(* CODESYS project 20260622.project

Project tree, tasks and I/O mapping:
  Device : AM522-0808TP/TN, Shenzhen Inovance Control Technology, version 3.5.11.50
      settings: PersistentStartAdddr = 0; PersistentStartEndAddr = 524287; Mode = 1; OPC UA Mode = 0
    application Application
      libraries: Standard, * (System); CmpEventMgr, 3.5.8.0 (System); Component Manager, 3.5.9.0 (System); CmpApp, 3.5.11.0 (System); CmpIecTask, 3.5.9.0 (System); SM3_Math, 4.10.0.0 (3S - Smart Software Solutions GmbH); SM3_Math, 4.10.0.0 (3S - Smart Software Solutions GmbH); HC_OmronUtils, 1.5.8.0 (Inovance); SM3_Basic, 4.10.13.1 (3S - Smart Software Solutions GmbH)
      task MainTask (cyclic, interval 10 ms, priority 1) calls PLC_MainPRG
      task ETHERCAT1 (cyclic, interval 4000 µs, priority 0) calls ETHERCAT1.EtherCAT_Task, PLC_Servo_伺服, PLC_HandWheel_手轮, PLC_CNC
      50_action/
        program PLC_Pump_泵管理 [ST]
        program PhotoScrape_L2 [ST]: A10_init_初始化, A32_cam_定位, A35_cam_回零, A34_cam_相机位, A33_cam_下压, A31_cam_移轴335, A40_scrape_刮取, A52_取料停旋转, A51_取料松压, A41_scrape_收尾
        program FeedLift_L2 [ST]: A11_feed_raise, A22_unload_bury, A12_feed_lower, A21_unload_ready
        program Sampling_L2 [ST]: A50_absorb_吸收液体, A31_放板移轴, A40_prep_上样准备, A32_放板定位, A20_clean_清洗, A10_init_初始化, A60_spray_点样, A61_喷涂移轴
        program Collect_L2 [ST]: A23_缩回升降下压, A22_伸缩伸出, A21_夹持夹紧, A30_collect_收集, A10_init_初始化, A42_伸缩缩回, A41_复位伸出, A43_松夹持
        program Rail_Sync [ST]
        program Rail_L2 [ST]
        program Develop_L2 [ST]: A31_放板缸回原点, A21_rinse_润洗展缸, A20_pipeline_清洗管路, A32_放板缸到动点, A22_up_liquid_上液, A10_init_初始化, A26_rinse_suction
        program Pump_L2 [ST]: A10_vacuum_on, A20_vacuum_off
      DifferentialMonitor
      25_FB_功能块/
        function block FB_Teach [ST]
        function block FB_SERVOAXIS [ST]
        function block FB_cylinder [ST]
        function block FB_HandWheel [ST]
        function block FB_RB_Control [ST]
        function block FB_Mode [ST]
      10_数据结构/
        data type HMI_Servo
        data type servo
        data type EN_功能块状态
      Symbols
      30_Ethercat任务/
        program PLC_Servo_伺服 [ST]: 伺服一键回原点, 伺服调用, 位置示教
        program PLC_CNC [CFC]
        program PLC_HandWheel_手轮 [ST]
      global variables PersistentVars
      20_变量Date/
        global variables HMI_Date
        global variables cyinder_date
        global variables IO
        global variables servoaxisdate
        global variables GVL
        global variables Host_Computer
        global variables RB_Date
      trace Trace (task ETHERCAT1): 玻璃上料轴1ZDATE.fActPos, 玻璃上料轴1ZDATE.fActVel
      CNC设置
      TaskEventPreStart
      text CNC_1
      40_Man/
        program Expand_process_展开流程 [ST]: Develop_L2_Dispatch, A00_initialization_初始化, A10_pipeline_cleaning_清洗管路, A20_clean_expand_润洗展缸, A40_up_liquid_上液, A30_silica_gel_plate_放硅胶板
        program Robotic_Process_机器人流程 [ST]: A30_取展缸硅胶板, A60_取收集器放暂存工位, A00_取放工具, A35_放拍照硅胶板, A65_放废料硅胶板, A41_取收集瓶组放暂存工位, A40_取收集器组放暂存工位, A15_放点样硅胶板, A55_取刮板收集器放到收集工位, A45_取暂存收集器放刮板位, A20_取点样硅胶板, A25_放展缸硅胶板, A50_取暂存收集瓶放收集工位, A71_取暂存收集瓶放仓库, A65_取收集瓶放暂存工位, A10_取升降机硅胶板, A70_取暂存收集器组放仓库, A32_取拍照硅胶板
        program Sample_point_sampling_上样点样 [ST]: A20_Place_materials_放硅胶板, A30_Sample_preparation_上样准备, A00_initialization_初始化, A50_Spray_sample_点样, A40_absorb_liquid_吸收液体, Sampling_L2_Dispatch, A10_clean_清洗
        program Collection_process_收集流程 [ST]: A20_collect_收集, A00_initialization_初始化, Collect_L2_Dispatch, A30_transport_物料搬运, A10_preparation_准备
        program PLC_MainPRG [ST]: A10_上下料伺服流程, A00_设备状态显示及控制, A20_机器人, A30_急停
        program initialization [ST]
        program Develop_TankDrain [ST]: A50_Expand_liquid_discharge_排液
        program Photo_scraper_拍照刮板 [ST]: A00_initialization_初始化, A10_Material_camera_拍照硅胶板, PhotoScrape_L2_Dispatch, A20_Scraper_collection_刮板收集, A30_Robot_material_retrieval_机器人取粉末收集器
        program PLC_Cyinder_气缸动作 [ST]
    ConfigStorage
    Network Configuration
      EtherCAT Config
      LocalBus Config
    Resources List
    HardWare Configuration
    Device Diagnosis
    EXP_A : 扩展卡, 汇川技术股份有限公司, version 00.00.00.10
    LocalHSIO : 本地高速IO, 汇川技术股份有限公司, version 2.0.0.0
        unmapped channels: %IB0 DigitalInput, DigitalOutput
      Counter0 : 高速计数器, 汇川技术股份有限公司, version 1.0.0.0
          settings: GeneralConfiguration.Value = 25; SignalSource.Value = 3; ResetPin.Value = 138; PresetPin.Value = 14; PositionComparePin.Value = 2; TouchProbePin1.Value = 10; TouchProbePin2.Value = 12
          unmapped channels: Statusword, Counter Value, Preset Status, Compare Status, Touch Probe Status1, Touch Probe Status2, Latch rising pos1, Latch rising pos2, Latch falling pos1, Latch falling pos2, Latch rising time1 low, Latch rising time1 high, Latch rising time2 low, Latch rising time2 high, Latch falling time1 low, Latch falling time1 high, Latch falling time2 low, Latch falling time2 high, Current frequency, ErrorCode, Controlword, Preset Value, Preset command, Compare Mode, Compare Parameter, Compare Value, Output Type, Output Parameter, Compare command, Touch probe command1, Touch probe command2
        Encoder : 编码器, 汇川技术股份有限公司, version 1.0.0.0
            settings: wDriveID = 0; 5050 = 10; Units = 1; LogicId = 0; AdrOffset_8010 = 64; BitOffset_8010 = 0; BitLength_8010 = 16; Address_ = '%QW32'; TYPE_ = 'WORD'; Address_Pointer = ADR(%QW32); AdrOffset_8020 = 72; BitOffset_8020 = 0; BitLength_8020 = 16; Address_ = '%QW36'; TYPE_ = 'WORD'; Address_Pointer = ADR(%QW36); AdrOffset_8030 = 68; BitOffset_8030 = 0; BitLength_8030 = 32; Address_ = '%QD17'; TYPE_ = 'DWORD'; Address_Pointer = ADR(%QD17); AdrOffset_8040 = 88; BitOffset_8040 = 0; BitLength_8040 = 16; Address_ = '%QW44'; TYPE_ = 'WORD'; Address_Pointer = ADR(%QW44); AdrOffset_8050 = 74; BitOffset_8050 = 0; BitLength_8050 = 16; Address_ = '%QW37'; TYPE_ = 'WORD'; Address_Pointer = ADR(%QW37); AdrOffset_8060 = 76; BitOffset_8060 = 0; BitLength_8060 = 32; Address_ = '%QD19'; TYPE_ = 'DWORD'; Address_Pointer = ADR(%QD19);
              AdrOffset_8070 = 80; BitOffset_8070 = 0; BitLength_8070 = 32; Address_ = '%QD20'; TYPE_ = 'DWORD'; Address_Pointer = ADR(%QD20); AdrOffset_8080 = 84; BitOffset_8080 = 0; BitLength_8080 = 16; Address_ = '%QW42'; TYPE_ = 'WORD'; Address_Pointer = ADR(%QW42); AdrOffset_8090 = 86; BitOffset_8090 = 0; BitLength_8090 = 16; Address_ = '%QW43'; TYPE_ = 'WORD'; Address_Pointer = ADR(%QW43); AdrOffset_8100 = 90; BitOffset_8100 = 0; BitLength_8100 = 16; Address_ = '%QW45'; TYPE_ = 'WORD'; Address_Pointer = ADR(%QW45); AdrOffset_8110 = 92; BitOffset_8110 = 0; BitLength_8110 = 16; Address_ = '%QW46'; TYPE_ = 'WORD'; Address_Pointer = ADR(%QW46); AdrOffset_8510 = 104; BitOffset_8510 = 0; BitLength_8510 = 16; Address_ = '%IW52'; TYPE_ = 'WORD'; Address_Pointer = ADR(%IW52); AdrOffset_8520 = 108; BitOffset_8520 = 0; BitLength_8520 = 32; Address_ = '%ID27';
              TYPE_ = 'DWORD'; Address_Pointer = ADR(%ID27); AdrOffset_8530 = 112; BitOffset_8530 = 0; BitLength_8530 = 16; Address_ = '%IW56'; TYPE_ = 'WORD'; Address_Pointer = ADR(%IW56); AdrOffset_8540 = 114; BitOffset_8540 = 0; BitLength_8540 = 16; Address_ = '%IW57'; TYPE_ = 'WORD'; Address_Pointer = ADR(%IW57); AdrOffset_8550 = 116; BitOffset_8550 = 0; BitLength_8550 = 16; Address_ = '%IW58'; TYPE_ = 'WORD'; Address_Pointer = ADR(%IW58); AdrOffset_8560 = 118; BitOffset_8560 = 0; BitLength_8560 = 16; Address_ = '%IW59'; TYPE_ = 'WORD'; Address_Pointer = ADR(%IW59); AdrOffset_8570 = 120; BitOffset_8570 = 0; BitLength_8570 = 32; Address_ = '%ID30'; TYPE_ = 'DWORD'; Address_Pointer = ADR(%ID30); AdrOffset_8580 = 124; BitOffset_8580 = 0; BitLength_8580 = 32; Address_ = '%ID31'; TYPE_ = 'DWORD'; Address_Pointer = ADR(%ID31); AdrOffset_8590 = 128; BitOffset_8590 = 0;
              BitLength_8590 = 32; Address_ = '%ID32'; TYPE_ = 'DWORD'; Address_Pointer = ADR(%ID32); AdrOffset_8600 = 132; BitOffset_8600 = 0; BitLength_8600 = 32; Address_ = '%ID33'; TYPE_ = 'DWORD'; Address_Pointer = ADR(%ID33); AdrOffset_8610 = 136; BitOffset_8610 = 0; BitLength_8610 = 32; Address_ = '%ID34'; TYPE_ = 'DWORD'; Address_Pointer = ADR(%ID34); AdrOffset_8620 = 140; BitOffset_8620 = 0; BitLength_8620 = 32; Address_ = '%ID35'; TYPE_ = 'DWORD'; Address_Pointer = ADR(%ID35); AdrOffset_8630 = 144; BitOffset_8630 = 0; BitLength_8630 = 32; Address_ = '%ID36'; TYPE_ = 'DWORD'; Address_Pointer = ADR(%ID36); AdrOffset_8640 = 148; BitOffset_8640 = 0; BitLength_8640 = 32; Address_ = '%ID37'; TYPE_ = 'DWORD'; Address_Pointer = ADR(%ID37); AdrOffset_8650 = 152; BitOffset_8650 = 0; BitLength_8650 = 32; Address_ = '%ID38'; TYPE_ = 'DWORD'; Address_Pointer = ADR(%ID38);
              AdrOffset_8660 = 156; BitOffset_8660 = 0; BitLength_8660 = 32; Address_ = '%ID39'; TYPE_ = 'DWORD'; Address_Pointer = ADR(%ID39); AdrOffset_8670 = 160; BitOffset_8670 = 0; BitLength_8670 = 32; Address_ = '%ID40'; TYPE_ = 'DWORD'; Address_Pointer = ADR(%ID40); AdrOffset_8680 = 164; BitOffset_8680 = 0; BitLength_8680 = 32; Address_ = '%ID41'; TYPE_ = 'DWORD'; Address_Pointer = ADR(%ID41); AdrOffset_8690 = 168; BitOffset_8690 = 0; BitLength_8690 = 32; Address_ = '%ID42'; TYPE_ = 'DWORD'; Address_Pointer = ADR(%ID42); AdrOffset_8700 = 172; BitOffset_8700 = 0; BitLength_8700 = 32; Address_ = '%ID43'; TYPE_ = 'DWORD'; Address_Pointer = ADR(%ID43)
    Serial : 串行接口, 汇川技术股份有限公司, version 00.00.00.10
      COM : Serial Port, Inovance, version 00.00.00.10
          settings: Device = AM522-0808TP/TN; devGuid = 'ea0913c2-01c3-4246-ae88-1c6b39cb02f1'
        串口自由协议 : 串口自由协议, inovance, version 00.00.00.10
            settings: Vendor.parameterset.Bit7 = FALSE; slave device set.RxCount = 1000; slave device set.RxAddrNum = 1001; slave device set.TxCount = 1300; slave device set.TxAddrNum = 1301
    EXP_B : 扩展卡, 汇川技术股份有限公司, version 00.00.00.10
    MODBUS_TCP_1 : ModbusTCP主站, inovance, version 00.00.00.10
        settings:  = 0
      modbusTcp : ModbusTCP Slave, Inovance, version 00.00.00.10 (disabled)
          settings: UseDec = True; ModbusTcpSlave.ChannelNum = 4; ModbusTcpSlave.EnableSlaveVariable = 3001; ModbusTcpSlave.IpAddr = 251701440; channel.PremeterSet.Bit2 = TRUE; channel.PremeterSet.Bit3 = TRUE; channel.PremeterSet.Bit4 = TRUE; channel.CycleTimes = 200; channel.ReadRegOffSet = 0; channel.WriteRegOffSet = 3100; channel.WriteRegLeg = 13; channel.IOChannel = 0; channel.ResendCount = 5; channel.ChannelName = 'write'; channel.ChannelNote = ''; channel.PremeterSet.Bit3 = TRUE; channel.CycleTimes = 200; channel.ReadRegOffSet = 3200; channel.ReadRegLeg = 13; channel.WriteRegOffSet = 0; channel.ResendCount = 5; channel.ChannelName = 'read'; channel.ChannelNote = ''; channel.PremeterSet.Bit2 = TRUE; channel.CycleTimes = 200; channel.ReadRegOffSet = 0; channel.ReadRegLeg = 12; channel.WriteRegOffSet = 0; channel.IOChannel = 2; channel.ResendCount = 5; channel.ChannelName = 'read_bool'; channel.ChannelNote = ''; channel.PremeterSet.Bit3 = TRUE; channel.PremeterSet.Bit4 = TRUE; channel.CycleTimes = 200; channel.ReadRegOffSet = 0; channel.WriteRegOffSet = 0; channel.WriteRegLeg = 7; channel.IOChannel = 3; channel.ResendCount = 5;
            channel.ChannelName = 'write_bool'; channel.ChannelNote = ''
          input  Application.Status : WORD  // read.read
          input  Application.Point : WORD  // read.read
          input  Application.ErrorID : WORD  // read.read
          input  Application.RO_ParameterList1 : WORD  // read.read
          input  Application.RO_ParameterList2 : WORD  // read.read
          input  Application.RO_ParameterList3 : WORD  // read.read
          input  Application.RO_ParameterList4 : WORD  // read.read
          input  Application.RO_ParameterList5 : WORD  // read.read
          input  Application.RO_ParameterList6 : WORD  // read.read
          input  Application.RO_ParameterList7 : WORD  // read.read
          input  Application.RO_ParameterList8 : WORD  // read.read
          input  Application.RO_ParameterList9 : WORD  // read.read
          input  Application.RO_ParameterList10 : WORD  // read.read
          output Application.Execute : WORD  // write.write
          output Application.Reset : WORD  // write.write
          output Application.FunctionID : WORD  // write.write
          output Application.ParameterList1 : WORD  // write.write
          output Application.ParameterList2 : WORD  // write.write
          output Application.ParameterList3 : WORD  // write.write
          output Application.ParameterList4 : WORD  // write.write
          output Application.ParameterList5 : WORD  // write.write
          output Application.ParameterList6 : WORD  // write.write
          output Application.ParameterList7 : WORD  // write.write
          output Application.ParameterList8 : WORD  // write.write
          output Application.ParameterList9 : WORD  // write.write
          output Application.ParameterList10 : WORD  // write.write
          unmapped channels: read, read_bool, write, write_bool
    ETHERCAT1 : EtherCAT Master SoftMotion, 3S - Smart Software Solutions GmbH, version 3.5.11.10
        settings:  = 0; NetworkName = 'eth1'; SelectNetworkByName = TRUE; DisableTaskGeneration = True; SyncOffset = 50; SlaveArrayName = ADR(_EC1_Node)
      InoSV660N_3 : SV660_1Axis_00915, Inovance, order no. InoSV660N, version Revision=16#00010000
          settings: FunCodeList = H02;H02-01;; WriteValueList = H02-01_8194_2_1_UINT_RW;; Number of Outputs = 6; Number of Inputs = 10; Number of Infos about Outputs = 6; Number of Infos about Inputs = 10; Configuration address of the slave = 5; Sync.Length = 18; Sync.Length = 32; FMMU.Length = 18; FMMU.Length = 32; AutoUpdate = False; DC sync0 cycletime = 4000; DC sync1 cycletime = 4000; Number of SDO = 10; Homing method.Index = 16#6098; Homing method.Subindex = 16#00; Homing method.Value = 27; Homing method.Size = 8; Homing method.AbortIfError = FALSE; Homing method.JumpToLine = FALSE; Homing method.Line = 0; Homing method.CompleteAccess = FALSE; Actual Position Calculation Method.Index = 16#60E6; Actual Position Calculation Method.Subindex = 16#00; Actual Position Calculation Method.Value = 0; Actual Position Calculation Method.Size = 8; Actual Position Calculation Method.AbortIfError = FALSE; Actual Position Calculation Method.JumpToLine = FALSE; Actual Position Calculation Method.Line = 0; Actual Position Calculation Method.CompleteAccess = FALSE; Speed during search for switch.Index = 16#6099; Speed during search for switch.Subindex = 16#01; Speed during search for switch.Value = 83886080; Speed during search for switch.Size = 32; Speed during search for switch.AbortIfError = FALSE; Speed during search for switch.JumpToLine = FALSE; Speed during search for switch.Line = 0; Speed during search for switch.CompleteAccess = FALSE; Homing acceleration.Index = 16#609A;
            Homing acceleration.Subindex = 16#00; Homing acceleration.Value = 279620266; Homing acceleration.Size = 32; Homing acceleration.AbortIfError = FALSE; Homing acceleration.JumpToLine = FALSE; Homing acceleration.Line = 0; Homing acceleration.CompleteAccess = FALSE; Speed during search for zero.Index = 16#6099; Speed during search for zero.Subindex = 16#02; Speed during search for zero.Value = 33554432; Speed during search for zero.Size = 32; Speed during search for zero.AbortIfError = FALSE; Speed during search for zero.JumpToLine = FALSE; Speed during search for zero.Line = 0; Speed during search for zero.CompleteAccess = FALSE; Time of home searching.Index = 16#2005; Time of home searching.Subindex = 16#24; Time of home searching.Value = 50000; Time of home searching.Size = 16; Time of home searching.AbortIfError = FALSE; Time of home searching.JumpToLine = FALSE; Time of home searching.Line = 0; Time of home searching.CompleteAccess = FALSE; Positive torque limit value.Index = 16#60E0; Positive torque limit value.Subindex = 16#00; Positive torque limit value.Value = 3500; Positive torque limit value.Size = 16; Positive torque limit value.AbortIfError = FALSE; Positive torque limit value.JumpToLine = FALSE; Positive torque limit value.Line = 0; Positive torque limit value.CompleteAccess = FALSE; Negative torque limit value.Index = 16#60E1; Negative torque limit value.Subindex = 16#00; Negative torque limit value.Value = 3500; Negative torque limit value.Size = 16; Negative torque limit value.AbortIfError = FALSE; Negative torque limit value.JumpToLine = FALSE; Negative torque limit value.Line = 0; Negative torque limit value.CompleteAccess = FALSE; Max profile velocity.Index = 16#607F;
            Max profile velocity.Subindex = 16#00; Max profile velocity.Value = 167772160; Max profile velocity.Size = 32; Max profile velocity.AbortIfError = FALSE; Max profile velocity.JumpToLine = FALSE; Max profile velocity.Line = 0; Max profile velocity.CompleteAccess = FALSE; RxTxPdo.NumberofEntries = 6; RxTxPdo.Sm = 2; Controlword.Index = 16#6040; Controlword.SubIndex = 0; Controlword.Size = 16; Controlword.DependOnSlot = false; Controlword.DependOnSlotGroup = false; Target position.Index = 16#607A; Target position.SubIndex = 0; Target position.Size = 32; Target position.DependOnSlot = false; Target position.DependOnSlotGroup = false; Touch probe function.Index = 16#60B8; Touch probe function.SubIndex = 0; Touch probe function.Size = 16; Touch probe function.DependOnSlot = false; Touch probe function.DependOnSlotGroup = false; Physical outputs.Index = 16#60FE; Physical outputs.SubIndex = 1; Physical outputs.Size = 32; Physical outputs.DependOnSlot = false; Physical outputs.DependOnSlotGroup = false; Target velocity.Index = 16#60FF; Target velocity.SubIndex = 0; Target velocity.Size = 32; Target velocity.DependOnSlot = false; Target velocity.DependOnSlotGroup = false; Target torque.Index = 16#6071; Target torque.SubIndex = 0; Target torque.Size = 16; Target torque.DependOnSlot = false; Target torque.DependOnSlotGroup = false; RxTxPdo.Sm = -1;
            RxTxPdo.NumberofEntries = 10; RxTxPdo.Sm = 3; Error code.Index = 16#603F; Error code.SubIndex = 0; Error code.Size = 16; Error code.DependOnSlot = false; Error code.DependOnSlotGroup = false; Statusword.Index = 16#6041; Statusword.SubIndex = 0; Statusword.Size = 16; Statusword.DependOnSlot = false; Statusword.DependOnSlotGroup = false; Position actual value.Index = 16#6064; Position actual value.SubIndex = 0; Position actual value.Size = 32; Position actual value.DependOnSlot = false; Position actual value.DependOnSlotGroup = false; Torque actual value.Index = 16#6077; Torque actual value.SubIndex = 0; Torque actual value.Size = 16; Torque actual value.DependOnSlot = false; Torque actual value.DependOnSlotGroup = false; Following error actual value.Index = 16#60F4; Following error actual value.SubIndex = 0; Following error actual value.Size = 32; Following error actual value.DependOnSlot = false; Following error actual value.DependOnSlotGroup = false; Touch probe status.Index = 16#60B9; Touch probe status.SubIndex = 0; Touch probe status.Size = 16; Touch probe status.DependOnSlot = false; Touch probe status.DependOnSlotGroup = false; Touch probe pos1 pos value.Index = 16#60BA; Touch probe pos1 pos value.SubIndex = 0; Touch probe pos1 pos value.Size = 32; Touch probe pos1 pos value.DependOnSlot = false; Touch probe pos1 pos value.DependOnSlotGroup = false; Touch probe pos2 pos value.Index = 16#60BC; Touch probe pos2 pos value.SubIndex = 0; Touch probe pos2 pos value.Size = 32;
            Touch probe pos2 pos value.DependOnSlot = false; Touch probe pos2 pos value.DependOnSlotGroup = false; Digital inputs.Index = 16#60FD; Digital inputs.SubIndex = 0; Digital inputs.Size = 32; Digital inputs.DependOnSlot = false; Digital inputs.DependOnSlotGroup = false; Velocity actual value.Index = 16#606C; Velocity actual value.SubIndex = 0; Velocity actual value.Size = 32; Velocity actual value.DependOnSlot = false; Velocity actual value.DependOnSlotGroup = false; RxTxPdo.Sm = -1; Controlword.Name = 'Controlword'; Controlword.DataType = 'UINT'; Target position.Name = 'Target position'; Target position.DataType = 'DINT'; Touch probe function.Name = 'Touch probe function'; Touch probe function.DataType = 'UINT'; Physical outputs.Name = 'Physical outputs'; Physical outputs.DataType = 'UDINT'; Target velocity.Name = 'Target velocity'; Target velocity.DataType = 'DINT'; Target torque.Name = 'Target torque'; Target torque.DataType = 'INT'; Error code.Name = 'Error code'; Error code.DataType = 'UINT'; Statusword.Name = 'Statusword'; Statusword.DataType = 'UINT'; Position actual value.Name = 'Position actual value'; Position actual value.DataType = 'DINT'; Torque actual value.Name = 'Torque actual value'; Torque actual value.DataType = 'INT'; Following error actual value.Name = 'Following error actual value'; Following error actual value.DataType = 'DINT'; Touch probe status.Name = 'Touch probe status'; Touch probe status.DataType = 'UINT'; Touch probe pos1 pos value.Name = 'Touch probe pos1 pos value'; Touch probe pos1 pos value.DataType = 'DINT'; Touch probe pos2 pos value.Name = 'Touch probe pos2 pos value';
            Touch probe pos2 pos value.DataType = 'DINT'; Digital inputs.Name = 'Digital inputs'; Digital inputs.DataType = 'UDINT'; Velocity actual value.Name = 'Velocity actual value'; Velocity actual value.DataType = 'DINT'
          unmapped channels: Controlword, Target position, Touch probe function, Physical outputs, Target velocity, Target torque, Error code, Statusword, Position actual value, Torque actual value, Following error actual value, Touch probe status, Touch probe pos1 pos value, Touch probe pos2 pos value, Digital inputs, Velocity actual value
        点样轴6X : Axis, Inovance, order no. 0, version 1.0.0.0
            settings: wDriveID = 3; dwRatioTechUnitsDenom = 8388608; iRatioTechUnitsNum = 5; iEncoderType = 1; iAbsEncoderOption = 2; HomingMode = 10; ZeroSignal = 0; StartDirction = 1; EndDirection = 1; PosLimitMode = 0; NegLimitMode = 0; HomingVelocity = 10; HomingApproachVelocity = 2; HomingAcceleration = 100; HomingDeceleration = 100; HomingJerk = 0; HomeMaskDistance = 0; HomePositionOffset = 0; HomePushTime = 0; HomeCompensation = 0; HomeTimeout = 0; HomeCompensationVelocity = 1000; 4000 = 1; 4001 = 0; 4003 = true; 4004 = 27; 4005 = 0; 4006 = 50.0; 4007 = 166.666666; 4008 = 20.0; 4009 = 50000; 4010 = 3500; 4011 = 3500; 4012 = 100.000000; ScalingIncs = 16#800000; 6005 = 5; AdrOffset_8010 = 2072; BitOffset_8010 = 0; BitLength_8010 = 16; Address_8010 = '%QW1036';
              Type_8010 = 'UINT'; AddressPointer_8010 = ADR(%QW1036); AdrOffset_8020 = 2076; BitOffset_8020 = 0; BitLength_8020 = 32; Address_8020 = '%QD519'; Type_8020 = 'DINT'; AddressPointer_8020 = ADR(%QD519); AdrOffset_8030 = 2088; BitOffset_8030 = 0; BitLength_8030 = 32; Address_8030 = '%QD522'; Type_8030 = 'DINT'; AddressPointer_8030 = ADR(%QD522); AdrOffset_8040 = 2092; BitOffset_8040 = 0; BitLength_8040 = 16; Address_8040 = '%QW1046'; Type_8040 = 'INT'; AddressPointer_8040 = ADR(%QW1046); AdrOffset_8050 = 4294967295; BitOffset_8050 = 0; BitLength_8050 = 0; Address_8050 = ''; Type_8050 = ''; AddressPointer_8050 = 0; AdrOffset_8060 = 2080; BitOffset_8060 = 0; BitLength_8060 = 16; Address_8060 = '%QW1040'; Type_8060 = 'UINT'; AddressPointer_8060 = ADR(%QW1040); AdrOffset_8070 = 4294967295; BitOffset_8070 = 0; BitLength_8070 = 0; Address_8070 = ''; Type_8070 = ''; AddressPointer_8070 = 0; AdrOffset_8080 = 4294967295; BitOffset_8080 = 0;
              BitLength_8080 = 0; Address_8080 = ''; Type_8080 = ''; AddressPointer_8080 = 0; AdrOffset_8090 = 2084; BitOffset_8090 = 0; BitLength_8090 = 32; Address_8090 = '%QD521'; Type_8090 = 'UDINT'; AddressPointer_8090 = ADR(%QD521); AdrOffset_8100 = 4294967295; BitOffset_8100 = 0; BitLength_8100 = 0; Address_8100 = ''; Type_8100 = ''; AddressPointer_8100 = 0; AdrOffset_8510 = 2110; BitOffset_8510 = 0; BitLength_8510 = 16; Address_8510 = '%IW1055'; Type_8510 = 'UINT'; AddressPointer_8510 = ADR(%IW1055); AdrOffset_8520 = 2112; BitOffset_8520 = 0; BitLength_8520 = 32; Address_8520 = '%ID528'; Type_8520 = 'DINT'; AddressPointer_8520 = ADR(%ID528); AdrOffset_8530 = 2140; BitOffset_8530 = 0; BitLength_8530 = 32; Address_8530 = '%ID535'; Type_8530 = 'DINT'; AddressPointer_8530 = ADR(%ID535); AdrOffset_8540 = 2116; BitOffset_8540 = 0; BitLength_8540 = 16; Address_8540 = '%IW1058'; Type_8540 = 'INT'; AddressPointer_8540 = ADR(%IW1058);
              AdrOffset_8550 = 4294967295; BitOffset_8550 = 0; BitLength_8550 = 0; Address_8550 = ''; Type_8550 = ''; AddressPointer_8550 = 0; AdrOffset_8560 = 2136; BitOffset_8560 = 0; BitLength_8560 = 32; Address_8560 = '%ID534'; Type_8560 = 'UDINT'; AddressPointer_8560 = ADR(%ID534); AdrOffset_8570 = 2124; BitOffset_8570 = 0; BitLength_8570 = 16; Address_8570 = '%IW1062'; Type_8570 = 'UINT'; AddressPointer_8570 = ADR(%IW1062); AdrOffset_8580 = 2128; BitOffset_8580 = 0; BitLength_8580 = 32; Address_8580 = '%ID532'; Type_8580 = 'DINT'; AddressPointer_8580 = ADR(%ID532); AdrOffset_8590 = 4294967295; BitOffset_8590 = 0; BitLength_8590 = 0; Address_8590 = ''; Type_8590 = ''; AddressPointer_8590 = 0; AdrOffset_8600 = 2132; BitOffset_8600 = 0; BitLength_8600 = 32; Address_8600 = '%ID533'; Type_8600 = 'DINT'; AddressPointer_8600 = ADR(%ID533); AdrOffset_8600 = 4294967295; BitOffset_8600 = 0; BitLength_8600 = 0; Address_8610 = '';
              Type_8610 = ''; AddressPointer_8610 = 0; AdrOffset_8620 = 2108; BitOffset_8620 = 0; BitLength_8620 = 16; Address_8620 = '%IW1054'; Type_8620 = 'UINT'; AddressPointer_8620 = ADR(%IW1054); IsValid = True; AxisNumber = 4; IsHostHoming = False; PulseSelectIndex = 4; SERVO_MAX_ID = 167772160
      InoSV660N_6 : SV660_1Axis_00915, Inovance, order no. InoSV660N, version Revision=16#00010000
          settings: FunCodeList = H02;H02-01;H03;H03-03;H03-05;; WriteValueList = H02-01_8194_2_1_UINT_RW;H03-03_8195_4_1_UINT_RW;H03-05_8195_6_1_UINT_RW;; Number of Outputs = 6; Number of Inputs = 10; Number of Infos about Outputs = 6; Number of Infos about Inputs = 10; Configuration address of the slave = 8; Sync.Length = 18; Sync.Length = 32; FMMU.Length = 18; FMMU.Length = 32; AutoUpdate = False; DC sync0 cycletime = 4000; DC sync1 cycletime = 4000; Number of SDO = 10; Homing method.Index = 16#6098; Homing method.Subindex = 16#00; Homing method.Value = 27; Homing method.Size = 8; Homing method.AbortIfError = FALSE; Homing method.JumpToLine = FALSE; Homing method.Line = 0; Homing method.CompleteAccess = FALSE; Actual Position Calculation Method.Index = 16#60E6; Actual Position Calculation Method.Subindex = 16#00; Actual Position Calculation Method.Value = 0; Actual Position Calculation Method.Size = 8; Actual Position Calculation Method.AbortIfError = FALSE; Actual Position Calculation Method.JumpToLine = FALSE; Actual Position Calculation Method.Line = 0; Actual Position Calculation Method.CompleteAccess = FALSE; Speed during search for switch.Index = 16#6099; Speed during search for switch.Subindex = 16#01; Speed during search for switch.Value = 15534459; Speed during search for switch.Size = 32; Speed during search for switch.AbortIfError = FALSE; Speed during search for switch.JumpToLine = FALSE; Speed during search for switch.Line = 0; Speed during search for switch.CompleteAccess = FALSE; Homing acceleration.Index = 16#609A;
            Homing acceleration.Subindex = 16#00; Homing acceleration.Value = 51781531; Homing acceleration.Size = 32; Homing acceleration.AbortIfError = FALSE; Homing acceleration.JumpToLine = FALSE; Homing acceleration.Line = 0; Homing acceleration.CompleteAccess = FALSE; Speed during search for zero.Index = 16#6099; Speed during search for zero.Subindex = 16#02; Speed during search for zero.Value = 6213784; Speed during search for zero.Size = 32; Speed during search for zero.AbortIfError = FALSE; Speed during search for zero.JumpToLine = FALSE; Speed during search for zero.Line = 0; Speed during search for zero.CompleteAccess = FALSE; Time of home searching.Index = 16#2005; Time of home searching.Subindex = 16#24; Time of home searching.Value = 50000; Time of home searching.Size = 16; Time of home searching.AbortIfError = FALSE; Time of home searching.JumpToLine = FALSE; Time of home searching.Line = 0; Time of home searching.CompleteAccess = FALSE; Positive torque limit value.Index = 16#60E0; Positive torque limit value.Subindex = 16#00; Positive torque limit value.Value = 3500; Positive torque limit value.Size = 16; Positive torque limit value.AbortIfError = FALSE; Positive torque limit value.JumpToLine = FALSE; Positive torque limit value.Line = 0; Positive torque limit value.CompleteAccess = FALSE; Negative torque limit value.Index = 16#60E1; Negative torque limit value.Subindex = 16#00; Negative torque limit value.Value = 3500; Negative torque limit value.Size = 16; Negative torque limit value.AbortIfError = FALSE; Negative torque limit value.JumpToLine = FALSE; Negative torque limit value.Line = 0; Negative torque limit value.CompleteAccess = FALSE; Max profile velocity.Index = 16#607F;
            Max profile velocity.Subindex = 16#00; Max profile velocity.Value = 31068919; Max profile velocity.Size = 32; Max profile velocity.AbortIfError = FALSE; Max profile velocity.JumpToLine = FALSE; Max profile velocity.Line = 0; Max profile velocity.CompleteAccess = FALSE; RxTxPdo.NumberofEntries = 6; RxTxPdo.Sm = 2; Controlword.Index = 16#6040; Controlword.SubIndex = 0; Controlword.Size = 16; Controlword.DependOnSlot = false; Controlword.DependOnSlotGroup = false; Target position.Index = 16#607A; Target position.SubIndex = 0; Target position.Size = 32; Target position.DependOnSlot = false; Target position.DependOnSlotGroup = false; Touch probe function.Index = 16#60B8; Touch probe function.SubIndex = 0; Touch probe function.Size = 16; Touch probe function.DependOnSlot = false; Touch probe function.DependOnSlotGroup = false; Physical outputs.Index = 16#60FE; Physical outputs.SubIndex = 1; Physical outputs.Size = 32; Physical outputs.DependOnSlot = false; Physical outputs.DependOnSlotGroup = false; Target velocity.Index = 16#60FF; Target velocity.SubIndex = 0; Target velocity.Size = 32; Target velocity.DependOnSlot = false; Target velocity.DependOnSlotGroup = false; Target torque.Index = 16#6071; Target torque.SubIndex = 0; Target torque.Size = 16; Target torque.DependOnSlot = false; Target torque.DependOnSlotGroup = false; RxTxPdo.Sm = -1;
            RxTxPdo.NumberofEntries = 10; RxTxPdo.Sm = 3; Error code.Index = 16#603F; Error code.SubIndex = 0; Error code.Size = 16; Error code.DependOnSlot = false; Error code.DependOnSlotGroup = false; Statusword.Index = 16#6041; Statusword.SubIndex = 0; Statusword.Size = 16; Statusword.DependOnSlot = false; Statusword.DependOnSlotGroup = false; Position actual value.Index = 16#6064; Position actual value.SubIndex = 0; Position actual value.Size = 32; Position actual value.DependOnSlot = false; Position actual value.DependOnSlotGroup = false; Torque actual value.Index = 16#6077; Torque actual value.SubIndex = 0; Torque actual value.Size = 16; Torque actual value.DependOnSlot = false; Torque actual value.DependOnSlotGroup = false; Following error actual value.Index = 16#60F4; Following error actual value.SubIndex = 0; Following error actual value.Size = 32; Following error actual value.DependOnSlot = false; Following error actual value.DependOnSlotGroup = false; Touch probe status.Index = 16#60B9; Touch probe status.SubIndex = 0; Touch probe status.Size = 16; Touch probe status.DependOnSlot = false; Touch probe status.DependOnSlotGroup = false; Touch probe pos1 pos value.Index = 16#60BA; Touch probe pos1 pos value.SubIndex = 0; Touch probe pos1 pos value.Size = 32; Touch probe pos1 pos value.DependOnSlot = false; Touch probe pos1 pos value.DependOnSlotGroup = false; Touch probe pos2 pos value.Index = 16#60BC; Touch probe pos2 pos value.SubIndex = 0; Touch probe pos2 pos value.Size = 32;
            Touch probe pos2 pos value.DependOnSlot = false; Touch probe pos2 pos value.DependOnSlotGroup = false; Digital inputs.Index = 16#60FD; Digital inputs.SubIndex = 0; Digital inputs.Size = 32; Digital inputs.DependOnSlot = false; Digital inputs.DependOnSlotGroup = false; Velocity actual value.Index = 16#606C; Velocity actual value.SubIndex = 0; Velocity actual value.Size = 32; Velocity actual value.DependOnSlot = false; Velocity actual value.DependOnSlotGroup = false; RxTxPdo.Sm = -1; Controlword.Name = 'Controlword'; Controlword.DataType = 'UINT'; Target position.Name = 'Target position'; Target position.DataType = 'DINT'; Touch probe function.Name = 'Touch probe function'; Touch probe function.DataType = 'UINT'; Physical outputs.Name = 'Physical outputs'; Physical outputs.DataType = 'UDINT'; Target velocity.Name = 'Target velocity'; Target velocity.DataType = 'DINT'; Target torque.Name = 'Target torque'; Target torque.DataType = 'INT'; Error code.Name = 'Error code'; Error code.DataType = 'UINT'; Statusword.Name = 'Statusword'; Statusword.DataType = 'UINT'; Position actual value.Name = 'Position actual value'; Position actual value.DataType = 'DINT'; Torque actual value.Name = 'Torque actual value'; Torque actual value.DataType = 'INT'; Following error actual value.Name = 'Following error actual value'; Following error actual value.DataType = 'DINT'; Touch probe status.Name = 'Touch probe status'; Touch probe status.DataType = 'UINT'; Touch probe pos1 pos value.Name = 'Touch probe pos1 pos value'; Touch probe pos1 pos value.DataType = 'DINT'; Touch probe pos2 pos value.Name = 'Touch probe pos2 pos value';
            Touch probe pos2 pos value.DataType = 'DINT'; Digital inputs.Name = 'Digital inputs'; Digital inputs.DataType = 'UDINT'; Velocity actual value.Name = 'Velocity actual value'; Velocity actual value.DataType = 'DINT'
          unmapped channels: Controlword, Target position, Touch probe function, Physical outputs, Target velocity, Target torque, Error code, Statusword, Position actual value, Torque actual value, Following error actual value, Touch probe status, Touch probe pos1 pos value, Touch probe pos2 pos value, Digital inputs, Velocity actual value
        刮板轴9X : Axis, Inovance, order no. 0, version 1.0.0.0
            settings: wDriveID = 6; dwRatioTechUnitsDenom = 8388608; iRatioTechUnitsNum = 27; iEncoderType = 1; iAbsEncoderOption = 2; HomingMode = 10; ZeroSignal = 0; StartDirction = 1; EndDirection = 1; PosLimitMode = 0; NegLimitMode = 0; HomingVelocity = 10; HomingApproachVelocity = 2; HomingAcceleration = 100; HomingDeceleration = 100; HomingJerk = 0; HomeMaskDistance = 0; HomePositionOffset = 0; HomePushTime = 0; HomeCompensation = 0; HomeTimeout = 0; HomeCompensationVelocity = 1000; 4000 = 1; 4001 = 0; 4003 = true; 4004 = 27; 4005 = 0; 4006 = 50.0; 4007 = 166.666666; 4008 = 20.0; 4009 = 50000; 4010 = 3500; 4011 = 3500; 4012 = 100.000000; ScalingIncs = 16#800000; 6005 = 27; AdrOffset_8010 = 2144; BitOffset_8010 = 0; BitLength_8010 = 16; Address_8010 = '%QW1072';
              Type_8010 = 'UINT'; AddressPointer_8010 = ADR(%QW1072); AdrOffset_8020 = 2148; BitOffset_8020 = 0; BitLength_8020 = 32; Address_8020 = '%QD537'; Type_8020 = 'DINT'; AddressPointer_8020 = ADR(%QD537); AdrOffset_8030 = 2160; BitOffset_8030 = 0; BitLength_8030 = 32; Address_8030 = '%QD540'; Type_8030 = 'DINT'; AddressPointer_8030 = ADR(%QD540); AdrOffset_8040 = 2164; BitOffset_8040 = 0; BitLength_8040 = 16; Address_8040 = '%QW1082'; Type_8040 = 'INT'; AddressPointer_8040 = ADR(%QW1082); AdrOffset_8050 = 4294967295; BitOffset_8050 = 0; BitLength_8050 = 0; Address_8050 = ''; Type_8050 = ''; AddressPointer_8050 = 0; AdrOffset_8060 = 2152; BitOffset_8060 = 0; BitLength_8060 = 16; Address_8060 = '%QW1076'; Type_8060 = 'UINT'; AddressPointer_8060 = ADR(%QW1076); AdrOffset_8070 = 4294967295; BitOffset_8070 = 0; BitLength_8070 = 0; Address_8070 = ''; Type_8070 = ''; AddressPointer_8070 = 0; AdrOffset_8080 = 4294967295; BitOffset_8080 = 0;
              BitLength_8080 = 0; Address_8080 = ''; Type_8080 = ''; AddressPointer_8080 = 0; AdrOffset_8090 = 2156; BitOffset_8090 = 0; BitLength_8090 = 32; Address_8090 = '%QD539'; Type_8090 = 'UDINT'; AddressPointer_8090 = ADR(%QD539); AdrOffset_8100 = 4294967295; BitOffset_8100 = 0; BitLength_8100 = 0; Address_8100 = ''; Type_8100 = ''; AddressPointer_8100 = 0; AdrOffset_8510 = 2218; BitOffset_8510 = 0; BitLength_8510 = 16; Address_8510 = '%IW1109'; Type_8510 = 'UINT'; AddressPointer_8510 = ADR(%IW1109); AdrOffset_8520 = 2220; BitOffset_8520 = 0; BitLength_8520 = 32; Address_8520 = '%ID555'; Type_8520 = 'DINT'; AddressPointer_8520 = ADR(%ID555); AdrOffset_8530 = 2248; BitOffset_8530 = 0; BitLength_8530 = 32; Address_8530 = '%ID562'; Type_8530 = 'DINT'; AddressPointer_8530 = ADR(%ID562); AdrOffset_8540 = 2224; BitOffset_8540 = 0; BitLength_8540 = 16; Address_8540 = '%IW1112'; Type_8540 = 'INT'; AddressPointer_8540 = ADR(%IW1112);
              AdrOffset_8550 = 4294967295; BitOffset_8550 = 0; BitLength_8550 = 0; Address_8550 = ''; Type_8550 = ''; AddressPointer_8550 = 0; AdrOffset_8560 = 2244; BitOffset_8560 = 0; BitLength_8560 = 32; Address_8560 = '%ID561'; Type_8560 = 'UDINT'; AddressPointer_8560 = ADR(%ID561); AdrOffset_8570 = 2232; BitOffset_8570 = 0; BitLength_8570 = 16; Address_8570 = '%IW1116'; Type_8570 = 'UINT'; AddressPointer_8570 = ADR(%IW1116); AdrOffset_8580 = 2236; BitOffset_8580 = 0; BitLength_8580 = 32; Address_8580 = '%ID559'; Type_8580 = 'DINT'; AddressPointer_8580 = ADR(%ID559); AdrOffset_8590 = 4294967295; BitOffset_8590 = 0; BitLength_8590 = 0; Address_8590 = ''; Type_8590 = ''; AddressPointer_8590 = 0; AdrOffset_8600 = 2240; BitOffset_8600 = 0; BitLength_8600 = 32; Address_8600 = '%ID560'; Type_8600 = 'DINT'; AddressPointer_8600 = ADR(%ID560); AdrOffset_8600 = 4294967295; BitOffset_8600 = 0; BitLength_8600 = 0; Address_8610 = '';
              Type_8610 = ''; AddressPointer_8610 = 0; AdrOffset_8620 = 2216; BitOffset_8620 = 0; BitLength_8620 = 16; Address_8620 = '%IW1108'; Type_8620 = 'UINT'; AddressPointer_8620 = ADR(%IW1108); IsValid = True; AxisNumber = 7; IsHostHoming = False; PulseSelectIndex = 4; SERVO_MAX_ID = 31068919
      InoSV660N_2 : SV660_1Axis_00915, Inovance, order no. InoSV660N, version Revision=16#00010000
          settings: FunCodeList = H02;H02-01;H03;H03-03;H03-05;; WriteValueList = H02-01_8194_2_1_UINT_RW;H03-03_8195_4_1_UINT_RW;H03-05_8195_6_1_UINT_RW;; Number of Outputs = 6; Number of Inputs = 10; Number of Infos about Outputs = 6; Number of Infos about Inputs = 10; Configuration address of the slave = 4; Sync.Length = 18; Sync.Length = 32; FMMU.Length = 18; FMMU.Length = 32; AutoUpdate = False; DC sync0 cycletime = 4000; DC sync1 cycletime = 4000; Number of SDO = 10; Homing method.Index = 16#6098; Homing method.Subindex = 16#00; Homing method.Value = 26; Homing method.Size = 8; Homing method.AbortIfError = FALSE; Homing method.JumpToLine = FALSE; Homing method.Line = 0; Homing method.CompleteAccess = FALSE; Actual Position Calculation Method.Index = 16#60E6; Actual Position Calculation Method.Subindex = 16#00; Actual Position Calculation Method.Value = 0; Actual Position Calculation Method.Size = 8; Actual Position Calculation Method.AbortIfError = FALSE; Actual Position Calculation Method.JumpToLine = FALSE; Actual Position Calculation Method.Line = 0; Actual Position Calculation Method.CompleteAccess = FALSE; Speed during search for switch.Index = 16#6099; Speed during search for switch.Subindex = 16#01; Speed during search for switch.Value = 15534459; Speed during search for switch.Size = 32; Speed during search for switch.AbortIfError = FALSE; Speed during search for switch.JumpToLine = FALSE; Speed during search for switch.Line = 0; Speed during search for switch.CompleteAccess = FALSE; Homing acceleration.Index = 16#609A;
            Homing acceleration.Subindex = 16#00; Homing acceleration.Value = 51781531; Homing acceleration.Size = 32; Homing acceleration.AbortIfError = FALSE; Homing acceleration.JumpToLine = FALSE; Homing acceleration.Line = 0; Homing acceleration.CompleteAccess = FALSE; Speed during search for zero.Index = 16#6099; Speed during search for zero.Subindex = 16#02; Speed during search for zero.Value = 6213784; Speed during search for zero.Size = 32; Speed during search for zero.AbortIfError = FALSE; Speed during search for zero.JumpToLine = FALSE; Speed during search for zero.Line = 0; Speed during search for zero.CompleteAccess = FALSE; Time of home searching.Index = 16#2005; Time of home searching.Subindex = 16#24; Time of home searching.Value = 50000; Time of home searching.Size = 16; Time of home searching.AbortIfError = FALSE; Time of home searching.JumpToLine = FALSE; Time of home searching.Line = 0; Time of home searching.CompleteAccess = FALSE; Positive torque limit value.Index = 16#60E0; Positive torque limit value.Subindex = 16#00; Positive torque limit value.Value = 3500; Positive torque limit value.Size = 16; Positive torque limit value.AbortIfError = FALSE; Positive torque limit value.JumpToLine = FALSE; Positive torque limit value.Line = 0; Positive torque limit value.CompleteAccess = FALSE; Negative torque limit value.Index = 16#60E1; Negative torque limit value.Subindex = 16#00; Negative torque limit value.Value = 3500; Negative torque limit value.Size = 16; Negative torque limit value.AbortIfError = FALSE; Negative torque limit value.JumpToLine = FALSE; Negative torque limit value.Line = 0; Negative torque limit value.CompleteAccess = FALSE; Max profile velocity.Index = 16#607F;
            Max profile velocity.Subindex = 16#00; Max profile velocity.Value = 31068919; Max profile velocity.Size = 32; Max profile velocity.AbortIfError = FALSE; Max profile velocity.JumpToLine = FALSE; Max profile velocity.Line = 0; Max profile velocity.CompleteAccess = FALSE; RxTxPdo.NumberofEntries = 6; RxTxPdo.Sm = 2; Controlword.Index = 16#6040; Controlword.SubIndex = 0; Controlword.Size = 16; Controlword.DependOnSlot = false; Controlword.DependOnSlotGroup = false; Target position.Index = 16#607A; Target position.SubIndex = 0; Target position.Size = 32; Target position.DependOnSlot = false; Target position.DependOnSlotGroup = false; Touch probe function.Index = 16#60B8; Touch probe function.SubIndex = 0; Touch probe function.Size = 16; Touch probe function.DependOnSlot = false; Touch probe function.DependOnSlotGroup = false; Physical outputs.Index = 16#60FE; Physical outputs.SubIndex = 1; Physical outputs.Size = 32; Physical outputs.DependOnSlot = false; Physical outputs.DependOnSlotGroup = false; Target velocity.Index = 16#60FF; Target velocity.SubIndex = 0; Target velocity.Size = 32; Target velocity.DependOnSlot = false; Target velocity.DependOnSlotGroup = false; Target torque.Index = 16#6071; Target torque.SubIndex = 0; Target torque.Size = 16; Target torque.DependOnSlot = false; Target torque.DependOnSlotGroup = false; RxTxPdo.Sm = -1;
            RxTxPdo.NumberofEntries = 10; RxTxPdo.Sm = 3; Error code.Index = 16#603F; Error code.SubIndex = 0; Error code.Size = 16; Error code.DependOnSlot = false; Error code.DependOnSlotGroup = false; Statusword.Index = 16#6041; Statusword.SubIndex = 0; Statusword.Size = 16; Statusword.DependOnSlot = false; Statusword.DependOnSlotGroup = false; Position actual value.Index = 16#6064; Position actual value.SubIndex = 0; Position actual value.Size = 32; Position actual value.DependOnSlot = false; Position actual value.DependOnSlotGroup = false; Torque actual value.Index = 16#6077; Torque actual value.SubIndex = 0; Torque actual value.Size = 16; Torque actual value.DependOnSlot = false; Torque actual value.DependOnSlotGroup = false; Following error actual value.Index = 16#60F4; Following error actual value.SubIndex = 0; Following error actual value.Size = 32; Following error actual value.DependOnSlot = false; Following error actual value.DependOnSlotGroup = false; Touch probe status.Index = 16#60B9; Touch probe status.SubIndex = 0; Touch probe status.Size = 16; Touch probe status.DependOnSlot = false; Touch probe status.DependOnSlotGroup = false; Touch probe pos1 pos value.Index = 16#60BA; Touch probe pos1 pos value.SubIndex = 0; Touch probe pos1 pos value.Size = 32; Touch probe pos1 pos value.DependOnSlot = false; Touch probe pos1 pos value.DependOnSlotGroup = false; Touch probe pos2 pos value.Index = 16#60BC; Touch probe pos2 pos value.SubIndex = 0; Touch probe pos2 pos value.Size = 32;
            Touch probe pos2 pos value.DependOnSlot = false; Touch probe pos2 pos value.DependOnSlotGroup = false; Digital inputs.Index = 16#60FD; Digital inputs.SubIndex = 0; Digital inputs.Size = 32; Digital inputs.DependOnSlot = false; Digital inputs.DependOnSlotGroup = false; Velocity actual value.Index = 16#606C; Velocity actual value.SubIndex = 0; Velocity actual value.Size = 32; Velocity actual value.DependOnSlot = false; Velocity actual value.DependOnSlotGroup = false; RxTxPdo.Sm = -1; Controlword.Name = 'Controlword'; Controlword.DataType = 'UINT'; Target position.Name = 'Target position'; Target position.DataType = 'DINT'; Touch probe function.Name = 'Touch probe function'; Touch probe function.DataType = 'UINT'; Physical outputs.Name = 'Physical outputs'; Physical outputs.DataType = 'UDINT'; Target velocity.Name = 'Target velocity'; Target velocity.DataType = 'DINT'; Target torque.Name = 'Target torque'; Target torque.DataType = 'INT'; Error code.Name = 'Error code'; Error code.DataType = 'UINT'; Statusword.Name = 'Statusword'; Statusword.DataType = 'UINT'; Position actual value.Name = 'Position actual value'; Position actual value.DataType = 'DINT'; Torque actual value.Name = 'Torque actual value'; Torque actual value.DataType = 'INT'; Following error actual value.Name = 'Following error actual value'; Following error actual value.DataType = 'DINT'; Touch probe status.Name = 'Touch probe status'; Touch probe status.DataType = 'UINT'; Touch probe pos1 pos value.Name = 'Touch probe pos1 pos value'; Touch probe pos1 pos value.DataType = 'DINT'; Touch probe pos2 pos value.Name = 'Touch probe pos2 pos value';
            Touch probe pos2 pos value.DataType = 'DINT'; Digital inputs.Name = 'Digital inputs'; Digital inputs.DataType = 'UDINT'; Velocity actual value.Name = 'Velocity actual value'; Velocity actual value.DataType = 'DINT'
          unmapped channels: Controlword, Target position, Touch probe function, Physical outputs, Target velocity, Target torque, Error code, Statusword, Position actual value, Torque actual value, Following error actual value, Touch probe status, Touch probe pos1 pos value, Touch probe pos2 pos value, Digital inputs, Velocity actual value
        打样瓶上料轴3Y : Axis, Inovance, order no. 0, version 1.0.0.0
            settings: wDriveID = 2; dwRatioTechUnitsDenom = 8388608; iRatioTechUnitsNum = -27; iEncoderType = 1; iAbsEncoderOption = 2; HomingMode = 10; ZeroSignal = 0; StartDirction = 1; EndDirection = 1; PosLimitMode = 0; NegLimitMode = 0; HomingVelocity = 10; HomingApproachVelocity = 2; HomingAcceleration = 100; HomingDeceleration = 100; HomingJerk = 0; HomeMaskDistance = 0; HomePositionOffset = 0; HomePushTime = 0; HomeCompensation = 0; HomeTimeout = 0; HomeCompensationVelocity = 1000; 4000 = 1; 4001 = 0; 4003 = true; 4004 = 26; 4005 = 0; 4006 = 50.0; 4007 = 166.666666; 4008 = 20.0; 4009 = 50000; 4010 = 3500; 4011 = 3500; 4012 = 100.000000; ScalingIncs = 16#800000; InvertDirection = TRUE; 6005 = 27; AdrOffset_8010 = 2048; BitOffset_8010 = 0; BitLength_8010 = 16;
              Address_8010 = '%QW1024'; Type_8010 = 'UINT'; AddressPointer_8010 = ADR(%QW1024); AdrOffset_8020 = 2052; BitOffset_8020 = 0; BitLength_8020 = 32; Address_8020 = '%QD513'; Type_8020 = 'DINT'; AddressPointer_8020 = ADR(%QD513); AdrOffset_8030 = 2064; BitOffset_8030 = 0; BitLength_8030 = 32; Address_8030 = '%QD516'; Type_8030 = 'DINT'; AddressPointer_8030 = ADR(%QD516); AdrOffset_8040 = 2068; BitOffset_8040 = 0; BitLength_8040 = 16; Address_8040 = '%QW1034'; Type_8040 = 'INT'; AddressPointer_8040 = ADR(%QW1034); AdrOffset_8050 = 4294967295; BitOffset_8050 = 0; BitLength_8050 = 0; Address_8050 = ''; Type_8050 = ''; AddressPointer_8050 = 0; AdrOffset_8060 = 2056; BitOffset_8060 = 0; BitLength_8060 = 16; Address_8060 = '%QW1028'; Type_8060 = 'UINT'; AddressPointer_8060 = ADR(%QW1028); AdrOffset_8070 = 4294967295; BitOffset_8070 = 0; BitLength_8070 = 0; Address_8070 = ''; Type_8070 = ''; AddressPointer_8070 = 0; AdrOffset_8080 = 4294967295;
              BitOffset_8080 = 0; BitLength_8080 = 0; Address_8080 = ''; Type_8080 = ''; AddressPointer_8080 = 0; AdrOffset_8090 = 2060; BitOffset_8090 = 0; BitLength_8090 = 32; Address_8090 = '%QD515'; Type_8090 = 'UDINT'; AddressPointer_8090 = ADR(%QD515); AdrOffset_8100 = 4294967295; BitOffset_8100 = 0; BitLength_8100 = 0; Address_8100 = ''; Type_8100 = ''; AddressPointer_8100 = 0; AdrOffset_8510 = 2074; BitOffset_8510 = 0; BitLength_8510 = 16; Address_8510 = '%IW1037'; Type_8510 = 'UINT'; AddressPointer_8510 = ADR(%IW1037); AdrOffset_8520 = 2076; BitOffset_8520 = 0; BitLength_8520 = 32; Address_8520 = '%ID519'; Type_8520 = 'DINT'; AddressPointer_8520 = ADR(%ID519); AdrOffset_8530 = 2104; BitOffset_8530 = 0; BitLength_8530 = 32; Address_8530 = '%ID526'; Type_8530 = 'DINT'; AddressPointer_8530 = ADR(%ID526); AdrOffset_8540 = 2080; BitOffset_8540 = 0; BitLength_8540 = 16; Address_8540 = '%IW1040'; Type_8540 = 'INT';
              AddressPointer_8540 = ADR(%IW1040); AdrOffset_8550 = 4294967295; BitOffset_8550 = 0; BitLength_8550 = 0; Address_8550 = ''; Type_8550 = ''; AddressPointer_8550 = 0; AdrOffset_8560 = 2100; BitOffset_8560 = 0; BitLength_8560 = 32; Address_8560 = '%ID525'; Type_8560 = 'UDINT'; AddressPointer_8560 = ADR(%ID525); AdrOffset_8570 = 2088; BitOffset_8570 = 0; BitLength_8570 = 16; Address_8570 = '%IW1044'; Type_8570 = 'UINT'; AddressPointer_8570 = ADR(%IW1044); AdrOffset_8580 = 2092; BitOffset_8580 = 0; BitLength_8580 = 32; Address_8580 = '%ID523'; Type_8580 = 'DINT'; AddressPointer_8580 = ADR(%ID523); AdrOffset_8590 = 4294967295; BitOffset_8590 = 0; BitLength_8590 = 0; Address_8590 = ''; Type_8590 = ''; AddressPointer_8590 = 0; AdrOffset_8600 = 2096; BitOffset_8600 = 0; BitLength_8600 = 32; Address_8600 = '%ID524'; Type_8600 = 'DINT'; AddressPointer_8600 = ADR(%ID524); AdrOffset_8600 = 4294967295; BitOffset_8600 = 0; BitLength_8600 = 0;
              Address_8610 = ''; Type_8610 = ''; AddressPointer_8610 = 0; AdrOffset_8620 = 2072; BitOffset_8620 = 0; BitLength_8620 = 16; Address_8620 = '%IW1036'; Type_8620 = 'UINT'; AddressPointer_8620 = ADR(%IW1036); IsValid = True; AxisNumber = 3; IsHostHoming = False; PulseSelectIndex = 4; SERVO_MAX_ID = 31068919
      InoSV660N_7 : SV660_1Axis_00915, Inovance, order no. InoSV660N, version Revision=16#00010000
          settings: FunCodeList = H02;H02-01;H03;H03-03;H03-05;; WriteValueList = H02-01_8194_2_1_UINT_RW;H03-03_8195_4_1_UINT_RW;H03-05_8195_6_1_UINT_RW;; Number of Outputs = 6; Number of Inputs = 10; Number of Infos about Outputs = 6; Number of Infos about Inputs = 10; Configuration address of the slave = 9; Sync.Length = 18; Sync.Length = 32; FMMU.Length = 18; FMMU.Length = 32; AutoUpdate = False; DC sync0 cycletime = 4000; DC sync1 cycletime = 4000; Number of SDO = 10; Homing method.Index = 16#6098; Homing method.Subindex = 16#00; Homing method.Value = 26; Homing method.Size = 8; Homing method.AbortIfError = FALSE; Homing method.JumpToLine = FALSE; Homing method.Line = 0; Homing method.CompleteAccess = FALSE; Actual Position Calculation Method.Index = 16#60E6; Actual Position Calculation Method.Subindex = 16#00; Actual Position Calculation Method.Value = 0; Actual Position Calculation Method.Size = 8; Actual Position Calculation Method.AbortIfError = FALSE; Actual Position Calculation Method.JumpToLine = FALSE; Actual Position Calculation Method.Line = 0; Actual Position Calculation Method.CompleteAccess = FALSE; Speed during search for switch.Index = 16#6099; Speed during search for switch.Subindex = 16#01; Speed during search for switch.Value = 83886080; Speed during search for switch.Size = 32; Speed during search for switch.AbortIfError = FALSE; Speed during search for switch.JumpToLine = FALSE; Speed during search for switch.Line = 0; Speed during search for switch.CompleteAccess = FALSE; Homing acceleration.Index = 16#609A;
            Homing acceleration.Subindex = 16#00; Homing acceleration.Value = 279620266; Homing acceleration.Size = 32; Homing acceleration.AbortIfError = FALSE; Homing acceleration.JumpToLine = FALSE; Homing acceleration.Line = 0; Homing acceleration.CompleteAccess = FALSE; Speed during search for zero.Index = 16#6099; Speed during search for zero.Subindex = 16#02; Speed during search for zero.Value = 33554432; Speed during search for zero.Size = 32; Speed during search for zero.AbortIfError = FALSE; Speed during search for zero.JumpToLine = FALSE; Speed during search for zero.Line = 0; Speed during search for zero.CompleteAccess = FALSE; Time of home searching.Index = 16#2005; Time of home searching.Subindex = 16#24; Time of home searching.Value = 50000; Time of home searching.Size = 16; Time of home searching.AbortIfError = FALSE; Time of home searching.JumpToLine = FALSE; Time of home searching.Line = 0; Time of home searching.CompleteAccess = FALSE; Positive torque limit value.Index = 16#60E0; Positive torque limit value.Subindex = 16#00; Positive torque limit value.Value = 3500; Positive torque limit value.Size = 16; Positive torque limit value.AbortIfError = FALSE; Positive torque limit value.JumpToLine = FALSE; Positive torque limit value.Line = 0; Positive torque limit value.CompleteAccess = FALSE; Negative torque limit value.Index = 16#60E1; Negative torque limit value.Subindex = 16#00; Negative torque limit value.Value = 3500; Negative torque limit value.Size = 16; Negative torque limit value.AbortIfError = FALSE; Negative torque limit value.JumpToLine = FALSE; Negative torque limit value.Line = 0; Negative torque limit value.CompleteAccess = FALSE; Max profile velocity.Index = 16#607F;
            Max profile velocity.Subindex = 16#00; Max profile velocity.Value = 167772160; Max profile velocity.Size = 32; Max profile velocity.AbortIfError = FALSE; Max profile velocity.JumpToLine = FALSE; Max profile velocity.Line = 0; Max profile velocity.CompleteAccess = FALSE; RxTxPdo.NumberofEntries = 6; RxTxPdo.Sm = 2; Controlword.Index = 16#6040; Controlword.SubIndex = 0; Controlword.Size = 16; Controlword.DependOnSlot = false; Controlword.DependOnSlotGroup = false; Target position.Index = 16#607A; Target position.SubIndex = 0; Target position.Size = 32; Target position.DependOnSlot = false; Target position.DependOnSlotGroup = false; Touch probe function.Index = 16#60B8; Touch probe function.SubIndex = 0; Touch probe function.Size = 16; Touch probe function.DependOnSlot = false; Touch probe function.DependOnSlotGroup = false; Physical outputs.Index = 16#60FE; Physical outputs.SubIndex = 1; Physical outputs.Size = 32; Physical outputs.DependOnSlot = false; Physical outputs.DependOnSlotGroup = false; Target velocity.Index = 16#60FF; Target velocity.SubIndex = 0; Target velocity.Size = 32; Target velocity.DependOnSlot = false; Target velocity.DependOnSlotGroup = false; Target torque.Index = 16#6071; Target torque.SubIndex = 0; Target torque.Size = 16; Target torque.DependOnSlot = false; Target torque.DependOnSlotGroup = false; RxTxPdo.Sm = -1;
            RxTxPdo.NumberofEntries = 10; RxTxPdo.Sm = 3; Error code.Index = 16#603F; Error code.SubIndex = 0; Error code.Size = 16; Error code.DependOnSlot = false; Error code.DependOnSlotGroup = false; Statusword.Index = 16#6041; Statusword.SubIndex = 0; Statusword.Size = 16; Statusword.DependOnSlot = false; Statusword.DependOnSlotGroup = false; Position actual value.Index = 16#6064; Position actual value.SubIndex = 0; Position actual value.Size = 32; Position actual value.DependOnSlot = false; Position actual value.DependOnSlotGroup = false; Torque actual value.Index = 16#6077; Torque actual value.SubIndex = 0; Torque actual value.Size = 16; Torque actual value.DependOnSlot = false; Torque actual value.DependOnSlotGroup = false; Following error actual value.Index = 16#60F4; Following error actual value.SubIndex = 0; Following error actual value.Size = 32; Following error actual value.DependOnSlot = false; Following error actual value.DependOnSlotGroup = false; Touch probe status.Index = 16#60B9; Touch probe status.SubIndex = 0; Touch probe status.Size = 16; Touch probe status.DependOnSlot = false; Touch probe status.DependOnSlotGroup = false; Touch probe pos1 pos value.Index = 16#60BA; Touch probe pos1 pos value.SubIndex = 0; Touch probe pos1 pos value.Size = 32; Touch probe pos1 pos value.DependOnSlot = false; Touch probe pos1 pos value.DependOnSlotGroup = false; Touch probe pos2 pos value.Index = 16#60BC; Touch probe pos2 pos value.SubIndex = 0; Touch probe pos2 pos value.Size = 32;
            Touch probe pos2 pos value.DependOnSlot = false; Touch probe pos2 pos value.DependOnSlotGroup = false; Digital inputs.Index = 16#60FD; Digital inputs.SubIndex = 0; Digital inputs.Size = 32; Digital inputs.DependOnSlot = false; Digital inputs.DependOnSlotGroup = false; Velocity actual value.Index = 16#606C; Velocity actual value.SubIndex = 0; Velocity actual value.Size = 32; Velocity actual value.DependOnSlot = false; Velocity actual value.DependOnSlotGroup = false; RxTxPdo.Sm = -1; Controlword.Name = 'Controlword'; Controlword.DataType = 'UINT'; Target position.Name = 'Target position'; Target position.DataType = 'DINT'; Touch probe function.Name = 'Touch probe function'; Touch probe function.DataType = 'UINT'; Physical outputs.Name = 'Physical outputs'; Physical outputs.DataType = 'UDINT'; Target velocity.Name = 'Target velocity'; Target velocity.DataType = 'DINT'; Target torque.Name = 'Target torque'; Target torque.DataType = 'INT'; Error code.Name = 'Error code'; Error code.DataType = 'UINT'; Statusword.Name = 'Statusword'; Statusword.DataType = 'UINT'; Position actual value.Name = 'Position actual value'; Position actual value.DataType = 'DINT'; Torque actual value.Name = 'Torque actual value'; Torque actual value.DataType = 'INT'; Following error actual value.Name = 'Following error actual value'; Following error actual value.DataType = 'DINT'; Touch probe status.Name = 'Touch probe status'; Touch probe status.DataType = 'UINT'; Touch probe pos1 pos value.Name = 'Touch probe pos1 pos value'; Touch probe pos1 pos value.DataType = 'DINT'; Touch probe pos2 pos value.Name = 'Touch probe pos2 pos value';
            Touch probe pos2 pos value.DataType = 'DINT'; Digital inputs.Name = 'Digital inputs'; Digital inputs.DataType = 'UDINT'; Velocity actual value.Name = 'Velocity actual value'; Velocity actual value.DataType = 'DINT'
          unmapped channels: Controlword, Target position, Touch probe function, Physical outputs, Target velocity, Target torque, Error code, Statusword, Position actual value, Torque actual value, Following error actual value, Touch probe status, Touch probe pos1 pos value, Touch probe pos2 pos value, Digital inputs, Velocity actual value
        刮板轴10Z : Axis, Inovance, order no. 0, version 1.0.0.0
            settings: wDriveID = 7; dwRatioTechUnitsDenom = 8388608; iRatioTechUnitsNum = -5; iEncoderType = 1; iAbsEncoderOption = 2; HomingMode = 10; ZeroSignal = 0; StartDirction = 1; EndDirection = 1; PosLimitMode = 0; NegLimitMode = 0; HomingVelocity = 10; HomingApproachVelocity = 2; HomingAcceleration = 100; HomingDeceleration = 100; HomingJerk = 0; HomeMaskDistance = 0; HomePositionOffset = 0; HomePushTime = 0; HomeCompensation = 0; HomeTimeout = 0; HomeCompensationVelocity = 1000; 4000 = 1; 4001 = 0; 4003 = true; 4004 = 26; 4005 = 0; 4006 = 50.0; 4007 = 166.666666; 4008 = 20.0; 4009 = 50000; 4010 = 3500; 4011 = 3500; 4012 = 100.000000; ScalingIncs = 16#800000; InvertDirection = TRUE; 6005 = 5; AdrOffset_8010 = 2168; BitOffset_8010 = 0; BitLength_8010 = 16;
              Address_8010 = '%QW1084'; Type_8010 = 'UINT'; AddressPointer_8010 = ADR(%QW1084); AdrOffset_8020 = 2172; BitOffset_8020 = 0; BitLength_8020 = 32; Address_8020 = '%QD543'; Type_8020 = 'DINT'; AddressPointer_8020 = ADR(%QD543); AdrOffset_8030 = 2184; BitOffset_8030 = 0; BitLength_8030 = 32; Address_8030 = '%QD546'; Type_8030 = 'DINT'; AddressPointer_8030 = ADR(%QD546); AdrOffset_8040 = 2188; BitOffset_8040 = 0; BitLength_8040 = 16; Address_8040 = '%QW1094'; Type_8040 = 'INT'; AddressPointer_8040 = ADR(%QW1094); AdrOffset_8050 = 4294967295; BitOffset_8050 = 0; BitLength_8050 = 0; Address_8050 = ''; Type_8050 = ''; AddressPointer_8050 = 0; AdrOffset_8060 = 2176; BitOffset_8060 = 0; BitLength_8060 = 16; Address_8060 = '%QW1088'; Type_8060 = 'UINT'; AddressPointer_8060 = ADR(%QW1088); AdrOffset_8070 = 4294967295; BitOffset_8070 = 0; BitLength_8070 = 0; Address_8070 = ''; Type_8070 = ''; AddressPointer_8070 = 0; AdrOffset_8080 = 4294967295;
              BitOffset_8080 = 0; BitLength_8080 = 0; Address_8080 = ''; Type_8080 = ''; AddressPointer_8080 = 0; AdrOffset_8090 = 2180; BitOffset_8090 = 0; BitLength_8090 = 32; Address_8090 = '%QD545'; Type_8090 = 'UDINT'; AddressPointer_8090 = ADR(%QD545); AdrOffset_8100 = 4294967295; BitOffset_8100 = 0; BitLength_8100 = 0; Address_8100 = ''; Type_8100 = ''; AddressPointer_8100 = 0; AdrOffset_8510 = 2254; BitOffset_8510 = 0; BitLength_8510 = 16; Address_8510 = '%IW1127'; Type_8510 = 'UINT'; AddressPointer_8510 = ADR(%IW1127); AdrOffset_8520 = 2256; BitOffset_8520 = 0; BitLength_8520 = 32; Address_8520 = '%ID564'; Type_8520 = 'DINT'; AddressPointer_8520 = ADR(%ID564); AdrOffset_8530 = 2284; BitOffset_8530 = 0; BitLength_8530 = 32; Address_8530 = '%ID571'; Type_8530 = 'DINT'; AddressPointer_8530 = ADR(%ID571); AdrOffset_8540 = 2260; BitOffset_8540 = 0; BitLength_8540 = 16; Address_8540 = '%IW1130'; Type_8540 = 'INT';
              AddressPointer_8540 = ADR(%IW1130); AdrOffset_8550 = 4294967295; BitOffset_8550 = 0; BitLength_8550 = 0; Address_8550 = ''; Type_8550 = ''; AddressPointer_8550 = 0; AdrOffset_8560 = 2280; BitOffset_8560 = 0; BitLength_8560 = 32; Address_8560 = '%ID570'; Type_8560 = 'UDINT'; AddressPointer_8560 = ADR(%ID570); AdrOffset_8570 = 2268; BitOffset_8570 = 0; BitLength_8570 = 16; Address_8570 = '%IW1134'; Type_8570 = 'UINT'; AddressPointer_8570 = ADR(%IW1134); AdrOffset_8580 = 2272; BitOffset_8580 = 0; BitLength_8580 = 32; Address_8580 = '%ID568'; Type_8580 = 'DINT'; AddressPointer_8580 = ADR(%ID568); AdrOffset_8590 = 4294967295; BitOffset_8590 = 0; BitLength_8590 = 0; Address_8590 = ''; Type_8590 = ''; AddressPointer_8590 = 0; AdrOffset_8600 = 2276; BitOffset_8600 = 0; BitLength_8600 = 32; Address_8600 = '%ID569'; Type_8600 = 'DINT'; AddressPointer_8600 = ADR(%ID569); AdrOffset_8600 = 4294967295; BitOffset_8600 = 0; BitLength_8600 = 0;
              Address_8610 = ''; Type_8610 = ''; AddressPointer_8610 = 0; AdrOffset_8620 = 2252; BitOffset_8620 = 0; BitLength_8620 = 16; Address_8620 = '%IW1126'; Type_8620 = 'UINT'; AddressPointer_8620 = ADR(%IW1126); IsValid = True; AxisNumber = 8; IsHostHoming = False; PulseSelectIndex = 4; SERVO_MAX_ID = 167772160
      InoSV660N : SV660_1Axis_00915, Inovance, order no. InoSV660N, version Revision=16#00010000
          settings: WriteValueList = H02-01_8194_2_1_UINT_RW;H03-03_8195_4_1_UINT_RW;H03-05_8195_6_1_UINT_RW;; Number of Outputs = 6; Number of Inputs = 10; Number of Infos about Outputs = 6; Number of Infos about Inputs = 10; StationAlias = 1002; Optional = False; DeviceIdenticationADO = 0; DeviceIdenticationMode = 0; Configuration address of the slave = 2; Sync.Length = 18; Sync.Length = 32; FMMU.Length = 18; FMMU.Length = 32; AutoUpdate = False; DC sync0 cycletime = 2000; DC sync0 cycletime = 4000000; DC sync1 cycletime = 2000; DC sync1 cycletime = 4000000; Number of SDO = 10; Homing method.Index = 16#6098; Homing method.Subindex = 16#00; Homing method.Value = 27; Homing method.Size = 8; Homing method.AbortIfError = FALSE; Homing method.JumpToLine = FALSE; Homing method.Line = 0; Homing method.CompleteAccess = FALSE; Actual Position Calculation Method.Index = 16#60E6; Actual Position Calculation Method.Subindex = 16#00; Actual Position Calculation Method.Value = 0; Actual Position Calculation Method.Size = 8; Actual Position Calculation Method.AbortIfError = FALSE; Actual Position Calculation Method.JumpToLine = FALSE; Actual Position Calculation Method.Line = 0; Actual Position Calculation Method.CompleteAccess = FALSE; Speed during search for switch.Index = 16#6099; Speed during search for switch.Subindex = 16#01; Speed during search for switch.Value = 83886080; Speed during search for switch.Size = 32;
            Speed during search for switch.AbortIfError = FALSE; Speed during search for switch.JumpToLine = FALSE; Speed during search for switch.Line = 0; Speed during search for switch.CompleteAccess = FALSE; Homing acceleration.Index = 16#609A; Homing acceleration.Subindex = 16#00; Homing acceleration.Value = 279620266; Homing acceleration.Size = 32; Homing acceleration.AbortIfError = FALSE; Homing acceleration.JumpToLine = FALSE; Homing acceleration.Line = 0; Homing acceleration.CompleteAccess = FALSE; Speed during search for zero.Index = 16#6099; Speed during search for zero.Subindex = 16#02; Speed during search for zero.Value = 33554432; Speed during search for zero.Size = 32; Speed during search for zero.AbortIfError = FALSE; Speed during search for zero.JumpToLine = FALSE; Speed during search for zero.Line = 0; Speed during search for zero.CompleteAccess = FALSE; Time of home searching.Index = 16#2005; Time of home searching.Subindex = 16#24; Time of home searching.Value = 50000; Time of home searching.Size = 16; Time of home searching.AbortIfError = FALSE; Time of home searching.JumpToLine = FALSE; Time of home searching.Line = 0; Time of home searching.CompleteAccess = FALSE; Positive torque limit value.Index = 16#60E0; Positive torque limit value.Subindex = 16#00; Positive torque limit value.Value = 3500; Positive torque limit value.Size = 16; Positive torque limit value.AbortIfError = FALSE; Positive torque limit value.JumpToLine = FALSE; Positive torque limit value.Line = 0; Positive torque limit value.CompleteAccess = FALSE; Negative torque limit value.Index = 16#60E1; Negative torque limit value.Subindex = 16#00; Negative torque limit value.Value = 3500; Negative torque limit value.Size = 16;
            Negative torque limit value.AbortIfError = FALSE; Negative torque limit value.JumpToLine = FALSE; Negative torque limit value.Line = 0; Negative torque limit value.CompleteAccess = FALSE; Max profile velocity.Index = 16#607F; Max profile velocity.Subindex = 16#00; Max profile velocity.Value = 167772160; Max profile velocity.Size = 32; Max profile velocity.AbortIfError = FALSE; Max profile velocity.JumpToLine = FALSE; Max profile velocity.Line = 0; Max profile velocity.CompleteAccess = FALSE; RxTxPdo.NumberofEntries = 6; RxTxPdo.Sm = 2; Controlword.Index = 16#6040; Controlword.SubIndex = 0; Controlword.Size = 16; Controlword.DependOnSlot = false; Controlword.DependOnSlotGroup = false; Target position.Index = 16#607A; Target position.SubIndex = 0; Target position.Size = 32; Target position.DependOnSlot = false; Target position.DependOnSlotGroup = false; Touch probe function.Index = 16#60B8; Touch probe function.SubIndex = 0; Touch probe function.Size = 16; Touch probe function.DependOnSlot = false; Touch probe function.DependOnSlotGroup = false; Physical outputs.Index = 16#60FE; Physical outputs.SubIndex = 1; Physical outputs.Size = 32; Physical outputs.DependOnSlot = false; Physical outputs.DependOnSlotGroup = false; Target velocity.Index = 16#60FF; Target velocity.SubIndex = 0; Target velocity.Size = 32; Target velocity.DependOnSlot = false; Target velocity.DependOnSlotGroup = false; Target torque.Index = 16#6071;
            Target torque.SubIndex = 0; Target torque.Size = 16; Target torque.DependOnSlot = false; Target torque.DependOnSlotGroup = false; RxTxPdo.Sm = -1; RxTxPdo.NumberofEntries = 10; RxTxPdo.Sm = 3; Error code.Index = 16#603F; Error code.SubIndex = 0; Error code.Size = 16; Error code.DependOnSlot = false; Error code.DependOnSlotGroup = false; Statusword.Index = 16#6041; Statusword.SubIndex = 0; Statusword.Size = 16; Statusword.DependOnSlot = false; Statusword.DependOnSlotGroup = false; Position actual value.Index = 16#6064; Position actual value.SubIndex = 0; Position actual value.Size = 32; Position actual value.DependOnSlot = false; Position actual value.DependOnSlotGroup = false; Torque actual value.Index = 16#6077; Torque actual value.SubIndex = 0; Torque actual value.Size = 16; Torque actual value.DependOnSlot = false; Torque actual value.DependOnSlotGroup = false; Following error actual value.Index = 16#60F4; Following error actual value.SubIndex = 0; Following error actual value.Size = 32; Following error actual value.DependOnSlot = false; Following error actual value.DependOnSlotGroup = false; Touch probe status.Index = 16#60B9; Touch probe status.SubIndex = 0; Touch probe status.Size = 16; Touch probe status.DependOnSlot = false; Touch probe status.DependOnSlotGroup = false; Touch probe pos1 pos value.Index = 16#60BA; Touch probe pos1 pos value.SubIndex = 0; Touch probe pos1 pos value.Size = 32;
            Touch probe pos1 pos value.DependOnSlot = false; Touch probe pos1 pos value.DependOnSlotGroup = false; Touch probe pos2 pos value.Index = 16#60BC; Touch probe pos2 pos value.SubIndex = 0; Touch probe pos2 pos value.Size = 32; Touch probe pos2 pos value.DependOnSlot = false; Touch probe pos2 pos value.DependOnSlotGroup = false; Digital inputs.Index = 16#60FD; Digital inputs.SubIndex = 0; Digital inputs.Size = 32; Digital inputs.DependOnSlot = false; Digital inputs.DependOnSlotGroup = false; Velocity actual value.Index = 16#606C; Velocity actual value.SubIndex = 0; Velocity actual value.Size = 32; Velocity actual value.DependOnSlot = false; Velocity actual value.DependOnSlotGroup = false; RxTxPdo.Sm = -1; Controlword.Name = 'Controlword'; Controlword.DataType = 'UINT'; Target position.Name = 'Target position'; Target position.DataType = 'DINT'; Touch probe function.Name = 'Touch probe function'; Touch probe function.DataType = 'UINT'; Physical outputs.Name = 'Physical outputs'; Physical outputs.DataType = 'UDINT'; Target velocity.Name = 'Target velocity'; Target velocity.DataType = 'DINT'; Target torque.Name = 'Target torque'; Target torque.DataType = 'INT'; Error code.Name = 'Error code'; Error code.DataType = 'UINT'; Statusword.Name = 'Statusword'; Statusword.DataType = 'UINT'; Position actual value.Name = 'Position actual value'; Position actual value.DataType = 'DINT'; Torque actual value.Name = 'Torque actual value'; Torque actual value.DataType = 'INT'; Following error actual value.Name = 'Following error actual value'; Following error actual value.DataType = 'DINT';
            Touch probe status.Name = 'Touch probe status'; Touch probe status.DataType = 'UINT'; Touch probe pos1 pos value.Name = 'Touch probe pos1 pos value'; Touch probe pos1 pos value.DataType = 'DINT'; Touch probe pos2 pos value.Name = 'Touch probe pos2 pos value'; Touch probe pos2 pos value.DataType = 'DINT'; Digital inputs.Name = 'Digital inputs'; Digital inputs.DataType = 'UDINT'; Velocity actual value.Name = 'Velocity actual value'; Velocity actual value.DataType = 'DINT'
          unmapped channels: %QW1000 Controlword, Target position, Touch probe function, Physical outputs, Target velocity, Target torque, %IW1000 Error code, Statusword, Position actual value, Torque actual value, Following error actual value, Touch probe status, Touch probe pos1 pos value, Touch probe pos2 pos value, Digital inputs, Velocity actual value
        玻璃上料轴1Z : Axis, Inovance, order no. 0, version 1.0.0.0
            settings: wDriveID = 0; dwRatioTechUnitsDenom = 8388608; iRatioTechUnitsNum = 5; iEncoderType = 1; iAbsEncoderOption = 2; HomingMode = 4; ZeroSignal = 0; StartDirction = -1; EndDirection = 1; PosLimitMode = 1; NegLimitMode = 1; HomingVelocity = 10; HomingApproachVelocity = 2; HomingAcceleration = 100; HomingDeceleration = 100; HomingJerk = 0; HomeMaskDistance = 0; HomePositionOffset = 0; HomePushTime = 0; HomeCompensation = 0; HomeTimeout = 0; HomeCompensationVelocity = 1000; 4000 = 1; 4001 = 0; 4003 = true; 4004 = 27; 4005 = 0; 4006 = 50.0; 4007 = 166.666666; 4008 = 20.0; 4009 = 50000; 4010 = 3500; 4011 = 3500; 4012 = 100.000000; ScalingIncs = 16#800000; 6005 = 5; AdrOffset_8010 = 2000; BitOffset_8010 = 0; BitLength_8010 = 16; Address_8010 = '%QW1000';
              Type_8010 = 'UINT'; AddressPointer_8010 = ADR(%QW1000); AdrOffset_8020 = 2004; BitOffset_8020 = 0; BitLength_8020 = 32; Address_8020 = '%QD501'; Type_8020 = 'DINT'; AddressPointer_8020 = ADR(%QD501); AdrOffset_8030 = 2016; BitOffset_8030 = 0; BitLength_8030 = 32; Address_8030 = '%QD504'; Type_8030 = 'DINT'; AddressPointer_8030 = ADR(%QD504); AdrOffset_8040 = 2020; BitOffset_8040 = 0; BitLength_8040 = 16; Address_8040 = '%QW1010'; Type_8040 = 'INT'; AddressPointer_8040 = ADR(%QW1010); AdrOffset_8050 = 4294967295; BitOffset_8050 = 0; BitLength_8050 = 0; Address_8050 = ''; Type_8050 = ''; AddressPointer_8050 = 0; AdrOffset_8060 = 2008; BitOffset_8060 = 0; BitLength_8060 = 16; Address_8060 = '%QW1004'; Type_8060 = 'UINT'; AddressPointer_8060 = ADR(%QW1004); AdrOffset_8070 = 4294967295; BitOffset_8070 = 0; BitLength_8070 = 0; Address_8070 = ''; Type_8070 = ''; AddressPointer_8070 = 0; AdrOffset_8080 = 4294967295; BitOffset_8080 = 0;
              BitLength_8080 = 0; Address_8080 = ''; Type_8080 = ''; AddressPointer_8080 = 0; AdrOffset_8090 = 2012; BitOffset_8090 = 0; BitLength_8090 = 32; Address_8090 = '%QD503'; Type_8090 = 'UDINT'; AddressPointer_8090 = ADR(%QD503); AdrOffset_8100 = 4294967295; BitOffset_8100 = 0; BitLength_8100 = 0; Address_8100 = ''; Type_8100 = ''; AddressPointer_8100 = 0; AdrOffset_8510 = 2002; BitOffset_8510 = 0; BitLength_8510 = 16; Address_8510 = '%IW1001'; Type_8510 = 'UINT'; AddressPointer_8510 = ADR(%IW1001); AdrOffset_8520 = 2004; BitOffset_8520 = 0; BitLength_8520 = 32; Address_8520 = '%ID501'; Type_8520 = 'DINT'; AddressPointer_8520 = ADR(%ID501); AdrOffset_8530 = 2032; BitOffset_8530 = 0; BitLength_8530 = 32; Address_8530 = '%ID508'; Type_8530 = 'DINT'; AddressPointer_8530 = ADR(%ID508); AdrOffset_8540 = 2008; BitOffset_8540 = 0; BitLength_8540 = 16; Address_8540 = '%IW1004'; Type_8540 = 'INT'; AddressPointer_8540 = ADR(%IW1004);
              AdrOffset_8550 = 4294967295; BitOffset_8550 = 0; BitLength_8550 = 0; Address_8550 = ''; Type_8550 = ''; AddressPointer_8550 = 0; AdrOffset_8560 = 2028; BitOffset_8560 = 0; BitLength_8560 = 32; Address_8560 = '%ID507'; Type_8560 = 'UDINT'; AddressPointer_8560 = ADR(%ID507); AdrOffset_8570 = 2016; BitOffset_8570 = 0; BitLength_8570 = 16; Address_8570 = '%IW1008'; Type_8570 = 'UINT'; AddressPointer_8570 = ADR(%IW1008); AdrOffset_8580 = 2020; BitOffset_8580 = 0; BitLength_8580 = 32; Address_8580 = '%ID505'; Type_8580 = 'DINT'; AddressPointer_8580 = ADR(%ID505); AdrOffset_8590 = 4294967295; BitOffset_8590 = 0; BitLength_8590 = 0; Address_8590 = ''; Type_8590 = ''; AddressPointer_8590 = 0; AdrOffset_8600 = 2024; BitOffset_8600 = 0; BitLength_8600 = 32; Address_8600 = '%ID506'; Type_8600 = 'DINT'; AddressPointer_8600 = ADR(%ID506); AdrOffset_8600 = 4294967295; BitOffset_8600 = 0; BitLength_8600 = 0; Address_8610 = '';
              Type_8610 = ''; AddressPointer_8610 = 0; AdrOffset_8620 = 2000; BitOffset_8620 = 0; BitLength_8620 = 16; Address_8620 = '%IW1000'; Type_8620 = 'UINT'; AddressPointer_8620 = ADR(%IW1000); IsValid = True; AxisNumber = 1; IsHostHoming = False; PulseSelectIndex = 4; SERVO_MAX_ID = 167772160
      CL3C_EC503_1 : CL3C-EC503(COE), Leadshine Technology Co.,Ltd., order no. CL3C-EC503, version Revision=16#00000001
          settings: Number of Outputs = 4; Number of Infos about Outputs = 4; Configuration address of the slave = 12; Sync.Length = 9; FMMU.Length = 9; AutoUpdate = False; DC sync0 cycletime = 4000; DC sync1 cycletime = 4000; RxTxPdo.NumberofEntries = 4; RxTxPdo.DependOnSlot = False; RxTxPdo.DependOnSlotGroup = False; RxTxPdo.OverwrittenByModule = False; Homing Method.Index = 16#6098; Homing Method.SubIndex = 0; Homing Method.Size = 8; Homing Method.Offset = 0; Homing Method.DependOnSlot = False; Homing Method.DependOnSlotGroup = False; Control Word.Index = 16#6040; Control Word.SubIndex = 0; Control Word.Size = 16; Control Word.Offset = 0; Control Word.DependOnSlot = False; Control Word.DependOnSlotGroup = False; Profile Target Position.Index = 16#607A; Profile Target Position.SubIndex = 0; Profile Target Position.Size = 32; Profile Target Position.Offset = 0; Profile Target Position.DependOnSlot = False; Profile Target Position.DependOnSlotGroup = False; Touch Probe Function.Index = 16#60B8; Touch Probe Function.SubIndex = 0; Touch Probe Function.Size = 16; Touch Probe Function.Offset = 0; Touch Probe Function.DependOnSlot = False; Touch Probe Function.DependOnSlotGroup = False; Homing Method.Name = 'Homing Method'; Homing Method.DataType = 'SINT'; Homing Method.Default = ''; Homing Method.Comment = '';
            Control Word.Name = 'Control Word'; Control Word.DataType = 'UINT'; Control Word.Default = ''; Control Word.Comment = ''; Profile Target Position.Name = 'Profile Target Position'; Profile Target Position.DataType = 'DINT'; Profile Target Position.Default = ''; Profile Target Position.Comment = ''; Touch Probe Function.Name = 'Touch Probe Function'; Touch Probe Function.DataType = 'UINT'; Touch Probe Function.Default = ''; Touch Probe Function.Comment = ''
          unmapped channels: Homing Method, Control Word, Profile Target Position, Touch Probe Function, Last Error Code, Status Word, Modes of Operation display, Position Actual Value, Touch Probe Status, Touch Probe 1 Positive Value, Digital Inputs
        上样轴5Z轴 : Axis, Inovance, order no. 0, version 4.0.0.0
            settings: wDriveID = 10; dwRatioTechUnitsDenom = 100; HomingMode = 4; ZeroSignal = 0; StartDirction = -1; EndDirection = -1; PosLimitMode = 1; NegLimitMode = 1; HomingVelocity = 10; HomingApproachVelocity = 2; HomingAcceleration = 100; HomingDeceleration = 100; HomingJerk = 0; HomeMaskDistance = 0; HomePositionOffset = 0; HomePushTime = 0; HomeCompensation = 0; HomeTimeout = 0; HomeCompensationVelocity = 1000; 4000 = 1; 4001 = 0; ScalingIncs = 7500; 6005 = 75; AdrOffset_8010 = 2230; BitOffset_8010 = 0; BitLength_8010 = 16; Address_8010 = '%QW1115'; Type_8010 = 'UINT'; AddressPointer_8010 = ADR(%QW1115); AdrOffset_8020 = 2232; BitOffset_8020 = 0; BitLength_8020 = 32; Address_8020 = '%QD558'; Type_8020 = 'DINT'; AddressPointer_8020 = ADR(%QD558); AdrOffset_8030 = 4294967295; BitOffset_8030 = 0; BitLength_8030 = 0; Address_8030 = ''; Type_8030 = '';
              AddressPointer_8030 = 0; AdrOffset_8040 = 4294967295; BitOffset_8040 = 0; BitLength_8040 = 0; Address_8040 = ''; Type_8040 = ''; AddressPointer_8040 = 0; AdrOffset_8050 = 4294967295; BitOffset_8050 = 0; BitLength_8050 = 0; Address_8050 = ''; Type_8050 = ''; AddressPointer_8050 = 0; AdrOffset_8060 = 2236; BitOffset_8060 = 0; BitLength_8060 = 16; Address_8060 = '%QW1118'; Type_8060 = 'UINT'; AddressPointer_8060 = ADR(%QW1118); AdrOffset_8070 = 4294967295; BitOffset_8070 = 0; BitLength_8070 = 0; Address_8070 = ''; Type_8070 = ''; AddressPointer_8070 = 0; AdrOffset_8080 = 4294967295; BitOffset_8080 = 0; BitLength_8080 = 0; Address_8080 = ''; Type_8080 = ''; AddressPointer_8080 = 0; AdrOffset_8090 = 4294967295; BitOffset_8090 = 0; BitLength_8090 = 0; Address_8090 = ''; Type_8090 = ''; AddressPointer_8090 = 0; AdrOffset_8100 = 4294967295; BitOffset_8100 = 0; BitLength_8100 = 0;
              Address_8100 = ''; Type_8100 = ''; AddressPointer_8100 = 0; AdrOffset_8510 = 2350; BitOffset_8510 = 0; BitLength_8510 = 16; Address_8510 = '%IW1175'; Type_8510 = 'UINT'; AddressPointer_8510 = ADR(%IW1175); AdrOffset_8520 = 2356; BitOffset_8520 = 0; BitLength_8520 = 32; Address_8520 = '%ID589'; Type_8520 = 'DINT'; AddressPointer_8520 = ADR(%ID589); AdrOffset_8530 = 4294967295; BitOffset_8530 = 0; BitLength_8530 = 0; Address_8530 = ''; Type_8530 = ''; AddressPointer_8530 = 0; AdrOffset_8540 = 4294967295; BitOffset_8540 = 0; BitLength_8540 = 0; Address_8540 = ''; Type_8540 = ''; AddressPointer_8540 = 0; AdrOffset_8550 = 2352; BitOffset_8550 = 0; BitLength_8550 = 8; Address_8550 = '%IB2352'; Type_8550 = 'SINT'; AddressPointer_8550 = ADR(%IB2352); AdrOffset_8560 = 2368; BitOffset_8560 = 0; BitLength_8560 = 32; Address_8560 = '%ID592'; Type_8560 = 'UDINT'; AddressPointer_8560 = ADR(%ID592); AdrOffset_8570 = 2360;
              BitOffset_8570 = 0; BitLength_8570 = 16; Address_8570 = '%IW1180'; Type_8570 = 'UINT'; AddressPointer_8570 = ADR(%IW1180); AdrOffset_8580 = 2364; BitOffset_8580 = 0; BitLength_8580 = 32; Address_8580 = '%ID591'; Type_8580 = 'DINT'; AddressPointer_8580 = ADR(%ID591); AdrOffset_8590 = 4294967295; BitOffset_8590 = 0; BitLength_8590 = 0; Address_8590 = ''; Type_8590 = ''; AddressPointer_8590 = 0; AdrOffset_8600 = 4294967295; BitOffset_8600 = 0; BitLength_8600 = 0; Address_8600 = ''; Type_8600 = ''; AddressPointer_8600 = 0; AdrOffset_8600 = 4294967295; BitOffset_8600 = 0; BitLength_8600 = 0; Address_8610 = ''; Type_8610 = ''; AddressPointer_8610 = 0; AdrOffset_8620 = 2348; BitOffset_8620 = 0; BitLength_8620 = 16; Address_8620 = '%IW1174'; Type_8620 = 'UINT'; AddressPointer_8620 = ADR(%IW1174); IsValid = True; AxisNumber = 11; IsHostHoming = True; PulseSelectIndex = 0
      InoSV660N_1 : SV660_1Axis_00915, Inovance, order no. InoSV660N, version Revision=16#00010000
          settings: FunCodeList = H02;H02-01;; WriteValueList = H02-01_8194_2_1_UINT_RW;; Number of Outputs = 6; Number of Inputs = 10; Number of Infos about Outputs = 6; Number of Infos about Inputs = 10; Configuration address of the slave = 3; Sync.Length = 18; Sync.Length = 32; FMMU.Length = 18; FMMU.Length = 32; AutoUpdate = False; DC sync0 cycletime = 4000; DC sync1 cycletime = 4000; Number of SDO = 10; Homing method.Index = 16#6098; Homing method.Subindex = 16#00; Homing method.Value = 27; Homing method.Size = 8; Homing method.AbortIfError = FALSE; Homing method.JumpToLine = FALSE; Homing method.Line = 0; Homing method.CompleteAccess = FALSE; Actual Position Calculation Method.Index = 16#60E6; Actual Position Calculation Method.Subindex = 16#00; Actual Position Calculation Method.Value = 0; Actual Position Calculation Method.Size = 8; Actual Position Calculation Method.AbortIfError = FALSE; Actual Position Calculation Method.JumpToLine = FALSE; Actual Position Calculation Method.Line = 0; Actual Position Calculation Method.CompleteAccess = FALSE; Speed during search for switch.Index = 16#6099; Speed during search for switch.Subindex = 16#01; Speed during search for switch.Value = 83886080; Speed during search for switch.Size = 32; Speed during search for switch.AbortIfError = FALSE; Speed during search for switch.JumpToLine = FALSE; Speed during search for switch.Line = 0; Speed during search for switch.CompleteAccess = FALSE; Homing acceleration.Index = 16#609A;
            Homing acceleration.Subindex = 16#00; Homing acceleration.Value = 279620266; Homing acceleration.Size = 32; Homing acceleration.AbortIfError = FALSE; Homing acceleration.JumpToLine = FALSE; Homing acceleration.Line = 0; Homing acceleration.CompleteAccess = FALSE; Speed during search for zero.Index = 16#6099; Speed during search for zero.Subindex = 16#02; Speed during search for zero.Value = 33554432; Speed during search for zero.Size = 32; Speed during search for zero.AbortIfError = FALSE; Speed during search for zero.JumpToLine = FALSE; Speed during search for zero.Line = 0; Speed during search for zero.CompleteAccess = FALSE; Time of home searching.Index = 16#2005; Time of home searching.Subindex = 16#24; Time of home searching.Value = 50000; Time of home searching.Size = 16; Time of home searching.AbortIfError = FALSE; Time of home searching.JumpToLine = FALSE; Time of home searching.Line = 0; Time of home searching.CompleteAccess = FALSE; Positive torque limit value.Index = 16#60E0; Positive torque limit value.Subindex = 16#00; Positive torque limit value.Value = 3500; Positive torque limit value.Size = 16; Positive torque limit value.AbortIfError = FALSE; Positive torque limit value.JumpToLine = FALSE; Positive torque limit value.Line = 0; Positive torque limit value.CompleteAccess = FALSE; Negative torque limit value.Index = 16#60E1; Negative torque limit value.Subindex = 16#00; Negative torque limit value.Value = 3500; Negative torque limit value.Size = 16; Negative torque limit value.AbortIfError = FALSE; Negative torque limit value.JumpToLine = FALSE; Negative torque limit value.Line = 0; Negative torque limit value.CompleteAccess = FALSE; Max profile velocity.Index = 16#607F;
            Max profile velocity.Subindex = 16#00; Max profile velocity.Value = 167772160; Max profile velocity.Size = 32; Max profile velocity.AbortIfError = FALSE; Max profile velocity.JumpToLine = FALSE; Max profile velocity.Line = 0; Max profile velocity.CompleteAccess = FALSE; RxTxPdo.NumberofEntries = 6; RxTxPdo.Sm = 2; Controlword.Index = 16#6040; Controlword.SubIndex = 0; Controlword.Size = 16; Controlword.DependOnSlot = false; Controlword.DependOnSlotGroup = false; Target position.Index = 16#607A; Target position.SubIndex = 0; Target position.Size = 32; Target position.DependOnSlot = false; Target position.DependOnSlotGroup = false; Touch probe function.Index = 16#60B8; Touch probe function.SubIndex = 0; Touch probe function.Size = 16; Touch probe function.DependOnSlot = false; Touch probe function.DependOnSlotGroup = false; Physical outputs.Index = 16#60FE; Physical outputs.SubIndex = 1; Physical outputs.Size = 32; Physical outputs.DependOnSlot = false; Physical outputs.DependOnSlotGroup = false; Target velocity.Index = 16#60FF; Target velocity.SubIndex = 0; Target velocity.Size = 32; Target velocity.DependOnSlot = false; Target velocity.DependOnSlotGroup = false; Target torque.Index = 16#6071; Target torque.SubIndex = 0; Target torque.Size = 16; Target torque.DependOnSlot = false; Target torque.DependOnSlotGroup = false; RxTxPdo.Sm = -1;
            RxTxPdo.NumberofEntries = 10; RxTxPdo.Sm = 3; Error code.Index = 16#603F; Error code.SubIndex = 0; Error code.Size = 16; Error code.DependOnSlot = false; Error code.DependOnSlotGroup = false; Statusword.Index = 16#6041; Statusword.SubIndex = 0; Statusword.Size = 16; Statusword.DependOnSlot = false; Statusword.DependOnSlotGroup = false; Position actual value.Index = 16#6064; Position actual value.SubIndex = 0; Position actual value.Size = 32; Position actual value.DependOnSlot = false; Position actual value.DependOnSlotGroup = false; Torque actual value.Index = 16#6077; Torque actual value.SubIndex = 0; Torque actual value.Size = 16; Torque actual value.DependOnSlot = false; Torque actual value.DependOnSlotGroup = false; Following error actual value.Index = 16#60F4; Following error actual value.SubIndex = 0; Following error actual value.Size = 32; Following error actual value.DependOnSlot = false; Following error actual value.DependOnSlotGroup = false; Touch probe status.Index = 16#60B9; Touch probe status.SubIndex = 0; Touch probe status.Size = 16; Touch probe status.DependOnSlot = false; Touch probe status.DependOnSlotGroup = false; Touch probe pos1 pos value.Index = 16#60BA; Touch probe pos1 pos value.SubIndex = 0; Touch probe pos1 pos value.Size = 32; Touch probe pos1 pos value.DependOnSlot = false; Touch probe pos1 pos value.DependOnSlotGroup = false; Touch probe pos2 pos value.Index = 16#60BC; Touch probe pos2 pos value.SubIndex = 0; Touch probe pos2 pos value.Size = 32;
            Touch probe pos2 pos value.DependOnSlot = false; Touch probe pos2 pos value.DependOnSlotGroup = false; Digital inputs.Index = 16#60FD; Digital inputs.SubIndex = 0; Digital inputs.Size = 32; Digital inputs.DependOnSlot = false; Digital inputs.DependOnSlotGroup = false; Velocity actual value.Index = 16#606C; Velocity actual value.SubIndex = 0; Velocity actual value.Size = 32; Velocity actual value.DependOnSlot = false; Velocity actual value.DependOnSlotGroup = false; RxTxPdo.Sm = -1; Controlword.Name = 'Controlword'; Controlword.DataType = 'UINT'; Target position.Name = 'Target position'; Target position.DataType = 'DINT'; Touch probe function.Name = 'Touch probe function'; Touch probe function.DataType = 'UINT'; Physical outputs.Name = 'Physical outputs'; Physical outputs.DataType = 'UDINT'; Target velocity.Name = 'Target velocity'; Target velocity.DataType = 'DINT'; Target torque.Name = 'Target torque'; Target torque.DataType = 'INT'; Error code.Name = 'Error code'; Error code.DataType = 'UINT'; Statusword.Name = 'Statusword'; Statusword.DataType = 'UINT'; Position actual value.Name = 'Position actual value'; Position actual value.DataType = 'DINT'; Torque actual value.Name = 'Torque actual value'; Torque actual value.DataType = 'INT'; Following error actual value.Name = 'Following error actual value'; Following error actual value.DataType = 'DINT'; Touch probe status.Name = 'Touch probe status'; Touch probe status.DataType = 'UINT'; Touch probe pos1 pos value.Name = 'Touch probe pos1 pos value'; Touch probe pos1 pos value.DataType = 'DINT'; Touch probe pos2 pos value.Name = 'Touch probe pos2 pos value';
            Touch probe pos2 pos value.DataType = 'DINT'; Digital inputs.Name = 'Digital inputs'; Digital inputs.DataType = 'UDINT'; Velocity actual value.Name = 'Velocity actual value'; Velocity actual value.DataType = 'DINT'
          unmapped channels: Controlword, Target position, Touch probe function, Physical outputs, Target velocity, Target torque, Error code, Statusword, Position actual value, Torque actual value, Following error actual value, Touch probe status, Touch probe pos1 pos value, Touch probe pos2 pos value, Digital inputs, Velocity actual value
        玻璃上料轴2Z : Axis, Inovance, order no. 0, version 1.0.0.0
            settings: dwRatioTechUnitsDenom = 8388608; iRatioTechUnitsNum = 5; iEncoderType = 1; iAbsEncoderOption = 2; HomingMode = 10; ZeroSignal = 0; StartDirction = 1; EndDirection = 1; PosLimitMode = 0; NegLimitMode = 0; HomingVelocity = 10; HomingApproachVelocity = 2; HomingAcceleration = 100; HomingDeceleration = 100; HomingJerk = 0; HomeMaskDistance = 0; HomePositionOffset = 0; HomePushTime = 0; HomeCompensation = 0; HomeTimeout = 0; HomeCompensationVelocity = 1000; 4000 = 1; 4001 = 0; 4003 = true; 4004 = 27; 4005 = 0; 4006 = 50.0; 4007 = 166.666666; 4008 = 20.0; 4009 = 50000; 4010 = 3500; 4011 = 3500; 4012 = 100.000000; ScalingIncs = 16#800000; 6005 = 5; AdrOffset_8010 = 2024; BitOffset_8010 = 0; BitLength_8010 = 16; Address_8010 = '%QW1012'; Type_8010 = 'UINT';
              AddressPointer_8010 = ADR(%QW1012); AdrOffset_8020 = 2028; BitOffset_8020 = 0; BitLength_8020 = 32; Address_8020 = '%QD507'; Type_8020 = 'DINT'; AddressPointer_8020 = ADR(%QD507); AdrOffset_8030 = 2040; BitOffset_8030 = 0; BitLength_8030 = 32; Address_8030 = '%QD510'; Type_8030 = 'DINT'; AddressPointer_8030 = ADR(%QD510); AdrOffset_8040 = 2044; BitOffset_8040 = 0; BitLength_8040 = 16; Address_8040 = '%QW1022'; Type_8040 = 'INT'; AddressPointer_8040 = ADR(%QW1022); AdrOffset_8050 = 4294967295; BitOffset_8050 = 0; BitLength_8050 = 0; Address_8050 = ''; Type_8050 = ''; AddressPointer_8050 = 0; AdrOffset_8060 = 2032; BitOffset_8060 = 0; BitLength_8060 = 16; Address_8060 = '%QW1016'; Type_8060 = 'UINT'; AddressPointer_8060 = ADR(%QW1016); AdrOffset_8070 = 4294967295; BitOffset_8070 = 0; BitLength_8070 = 0; Address_8070 = ''; Type_8070 = ''; AddressPointer_8070 = 0; AdrOffset_8080 = 4294967295; BitOffset_8080 = 0; BitLength_8080 = 0;
              Address_8080 = ''; Type_8080 = ''; AddressPointer_8080 = 0; AdrOffset_8090 = 2036; BitOffset_8090 = 0; BitLength_8090 = 32; Address_8090 = '%QD509'; Type_8090 = 'UDINT'; AddressPointer_8090 = ADR(%QD509); AdrOffset_8100 = 4294967295; BitOffset_8100 = 0; BitLength_8100 = 0; Address_8100 = ''; Type_8100 = ''; AddressPointer_8100 = 0; AdrOffset_8510 = 2038; BitOffset_8510 = 0; BitLength_8510 = 16; Address_8510 = '%IW1019'; Type_8510 = 'UINT'; AddressPointer_8510 = ADR(%IW1019); AdrOffset_8520 = 2040; BitOffset_8520 = 0; BitLength_8520 = 32; Address_8520 = '%ID510'; Type_8520 = 'DINT'; AddressPointer_8520 = ADR(%ID510); AdrOffset_8530 = 2068; BitOffset_8530 = 0; BitLength_8530 = 32; Address_8530 = '%ID517'; Type_8530 = 'DINT'; AddressPointer_8530 = ADR(%ID517); AdrOffset_8540 = 2044; BitOffset_8540 = 0; BitLength_8540 = 16; Address_8540 = '%IW1022'; Type_8540 = 'INT'; AddressPointer_8540 = ADR(%IW1022); AdrOffset_8550 = 4294967295;
              BitOffset_8550 = 0; BitLength_8550 = 0; Address_8550 = ''; Type_8550 = ''; AddressPointer_8550 = 0; AdrOffset_8560 = 2064; BitOffset_8560 = 0; BitLength_8560 = 32; Address_8560 = '%ID516'; Type_8560 = 'UDINT'; AddressPointer_8560 = ADR(%ID516); AdrOffset_8570 = 2052; BitOffset_8570 = 0; BitLength_8570 = 16; Address_8570 = '%IW1026'; Type_8570 = 'UINT'; AddressPointer_8570 = ADR(%IW1026); AdrOffset_8580 = 2056; BitOffset_8580 = 0; BitLength_8580 = 32; Address_8580 = '%ID514'; Type_8580 = 'DINT'; AddressPointer_8580 = ADR(%ID514); AdrOffset_8590 = 4294967295; BitOffset_8590 = 0; BitLength_8590 = 0; Address_8590 = ''; Type_8590 = ''; AddressPointer_8590 = 0; AdrOffset_8600 = 2060; BitOffset_8600 = 0; BitLength_8600 = 32; Address_8600 = '%ID515'; Type_8600 = 'DINT'; AddressPointer_8600 = ADR(%ID515); AdrOffset_8600 = 4294967295; BitOffset_8600 = 0; BitLength_8600 = 0; Address_8610 = ''; Type_8610 = '';
              AddressPointer_8610 = 0; AdrOffset_8620 = 2036; BitOffset_8620 = 0; BitLength_8620 = 16; Address_8620 = '%IW1018'; Type_8620 = 'UINT'; AddressPointer_8620 = ADR(%IW1018); IsValid = True; AxisNumber = 2; IsHostHoming = False; PulseSelectIndex = 4; SERVO_MAX_ID = 167772160
      CL3C_EC503 : CL3C-EC503(COE), Leadshine Technology Co.,Ltd., order no. CL3C-EC503, version Revision=16#00000001
          settings: Number of Outputs = 4; Number of Infos about Outputs = 4; Configuration address of the slave = 11; Sync.Length = 9; FMMU.Length = 9; Number of RxPDOs of the Slave = 1; Number of TxPDOs of the Slave = 1; AutoUpdate = False; DC sync0 cycletime = 4000; DC sync1 cycletime = 4000; Number of SDO = 1; Modes of Operation.Index = 16#6060; Modes of Operation.Subindex = 16#00; Modes of Operation.Value = 8; Modes of Operation.Size = 8; Modes of Operation.AbortIfError = FALSE; Modes of Operation.JumpToLine = FALSE; Modes of Operation.Line = 0; Modes of Operation.CompleteAccess = False; RxTxPdo.NumberofExcludes = 0; RxTxPdo.NumberofEntries = 4; RxTxPdo.Index = 16#1600; RxTxPdo.Fixed = False; RxTxPdo.Mandatory = False; RxTxPdo.Virtual = False; RxTxPdo.Sm = 2; RxTxPdo.Su = 0; RxTxPdo.Name = 'RXPDO 1 Mapping Parameter'; RxTxPdo.DependOnSlot = False; RxTxPdo.DependOnSlotGroup = False; RxTxPdo.OverwrittenByModule = False; Homing Method.Index = 16#6098; Homing Method.SubIndex = 0; Homing Method.Size = 8; Homing Method.Offset = 0; Homing Method.DependOnSlot = False; Homing Method.DependOnSlotGroup = False; Control Word.Index = 16#6040; Control Word.SubIndex = 0; Control Word.Size = 16;
            Control Word.Offset = 0; Control Word.DependOnSlot = False; Control Word.DependOnSlotGroup = False; Profile Target Position.Index = 16#607A; Profile Target Position.SubIndex = 0; Profile Target Position.Size = 32; Profile Target Position.Offset = 0; Profile Target Position.DependOnSlot = False; Profile Target Position.DependOnSlotGroup = False; Touch Probe Function.Index = 16#60B8; Touch Probe Function.SubIndex = 0; Touch Probe Function.Size = 16; Touch Probe Function.Offset = 0; Touch Probe Function.DependOnSlot = False; Touch Probe Function.DependOnSlotGroup = False; RxTxPdo.NumberofExcludes = 0; RxTxPdo.NumberofEntries = 7; RxTxPdo.Index = 16#1A00; RxTxPdo.Fixed = False; RxTxPdo.Mandatory = False; RxTxPdo.Virtual = False; RxTxPdo.Sm = 3; RxTxPdo.Su = 0; RxTxPdo.Name = 'TXPDO 1 Mapping Parameter'; RxTxPdo.DependOnSlot = False; RxTxPdo.DependOnSlotGroup = False; RxTxPdo.OverwrittenByModule = False; Last Error Code.Index = 16#603F; Last Error Code.SubIndex = 0; Last Error Code.Size = 16; Last Error Code.Offset = 0; Last Error Code.DependOnSlot = False; Last Error Code.DependOnSlotGroup = False; Status Word.Index = 16#6041; Status Word.SubIndex = 0; Status Word.Size = 16; Status Word.Offset = 0; Status Word.DependOnSlot = False; Status Word.DependOnSlotGroup = False; Modes of Operation Display.Index = 16#6061;
            Modes of Operation Display.SubIndex = 0; Modes of Operation Display.Size = 8; Modes of Operation Display.Offset = 0; Modes of Operation Display.DependOnSlot = False; Modes of Operation Display.DependOnSlotGroup = False; Actual Position.Index = 16#6064; Actual Position.SubIndex = 0; Actual Position.Size = 32; Actual Position.Offset = 0; Actual Position.DependOnSlot = False; Actual Position.DependOnSlotGroup = False; Touch Probe Status.Index = 16#60B9; Touch Probe Status.SubIndex = 0; Touch Probe Status.Size = 16; Touch Probe Status.Offset = 0; Touch Probe Status.DependOnSlot = False; Touch Probe Status.DependOnSlotGroup = False; Touch Probe 1 Positive Value.Index = 16#60BA; Touch Probe 1 Positive Value.SubIndex = 0; Touch Probe 1 Positive Value.Size = 32; Touch Probe 1 Positive Value.Offset = 0; Touch Probe 1 Positive Value.DependOnSlot = False; Touch Probe 1 Positive Value.DependOnSlotGroup = False; Digital Inputs.Index = 16#60FD; Digital Inputs.SubIndex = 0; Digital Inputs.Size = 32; Digital Inputs.Offset = 0; Digital Inputs.DependOnSlot = False; Digital Inputs.DependOnSlotGroup = False; Homing Method.Name = 'Homing Method'; Homing Method.DataType = 'SINT'; Homing Method.Default = ''; Homing Method.Comment = ''; Control Word.Name = 'Control Word'; Control Word.DataType = 'UINT'; Control Word.Default = ''; Control Word.Comment = ''; Profile Target Position.Name = 'Profile Target Position'; Profile Target Position.DataType = 'DINT'; Profile Target Position.Default = '';
            Profile Target Position.Comment = ''; Touch Probe Function.Name = 'Touch Probe Function'; Touch Probe Function.DataType = 'UINT'; Touch Probe Function.Default = ''; Touch Probe Function.Comment = ''; Last Error Code.Name = 'Last Error Code'; Last Error Code.DataType = 'UINT'; Last Error Code.Default = ''; Last Error Code.Comment = ''; Status Word.Name = 'Status Word'; Status Word.DataType = 'UINT'; Status Word.Default = ''; Status Word.Comment = ''; Modes of Operation Display.Name = 'Modes of Operation Display'; Modes of Operation Display.DataType = 'SINT'; Modes of Operation Display.Default = ''; Modes of Operation Display.Comment = ''; Actual Position.Name = 'Actual Position'; Actual Position.DataType = 'DINT'; Actual Position.Default = ''; Actual Position.Comment = ''; Touch Probe Status.Name = 'Touch Probe Status'; Touch Probe Status.DataType = 'UINT'; Touch Probe Status.Default = ''; Touch Probe Status.Comment = ''; Touch Probe 1 Positive Value.Name = 'Touch Probe 1 Positive Value'; Touch Probe 1 Positive Value.DataType = 'DINT'; Touch Probe 1 Positive Value.Default = ''; Touch Probe 1 Positive Value.Comment = ''; Digital Inputs.Name = 'Digital Inputs'; Digital Inputs.DataType = 'UDINT'; Digital Inputs.Default = ''; Digital Inputs.Comment = ''
          unmapped channels: Homing Method, Control Word, Profile Target Position, Touch Probe Function, Last Error Code, Status Word, Modes of Operation Display, Actual Position, Touch Probe Status, Touch Probe 1 Positive Value, Digital Inputs
        上样轴4X轴 : Axis, Inovance, order no. 0, version 4.0.0.0
            settings: wDriveID = 9; dwRatioTechUnitsDenom = 2800; iRatioTechUnitsNum = 3; HomingMode = 4; ZeroSignal = 0; StartDirction = -1; EndDirection = -1; PosLimitMode = 1; NegLimitMode = 1; HomingVelocity = 10; HomingApproachVelocity = 2; HomingAcceleration = 100; HomingDeceleration = 100; HomingJerk = 0; HomeMaskDistance = 0; HomePositionOffset = 0; HomePushTime = 0; HomeCompensation = 0; HomeTimeout = 0; HomeCompensationVelocity = 1000; 4000 = 1; 4001 = 0; ScalingIncs = 35000; 6005 = 37.5; AdrOffset_8010 = 2218; BitOffset_8010 = 0; BitLength_8010 = 16; Address_8010 = '%QW1109'; Type_8010 = 'UINT'; AddressPointer_8010 = ADR(%QW1109); AdrOffset_8020 = 2220; BitOffset_8020 = 0; BitLength_8020 = 32; Address_8020 = '%QD555'; Type_8020 = 'DINT'; AddressPointer_8020 = ADR(%QD555); AdrOffset_8030 = 4294967295; BitOffset_8030 = 0; BitLength_8030 = 0; Address_8030 = '';
              Type_8030 = ''; AddressPointer_8030 = 0; AdrOffset_8040 = 4294967295; BitOffset_8040 = 0; BitLength_8040 = 0; Address_8040 = ''; Type_8040 = ''; AddressPointer_8040 = 0; AdrOffset_8050 = 4294967295; BitOffset_8050 = 0; BitLength_8050 = 0; Address_8050 = ''; Type_8050 = ''; AddressPointer_8050 = 0; AdrOffset_8060 = 2224; BitOffset_8060 = 0; BitLength_8060 = 16; Address_8060 = '%QW1112'; Type_8060 = 'UINT'; AddressPointer_8060 = ADR(%QW1112); AdrOffset_8070 = 4294967295; BitOffset_8070 = 0; BitLength_8070 = 0; Address_8070 = ''; Type_8070 = ''; AddressPointer_8070 = 0; AdrOffset_8080 = 4294967295; BitOffset_8080 = 0; BitLength_8080 = 0; Address_8080 = ''; Type_8080 = ''; AddressPointer_8080 = 0; AdrOffset_8090 = 4294967295; BitOffset_8090 = 0; BitLength_8090 = 0; Address_8090 = ''; Type_8090 = ''; AddressPointer_8090 = 0; AdrOffset_8100 = 4294967295; BitOffset_8100 = 0;
              BitLength_8100 = 0; Address_8100 = ''; Type_8100 = ''; AddressPointer_8100 = 0; AdrOffset_8510 = 2326; BitOffset_8510 = 0; BitLength_8510 = 16; Address_8510 = '%IW1163'; Type_8510 = 'UINT'; AddressPointer_8510 = ADR(%IW1163); AdrOffset_8520 = 2332; BitOffset_8520 = 0; BitLength_8520 = 32; Address_8520 = '%ID583'; Type_8520 = 'DINT'; AddressPointer_8520 = ADR(%ID583); AdrOffset_8530 = 4294967295; BitOffset_8530 = 0; BitLength_8530 = 0; Address_8530 = ''; Type_8530 = ''; AddressPointer_8530 = 0; AdrOffset_8540 = 4294967295; BitOffset_8540 = 0; BitLength_8540 = 0; Address_8540 = ''; Type_8540 = ''; AddressPointer_8540 = 0; AdrOffset_8550 = 2328; BitOffset_8550 = 0; BitLength_8550 = 8; Address_8550 = '%IB2328'; Type_8550 = 'SINT'; AddressPointer_8550 = ADR(%IB2328); AdrOffset_8560 = 2344; BitOffset_8560 = 0; BitLength_8560 = 32; Address_8560 = '%ID586'; Type_8560 = 'UDINT'; AddressPointer_8560 = ADR(%ID586);
              AdrOffset_8570 = 2336; BitOffset_8570 = 0; BitLength_8570 = 16; Address_8570 = '%IW1168'; Type_8570 = 'UINT'; AddressPointer_8570 = ADR(%IW1168); AdrOffset_8580 = 2340; BitOffset_8580 = 0; BitLength_8580 = 32; Address_8580 = '%ID585'; Type_8580 = 'DINT'; AddressPointer_8580 = ADR(%ID585); AdrOffset_8590 = 4294967295; BitOffset_8590 = 0; BitLength_8590 = 0; Address_8590 = ''; Type_8590 = ''; AddressPointer_8590 = 0; AdrOffset_8600 = 4294967295; BitOffset_8600 = 0; BitLength_8600 = 0; Address_8600 = ''; Type_8600 = ''; AddressPointer_8600 = 0; AdrOffset_8600 = 4294967295; BitOffset_8600 = 0; BitLength_8600 = 0; Address_8610 = ''; Type_8610 = ''; AddressPointer_8610 = 0; AdrOffset_8620 = 2324; BitOffset_8620 = 0; BitLength_8620 = 16; Address_8620 = '%IW1162'; Type_8620 = 'UINT'; AddressPointer_8620 = ADR(%IW1162); Automatic Mapping = True; IsValid = True; AxisNumber = 10; IsHostHoming = True;
              PulseSelectIndex = 0
      AU7_877_ECT22_H : AU7 877-ECT22-H, AUTO, order no. AU7 877-ECT22-H, version Revision=16#00001000
          settings:  = '30d8641a-a89f-41d9-9860-5b1d09cb5afa';  = '30d8641a-a89f-41d9-9860-5b1d09cb5afa';  = '30d8641a-a89f-41d9-9860-5b1d09cb5afa';  = '30d8641a-a89f-41d9-9860-5b1d09cb5afa';  = '30d8641a-a89f-41d9-9860-5b1d09cb5afa';  = '2b5b7a91-b0ea-458b-8a5e-2a35da436682';  = '2b5b7a91-b0ea-458b-8a5e-2a35da436682';  = '2b5b7a91-b0ea-458b-8a5e-2a35da436682';  = '2b5b7a91-b0ea-458b-8a5e-2a35da436682';  = '2b5b7a91-b0ea-458b-8a5e-2a35da436682';  = '1e06bf35-6cb5-4a2d-8bf5-5f44f972a574';  = '1e06bf35-6cb5-4a2d-8bf5-5f44f972a574';  = '1e06bf35-6cb5-4a2d-8bf5-5f44f972a574';  = '1e06bf35-6cb5-4a2d-8bf5-5f44f972a574';  = '1e06bf35-6cb5-4a2d-8bf5-5f44f972a574';  = 'd126d70a-8f54-4883-a11e-5bdc58f1a2b5';  = 'd126d70a-8f54-4883-a11e-5bdc58f1a2b5';  = 'd126d70a-8f54-4883-a11e-5bdc58f1a2b5';  = 'd126d70a-8f54-4883-a11e-5bdc58f1a2b5';  = 'd126d70a-8f54-4883-a11e-5bdc58f1a2b5';  = '3ad5e0e7-27d0-4bc5-8bf1-3c35b9d3bbe6';  = '3ad5e0e7-27d0-4bc5-8bf1-3c35b9d3bbe6';  = '3ad5e0e7-27d0-4bc5-8bf1-3c35b9d3bbe6';  = '3ad5e0e7-27d0-4bc5-8bf1-3c35b9d3bbe6';  = '3ad5e0e7-27d0-4bc5-8bf1-3c35b9d3bbe6';  = '30d8641a-a89f-41d9-9860-5b1d09cb5afa';  = '30d8641a-a89f-41d9-9860-5b1d09cb5afa';  = '30d8641a-a89f-41d9-9860-5b1d09cb5afa';  = '30d8641a-a89f-41d9-9860-5b1d09cb5afa';  = '30d8641a-a89f-41d9-9860-5b1d09cb5afa';  = '2b5b7a91-b0ea-458b-8a5e-2a35da436682';  = '2b5b7a91-b0ea-458b-8a5e-2a35da436682';  = '2b5b7a91-b0ea-458b-8a5e-2a35da436682';  = '2b5b7a91-b0ea-458b-8a5e-2a35da436682';  = '2b5b7a91-b0ea-458b-8a5e-2a35da436682';  = '1e06bf35-6cb5-4a2d-8bf5-5f44f972a574';  = '1e06bf35-6cb5-4a2d-8bf5-5f44f972a574';  = '1e06bf35-6cb5-4a2d-8bf5-5f44f972a574';  = '1e06bf35-6cb5-4a2d-8bf5-5f44f972a574';  = '1e06bf35-6cb5-4a2d-8bf5-5f44f972a574';
             = 'd126d70a-8f54-4883-a11e-5bdc58f1a2b5';  = 'd126d70a-8f54-4883-a11e-5bdc58f1a2b5';  = 'd126d70a-8f54-4883-a11e-5bdc58f1a2b5';  = 'd126d70a-8f54-4883-a11e-5bdc58f1a2b5';  = 'd126d70a-8f54-4883-a11e-5bdc58f1a2b5';  = '3ad5e0e7-27d0-4bc5-8bf1-3c35b9d3bbe6';  = '3ad5e0e7-27d0-4bc5-8bf1-3c35b9d3bbe6';  = '3ad5e0e7-27d0-4bc5-8bf1-3c35b9d3bbe6';  = '3ad5e0e7-27d0-4bc5-8bf1-3c35b9d3bbe6';  = '3ad5e0e7-27d0-4bc5-8bf1-3c35b9d3bbe6'; Number of Outputs = 80; Number of Inputs = 81; IOModuleSize = 5; IOModuleName = "AU7_823_1ML22_MIL,AU7_823_1ML22_MIL_1,AU7_823_1ML22_MIL_2,AU7_823_1ML22_MIL_3,AU7_823_1ML22_MIL_4"; Number of Infos about Outputs = 80; Number of Infos about Inputs = 81; Configuration address of the slave = 1; Sync.Length = 10; Sync.Length = 12; FMMU.Length = 10; FMMU.Length = 12; Number of RxPDOs of the Slave = 25; Number of TxPDOs of the Slave = 26; AutoUpdate = False; DC sync0 cycletime = 4000; DC sync1 cycletime = 4000; Number of SDO = 5; Command_0.Index = 16#8000; Command_0.Subindex = 16#01; Command_0.Value = 4256; Command_0.Size = 16; Command_0.AbortIfError = FALSE; Command_0.JumpToLine = FALSE; Command_0.Line = 0; Command_0.CompleteAccess = False; Command_0.Index = 16#8010; Command_0.Subindex = 16#01; Command_0.Value = 4256; Command_0.Size = 16; Command_0.AbortIfError = FALSE;
            Command_0.JumpToLine = FALSE; Command_0.Line = 0; Command_0.CompleteAccess = False; Command_0.Index = 16#8020; Command_0.Subindex = 16#01; Command_0.Value = 4256; Command_0.Size = 16; Command_0.AbortIfError = FALSE; Command_0.JumpToLine = FALSE; Command_0.Line = 0; Command_0.CompleteAccess = False; Command_0.Index = 16#8030; Command_0.Subindex = 16#01; Command_0.Value = 4256; Command_0.Size = 16; Command_0.AbortIfError = FALSE; Command_0.JumpToLine = FALSE; Command_0.Line = 0; Command_0.CompleteAccess = False; Command_0.Index = 16#8040; Command_0.Subindex = 16#01; Command_0.Value = 4256; Command_0.Size = 16; Command_0.AbortIfError = FALSE; Command_0.JumpToLine = FALSE; Command_0.Line = 0; Command_0.CompleteAccess = False; RxTxPdo.NumberofExcludes = 4; RxTxPdo.NumberofEntries = 16; RxTxPdo.Index = 16#1660; RxTxPdo.Fixed = True; RxTxPdo.Mandatory = False; RxTxPdo.Virtual = False; RxTxPdo.Sm = 2; RxTxPdo.Su = 0; RxTxPdo.Name = 'Digital Outputs(Bit)'; RxTxPdo.DependOnSlot = True; RxTxPdo.DependOnSlotGroup = False; RxTxPdo.OverwrittenByModule = True; Exclude = [16#1661,16#1662,16#1663,16#1664];
            AU7_823_1ML22_MIL Channel 1.Index = 16#7600; AU7_823_1ML22_MIL Channel 1.SubIndex = 1; AU7_823_1ML22_MIL Channel 1.Size = 1; AU7_823_1ML22_MIL Channel 1.Offset = 0; AU7_823_1ML22_MIL Channel 1.DependOnSlot = True; AU7_823_1ML22_MIL Channel 1.DependOnSlotGroup = False; AU7_823_1ML22_MIL Channel 2.Index = 16#7600; AU7_823_1ML22_MIL Channel 2.SubIndex = 2; AU7_823_1ML22_MIL Channel 2.Size = 1; AU7_823_1ML22_MIL Channel 2.Offset = 0; AU7_823_1ML22_MIL Channel 2.DependOnSlot = True; AU7_823_1ML22_MIL Channel 2.DependOnSlotGroup = False; AU7_823_1ML22_MIL Channel 3.Index = 16#7600; AU7_823_1ML22_MIL Channel 3.SubIndex = 3; AU7_823_1ML22_MIL Channel 3.Size = 1; AU7_823_1ML22_MIL Channel 3.Offset = 0; AU7_823_1ML22_MIL Channel 3.DependOnSlot = True; AU7_823_1ML22_MIL Channel 3.DependOnSlotGroup = False; AU7_823_1ML22_MIL Channel 4.Index = 16#7600; AU7_823_1ML22_MIL Channel 4.SubIndex = 4; AU7_823_1ML22_MIL Channel 4.Size = 1; AU7_823_1ML22_MIL Channel 4.Offset = 0; AU7_823_1ML22_MIL Channel 4.DependOnSlot = True; AU7_823_1ML22_MIL Channel 4.DependOnSlotGroup = False; AU7_823_1ML22_MIL Channel 5.Index = 16#7600; AU7_823_1ML22_MIL Channel 5.SubIndex = 5; AU7_823_1ML22_MIL Channel 5.Size = 1; AU7_823_1ML22_MIL Channel 5.Offset = 0; AU7_823_1ML22_MIL Channel 5.DependOnSlot = True; AU7_823_1ML22_MIL Channel 5.DependOnSlotGroup = False; AU7_823_1ML22_MIL Channel 6.Index = 16#7600; AU7_823_1ML22_MIL Channel 6.SubIndex = 6; AU7_823_1ML22_MIL Channel 6.Size = 1; AU7_823_1ML22_MIL Channel 6.Offset = 0; AU7_823_1ML22_MIL Channel 6.DependOnSlot = True; AU7_823_1ML22_MIL Channel 6.DependOnSlotGroup = False; AU7_823_1ML22_MIL Channel 7.Index = 16#7600; AU7_823_1ML22_MIL Channel 7.SubIndex = 7; AU7_823_1ML22_MIL Channel 7.Size = 1; AU7_823_1ML22_MIL Channel 7.Offset = 0;
            AU7_823_1ML22_MIL Channel 7.DependOnSlot = True; AU7_823_1ML22_MIL Channel 7.DependOnSlotGroup = False; AU7_823_1ML22_MIL Channel 8.Index = 16#7600; AU7_823_1ML22_MIL Channel 8.SubIndex = 8; AU7_823_1ML22_MIL Channel 8.Size = 1; AU7_823_1ML22_MIL Channel 8.Offset = 0; AU7_823_1ML22_MIL Channel 8.DependOnSlot = True; AU7_823_1ML22_MIL Channel 8.DependOnSlotGroup = False; AU7_823_1ML22_MIL Channel 9.Index = 16#7600; AU7_823_1ML22_MIL Channel 9.SubIndex = 9; AU7_823_1ML22_MIL Channel 9.Size = 1; AU7_823_1ML22_MIL Channel 9.Offset = 0; AU7_823_1ML22_MIL Channel 9.DependOnSlot = True; AU7_823_1ML22_MIL Channel 9.DependOnSlotGroup = False; AU7_823_1ML22_MIL Channel 10.Index = 16#7600; AU7_823_1ML22_MIL Channel 10.SubIndex = 10; AU7_823_1ML22_MIL Channel 10.Size = 1; AU7_823_1ML22_MIL Channel 10.Offset = 0; AU7_823_1ML22_MIL Channel 10.DependOnSlot = True; AU7_823_1ML22_MIL Channel 10.DependOnSlotGroup = False; AU7_823_1ML22_MIL Channel 11.Index = 16#7600; AU7_823_1ML22_MIL Channel 11.SubIndex = 11; AU7_823_1ML22_MIL Channel 11.Size = 1; AU7_823_1ML22_MIL Channel 11.Offset = 0; AU7_823_1ML22_MIL Channel 11.DependOnSlot = True; AU7_823_1ML22_MIL Channel 11.DependOnSlotGroup = False; AU7_823_1ML22_MIL Channel 12.Index = 16#7600; AU7_823_1ML22_MIL Channel 12.SubIndex = 12; AU7_823_1ML22_MIL Channel 12.Size = 1; AU7_823_1ML22_MIL Channel 12.Offset = 0; AU7_823_1ML22_MIL Channel 12.DependOnSlot = True; AU7_823_1ML22_MIL Channel 12.DependOnSlotGroup = False; AU7_823_1ML22_MIL Channel 13.Index = 16#7600; AU7_823_1ML22_MIL Channel 13.SubIndex = 13; AU7_823_1ML22_MIL Channel 13.Size = 1; AU7_823_1ML22_MIL Channel 13.Offset = 0; AU7_823_1ML22_MIL Channel 13.DependOnSlot = True; AU7_823_1ML22_MIL Channel 13.DependOnSlotGroup = False; AU7_823_1ML22_MIL Channel 14.Index = 16#7600; AU7_823_1ML22_MIL Channel 14.SubIndex = 14;
            AU7_823_1ML22_MIL Channel 14.Size = 1; AU7_823_1ML22_MIL Channel 14.Offset = 0; AU7_823_1ML22_MIL Channel 14.DependOnSlot = True; AU7_823_1ML22_MIL Channel 14.DependOnSlotGroup = False; AU7_823_1ML22_MIL Channel 15.Index = 16#7600; AU7_823_1ML22_MIL Channel 15.SubIndex = 15; AU7_823_1ML22_MIL Channel 15.Size = 1; AU7_823_1ML22_MIL Channel 15.Offset = 0; AU7_823_1ML22_MIL Channel 15.DependOnSlot = True; AU7_823_1ML22_MIL Channel 15.DependOnSlotGroup = False; AU7_823_1ML22_MIL Channel 16.Index = 16#7600; AU7_823_1ML22_MIL Channel 16.SubIndex = 16; AU7_823_1ML22_MIL Channel 16.Size = 1; AU7_823_1ML22_MIL Channel 16.Offset = 0; AU7_823_1ML22_MIL Channel 16.DependOnSlot = True; AU7_823_1ML22_MIL Channel 16.DependOnSlotGroup = False; RxTxPdo.NumberofExcludes = 4; RxTxPdo.NumberofEntries = 2; RxTxPdo.Index = 16#1661; RxTxPdo.Fixed = True; RxTxPdo.Mandatory = False; RxTxPdo.Virtual = False; RxTxPdo.Sm = -1; RxTxPdo.Su = 0; RxTxPdo.Name = 'Digital Outputs(Byte)'; RxTxPdo.DependOnSlot = True; RxTxPdo.DependOnSlotGroup = False; RxTxPdo.OverwrittenByModule = True; Exclude = [16#1660,16#1662,16#1663,16#1664]; AU7_823_1ML22_MIL Channel 1-8.Index = 16#7601; AU7_823_1ML22_MIL Channel 1-8.SubIndex = 1; AU7_823_1ML22_MIL Channel 1-8.Size = 8; AU7_823_1ML22_MIL Channel 1-8.Offset = 0; AU7_823_1ML22_MIL Channel 1-8.DependOnSlot = True; AU7_823_1ML22_MIL Channel 1-8.DependOnSlotGroup = False; AU7_823_1ML22_MIL Channel 9-16.Index = 16#7601; AU7_823_1ML22_MIL Channel 9-16.SubIndex = 2; AU7_823_1ML22_MIL Channel 9-16.Size = 8; AU7_823_1ML22_MIL Channel 9-16.Offset = 0; AU7_823_1ML22_MIL Channel 9-16.DependOnSlot = True;
            AU7_823_1ML22_MIL Channel 9-16.DependOnSlotGroup = False; RxTxPdo.NumberofExcludes = 4; RxTxPdo.NumberofEntries = 2; RxTxPdo.Index = 16#1662; RxTxPdo.Fixed = True; RxTxPdo.Mandatory = False; RxTxPdo.Virtual = False; RxTxPdo.Sm = -1; RxTxPdo.Su = 0; RxTxPdo.Name = 'Digital Outputs(Arr 8Bit)'; RxTxPdo.DependOnSlot = True; RxTxPdo.DependOnSlotGroup = False; RxTxPdo.OverwrittenByModule = True; Exclude = [16#1660,16#1661,16#1663,16#1664]; AU7_823_1ML22_MIL Channel 1-8.Index = 16#7602; AU7_823_1ML22_MIL Channel 1-8.SubIndex = 1; AU7_823_1ML22_MIL Channel 1-8.Size = 8; AU7_823_1ML22_MIL Channel 1-8.Offset = 0; AU7_823_1ML22_MIL Channel 1-8.DependOnSlot = True; AU7_823_1ML22_MIL Channel 1-8.DependOnSlotGroup = False; AU7_823_1ML22_MIL Channel 9-16.Index = 16#7602; AU7_823_1ML22_MIL Channel 9-16.SubIndex = 2; AU7_823_1ML22_MIL Channel 9-16.Size = 8; AU7_823_1ML22_MIL Channel 9-16.Offset = 0; AU7_823_1ML22_MIL Channel 9-16.DependOnSlot = True; AU7_823_1ML22_MIL Channel 9-16.DependOnSlotGroup = False; RxTxPdo.NumberofExcludes = 4; RxTxPdo.NumberofEntries = 1; RxTxPdo.Index = 16#1663; RxTxPdo.Fixed = True; RxTxPdo.Mandatory = False; RxTxPdo.Virtual = False; RxTxPdo.Sm = -1; RxTxPdo.Su = 0; RxTxPdo.Name = 'Digital Outputs(Arr 16Bit)'; RxTxPdo.DependOnSlot = True; RxTxPdo.DependOnSlotGroup = False; RxTxPdo.OverwrittenByModule = True; Exclude = [16#1660,16#1661,16#1662,16#1664]; AU7_823_1ML22_MIL Channel 1-16.Index = 16#7603;
            AU7_823_1ML22_MIL Channel 1-16.SubIndex = 1; AU7_823_1ML22_MIL Channel 1-16.Size = 16; AU7_823_1ML22_MIL Channel 1-16.Offset = 0; AU7_823_1ML22_MIL Channel 1-16.DependOnSlot = True; AU7_823_1ML22_MIL Channel 1-16.DependOnSlotGroup = False; RxTxPdo.NumberofExcludes = 4; RxTxPdo.NumberofEntries = 1; RxTxPdo.Index = 16#1664; RxTxPdo.Fixed = True; RxTxPdo.Mandatory = False; RxTxPdo.Virtual = False; RxTxPdo.Sm = -1; RxTxPdo.Su = 0; RxTxPdo.Name = 'Digital Outputs(Word)'; RxTxPdo.DependOnSlot = True; RxTxPdo.DependOnSlotGroup = False; RxTxPdo.OverwrittenByModule = True; Exclude = [16#1660,16#1661,16#1662,16#1663]; AU7_823_1ML22_MIL Channel 1-16.Index = 16#7604; AU7_823_1ML22_MIL Channel 1-16.SubIndex = 1; AU7_823_1ML22_MIL Channel 1-16.Size = 16; AU7_823_1ML22_MIL Channel 1-16.Offset = 0; AU7_823_1ML22_MIL Channel 1-16.DependOnSlot = True; AU7_823_1ML22_MIL Channel 1-16.DependOnSlotGroup = False; RxTxPdo.NumberofExcludes = 4; RxTxPdo.NumberofEntries = 16; RxTxPdo.Index = 16#1665; RxTxPdo.Fixed = True; RxTxPdo.Mandatory = False; RxTxPdo.Virtual = False; RxTxPdo.Sm = 2; RxTxPdo.Su = 0; RxTxPdo.Name = 'Digital Outputs(Bit)'; RxTxPdo.DependOnSlot = True; RxTxPdo.DependOnSlotGroup = False; RxTxPdo.OverwrittenByModule = True; Exclude = [16#1666,16#1667,16#1668,16#1669]; AU7_823_1ML22_MIL_1 Channel 1.Index = 16#7610; AU7_823_1ML22_MIL_1 Channel 1.SubIndex = 1; AU7_823_1ML22_MIL_1 Channel 1.Size = 1;
            AU7_823_1ML22_MIL_1 Channel 1.Offset = 0; AU7_823_1ML22_MIL_1 Channel 1.DependOnSlot = True; AU7_823_1ML22_MIL_1 Channel 1.DependOnSlotGroup = False; AU7_823_1ML22_MIL_1 Channel 2.Index = 16#7610; AU7_823_1ML22_MIL_1 Channel 2.SubIndex = 2; AU7_823_1ML22_MIL_1 Channel 2.Size = 1; AU7_823_1ML22_MIL_1 Channel 2.Offset = 0; AU7_823_1ML22_MIL_1 Channel 2.DependOnSlot = True; AU7_823_1ML22_MIL_1 Channel 2.DependOnSlotGroup = False; AU7_823_1ML22_MIL_1 Channel 3.Index = 16#7610; AU7_823_1ML22_MIL_1 Channel 3.SubIndex = 3; AU7_823_1ML22_MIL_1 Channel 3.Size = 1; AU7_823_1ML22_MIL_1 Channel 3.Offset = 0; AU7_823_1ML22_MIL_1 Channel 3.DependOnSlot = True; AU7_823_1ML22_MIL_1 Channel 3.DependOnSlotGroup = False; AU7_823_1ML22_MIL_1 Channel 4.Index = 16#7610; AU7_823_1ML22_MIL_1 Channel 4.SubIndex = 4; AU7_823_1ML22_MIL_1 Channel 4.Size = 1; AU7_823_1ML22_MIL_1 Channel 4.Offset = 0; AU7_823_1ML22_MIL_1 Channel 4.DependOnSlot = True; AU7_823_1ML22_MIL_1 Channel 4.DependOnSlotGroup = False; AU7_823_1ML22_MIL_1 Channel 5.Index = 16#7610; AU7_823_1ML22_MIL_1 Channel 5.SubIndex = 5; AU7_823_1ML22_MIL_1 Channel 5.Size = 1; AU7_823_1ML22_MIL_1 Channel 5.Offset = 0; AU7_823_1ML22_MIL_1 Channel 5.DependOnSlot = True; AU7_823_1ML22_MIL_1 Channel 5.DependOnSlotGroup = False; AU7_823_1ML22_MIL_1 Channel 6.Index = 16#7610; AU7_823_1ML22_MIL_1 Channel 6.SubIndex = 6; AU7_823_1ML22_MIL_1 Channel 6.Size = 1; AU7_823_1ML22_MIL_1 Channel 6.Offset = 0; AU7_823_1ML22_MIL_1 Channel 6.DependOnSlot = True; AU7_823_1ML22_MIL_1 Channel 6.DependOnSlotGroup = False; AU7_823_1ML22_MIL_1 Channel 7.Index = 16#7610; AU7_823_1ML22_MIL_1 Channel 7.SubIndex = 7; AU7_823_1ML22_MIL_1 Channel 7.Size = 1; AU7_823_1ML22_MIL_1 Channel 7.Offset = 0; AU7_823_1ML22_MIL_1 Channel 7.DependOnSlot = True; AU7_823_1ML22_MIL_1 Channel 7.DependOnSlotGroup = False; AU7_823_1ML22_MIL_1 Channel 8.Index = 16#7610;
            AU7_823_1ML22_MIL_1 Channel 8.SubIndex = 8; AU7_823_1ML22_MIL_1 Channel 8.Size = 1; AU7_823_1ML22_MIL_1 Channel 8.Offset = 0; AU7_823_1ML22_MIL_1 Channel 8.DependOnSlot = True; AU7_823_1ML22_MIL_1 Channel 8.DependOnSlotGroup = False; AU7_823_1ML22_MIL_1 Channel 9.Index = 16#7610; AU7_823_1ML22_MIL_1 Channel 9.SubIndex = 9; AU7_823_1ML22_MIL_1 Channel 9.Size = 1; AU7_823_1ML22_MIL_1 Channel 9.Offset = 0; AU7_823_1ML22_MIL_1 Channel 9.DependOnSlot = True; AU7_823_1ML22_MIL_1 Channel 9.DependOnSlotGroup = False; AU7_823_1ML22_MIL_1 Channel 10.Index = 16#7610; AU7_823_1ML22_MIL_1 Channel 10.SubIndex = 10; AU7_823_1ML22_MIL_1 Channel 10.Size = 1; AU7_823_1ML22_MIL_1 Channel 10.Offset = 0; AU7_823_1ML22_MIL_1 Channel 10.DependOnSlot = True; AU7_823_1ML22_MIL_1 Channel 10.DependOnSlotGroup = False; AU7_823_1ML22_MIL_1 Channel 11.Index = 16#7610; AU7_823_1ML22_MIL_1 Channel 11.SubIndex = 11; AU7_823_1ML22_MIL_1 Channel 11.Size = 1; AU7_823_1ML22_MIL_1 Channel 11.Offset = 0; AU7_823_1ML22_MIL_1 Channel 11.DependOnSlot = True; AU7_823_1ML22_MIL_1 Channel 11.DependOnSlotGroup = False; AU7_823_1ML22_MIL_1 Channel 12.Index = 16#7610; AU7_823_1ML22_MIL_1 Channel 12.SubIndex = 12; AU7_823_1ML22_MIL_1 Channel 12.Size = 1; AU7_823_1ML22_MIL_1 Channel 12.Offset = 0; AU7_823_1ML22_MIL_1 Channel 12.DependOnSlot = True; AU7_823_1ML22_MIL_1 Channel 12.DependOnSlotGroup = False; AU7_823_1ML22_MIL_1 Channel 13.Index = 16#7610; AU7_823_1ML22_MIL_1 Channel 13.SubIndex = 13; AU7_823_1ML22_MIL_1 Channel 13.Size = 1; AU7_823_1ML22_MIL_1 Channel 13.Offset = 0; AU7_823_1ML22_MIL_1 Channel 13.DependOnSlot = True; AU7_823_1ML22_MIL_1 Channel 13.DependOnSlotGroup = False; AU7_823_1ML22_MIL_1 Channel 14.Index = 16#7610; AU7_823_1ML22_MIL_1 Channel 14.SubIndex = 14; AU7_823_1ML22_MIL_1 Channel 14.Size = 1; AU7_823_1ML22_MIL_1 Channel 14.Offset = 0; AU7_823_1ML22_MIL_1 Channel 14.DependOnSlot = True;
            AU7_823_1ML22_MIL_1 Channel 14.DependOnSlotGroup = False; AU7_823_1ML22_MIL_1 Channel 15.Index = 16#7610; AU7_823_1ML22_MIL_1 Channel 15.SubIndex = 15; AU7_823_1ML22_MIL_1 Channel 15.Size = 1; AU7_823_1ML22_MIL_1 Channel 15.Offset = 0; AU7_823_1ML22_MIL_1 Channel 15.DependOnSlot = True; AU7_823_1ML22_MIL_1 Channel 15.DependOnSlotGroup = False; AU7_823_1ML22_MIL_1 Channel 16.Index = 16#7610; AU7_823_1ML22_MIL_1 Channel 16.SubIndex = 16; AU7_823_1ML22_MIL_1 Channel 16.Size = 1; AU7_823_1ML22_MIL_1 Channel 16.Offset = 0; AU7_823_1ML22_MIL_1 Channel 16.DependOnSlot = True; AU7_823_1ML22_MIL_1 Channel 16.DependOnSlotGroup = False; RxTxPdo.NumberofExcludes = 4; RxTxPdo.NumberofEntries = 2; RxTxPdo.Index = 16#1666; RxTxPdo.Fixed = True; RxTxPdo.Mandatory = False; RxTxPdo.Virtual = False; RxTxPdo.Sm = -1; RxTxPdo.Su = 0; RxTxPdo.Name = 'Digital Outputs(Byte)'; RxTxPdo.DependOnSlot = True; RxTxPdo.DependOnSlotGroup = False; RxTxPdo.OverwrittenByModule = True; Exclude = [16#1665,16#1667,16#1668,16#1669]; AU7_823_1ML22_MIL_1 Channel 1-8.Index = 16#7611; AU7_823_1ML22_MIL_1 Channel 1-8.SubIndex = 1; AU7_823_1ML22_MIL_1 Channel 1-8.Size = 8; AU7_823_1ML22_MIL_1 Channel 1-8.Offset = 0; AU7_823_1ML22_MIL_1 Channel 1-8.DependOnSlot = True; AU7_823_1ML22_MIL_1 Channel 1-8.DependOnSlotGroup = False; AU7_823_1ML22_MIL_1 Channel 9-16.Index = 16#7611; AU7_823_1ML22_MIL_1 Channel 9-16.SubIndex = 2; AU7_823_1ML22_MIL_1 Channel 9-16.Size = 8; AU7_823_1ML22_MIL_1 Channel 9-16.Offset = 0; AU7_823_1ML22_MIL_1 Channel 9-16.DependOnSlot = True; AU7_823_1ML22_MIL_1 Channel 9-16.DependOnSlotGroup = False; RxTxPdo.NumberofExcludes = 4; RxTxPdo.NumberofEntries = 2;
            RxTxPdo.Index = 16#1667; RxTxPdo.Fixed = True; RxTxPdo.Mandatory = False; RxTxPdo.Virtual = False; RxTxPdo.Sm = -1; RxTxPdo.Su = 0; RxTxPdo.Name = 'Digital Outputs(Arr 8Bit)'; RxTxPdo.DependOnSlot = True; RxTxPdo.DependOnSlotGroup = False; RxTxPdo.OverwrittenByModule = True; Exclude = [16#1665,16#1666,16#1668,16#1669]; AU7_823_1ML22_MIL_1 Channel 1-8.Index = 16#7612; AU7_823_1ML22_MIL_1 Channel 1-8.SubIndex = 1; AU7_823_1ML22_MIL_1 Channel 1-8.Size = 8; AU7_823_1ML22_MIL_1 Channel 1-8.Offset = 0; AU7_823_1ML22_MIL_1 Channel 1-8.DependOnSlot = True; AU7_823_1ML22_MIL_1 Channel 1-8.DependOnSlotGroup = False; AU7_823_1ML22_MIL_1 Channel 9-16.Index = 16#7612; AU7_823_1ML22_MIL_1 Channel 9-16.SubIndex = 2; AU7_823_1ML22_MIL_1 Channel 9-16.Size = 8; AU7_823_1ML22_MIL_1 Channel 9-16.Offset = 0; AU7_823_1ML22_MIL_1 Channel 9-16.DependOnSlot = True; AU7_823_1ML22_MIL_1 Channel 9-16.DependOnSlotGroup = False; RxTxPdo.NumberofExcludes = 4; RxTxPdo.NumberofEntries = 1; RxTxPdo.Index = 16#1668; RxTxPdo.Fixed = True; RxTxPdo.Mandatory = False; RxTxPdo.Virtual = False; RxTxPdo.Sm = -1; RxTxPdo.Su = 0; RxTxPdo.Name = 'Digital Outputs(Arr 16Bit)'; RxTxPdo.DependOnSlot = True; RxTxPdo.DependOnSlotGroup = False; RxTxPdo.OverwrittenByModule = True; Exclude = [16#1665,16#1666,16#1667,16#1669]; AU7_823_1ML22_MIL_1 Channel 1-16.Index = 16#7613; AU7_823_1ML22_MIL_1 Channel 1-16.SubIndex = 1; AU7_823_1ML22_MIL_1 Channel 1-16.Size = 16; AU7_823_1ML22_MIL_1 Channel 1-16.Offset = 0;
            AU7_823_1ML22_MIL_1 Channel 1-16.DependOnSlot = True; AU7_823_1ML22_MIL_1 Channel 1-16.DependOnSlotGroup = False; RxTxPdo.NumberofExcludes = 4; RxTxPdo.NumberofEntries = 1; RxTxPdo.Index = 16#1669; RxTxPdo.Fixed = True; RxTxPdo.Mandatory = False; RxTxPdo.Virtual = False; RxTxPdo.Sm = -1; RxTxPdo.Su = 0; RxTxPdo.Name = 'Digital Outputs(Word)'; RxTxPdo.DependOnSlot = True; RxTxPdo.DependOnSlotGroup = False; RxTxPdo.OverwrittenByModule = True; Exclude = [16#1665,16#1666,16#1667,16#1668]; AU7_823_1ML22_MIL_1 Channel 1-16.Index = 16#7614; AU7_823_1ML22_MIL_1 Channel 1-16.SubIndex = 1; AU7_823_1ML22_MIL_1 Channel 1-16.Size = 16; AU7_823_1ML22_MIL_1 Channel 1-16.Offset = 0; AU7_823_1ML22_MIL_1 Channel 1-16.DependOnSlot = True; AU7_823_1ML22_MIL_1 Channel 1-16.DependOnSlotGroup = False; RxTxPdo.NumberofExcludes = 4; RxTxPdo.NumberofEntries = 16; RxTxPdo.Index = 16#166A; RxTxPdo.Fixed = True; RxTxPdo.Mandatory = False; RxTxPdo.Virtual = False; RxTxPdo.Sm = 2; RxTxPdo.Su = 0; RxTxPdo.Name = 'Digital Outputs(Bit)'; RxTxPdo.DependOnSlot = True; RxTxPdo.DependOnSlotGroup = False; RxTxPdo.OverwrittenByModule = True; Exclude = [16#166B,16#166C,16#166D,16#166E]; AU7_823_1ML22_MIL_2 Channel 1.Index = 16#7620; AU7_823_1ML22_MIL_2 Channel 1.SubIndex = 1; AU7_823_1ML22_MIL_2 Channel 1.Size = 1; AU7_823_1ML22_MIL_2 Channel 1.Offset = 0; AU7_823_1ML22_MIL_2 Channel 1.DependOnSlot = True; AU7_823_1ML22_MIL_2 Channel 1.DependOnSlotGroup = False;
            AU7_823_1ML22_MIL_2 Channel 2.Index = 16#7620; AU7_823_1ML22_MIL_2 Channel 2.SubIndex = 2; AU7_823_1ML22_MIL_2 Channel 2.Size = 1; AU7_823_1ML22_MIL_2 Channel 2.Offset = 0; AU7_823_1ML22_MIL_2 Channel 2.DependOnSlot = True; AU7_823_1ML22_MIL_2 Channel 2.DependOnSlotGroup = False; AU7_823_1ML22_MIL_2 Channel 3.Index = 16#7620; AU7_823_1ML22_MIL_2 Channel 3.SubIndex = 3; AU7_823_1ML22_MIL_2 Channel 3.Size = 1; AU7_823_1ML22_MIL_2 Channel 3.Offset = 0; AU7_823_1ML22_MIL_2 Channel 3.DependOnSlot = True; AU7_823_1ML22_MIL_2 Channel 3.DependOnSlotGroup = False; AU7_823_1ML22_MIL_2 Channel 4.Index = 16#7620; AU7_823_1ML22_MIL_2 Channel 4.SubIndex = 4; AU7_823_1ML22_MIL_2 Channel 4.Size = 1; AU7_823_1ML22_MIL_2 Channel 4.Offset = 0; AU7_823_1ML22_MIL_2 Channel 4.DependOnSlot = True; AU7_823_1ML22_MIL_2 Channel 4.DependOnSlotGroup = False; AU7_823_1ML22_MIL_2 Channel 5.Index = 16#7620; AU7_823_1ML22_MIL_2 Channel 5.SubIndex = 5; AU7_823_1ML22_MIL_2 Channel 5.Size = 1; AU7_823_1ML22_MIL_2 Channel 5.Offset = 0; AU7_823_1ML22_MIL_2 Channel 5.DependOnSlot = True; AU7_823_1ML22_MIL_2 Channel 5.DependOnSlotGroup = False; AU7_823_1ML22_MIL_2 Channel 6.Index = 16#7620; AU7_823_1ML22_MIL_2 Channel 6.SubIndex = 6; AU7_823_1ML22_MIL_2 Channel 6.Size = 1; AU7_823_1ML22_MIL_2 Channel 6.Offset = 0; AU7_823_1ML22_MIL_2 Channel 6.DependOnSlot = True; AU7_823_1ML22_MIL_2 Channel 6.DependOnSlotGroup = False; AU7_823_1ML22_MIL_2 Channel 7.Index = 16#7620; AU7_823_1ML22_MIL_2 Channel 7.SubIndex = 7; AU7_823_1ML22_MIL_2 Channel 7.Size = 1; AU7_823_1ML22_MIL_2 Channel 7.Offset = 0; AU7_823_1ML22_MIL_2 Channel 7.DependOnSlot = True; AU7_823_1ML22_MIL_2 Channel 7.DependOnSlotGroup = False; AU7_823_1ML22_MIL_2 Channel 8.Index = 16#7620; AU7_823_1ML22_MIL_2 Channel 8.SubIndex = 8; AU7_823_1ML22_MIL_2 Channel 8.Size = 1; AU7_823_1ML22_MIL_2 Channel 8.Offset = 0;
            AU7_823_1ML22_MIL_2 Channel 8.DependOnSlot = True; AU7_823_1ML22_MIL_2 Channel 8.DependOnSlotGroup = False; AU7_823_1ML22_MIL_2 Channel 9.Index = 16#7620; AU7_823_1ML22_MIL_2 Channel 9.SubIndex = 9; AU7_823_1ML22_MIL_2 Channel 9.Size = 1; AU7_823_1ML22_MIL_2 Channel 9.Offset = 0; AU7_823_1ML22_MIL_2 Channel 9.DependOnSlot = True; AU7_823_1ML22_MIL_2 Channel 9.DependOnSlotGroup = False; AU7_823_1ML22_MIL_2 Channel 10.Index = 16#7620; AU7_823_1ML22_MIL_2 Channel 10.SubIndex = 10; AU7_823_1ML22_MIL_2 Channel 10.Size = 1; AU7_823_1ML22_MIL_2 Channel 10.Offset = 0; AU7_823_1ML22_MIL_2 Channel 10.DependOnSlot = True; AU7_823_1ML22_MIL_2 Channel 10.DependOnSlotGroup = False; AU7_823_1ML22_MIL_2 Channel 11.Index = 16#7620; AU7_823_1ML22_MIL_2 Channel 11.SubIndex = 11; AU7_823_1ML22_MIL_2 Channel 11.Size = 1; AU7_823_1ML22_MIL_2 Channel 11.Offset = 0; AU7_823_1ML22_MIL_2 Channel 11.DependOnSlot = True; AU7_823_1ML22_MIL_2 Channel 11.DependOnSlotGroup = False; AU7_823_1ML22_MIL_2 Channel 12.Index = 16#7620; AU7_823_1ML22_MIL_2 Channel 12.SubIndex = 12; AU7_823_1ML22_MIL_2 Channel 12.Size = 1; AU7_823_1ML22_MIL_2 Channel 12.Offset = 0; AU7_823_1ML22_MIL_2 Channel 12.DependOnSlot = True; AU7_823_1ML22_MIL_2 Channel 12.DependOnSlotGroup = False; AU7_823_1ML22_MIL_2 Channel 13.Index = 16#7620; AU7_823_1ML22_MIL_2 Channel 13.SubIndex = 13; AU7_823_1ML22_MIL_2 Channel 13.Size = 1; AU7_823_1ML22_MIL_2 Channel 13.Offset = 0; AU7_823_1ML22_MIL_2 Channel 13.DependOnSlot = True; AU7_823_1ML22_MIL_2 Channel 13.DependOnSlotGroup = False; AU7_823_1ML22_MIL_2 Channel 14.Index = 16#7620; AU7_823_1ML22_MIL_2 Channel 14.SubIndex = 14; AU7_823_1ML22_MIL_2 Channel 14.Size = 1; AU7_823_1ML22_MIL_2 Channel 14.Offset = 0; AU7_823_1ML22_MIL_2 Channel 14.DependOnSlot = True; AU7_823_1ML22_MIL_2 Channel 14.DependOnSlotGroup = False; AU7_823_1ML22_MIL_2 Channel 15.Index = 16#7620; AU7_823_1ML22_MIL_2 Channel 15.SubIndex = 15;
            AU7_823_1ML22_MIL_2 Channel 15.Size = 1; AU7_823_1ML22_MIL_2 Channel 15.Offset = 0; AU7_823_1ML22_MIL_2 Channel 15.DependOnSlot = True; AU7_823_1ML22_MIL_2 Channel 15.DependOnSlotGroup = False; AU7_823_1ML22_MIL_2 Channel 16.Index = 16#7620; AU7_823_1ML22_MIL_2 Channel 16.SubIndex = 16; AU7_823_1ML22_MIL_2 Channel 16.Size = 1; AU7_823_1ML22_MIL_2 Channel 16.Offset = 0; AU7_823_1ML22_MIL_2 Channel 16.DependOnSlot = True; AU7_823_1ML22_MIL_2 Channel 16.DependOnSlotGroup = False; RxTxPdo.NumberofExcludes = 4; RxTxPdo.NumberofEntries = 2; RxTxPdo.Index = 16#166B; RxTxPdo.Fixed = True; RxTxPdo.Mandatory = False; RxTxPdo.Virtual = False; RxTxPdo.Sm = -1; RxTxPdo.Su = 0; RxTxPdo.Name = 'Digital Outputs(Byte)'; RxTxPdo.DependOnSlot = True; RxTxPdo.DependOnSlotGroup = False; RxTxPdo.OverwrittenByModule = True; Exclude = [16#166A,16#166C,16#166D,16#166E]; AU7_823_1ML22_MIL_2 Channel 1-8.Index = 16#7621; AU7_823_1ML22_MIL_2 Channel 1-8.SubIndex = 1; AU7_823_1ML22_MIL_2 Channel 1-8.Size = 8; AU7_823_1ML22_MIL_2 Channel 1-8.Offset = 0; AU7_823_1ML22_MIL_2 Channel 1-8.DependOnSlot = True; AU7_823_1ML22_MIL_2 Channel 1-8.DependOnSlotGroup = False; AU7_823_1ML22_MIL_2 Channel 9-16.Index = 16#7621; AU7_823_1ML22_MIL_2 Channel 9-16.SubIndex = 2; AU7_823_1ML22_MIL_2 Channel 9-16.Size = 8; AU7_823_1ML22_MIL_2 Channel 9-16.Offset = 0; AU7_823_1ML22_MIL_2 Channel 9-16.DependOnSlot = True; AU7_823_1ML22_MIL_2 Channel 9-16.DependOnSlotGroup = False; RxTxPdo.NumberofExcludes = 4; RxTxPdo.NumberofEntries = 2; RxTxPdo.Index = 16#166C; RxTxPdo.Fixed = True; RxTxPdo.Mandatory = False;
            RxTxPdo.Virtual = False; RxTxPdo.Sm = -1; RxTxPdo.Su = 0; RxTxPdo.Name = 'Digital Outputs(Arr 8Bit)'; RxTxPdo.DependOnSlot = True; RxTxPdo.DependOnSlotGroup = False; RxTxPdo.OverwrittenByModule = True; Exclude = [16#166A,16#166B,16#166D,16#166E]; AU7_823_1ML22_MIL_2 Channel 1-8.Index = 16#7622; AU7_823_1ML22_MIL_2 Channel 1-8.SubIndex = 1; AU7_823_1ML22_MIL_2 Channel 1-8.Size = 8; AU7_823_1ML22_MIL_2 Channel 1-8.Offset = 0; AU7_823_1ML22_MIL_2 Channel 1-8.DependOnSlot = True; AU7_823_1ML22_MIL_2 Channel 1-8.DependOnSlotGroup = False; AU7_823_1ML22_MIL_2 Channel 9-16.Index = 16#7622; AU7_823_1ML22_MIL_2 Channel 9-16.SubIndex = 2; AU7_823_1ML22_MIL_2 Channel 9-16.Size = 8; AU7_823_1ML22_MIL_2 Channel 9-16.Offset = 0; AU7_823_1ML22_MIL_2 Channel 9-16.DependOnSlot = True; AU7_823_1ML22_MIL_2 Channel 9-16.DependOnSlotGroup = False; RxTxPdo.NumberofExcludes = 4; RxTxPdo.NumberofEntries = 1; RxTxPdo.Index = 16#166D; RxTxPdo.Fixed = True; RxTxPdo.Mandatory = False; RxTxPdo.Virtual = False; RxTxPdo.Sm = -1; RxTxPdo.Su = 0; RxTxPdo.Name = 'Digital Outputs(Arr 16Bit)'; RxTxPdo.DependOnSlot = True; RxTxPdo.DependOnSlotGroup = False; RxTxPdo.OverwrittenByModule = True; Exclude = [16#166A,16#166B,16#166C,16#166E]; AU7_823_1ML22_MIL_2 Channel 1-16.Index = 16#7623; AU7_823_1ML22_MIL_2 Channel 1-16.SubIndex = 1; AU7_823_1ML22_MIL_2 Channel 1-16.Size = 16; AU7_823_1ML22_MIL_2 Channel 1-16.Offset = 0; AU7_823_1ML22_MIL_2 Channel 1-16.DependOnSlot = True; AU7_823_1ML22_MIL_2 Channel 1-16.DependOnSlotGroup = False; RxTxPdo.NumberofExcludes = 4;
            RxTxPdo.NumberofEntries = 1; RxTxPdo.Index = 16#166E; RxTxPdo.Fixed = True; RxTxPdo.Mandatory = False; RxTxPdo.Virtual = False; RxTxPdo.Sm = -1; RxTxPdo.Su = 0; RxTxPdo.Name = 'Digital Outputs(Word)'; RxTxPdo.DependOnSlot = True; RxTxPdo.DependOnSlotGroup = False; RxTxPdo.OverwrittenByModule = True; Exclude = [16#166A,16#166B,16#166C,16#166D]; AU7_823_1ML22_MIL_2 Channel 1-16.Index = 16#7624; AU7_823_1ML22_MIL_2 Channel 1-16.SubIndex = 1; AU7_823_1ML22_MIL_2 Channel 1-16.Size = 16; AU7_823_1ML22_MIL_2 Channel 1-16.Offset = 0; AU7_823_1ML22_MIL_2 Channel 1-16.DependOnSlot = True; AU7_823_1ML22_MIL_2 Channel 1-16.DependOnSlotGroup = False; RxTxPdo.NumberofExcludes = 4; RxTxPdo.NumberofEntries = 16; RxTxPdo.Index = 16#166F; RxTxPdo.Fixed = True; RxTxPdo.Mandatory = False; RxTxPdo.Virtual = False; RxTxPdo.Sm = 2; RxTxPdo.Su = 0; RxTxPdo.Name = 'Digital Outputs(Bit)'; RxTxPdo.DependOnSlot = True; RxTxPdo.DependOnSlotGroup = False; RxTxPdo.OverwrittenByModule = True; Exclude = [16#1670,16#1671,16#1672,16#1673]; AU7_823_1ML22_MIL_3 Channel 1.Index = 16#7630; AU7_823_1ML22_MIL_3 Channel 1.SubIndex = 1; AU7_823_1ML22_MIL_3 Channel 1.Size = 1; AU7_823_1ML22_MIL_3 Channel 1.Offset = 0; AU7_823_1ML22_MIL_3 Channel 1.DependOnSlot = True; AU7_823_1ML22_MIL_3 Channel 1.DependOnSlotGroup = False; AU7_823_1ML22_MIL_3 Channel 2.Index = 16#7630; AU7_823_1ML22_MIL_3 Channel 2.SubIndex = 2; AU7_823_1ML22_MIL_3 Channel 2.Size = 1;
            AU7_823_1ML22_MIL_3 Channel 2.Offset = 0; AU7_823_1ML22_MIL_3 Channel 2.DependOnSlot = True; AU7_823_1ML22_MIL_3 Channel 2.DependOnSlotGroup = False; AU7_823_1ML22_MIL_3 Channel 3.Index = 16#7630; AU7_823_1ML22_MIL_3 Channel 3.SubIndex = 3; AU7_823_1ML22_MIL_3 Channel 3.Size = 1; AU7_823_1ML22_MIL_3 Channel 3.Offset = 0; AU7_823_1ML22_MIL_3 Channel 3.DependOnSlot = True; AU7_823_1ML22_MIL_3 Channel 3.DependOnSlotGroup = False; AU7_823_1ML22_MIL_3 Channel 4.Index = 16#7630; AU7_823_1ML22_MIL_3 Channel 4.SubIndex = 4; AU7_823_1ML22_MIL_3 Channel 4.Size = 1; AU7_823_1ML22_MIL_3 Channel 4.Offset = 0; AU7_823_1ML22_MIL_3 Channel 4.DependOnSlot = True; AU7_823_1ML22_MIL_3 Channel 4.DependOnSlotGroup = False; AU7_823_1ML22_MIL_3 Channel 5.Index = 16#7630; AU7_823_1ML22_MIL_3 Channel 5.SubIndex = 5; AU7_823_1ML22_MIL_3 Channel 5.Size = 1; AU7_823_1ML22_MIL_3 Channel 5.Offset = 0; AU7_823_1ML22_MIL_3 Channel 5.DependOnSlot = True; AU7_823_1ML22_MIL_3 Channel 5.DependOnSlotGroup = False; AU7_823_1ML22_MIL_3 Channel 6.Index = 16#7630; AU7_823_1ML22_MIL_3 Channel 6.SubIndex = 6; AU7_823_1ML22_MIL_3 Channel 6.Size = 1; AU7_823_1ML22_MIL_3 Channel 6.Offset = 0; AU7_823_1ML22_MIL_3 Channel 6.DependOnSlot = True; AU7_823_1ML22_MIL_3 Channel 6.DependOnSlotGroup = False; AU7_823_1ML22_MIL_3 Channel 7.Index = 16#7630; AU7_823_1ML22_MIL_3 Channel 7.SubIndex = 7; AU7_823_1ML22_MIL_3 Channel 7.Size = 1; AU7_823_1ML22_MIL_3 Channel 7.Offset = 0; AU7_823_1ML22_MIL_3 Channel 7.DependOnSlot = True; AU7_823_1ML22_MIL_3 Channel 7.DependOnSlotGroup = False; AU7_823_1ML22_MIL_3 Channel 8.Index = 16#7630; AU7_823_1ML22_MIL_3 Channel 8.SubIndex = 8; AU7_823_1ML22_MIL_3 Channel 8.Size = 1; AU7_823_1ML22_MIL_3 Channel 8.Offset = 0; AU7_823_1ML22_MIL_3 Channel 8.DependOnSlot = True; AU7_823_1ML22_MIL_3 Channel 8.DependOnSlotGroup = False; AU7_823_1ML22_MIL_3 Channel 9.Index = 16#7630;
            AU7_823_1ML22_MIL_3 Channel 9.SubIndex = 9; AU7_823_1ML22_MIL_3 Channel 9.Size = 1; AU7_823_1ML22_MIL_3 Channel 9.Offset = 0; AU7_823_1ML22_MIL_3 Channel 9.DependOnSlot = True; AU7_823_1ML22_MIL_3 Channel 9.DependOnSlotGroup = False; AU7_823_1ML22_MIL_3 Channel 10.Index = 16#7630; AU7_823_1ML22_MIL_3 Channel 10.SubIndex = 10; AU7_823_1ML22_MIL_3 Channel 10.Size = 1; AU7_823_1ML22_MIL_3 Channel 10.Offset = 0; AU7_823_1ML22_MIL_3 Channel 10.DependOnSlot = True; AU7_823_1ML22_MIL_3 Channel 10.DependOnSlotGroup = False; AU7_823_1ML22_MIL_3 Channel 11.Index = 16#7630; AU7_823_1ML22_MIL_3 Channel 11.SubIndex = 11; AU7_823_1ML22_MIL_3 Channel 11.Size = 1; AU7_823_1ML22_MIL_3 Channel 11.Offset = 0; AU7_823_1ML22_MIL_3 Channel 11.DependOnSlot = True; AU7_823_1ML22_MIL_3 Channel 11.DependOnSlotGroup = False; AU7_823_1ML22_MIL_3 Channel 12.Index = 16#7630; AU7_823_1ML22_MIL_3 Channel 12.SubIndex = 12; AU7_823_1ML22_MIL_3 Channel 12.Size = 1; AU7_823_1ML22_MIL_3 Channel 12.Offset = 0; AU7_823_1ML22_MIL_3 Channel 12.DependOnSlot = True; AU7_823_1ML22_MIL_3 Channel 12.DependOnSlotGroup = False; AU7_823_1ML22_MIL_3 Channel 13.Index = 16#7630; AU7_823_1ML22_MIL_3 Channel 13.SubIndex = 13; AU7_823_1ML22_MIL_3 Channel 13.Size = 1; AU7_823_1ML22_MIL_3 Channel 13.Offset = 0; AU7_823_1ML22_MIL_3 Channel 13.DependOnSlot = True; AU7_823_1ML22_MIL_3 Channel 13.DependOnSlotGroup = False; AU7_823_1ML22_MIL_3 Channel 14.Index = 16#7630; AU7_823_1ML22_MIL_3 Channel 14.SubIndex = 14; AU7_823_1ML22_MIL_3 Channel 14.Size = 1; AU7_823_1ML22_MIL_3 Channel 14.Offset = 0; AU7_823_1ML22_MIL_3 Channel 14.DependOnSlot = True; AU7_823_1ML22_MIL_3 Channel 14.DependOnSlotGroup = False; AU7_823_1ML22_MIL_3 Channel 15.Index = 16#7630; AU7_823_1ML22_MIL_3 Channel 15.SubIndex = 15; AU7_823_1ML22_MIL_3 Channel 15.Size = 1; AU7_823_1ML22_MIL_3 Channel 15.Offset = 0; AU7_823_1ML22_MIL_3 Channel 15.DependOnSlot = True;
            AU7_823_1ML22_MIL_3 Channel 15.DependOnSlotGroup = False; AU7_823_1ML22_MIL_3 Channel 16.Index = 16#7630; AU7_823_1ML22_MIL_3 Channel 16.SubIndex = 16; AU7_823_1ML22_MIL_3 Channel 16.Size = 1; AU7_823_1ML22_MIL_3 Channel 16.Offset = 0; AU7_823_1ML22_MIL_3 Channel 16.DependOnSlot = True; AU7_823_1ML22_MIL_3 Channel 16.DependOnSlotGroup = False; RxTxPdo.NumberofExcludes = 4; RxTxPdo.NumberofEntries = 2; RxTxPdo.Index = 16#1670; RxTxPdo.Fixed = True; RxTxPdo.Mandatory = False; RxTxPdo.Virtual = False; RxTxPdo.Sm = -1; RxTxPdo.Su = 0; RxTxPdo.Name = 'Digital Outputs(Byte)'; RxTxPdo.DependOnSlot = True; RxTxPdo.DependOnSlotGroup = False; RxTxPdo.OverwrittenByModule = True; Exclude = [16#166F,16#1671,16#1672,16#1673]; AU7_823_1ML22_MIL_3 Channel 1-8.Index = 16#7631; AU7_823_1ML22_MIL_3 Channel 1-8.SubIndex = 1; AU7_823_1ML22_MIL_3 Channel 1-8.Size = 8; AU7_823_1ML22_MIL_3 Channel 1-8.Offset = 0; AU7_823_1ML22_MIL_3 Channel 1-8.DependOnSlot = True; AU7_823_1ML22_MIL_3 Channel 1-8.DependOnSlotGroup = False; AU7_823_1ML22_MIL_3 Channel 9-16.Index = 16#7631; AU7_823_1ML22_MIL_3 Channel 9-16.SubIndex = 2; AU7_823_1ML22_MIL_3 Channel 9-16.Size = 8; AU7_823_1ML22_MIL_3 Channel 9-16.Offset = 0; AU7_823_1ML22_MIL_3 Channel 9-16.DependOnSlot = True; AU7_823_1ML22_MIL_3 Channel 9-16.DependOnSlotGroup = False; RxTxPdo.NumberofExcludes = 4; RxTxPdo.NumberofEntries = 2; RxTxPdo.Index = 16#1671; RxTxPdo.Fixed = True; RxTxPdo.Mandatory = False; RxTxPdo.Virtual = False; RxTxPdo.Sm = -1; RxTxPdo.Su = 0;
            RxTxPdo.Name = 'Digital Outputs(Arr 8Bit)'; RxTxPdo.DependOnSlot = True; RxTxPdo.DependOnSlotGroup = False; RxTxPdo.OverwrittenByModule = True; Exclude = [16#166F,16#1670,16#1672,16#1673]; AU7_823_1ML22_MIL_3 Channel 1-8.Index = 16#7632; AU7_823_1ML22_MIL_3 Channel 1-8.SubIndex = 1; AU7_823_1ML22_MIL_3 Channel 1-8.Size = 8; AU7_823_1ML22_MIL_3 Channel 1-8.Offset = 0; AU7_823_1ML22_MIL_3 Channel 1-8.DependOnSlot = True; AU7_823_1ML22_MIL_3 Channel 1-8.DependOnSlotGroup = False; AU7_823_1ML22_MIL_3 Channel 9-16.Index = 16#7632; AU7_823_1ML22_MIL_3 Channel 9-16.SubIndex = 2; AU7_823_1ML22_MIL_3 Channel 9-16.Size = 8; AU7_823_1ML22_MIL_3 Channel 9-16.Offset = 0; AU7_823_1ML22_MIL_3 Channel 9-16.DependOnSlot = True; AU7_823_1ML22_MIL_3 Channel 9-16.DependOnSlotGroup = False; RxTxPdo.NumberofExcludes = 4; RxTxPdo.NumberofEntries = 1; RxTxPdo.Index = 16#1672; RxTxPdo.Fixed = True; RxTxPdo.Mandatory = False; RxTxPdo.Virtual = False; RxTxPdo.Sm = -1; RxTxPdo.Su = 0; RxTxPdo.Name = 'Digital Outputs(Arr 16Bit)'; RxTxPdo.DependOnSlot = True; RxTxPdo.DependOnSlotGroup = False; RxTxPdo.OverwrittenByModule = True; Exclude = [16#166F,16#1670,16#1671,16#1673]; AU7_823_1ML22_MIL_3 Channel 1-16.Index = 16#7633; AU7_823_1ML22_MIL_3 Channel 1-16.SubIndex = 1; AU7_823_1ML22_MIL_3 Channel 1-16.Size = 16; AU7_823_1ML22_MIL_3 Channel 1-16.Offset = 0; AU7_823_1ML22_MIL_3 Channel 1-16.DependOnSlot = True; AU7_823_1ML22_MIL_3 Channel 1-16.DependOnSlotGroup = False; RxTxPdo.NumberofExcludes = 4; RxTxPdo.NumberofEntries = 1; RxTxPdo.Index = 16#1673; RxTxPdo.Fixed = True;
            RxTxPdo.Mandatory = False; RxTxPdo.Virtual = False; RxTxPdo.Sm = -1; RxTxPdo.Su = 0; RxTxPdo.Name = 'Digital Outputs(Word)'; RxTxPdo.DependOnSlot = True; RxTxPdo.DependOnSlotGroup = False; RxTxPdo.OverwrittenByModule = True; Exclude = [16#166F,16#1670,16#1671,16#1672]; AU7_823_1ML22_MIL_3 Channel 1-16.Index = 16#7634; AU7_823_1ML22_MIL_3 Channel 1-16.SubIndex = 1; AU7_823_1ML22_MIL_3 Channel 1-16.Size = 16; AU7_823_1ML22_MIL_3 Channel 1-16.Offset = 0; AU7_823_1ML22_MIL_3 Channel 1-16.DependOnSlot = True; AU7_823_1ML22_MIL_3 Channel 1-16.DependOnSlotGroup = False; RxTxPdo.NumberofExcludes = 4; RxTxPdo.NumberofEntries = 16; RxTxPdo.Index = 16#1674; RxTxPdo.Fixed = True; RxTxPdo.Mandatory = False; RxTxPdo.Virtual = False; RxTxPdo.Sm = 2; RxTxPdo.Su = 0; RxTxPdo.Name = 'Digital Outputs(Bit)'; RxTxPdo.DependOnSlot = True; RxTxPdo.DependOnSlotGroup = False; RxTxPdo.OverwrittenByModule = True; Exclude = [16#1675,16#1676,16#1677,16#1678]; AU7_823_1ML22_MIL_4 Channel 1.Index = 16#7640; AU7_823_1ML22_MIL_4 Channel 1.SubIndex = 1; AU7_823_1ML22_MIL_4 Channel 1.Size = 1; AU7_823_1ML22_MIL_4 Channel 1.Offset = 0; AU7_823_1ML22_MIL_4 Channel 1.DependOnSlot = True; AU7_823_1ML22_MIL_4 Channel 1.DependOnSlotGroup = False; AU7_823_1ML22_MIL_4 Channel 2.Index = 16#7640; AU7_823_1ML22_MIL_4 Channel 2.SubIndex = 2; AU7_823_1ML22_MIL_4 Channel 2.Size = 1; AU7_823_1ML22_MIL_4 Channel 2.Offset = 0; AU7_823_1ML22_MIL_4 Channel 2.DependOnSlot = True; AU7_823_1ML22_MIL_4 Channel 2.DependOnSlotGroup = False;
            AU7_823_1ML22_MIL_4 Channel 3.Index = 16#7640; AU7_823_1ML22_MIL_4 Channel 3.SubIndex = 3; AU7_823_1ML22_MIL_4 Channel 3.Size = 1; AU7_823_1ML22_MIL_4 Channel 3.Offset = 0; AU7_823_1ML22_MIL_4 Channel 3.DependOnSlot = True; AU7_823_1ML22_MIL_4 Channel 3.DependOnSlotGroup = False; AU7_823_1ML22_MIL_4 Channel 4.Index = 16#7640; AU7_823_1ML22_MIL_4 Channel 4.SubIndex = 4; AU7_823_1ML22_MIL_4 Channel 4.Size = 1; AU7_823_1ML22_MIL_4 Channel 4.Offset = 0; AU7_823_1ML22_MIL_4 Channel 4.DependOnSlot = True; AU7_823_1ML22_MIL_4 Channel 4.DependOnSlotGroup = False; AU7_823_1ML22_MIL_4 Channel 5.Index = 16#7640; AU7_823_1ML22_MIL_4 Channel 5.SubIndex = 5; AU7_823_1ML22_MIL_4 Channel 5.Size = 1; AU7_823_1ML22_MIL_4 Channel 5.Offset = 0; AU7_823_1ML22_MIL_4 Channel 5.DependOnSlot = True; AU7_823_1ML22_MIL_4 Channel 5.DependOnSlotGroup = False; AU7_823_1ML22_MIL_4 Channel 6.Index = 16#7640; AU7_823_1ML22_MIL_4 Channel 6.SubIndex = 6; AU7_823_1ML22_MIL_4 Channel 6.Size = 1; AU7_823_1ML22_MIL_4 Channel 6.Offset = 0; AU7_823_1ML22_MIL_4 Channel 6.DependOnSlot = True; AU7_823_1ML22_MIL_4 Channel 6.DependOnSlotGroup = False; AU7_823_1ML22_MIL_4 Channel 7.Index = 16#7640; AU7_823_1ML22_MIL_4 Channel 7.SubIndex = 7; AU7_823_1ML22_MIL_4 Channel 7.Size = 1; AU7_823_1ML22_MIL_4 Channel 7.Offset = 0; AU7_823_1ML22_MIL_4 Channel 7.DependOnSlot = True; AU7_823_1ML22_MIL_4 Channel 7.DependOnSlotGroup = False; AU7_823_1ML22_MIL_4 Channel 8.Index = 16#7640; AU7_823_1ML22_MIL_4 Channel 8.SubIndex = 8; AU7_823_1ML22_MIL_4 Channel 8.Size = 1; AU7_823_1ML22_MIL_4 Channel 8.Offset = 0; AU7_823_1ML22_MIL_4 Channel 8.DependOnSlot = True; AU7_823_1ML22_MIL_4 Channel 8.DependOnSlotGroup = False; AU7_823_1ML22_MIL_4 Channel 9.Index = 16#7640; AU7_823_1ML22_MIL_4 Channel 9.SubIndex = 9; AU7_823_1ML22_MIL_4 Channel 9.Size = 1; AU7_823_1ML22_MIL_4 Channel 9.Offset = 0;
            AU7_823_1ML22_MIL_4 Channel 9.DependOnSlot = True; AU7_823_1ML22_MIL_4 Channel 9.DependOnSlotGroup = False; AU7_823_1ML22_MIL_4 Channel 10.Index = 16#7640; AU7_823_1ML22_MIL_4 Channel 10.SubIndex = 10; AU7_823_1ML22_MIL_4 Channel 10.Size = 1; AU7_823_1ML22_MIL_4 Channel 10.Offset = 0; AU7_823_1ML22_MIL_4 Channel 10.DependOnSlot = True; AU7_823_1ML22_MIL_4 Channel 10.DependOnSlotGroup = False; AU7_823_1ML22_MIL_4 Channel 11.Index = 16#7640; AU7_823_1ML22_MIL_4 Channel 11.SubIndex = 11; AU7_823_1ML22_MIL_4 Channel 11.Size = 1; AU7_823_1ML22_MIL_4 Channel 11.Offset = 0; AU7_823_1ML22_MIL_4 Channel 11.DependOnSlot = True; AU7_823_1ML22_MIL_4 Channel 11.DependOnSlotGroup = False; AU7_823_1ML22_MIL_4 Channel 12.Index = 16#7640; AU7_823_1ML22_MIL_4 Channel 12.SubIndex = 12; AU7_823_1ML22_MIL_4 Channel 12.Size = 1; AU7_823_1ML22_MIL_4 Channel 12.Offset = 0; AU7_823_1ML22_MIL_4 Channel 12.DependOnSlot = True; AU7_823_1ML22_MIL_4 Channel 12.DependOnSlotGroup = False; AU7_823_1ML22_MIL_4 Channel 13.Index = 16#7640; AU7_823_1ML22_MIL_4 Channel 13.SubIndex = 13; AU7_823_1ML22_MIL_4 Channel 13.Size = 1; AU7_823_1ML22_MIL_4 Channel 13.Offset = 0; AU7_823_1ML22_MIL_4 Channel 13.DependOnSlot = True; AU7_823_1ML22_MIL_4 Channel 13.DependOnSlotGroup = False; AU7_823_1ML22_MIL_4 Channel 14.Index = 16#7640; AU7_823_1ML22_MIL_4 Channel 14.SubIndex = 14; AU7_823_1ML22_MIL_4 Channel 14.Size = 1; AU7_823_1ML22_MIL_4 Channel 14.Offset = 0; AU7_823_1ML22_MIL_4 Channel 14.DependOnSlot = True; AU7_823_1ML22_MIL_4 Channel 14.DependOnSlotGroup = False; AU7_823_1ML22_MIL_4 Channel 15.Index = 16#7640; AU7_823_1ML22_MIL_4 Channel 15.SubIndex = 15; AU7_823_1ML22_MIL_4 Channel 15.Size = 1; AU7_823_1ML22_MIL_4 Channel 15.Offset = 0; AU7_823_1ML22_MIL_4 Channel 15.DependOnSlot = True; AU7_823_1ML22_MIL_4 Channel 15.DependOnSlotGroup = False; AU7_823_1ML22_MIL_4 Channel 16.Index = 16#7640; AU7_823_1ML22_MIL_4 Channel 16.SubIndex = 16;
            AU7_823_1ML22_MIL_4 Channel 16.Size = 1; AU7_823_1ML22_MIL_4 Channel 16.Offset = 0; AU7_823_1ML22_MIL_4 Channel 16.DependOnSlot = True; AU7_823_1ML22_MIL_4 Channel 16.DependOnSlotGroup = False; RxTxPdo.NumberofExcludes = 4; RxTxPdo.NumberofEntries = 2; RxTxPdo.Index = 16#1675; RxTxPdo.Fixed = True; RxTxPdo.Mandatory = False; RxTxPdo.Virtual = False; RxTxPdo.Sm = -1; RxTxPdo.Su = 0; RxTxPdo.Name = 'Digital Outputs(Byte)'; RxTxPdo.DependOnSlot = True; RxTxPdo.DependOnSlotGroup = False; RxTxPdo.OverwrittenByModule = True; Exclude = [16#1674,16#1676,16#1677,16#1678]; AU7_823_1ML22_MIL_4 Channel 1-8.Index = 16#7641; AU7_823_1ML22_MIL_4 Channel 1-8.SubIndex = 1; AU7_823_1ML22_MIL_4 Channel 1-8.Size = 8; AU7_823_1ML22_MIL_4 Channel 1-8.Offset = 0; AU7_823_1ML22_MIL_4 Channel 1-8.DependOnSlot = True; AU7_823_1ML22_MIL_4 Channel 1-8.DependOnSlotGroup = False; AU7_823_1ML22_MIL_4 Channel 9-16.Index = 16#7641; AU7_823_1ML22_MIL_4 Channel 9-16.SubIndex = 2; AU7_823_1ML22_MIL_4 Channel 9-16.Size = 8; AU7_823_1ML22_MIL_4 Channel 9-16.Offset = 0; AU7_823_1ML22_MIL_4 Channel 9-16.DependOnSlot = True; AU7_823_1ML22_MIL_4 Channel 9-16.DependOnSlotGroup = False; RxTxPdo.NumberofExcludes = 4; RxTxPdo.NumberofEntries = 2; RxTxPdo.Index = 16#1676; RxTxPdo.Fixed = True; RxTxPdo.Mandatory = False; RxTxPdo.Virtual = False; RxTxPdo.Sm = -1; RxTxPdo.Su = 0; RxTxPdo.Name = 'Digital Outputs(Arr 8Bit)'; RxTxPdo.DependOnSlot = True; RxTxPdo.DependOnSlotGroup = False;
            RxTxPdo.OverwrittenByModule = True; Exclude = [16#1674,16#1675,16#1677,16#1678]; AU7_823_1ML22_MIL_4 Channel 1-8.Index = 16#7642; AU7_823_1ML22_MIL_4 Channel 1-8.SubIndex = 1; AU7_823_1ML22_MIL_4 Channel 1-8.Size = 8; AU7_823_1ML22_MIL_4 Channel 1-8.Offset = 0; AU7_823_1ML22_MIL_4 Channel 1-8.DependOnSlot = True; AU7_823_1ML22_MIL_4 Channel 1-8.DependOnSlotGroup = False; AU7_823_1ML22_MIL_4 Channel 9-16.Index = 16#7642; AU7_823_1ML22_MIL_4 Channel 9-16.SubIndex = 2; AU7_823_1ML22_MIL_4 Channel 9-16.Size = 8; AU7_823_1ML22_MIL_4 Channel 9-16.Offset = 0; AU7_823_1ML22_MIL_4 Channel 9-16.DependOnSlot = True; AU7_823_1ML22_MIL_4 Channel 9-16.DependOnSlotGroup = False; RxTxPdo.NumberofExcludes = 4; RxTxPdo.NumberofEntries = 1; RxTxPdo.Index = 16#1677; RxTxPdo.Fixed = True; RxTxPdo.Mandatory = False; RxTxPdo.Virtual = False; RxTxPdo.Sm = -1; RxTxPdo.Su = 0; RxTxPdo.Name = 'Digital Outputs(Arr 16Bit)'; RxTxPdo.DependOnSlot = True; RxTxPdo.DependOnSlotGroup = False; RxTxPdo.OverwrittenByModule = True; Exclude = [16#1674,16#1675,16#1676,16#1678]; AU7_823_1ML22_MIL_4 Channel 1-16.Index = 16#7643; AU7_823_1ML22_MIL_4 Channel 1-16.SubIndex = 1; AU7_823_1ML22_MIL_4 Channel 1-16.Size = 16; AU7_823_1ML22_MIL_4 Channel 1-16.Offset = 0; AU7_823_1ML22_MIL_4 Channel 1-16.DependOnSlot = True; AU7_823_1ML22_MIL_4 Channel 1-16.DependOnSlotGroup = False; RxTxPdo.NumberofExcludes = 4; RxTxPdo.NumberofEntries = 1; RxTxPdo.Index = 16#1678; RxTxPdo.Fixed = True; RxTxPdo.Mandatory = False; RxTxPdo.Virtual = False; RxTxPdo.Sm = -1;
            RxTxPdo.Su = 0; RxTxPdo.Name = 'Digital Outputs(Word)'; RxTxPdo.DependOnSlot = True; RxTxPdo.DependOnSlotGroup = False; RxTxPdo.OverwrittenByModule = True; Exclude = [16#1674,16#1675,16#1676,16#1677]; AU7_823_1ML22_MIL_4 Channel 1-16.Index = 16#7644; AU7_823_1ML22_MIL_4 Channel 1-16.SubIndex = 1; AU7_823_1ML22_MIL_4 Channel 1-16.Size = 16; AU7_823_1ML22_MIL_4 Channel 1-16.Offset = 0; AU7_823_1ML22_MIL_4 Channel 1-16.DependOnSlot = True; AU7_823_1ML22_MIL_4 Channel 1-16.DependOnSlotGroup = False; RxTxPdo.NumberofExcludes = 0; RxTxPdo.NumberofEntries = 1; RxTxPdo.Index = 16#1A00; RxTxPdo.Fixed = True; RxTxPdo.Mandatory = True; RxTxPdo.Virtual = False; RxTxPdo.Sm = 3; RxTxPdo.Su = 3; RxTxPdo.Name = 'ID'; RxTxPdo.DependOnSlot = False; RxTxPdo.DependOnSlotGroup = False; RxTxPdo.OverwrittenByModule = False; ID.Index = 16#6000; ID.SubIndex = 1; ID.Size = 16; ID.Offset = 0; ID.DependOnSlot = False; ID.DependOnSlotGroup = False; RxTxPdo.NumberofExcludes = 4; RxTxPdo.NumberofEntries = 16; RxTxPdo.Index = 16#1A60; RxTxPdo.Fixed = True; RxTxPdo.Mandatory = False; RxTxPdo.Virtual = False; RxTxPdo.Sm = 3; RxTxPdo.Su = 0; RxTxPdo.Name = 'Digital Inputs(Bit)'; RxTxPdo.DependOnSlot = True;
            RxTxPdo.DependOnSlotGroup = False; RxTxPdo.OverwrittenByModule = True; Exclude = [16#1A61,16#1A62,16#1A63,16#1A64]; AU7_823_1ML22_MIL Channel 1.Index = 16#6600; AU7_823_1ML22_MIL Channel 1.SubIndex = 1; AU7_823_1ML22_MIL Channel 1.Size = 1; AU7_823_1ML22_MIL Channel 1.Offset = 0; AU7_823_1ML22_MIL Channel 1.DependOnSlot = True; AU7_823_1ML22_MIL Channel 1.DependOnSlotGroup = False; AU7_823_1ML22_MIL Channel 2.Index = 16#6600; AU7_823_1ML22_MIL Channel 2.SubIndex = 2; AU7_823_1ML22_MIL Channel 2.Size = 1; AU7_823_1ML22_MIL Channel 2.Offset = 0; AU7_823_1ML22_MIL Channel 2.DependOnSlot = True; AU7_823_1ML22_MIL Channel 2.DependOnSlotGroup = False; AU7_823_1ML22_MIL Channel 3.Index = 16#6600; AU7_823_1ML22_MIL Channel 3.SubIndex = 3; AU7_823_1ML22_MIL Channel 3.Size = 1; AU7_823_1ML22_MIL Channel 3.Offset = 0; AU7_823_1ML22_MIL Channel 3.DependOnSlot = True; AU7_823_1ML22_MIL Channel 3.DependOnSlotGroup = False; AU7_823_1ML22_MIL Channel 4.Index = 16#6600; AU7_823_1ML22_MIL Channel 4.SubIndex = 4; AU7_823_1ML22_MIL Channel 4.Size = 1; AU7_823_1ML22_MIL Channel 4.Offset = 0; AU7_823_1ML22_MIL Channel 4.DependOnSlot = True; AU7_823_1ML22_MIL Channel 4.DependOnSlotGroup = False; AU7_823_1ML22_MIL Channel 5.Index = 16#6600; AU7_823_1ML22_MIL Channel 5.SubIndex = 5; AU7_823_1ML22_MIL Channel 5.Size = 1; AU7_823_1ML22_MIL Channel 5.Offset = 0; AU7_823_1ML22_MIL Channel 5.DependOnSlot = True; AU7_823_1ML22_MIL Channel 5.DependOnSlotGroup = False; AU7_823_1ML22_MIL Channel 6.Index = 16#6600; AU7_823_1ML22_MIL Channel 6.SubIndex = 6; AU7_823_1ML22_MIL Channel 6.Size = 1; AU7_823_1ML22_MIL Channel 6.Offset = 0; AU7_823_1ML22_MIL Channel 6.DependOnSlot = True; AU7_823_1ML22_MIL Channel 6.DependOnSlotGroup = False; AU7_823_1ML22_MIL Channel 7.Index = 16#6600;
            AU7_823_1ML22_MIL Channel 7.SubIndex = 7; AU7_823_1ML22_MIL Channel 7.Size = 1; AU7_823_1ML22_MIL Channel 7.Offset = 0; AU7_823_1ML22_MIL Channel 7.DependOnSlot = True; AU7_823_1ML22_MIL Channel 7.DependOnSlotGroup = False; AU7_823_1ML22_MIL Channel 8.Index = 16#6600; AU7_823_1ML22_MIL Channel 8.SubIndex = 8; AU7_823_1ML22_MIL Channel 8.Size = 1; AU7_823_1ML22_MIL Channel 8.Offset = 0; AU7_823_1ML22_MIL Channel 8.DependOnSlot = True; AU7_823_1ML22_MIL Channel 8.DependOnSlotGroup = False; AU7_823_1ML22_MIL Channel 9.Index = 16#6600; AU7_823_1ML22_MIL Channel 9.SubIndex = 9; AU7_823_1ML22_MIL Channel 9.Size = 1; AU7_823_1ML22_MIL Channel 9.Offset = 0; AU7_823_1ML22_MIL Channel 9.DependOnSlot = True; AU7_823_1ML22_MIL Channel 9.DependOnSlotGroup = False; AU7_823_1ML22_MIL Channel 10.Index = 16#6600; AU7_823_1ML22_MIL Channel 10.SubIndex = 10; AU7_823_1ML22_MIL Channel 10.Size = 1; AU7_823_1ML22_MIL Channel 10.Offset = 0; AU7_823_1ML22_MIL Channel 10.DependOnSlot = True; AU7_823_1ML22_MIL Channel 10.DependOnSlotGroup = False; AU7_823_1ML22_MIL Channel 11.Index = 16#6600; AU7_823_1ML22_MIL Channel 11.SubIndex = 11; AU7_823_1ML22_MIL Channel 11.Size = 1; AU7_823_1ML22_MIL Channel 11.Offset = 0; AU7_823_1ML22_MIL Channel 11.DependOnSlot = True; AU7_823_1ML22_MIL Channel 11.DependOnSlotGroup = False; AU7_823_1ML22_MIL Channel 12.Index = 16#6600; AU7_823_1ML22_MIL Channel 12.SubIndex = 12; AU7_823_1ML22_MIL Channel 12.Size = 1; AU7_823_1ML22_MIL Channel 12.Offset = 0; AU7_823_1ML22_MIL Channel 12.DependOnSlot = True; AU7_823_1ML22_MIL Channel 12.DependOnSlotGroup = False; AU7_823_1ML22_MIL Channel 13.Index = 16#6600; AU7_823_1ML22_MIL Channel 13.SubIndex = 13; AU7_823_1ML22_MIL Channel 13.Size = 1; AU7_823_1ML22_MIL Channel 13.Offset = 0; AU7_823_1ML22_MIL Channel 13.DependOnSlot = True;
            AU7_823_1ML22_MIL Channel 13.DependOnSlotGroup = False; AU7_823_1ML22_MIL Channel 14.Index = 16#6600; AU7_823_1ML22_MIL Channel 14.SubIndex = 14; AU7_823_1ML22_MIL Channel 14.Size = 1; AU7_823_1ML22_MIL Channel 14.Offset = 0; AU7_823_1ML22_MIL Channel 14.DependOnSlot = True; AU7_823_1ML22_MIL Channel 14.DependOnSlotGroup = False; AU7_823_1ML22_MIL Channel 15.Index = 16#6600; AU7_823_1ML22_MIL Channel 15.SubIndex = 15; AU7_823_1ML22_MIL Channel 15.Size = 1; AU7_823_1ML22_MIL Channel 15.Offset = 0; AU7_823_1ML22_MIL Channel 15.DependOnSlot = True; AU7_823_1ML22_MIL Channel 15.DependOnSlotGroup = False; AU7_823_1ML22_MIL Channel 16.Index = 16#6600; AU7_823_1ML22_MIL Channel 16.SubIndex = 16; AU7_823_1ML22_MIL Channel 16.Size = 1; AU7_823_1ML22_MIL Channel 16.Offset = 0; AU7_823_1ML22_MIL Channel 16.DependOnSlot = True; AU7_823_1ML22_MIL Channel 16.DependOnSlotGroup = False; RxTxPdo.NumberofExcludes = 4; RxTxPdo.NumberofEntries = 2; RxTxPdo.Index = 16#1A61; RxTxPdo.Fixed = True; RxTxPdo.Mandatory = False; RxTxPdo.Virtual = False; RxTxPdo.Sm = -1; RxTxPdo.Su = 0; RxTxPdo.Name = 'Digital Inputs(Byte)'; RxTxPdo.DependOnSlot = True; RxTxPdo.DependOnSlotGroup = False; RxTxPdo.OverwrittenByModule = True; Exclude = [16#1A60,16#1A62,16#1A63,16#1A64]; AU7_823_1ML22_MIL Channel 1-8.Index = 16#6601; AU7_823_1ML22_MIL Channel 1-8.SubIndex = 1; AU7_823_1ML22_MIL Channel 1-8.Size = 8; AU7_823_1ML22_MIL Channel 1-8.Offset = 0; AU7_823_1ML22_MIL Channel 1-8.DependOnSlot = True; AU7_823_1ML22_MIL Channel 1-8.DependOnSlotGroup = False; AU7_823_1ML22_MIL Channel 9-16.Index = 16#6601; AU7_823_1ML22_MIL Channel 9-16.SubIndex = 2;
            AU7_823_1ML22_MIL Channel 9-16.Size = 8; AU7_823_1ML22_MIL Channel 9-16.Offset = 0; AU7_823_1ML22_MIL Channel 9-16.DependOnSlot = True; AU7_823_1ML22_MIL Channel 9-16.DependOnSlotGroup = False; RxTxPdo.NumberofExcludes = 4; RxTxPdo.NumberofEntries = 2; RxTxPdo.Index = 16#1A62; RxTxPdo.Fixed = True; RxTxPdo.Mandatory = False; RxTxPdo.Virtual = False; RxTxPdo.Sm = -1; RxTxPdo.Su = 0; RxTxPdo.Name = 'Digital Inputs(Arr 8Bit)'; RxTxPdo.DependOnSlot = True; RxTxPdo.DependOnSlotGroup = False; RxTxPdo.OverwrittenByModule = True; Exclude = [16#1A60,16#1A61,16#1A63,16#1A64]; AU7_823_1ML22_MIL Channel 1-8.Index = 16#6602; AU7_823_1ML22_MIL Channel 1-8.SubIndex = 1; AU7_823_1ML22_MIL Channel 1-8.Size = 8; AU7_823_1ML22_MIL Channel 1-8.Offset = 0; AU7_823_1ML22_MIL Channel 1-8.DependOnSlot = True; AU7_823_1ML22_MIL Channel 1-8.DependOnSlotGroup = False; AU7_823_1ML22_MIL Channel 9-16.Index = 16#6602; AU7_823_1ML22_MIL Channel 9-16.SubIndex = 2; AU7_823_1ML22_MIL Channel 9-16.Size = 8; AU7_823_1ML22_MIL Channel 9-16.Offset = 0; AU7_823_1ML22_MIL Channel 9-16.DependOnSlot = True; AU7_823_1ML22_MIL Channel 9-16.DependOnSlotGroup = False; RxTxPdo.NumberofExcludes = 4; RxTxPdo.NumberofEntries = 1; RxTxPdo.Index = 16#1A63; RxTxPdo.Fixed = True; RxTxPdo.Mandatory = False; RxTxPdo.Virtual = False; RxTxPdo.Sm = -1; RxTxPdo.Su = 0; RxTxPdo.Name = 'Digital Inputs(Arr 16Bit)'; RxTxPdo.DependOnSlot = True; RxTxPdo.DependOnSlotGroup = False;
            RxTxPdo.OverwrittenByModule = True; Exclude = [16#1A60,16#1A61,16#1A62,16#1A64]; AU7_823_1ML22_MIL Channel 1-16.Index = 16#6603; AU7_823_1ML22_MIL Channel 1-16.SubIndex = 1; AU7_823_1ML22_MIL Channel 1-16.Size = 16; AU7_823_1ML22_MIL Channel 1-16.Offset = 0; AU7_823_1ML22_MIL Channel 1-16.DependOnSlot = True; AU7_823_1ML22_MIL Channel 1-16.DependOnSlotGroup = False; RxTxPdo.NumberofExcludes = 4; RxTxPdo.NumberofEntries = 1; RxTxPdo.Index = 16#1A64; RxTxPdo.Fixed = True; RxTxPdo.Mandatory = False; RxTxPdo.Virtual = False; RxTxPdo.Sm = -1; RxTxPdo.Su = 0; RxTxPdo.Name = 'Digital Inputs(Word)'; RxTxPdo.DependOnSlot = True; RxTxPdo.DependOnSlotGroup = False; RxTxPdo.OverwrittenByModule = True; Exclude = [16#1A60,16#1A61,16#1A62,16#1A63]; AU7_823_1ML22_MIL Channel 1-16.Index = 16#6604; AU7_823_1ML22_MIL Channel 1-16.SubIndex = 1; AU7_823_1ML22_MIL Channel 1-16.Size = 16; AU7_823_1ML22_MIL Channel 1-16.Offset = 0; AU7_823_1ML22_MIL Channel 1-16.DependOnSlot = True; AU7_823_1ML22_MIL Channel 1-16.DependOnSlotGroup = False; RxTxPdo.NumberofExcludes = 4; RxTxPdo.NumberofEntries = 16; RxTxPdo.Index = 16#1A65; RxTxPdo.Fixed = True; RxTxPdo.Mandatory = False; RxTxPdo.Virtual = False; RxTxPdo.Sm = 3; RxTxPdo.Su = 0; RxTxPdo.Name = 'Digital Inputs(Bit)'; RxTxPdo.DependOnSlot = True; RxTxPdo.DependOnSlotGroup = False; RxTxPdo.OverwrittenByModule = True; Exclude = [16#1A66,16#1A67,16#1A68,16#1A69];
            AU7_823_1ML22_MIL_1 Channel 1.Index = 16#6610; AU7_823_1ML22_MIL_1 Channel 1.SubIndex = 1; AU7_823_1ML22_MIL_1 Channel 1.Size = 1; AU7_823_1ML22_MIL_1 Channel 1.Offset = 0; AU7_823_1ML22_MIL_1 Channel 1.DependOnSlot = True; AU7_823_1ML22_MIL_1 Channel 1.DependOnSlotGroup = False; AU7_823_1ML22_MIL_1 Channel 2.Index = 16#6610; AU7_823_1ML22_MIL_1 Channel 2.SubIndex = 2; AU7_823_1ML22_MIL_1 Channel 2.Size = 1; AU7_823_1ML22_MIL_1 Channel 2.Offset = 0; AU7_823_1ML22_MIL_1 Channel 2.DependOnSlot = True; AU7_823_1ML22_MIL_1 Channel 2.DependOnSlotGroup = False; AU7_823_1ML22_MIL_1 Channel 3.Index = 16#6610; AU7_823_1ML22_MIL_1 Channel 3.SubIndex = 3; AU7_823_1ML22_MIL_1 Channel 3.Size = 1; AU7_823_1ML22_MIL_1 Channel 3.Offset = 0; AU7_823_1ML22_MIL_1 Channel 3.DependOnSlot = True; AU7_823_1ML22_MIL_1 Channel 3.DependOnSlotGroup = False; AU7_823_1ML22_MIL_1 Channel 4.Index = 16#6610; AU7_823_1ML22_MIL_1 Channel 4.SubIndex = 4; AU7_823_1ML22_MIL_1 Channel 4.Size = 1; AU7_823_1ML22_MIL_1 Channel 4.Offset = 0; AU7_823_1ML22_MIL_1 Channel 4.DependOnSlot = True; AU7_823_1ML22_MIL_1 Channel 4.DependOnSlotGroup = False; AU7_823_1ML22_MIL_1 Channel 5.Index = 16#6610; AU7_823_1ML22_MIL_1 Channel 5.SubIndex = 5; AU7_823_1ML22_MIL_1 Channel 5.Size = 1; AU7_823_1ML22_MIL_1 Channel 5.Offset = 0; AU7_823_1ML22_MIL_1 Channel 5.DependOnSlot = True; AU7_823_1ML22_MIL_1 Channel 5.DependOnSlotGroup = False; AU7_823_1ML22_MIL_1 Channel 6.Index = 16#6610; AU7_823_1ML22_MIL_1 Channel 6.SubIndex = 6; AU7_823_1ML22_MIL_1 Channel 6.Size = 1; AU7_823_1ML22_MIL_1 Channel 6.Offset = 0; AU7_823_1ML22_MIL_1 Channel 6.DependOnSlot = True; AU7_823_1ML22_MIL_1 Channel 6.DependOnSlotGroup = False; AU7_823_1ML22_MIL_1 Channel 7.Index = 16#6610; AU7_823_1ML22_MIL_1 Channel 7.SubIndex = 7; AU7_823_1ML22_MIL_1 Channel 7.Size = 1; AU7_823_1ML22_MIL_1 Channel 7.Offset = 0;
            AU7_823_1ML22_MIL_1 Channel 7.DependOnSlot = True; AU7_823_1ML22_MIL_1 Channel 7.DependOnSlotGroup = False; AU7_823_1ML22_MIL_1 Channel 8.Index = 16#6610; AU7_823_1ML22_MIL_1 Channel 8.SubIndex = 8; AU7_823_1ML22_MIL_1 Channel 8.Size = 1; AU7_823_1ML22_MIL_1 Channel 8.Offset = 0; AU7_823_1ML22_MIL_1 Channel 8.DependOnSlot = True; AU7_823_1ML22_MIL_1 Channel 8.DependOnSlotGroup = False; AU7_823_1ML22_MIL_1 Channel 9.Index = 16#6610; AU7_823_1ML22_MIL_1 Channel 9.SubIndex = 9; AU7_823_1ML22_MIL_1 Channel 9.Size = 1; AU7_823_1ML22_MIL_1 Channel 9.Offset = 0; AU7_823_1ML22_MIL_1 Channel 9.DependOnSlot = True; AU7_823_1ML22_MIL_1 Channel 9.DependOnSlotGroup = False; AU7_823_1ML22_MIL_1 Channel 10.Index = 16#6610; AU7_823_1ML22_MIL_1 Channel 10.SubIndex = 10; AU7_823_1ML22_MIL_1 Channel 10.Size = 1; AU7_823_1ML22_MIL_1 Channel 10.Offset = 0; AU7_823_1ML22_MIL_1 Channel 10.DependOnSlot = True; AU7_823_1ML22_MIL_1 Channel 10.DependOnSlotGroup = False; AU7_823_1ML22_MIL_1 Channel 11.Index = 16#6610; AU7_823_1ML22_MIL_1 Channel 11.SubIndex = 11; AU7_823_1ML22_MIL_1 Channel 11.Size = 1; AU7_823_1ML22_MIL_1 Channel 11.Offset = 0; AU7_823_1ML22_MIL_1 Channel 11.DependOnSlot = True; AU7_823_1ML22_MIL_1 Channel 11.DependOnSlotGroup = False; AU7_823_1ML22_MIL_1 Channel 12.Index = 16#6610; AU7_823_1ML22_MIL_1 Channel 12.SubIndex = 12; AU7_823_1ML22_MIL_1 Channel 12.Size = 1; AU7_823_1ML22_MIL_1 Channel 12.Offset = 0; AU7_823_1ML22_MIL_1 Channel 12.DependOnSlot = True; AU7_823_1ML22_MIL_1 Channel 12.DependOnSlotGroup = False; AU7_823_1ML22_MIL_1 Channel 13.Index = 16#6610; AU7_823_1ML22_MIL_1 Channel 13.SubIndex = 13; AU7_823_1ML22_MIL_1 Channel 13.Size = 1; AU7_823_1ML22_MIL_1 Channel 13.Offset = 0; AU7_823_1ML22_MIL_1 Channel 13.DependOnSlot = True; AU7_823_1ML22_MIL_1 Channel 13.DependOnSlotGroup = False; AU7_823_1ML22_MIL_1 Channel 14.Index = 16#6610; AU7_823_1ML22_MIL_1 Channel 14.SubIndex = 14;
            AU7_823_1ML22_MIL_1 Channel 14.Size = 1; AU7_823_1ML22_MIL_1 Channel 14.Offset = 0; AU7_823_1ML22_MIL_1 Channel 14.DependOnSlot = True; AU7_823_1ML22_MIL_1 Channel 14.DependOnSlotGroup = False; AU7_823_1ML22_MIL_1 Channel 15.Index = 16#6610; AU7_823_1ML22_MIL_1 Channel 15.SubIndex = 15; AU7_823_1ML22_MIL_1 Channel 15.Size = 1; AU7_823_1ML22_MIL_1 Channel 15.Offset = 0; AU7_823_1ML22_MIL_1 Channel 15.DependOnSlot = True; AU7_823_1ML22_MIL_1 Channel 15.DependOnSlotGroup = False; AU7_823_1ML22_MIL_1 Channel 16.Index = 16#6610; AU7_823_1ML22_MIL_1 Channel 16.SubIndex = 16; AU7_823_1ML22_MIL_1 Channel 16.Size = 1; AU7_823_1ML22_MIL_1 Channel 16.Offset = 0; AU7_823_1ML22_MIL_1 Channel 16.DependOnSlot = True; AU7_823_1ML22_MIL_1 Channel 16.DependOnSlotGroup = False; RxTxPdo.NumberofExcludes = 4; RxTxPdo.NumberofEntries = 2; RxTxPdo.Index = 16#1A66; RxTxPdo.Fixed = True; RxTxPdo.Mandatory = False; RxTxPdo.Virtual = False; RxTxPdo.Sm = -1; RxTxPdo.Su = 0; RxTxPdo.Name = 'Digital Inputs(Byte)'; RxTxPdo.DependOnSlot = True; RxTxPdo.DependOnSlotGroup = False; RxTxPdo.OverwrittenByModule = True; Exclude = [16#1A65,16#1A67,16#1A68,16#1A69]; AU7_823_1ML22_MIL_1 Channel 1-8.Index = 16#6611; AU7_823_1ML22_MIL_1 Channel 1-8.SubIndex = 1; AU7_823_1ML22_MIL_1 Channel 1-8.Size = 8; AU7_823_1ML22_MIL_1 Channel 1-8.Offset = 0; AU7_823_1ML22_MIL_1 Channel 1-8.DependOnSlot = True; AU7_823_1ML22_MIL_1 Channel 1-8.DependOnSlotGroup = False; AU7_823_1ML22_MIL_1 Channel 9-16.Index = 16#6611; AU7_823_1ML22_MIL_1 Channel 9-16.SubIndex = 2; AU7_823_1ML22_MIL_1 Channel 9-16.Size = 8; AU7_823_1ML22_MIL_1 Channel 9-16.Offset = 0; AU7_823_1ML22_MIL_1 Channel 9-16.DependOnSlot = True;
            AU7_823_1ML22_MIL_1 Channel 9-16.DependOnSlotGroup = False; RxTxPdo.NumberofExcludes = 4; RxTxPdo.NumberofEntries = 2; RxTxPdo.Index = 16#1A67; RxTxPdo.Fixed = True; RxTxPdo.Mandatory = False; RxTxPdo.Virtual = False; RxTxPdo.Sm = -1; RxTxPdo.Su = 0; RxTxPdo.Name = 'Digital Inputs(Arr 8Bit)'; RxTxPdo.DependOnSlot = True; RxTxPdo.DependOnSlotGroup = False; RxTxPdo.OverwrittenByModule = True; Exclude = [16#1A65,16#1A66,16#1A68,16#1A69]; AU7_823_1ML22_MIL_1 Channel 1-8.Index = 16#6612; AU7_823_1ML22_MIL_1 Channel 1-8.SubIndex = 1; AU7_823_1ML22_MIL_1 Channel 1-8.Size = 8; AU7_823_1ML22_MIL_1 Channel 1-8.Offset = 0; AU7_823_1ML22_MIL_1 Channel 1-8.DependOnSlot = True; AU7_823_1ML22_MIL_1 Channel 1-8.DependOnSlotGroup = False; AU7_823_1ML22_MIL_1 Channel 9-16.Index = 16#6612; AU7_823_1ML22_MIL_1 Channel 9-16.SubIndex = 2; AU7_823_1ML22_MIL_1 Channel 9-16.Size = 8; AU7_823_1ML22_MIL_1 Channel 9-16.Offset = 0; AU7_823_1ML22_MIL_1 Channel 9-16.DependOnSlot = True; AU7_823_1ML22_MIL_1 Channel 9-16.DependOnSlotGroup = False; RxTxPdo.NumberofExcludes = 4; RxTxPdo.NumberofEntries = 1; RxTxPdo.Index = 16#1A68; RxTxPdo.Fixed = True; RxTxPdo.Mandatory = False; RxTxPdo.Virtual = False; RxTxPdo.Sm = -1; RxTxPdo.Su = 0; RxTxPdo.Name = 'Digital Inputs(Arr 16Bit)'; RxTxPdo.DependOnSlot = True; RxTxPdo.DependOnSlotGroup = False; RxTxPdo.OverwrittenByModule = True; Exclude = [16#1A65,16#1A66,16#1A67,16#1A69]; AU7_823_1ML22_MIL_1 Channel 1-16.Index = 16#6613;
            AU7_823_1ML22_MIL_1 Channel 1-16.SubIndex = 1; AU7_823_1ML22_MIL_1 Channel 1-16.Size = 16; AU7_823_1ML22_MIL_1 Channel 1-16.Offset = 0; AU7_823_1ML22_MIL_1 Channel 1-16.DependOnSlot = True; AU7_823_1ML22_MIL_1 Channel 1-16.DependOnSlotGroup = False; RxTxPdo.NumberofExcludes = 4; RxTxPdo.NumberofEntries = 1; RxTxPdo.Index = 16#1A69; RxTxPdo.Fixed = True; RxTxPdo.Mandatory = False; RxTxPdo.Virtual = False; RxTxPdo.Sm = -1; RxTxPdo.Su = 0; RxTxPdo.Name = 'Digital Inputs(Word)'; RxTxPdo.DependOnSlot = True; RxTxPdo.DependOnSlotGroup = False; RxTxPdo.OverwrittenByModule = True; Exclude = [16#1A65,16#1A66,16#1A67,16#1A68]; AU7_823_1ML22_MIL_1 Channel 1-16.Index = 16#6614; AU7_823_1ML22_MIL_1 Channel 1-16.SubIndex = 1; AU7_823_1ML22_MIL_1 Channel 1-16.Size = 16; AU7_823_1ML22_MIL_1 Channel 1-16.Offset = 0; AU7_823_1ML22_MIL_1 Channel 1-16.DependOnSlot = True; AU7_823_1ML22_MIL_1 Channel 1-16.DependOnSlotGroup = False; RxTxPdo.NumberofExcludes = 4; RxTxPdo.NumberofEntries = 16; RxTxPdo.Index = 16#1A6A; RxTxPdo.Fixed = True; RxTxPdo.Mandatory = False; RxTxPdo.Virtual = False; RxTxPdo.Sm = 3; RxTxPdo.Su = 0; RxTxPdo.Name = 'Digital Inputs(Bit)'; RxTxPdo.DependOnSlot = True; RxTxPdo.DependOnSlotGroup = False; RxTxPdo.OverwrittenByModule = True; Exclude = [16#1A6B,16#1A6C,16#1A6D,16#1A6E]; AU7_823_1ML22_MIL_2 Channel 1.Index = 16#6620; AU7_823_1ML22_MIL_2 Channel 1.SubIndex = 1; AU7_823_1ML22_MIL_2 Channel 1.Size = 1;
            AU7_823_1ML22_MIL_2 Channel 1.Offset = 0; AU7_823_1ML22_MIL_2 Channel 1.DependOnSlot = True; AU7_823_1ML22_MIL_2 Channel 1.DependOnSlotGroup = False; AU7_823_1ML22_MIL_2 Channel 2.Index = 16#6620; AU7_823_1ML22_MIL_2 Channel 2.SubIndex = 2; AU7_823_1ML22_MIL_2 Channel 2.Size = 1; AU7_823_1ML22_MIL_2 Channel 2.Offset = 0; AU7_823_1ML22_MIL_2 Channel 2.DependOnSlot = True; AU7_823_1ML22_MIL_2 Channel 2.DependOnSlotGroup = False; AU7_823_1ML22_MIL_2 Channel 3.Index = 16#6620; AU7_823_1ML22_MIL_2 Channel 3.SubIndex = 3; AU7_823_1ML22_MIL_2 Channel 3.Size = 1; AU7_823_1ML22_MIL_2 Channel 3.Offset = 0; AU7_823_1ML22_MIL_2 Channel 3.DependOnSlot = True; AU7_823_1ML22_MIL_2 Channel 3.DependOnSlotGroup = False; AU7_823_1ML22_MIL_2 Channel 4.Index = 16#6620; AU7_823_1ML22_MIL_2 Channel 4.SubIndex = 4; AU7_823_1ML22_MIL_2 Channel 4.Size = 1; AU7_823_1ML22_MIL_2 Channel 4.Offset = 0; AU7_823_1ML22_MIL_2 Channel 4.DependOnSlot = True; AU7_823_1ML22_MIL_2 Channel 4.DependOnSlotGroup = False; AU7_823_1ML22_MIL_2 Channel 5.Index = 16#6620; AU7_823_1ML22_MIL_2 Channel 5.SubIndex = 5; AU7_823_1ML22_MIL_2 Channel 5.Size = 1; AU7_823_1ML22_MIL_2 Channel 5.Offset = 0; AU7_823_1ML22_MIL_2 Channel 5.DependOnSlot = True; AU7_823_1ML22_MIL_2 Channel 5.DependOnSlotGroup = False; AU7_823_1ML22_MIL_2 Channel 6.Index = 16#6620; AU7_823_1ML22_MIL_2 Channel 6.SubIndex = 6; AU7_823_1ML22_MIL_2 Channel 6.Size = 1; AU7_823_1ML22_MIL_2 Channel 6.Offset = 0; AU7_823_1ML22_MIL_2 Channel 6.DependOnSlot = True; AU7_823_1ML22_MIL_2 Channel 6.DependOnSlotGroup = False; AU7_823_1ML22_MIL_2 Channel 7.Index = 16#6620; AU7_823_1ML22_MIL_2 Channel 7.SubIndex = 7; AU7_823_1ML22_MIL_2 Channel 7.Size = 1; AU7_823_1ML22_MIL_2 Channel 7.Offset = 0; AU7_823_1ML22_MIL_2 Channel 7.DependOnSlot = True; AU7_823_1ML22_MIL_2 Channel 7.DependOnSlotGroup = False; AU7_823_1ML22_MIL_2 Channel 8.Index = 16#6620;
            AU7_823_1ML22_MIL_2 Channel 8.SubIndex = 8; AU7_823_1ML22_MIL_2 Channel 8.Size = 1; AU7_823_1ML22_MIL_2 Channel 8.Offset = 0; AU7_823_1ML22_MIL_2 Channel 8.DependOnSlot = True; AU7_823_1ML22_MIL_2 Channel 8.DependOnSlotGroup = False; AU7_823_1ML22_MIL_2 Channel 9.Index = 16#6620; AU7_823_1ML22_MIL_2 Channel 9.SubIndex = 9; AU7_823_1ML22_MIL_2 Channel 9.Size = 1; AU7_823_1ML22_MIL_2 Channel 9.Offset = 0; AU7_823_1ML22_MIL_2 Channel 9.DependOnSlot = True; AU7_823_1ML22_MIL_2 Channel 9.DependOnSlotGroup = False; AU7_823_1ML22_MIL_2 Channel 10.Index = 16#6620; AU7_823_1ML22_MIL_2 Channel 10.SubIndex = 10; AU7_823_1ML22_MIL_2 Channel 10.Size = 1; AU7_823_1ML22_MIL_2 Channel 10.Offset = 0; AU7_823_1ML22_MIL_2 Channel 10.DependOnSlot = True; AU7_823_1ML22_MIL_2 Channel 10.DependOnSlotGroup = False; AU7_823_1ML22_MIL_2 Channel 11.Index = 16#6620; AU7_823_1ML22_MIL_2 Channel 11.SubIndex = 11; AU7_823_1ML22_MIL_2 Channel 11.Size = 1; AU7_823_1ML22_MIL_2 Channel 11.Offset = 0; AU7_823_1ML22_MIL_2 Channel 11.DependOnSlot = True; AU7_823_1ML22_MIL_2 Channel 11.DependOnSlotGroup = False; AU7_823_1ML22_MIL_2 Channel 12.Index = 16#6620; AU7_823_1ML22_MIL_2 Channel 12.SubIndex = 12; AU7_823_1ML22_MIL_2 Channel 12.Size = 1; AU7_823_1ML22_MIL_2 Channel 12.Offset = 0; AU7_823_1ML22_MIL_2 Channel 12.DependOnSlot = True; AU7_823_1ML22_MIL_2 Channel 12.DependOnSlotGroup = False; AU7_823_1ML22_MIL_2 Channel 13.Index = 16#6620; AU7_823_1ML22_MIL_2 Channel 13.SubIndex = 13; AU7_823_1ML22_MIL_2 Channel 13.Size = 1; AU7_823_1ML22_MIL_2 Channel 13.Offset = 0; AU7_823_1ML22_MIL_2 Channel 13.DependOnSlot = True; AU7_823_1ML22_MIL_2 Channel 13.DependOnSlotGroup = False; AU7_823_1ML22_MIL_2 Channel 14.Index = 16#6620; AU7_823_1ML22_MIL_2 Channel 14.SubIndex = 14; AU7_823_1ML22_MIL_2 Channel 14.Size = 1; AU7_823_1ML22_MIL_2 Channel 14.Offset = 0; AU7_823_1ML22_MIL_2 Channel 14.DependOnSlot = True;
            AU7_823_1ML22_MIL_2 Channel 14.DependOnSlotGroup = False; AU7_823_1ML22_MIL_2 Channel 15.Index = 16#6620; AU7_823_1ML22_MIL_2 Channel 15.SubIndex = 15; AU7_823_1ML22_MIL_2 Channel 15.Size = 1; AU7_823_1ML22_MIL_2 Channel 15.Offset = 0; AU7_823_1ML22_MIL_2 Channel 15.DependOnSlot = True; AU7_823_1ML22_MIL_2 Channel 15.DependOnSlotGroup = False; AU7_823_1ML22_MIL_2 Channel 16.Index = 16#6620; AU7_823_1ML22_MIL_2 Channel 16.SubIndex = 16; AU7_823_1ML22_MIL_2 Channel 16.Size = 1; AU7_823_1ML22_MIL_2 Channel 16.Offset = 0; AU7_823_1ML22_MIL_2 Channel 16.DependOnSlot = True; AU7_823_1ML22_MIL_2 Channel 16.DependOnSlotGroup = False; RxTxPdo.NumberofExcludes = 4; RxTxPdo.NumberofEntries = 2; RxTxPdo.Index = 16#1A6B; RxTxPdo.Fixed = True; RxTxPdo.Mandatory = False; RxTxPdo.Virtual = False; RxTxPdo.Sm = -1; RxTxPdo.Su = 0; RxTxPdo.Name = 'Digital Inputs(Byte)'; RxTxPdo.DependOnSlot = True; RxTxPdo.DependOnSlotGroup = False; RxTxPdo.OverwrittenByModule = True; Exclude = [16#1A6A,16#1A6C,16#1A6D,16#1A6E]; AU7_823_1ML22_MIL_2 Channel 1-8.Index = 16#6621; AU7_823_1ML22_MIL_2 Channel 1-8.SubIndex = 1; AU7_823_1ML22_MIL_2 Channel 1-8.Size = 8; AU7_823_1ML22_MIL_2 Channel 1-8.Offset = 0; AU7_823_1ML22_MIL_2 Channel 1-8.DependOnSlot = True; AU7_823_1ML22_MIL_2 Channel 1-8.DependOnSlotGroup = False; AU7_823_1ML22_MIL_2 Channel 9-16.Index = 16#6621; AU7_823_1ML22_MIL_2 Channel 9-16.SubIndex = 2; AU7_823_1ML22_MIL_2 Channel 9-16.Size = 8; AU7_823_1ML22_MIL_2 Channel 9-16.Offset = 0; AU7_823_1ML22_MIL_2 Channel 9-16.DependOnSlot = True; AU7_823_1ML22_MIL_2 Channel 9-16.DependOnSlotGroup = False; RxTxPdo.NumberofExcludes = 4; RxTxPdo.NumberofEntries = 2;
            RxTxPdo.Index = 16#1A6C; RxTxPdo.Fixed = True; RxTxPdo.Mandatory = False; RxTxPdo.Virtual = False; RxTxPdo.Sm = -1; RxTxPdo.Su = 0; RxTxPdo.Name = 'Digital Inputs(Arr 8Bit)'; RxTxPdo.DependOnSlot = True; RxTxPdo.DependOnSlotGroup = False; RxTxPdo.OverwrittenByModule = True; Exclude = [16#1A6A,16#1A6B,16#1A6D,16#1A6E]; AU7_823_1ML22_MIL_2 Channel 1-8.Index = 16#6622; AU7_823_1ML22_MIL_2 Channel 1-8.SubIndex = 1; AU7_823_1ML22_MIL_2 Channel 1-8.Size = 8; AU7_823_1ML22_MIL_2 Channel 1-8.Offset = 0; AU7_823_1ML22_MIL_2 Channel 1-8.DependOnSlot = True; AU7_823_1ML22_MIL_2 Channel 1-8.DependOnSlotGroup = False; AU7_823_1ML22_MIL_2 Channel 9-16.Index = 16#6622; AU7_823_1ML22_MIL_2 Channel 9-16.SubIndex = 2; AU7_823_1ML22_MIL_2 Channel 9-16.Size = 8; AU7_823_1ML22_MIL_2 Channel 9-16.Offset = 0; AU7_823_1ML22_MIL_2 Channel 9-16.DependOnSlot = True; AU7_823_1ML22_MIL_2 Channel 9-16.DependOnSlotGroup = False; RxTxPdo.NumberofExcludes = 4; RxTxPdo.NumberofEntries = 1; RxTxPdo.Index = 16#1A6D; RxTxPdo.Fixed = True; RxTxPdo.Mandatory = False; RxTxPdo.Virtual = False; RxTxPdo.Sm = -1; RxTxPdo.Su = 0; RxTxPdo.Name = 'Digital Inputs(Arr 16Bit)'; RxTxPdo.DependOnSlot = True; RxTxPdo.DependOnSlotGroup = False; RxTxPdo.OverwrittenByModule = True; Exclude = [16#1A6A,16#1A6B,16#1A6C,16#1A6E]; AU7_823_1ML22_MIL_2 Channel 1-16.Index = 16#6623; AU7_823_1ML22_MIL_2 Channel 1-16.SubIndex = 1; AU7_823_1ML22_MIL_2 Channel 1-16.Size = 16; AU7_823_1ML22_MIL_2 Channel 1-16.Offset = 0;
            AU7_823_1ML22_MIL_2 Channel 1-16.DependOnSlot = True; AU7_823_1ML22_MIL_2 Channel 1-16.DependOnSlotGroup = False; RxTxPdo.NumberofExcludes = 4; RxTxPdo.NumberofEntries = 1; RxTxPdo.Index = 16#1A6E; RxTxPdo.Fixed = True; RxTxPdo.Mandatory = False; RxTxPdo.Virtual = False; RxTxPdo.Sm = -1; RxTxPdo.Su = 0; RxTxPdo.Name = 'Digital Inputs(Word)'; RxTxPdo.DependOnSlot = True; RxTxPdo.DependOnSlotGroup = False; RxTxPdo.OverwrittenByModule = True; Exclude = [16#1A6A,16#1A6B,16#1A6C,16#1A6D]; AU7_823_1ML22_MIL_2 Channel 1-16.Index = 16#6624; AU7_823_1ML22_MIL_2 Channel 1-16.SubIndex = 1; AU7_823_1ML22_MIL_2 Channel 1-16.Size = 16; AU7_823_1ML22_MIL_2 Channel 1-16.Offset = 0; AU7_823_1ML22_MIL_2 Channel 1-16.DependOnSlot = True; AU7_823_1ML22_MIL_2 Channel 1-16.DependOnSlotGroup = False; RxTxPdo.NumberofExcludes = 4; RxTxPdo.NumberofEntries = 16; RxTxPdo.Index = 16#1A6F; RxTxPdo.Fixed = True; RxTxPdo.Mandatory = False; RxTxPdo.Virtual = False; RxTxPdo.Sm = 3; RxTxPdo.Su = 0; RxTxPdo.Name = 'Digital Inputs(Bit)'; RxTxPdo.DependOnSlot = True; RxTxPdo.DependOnSlotGroup = False; RxTxPdo.OverwrittenByModule = True; Exclude = [16#1A70,16#1A71,16#1A72,16#1A73]; AU7_823_1ML22_MIL_3 Channel 1.Index = 16#6630; AU7_823_1ML22_MIL_3 Channel 1.SubIndex = 1; AU7_823_1ML22_MIL_3 Channel 1.Size = 1; AU7_823_1ML22_MIL_3 Channel 1.Offset = 0; AU7_823_1ML22_MIL_3 Channel 1.DependOnSlot = True; AU7_823_1ML22_MIL_3 Channel 1.DependOnSlotGroup = False;
            AU7_823_1ML22_MIL_3 Channel 2.Index = 16#6630; AU7_823_1ML22_MIL_3 Channel 2.SubIndex = 2; AU7_823_1ML22_MIL_3 Channel 2.Size = 1; AU7_823_1ML22_MIL_3 Channel 2.Offset = 0; AU7_823_1ML22_MIL_3 Channel 2.DependOnSlot = True; AU7_823_1ML22_MIL_3 Channel 2.DependOnSlotGroup = False; AU7_823_1ML22_MIL_3 Channel 3.Index = 16#6630; AU7_823_1ML22_MIL_3 Channel 3.SubIndex = 3; AU7_823_1ML22_MIL_3 Channel 3.Size = 1; AU7_823_1ML22_MIL_3 Channel 3.Offset = 0; AU7_823_1ML22_MIL_3 Channel 3.DependOnSlot = True; AU7_823_1ML22_MIL_3 Channel 3.DependOnSlotGroup = False; AU7_823_1ML22_MIL_3 Channel 4.Index = 16#6630; AU7_823_1ML22_MIL_3 Channel 4.SubIndex = 4; AU7_823_1ML22_MIL_3 Channel 4.Size = 1; AU7_823_1ML22_MIL_3 Channel 4.Offset = 0; AU7_823_1ML22_MIL_3 Channel 4.DependOnSlot = True; AU7_823_1ML22_MIL_3 Channel 4.DependOnSlotGroup = False; AU7_823_1ML22_MIL_3 Channel 5.Index = 16#6630; AU7_823_1ML22_MIL_3 Channel 5.SubIndex = 5; AU7_823_1ML22_MIL_3 Channel 5.Size = 1; AU7_823_1ML22_MIL_3 Channel 5.Offset = 0; AU7_823_1ML22_MIL_3 Channel 5.DependOnSlot = True; AU7_823_1ML22_MIL_3 Channel 5.DependOnSlotGroup = False; AU7_823_1ML22_MIL_3 Channel 6.Index = 16#6630; AU7_823_1ML22_MIL_3 Channel 6.SubIndex = 6; AU7_823_1ML22_MIL_3 Channel 6.Size = 1; AU7_823_1ML22_MIL_3 Channel 6.Offset = 0; AU7_823_1ML22_MIL_3 Channel 6.DependOnSlot = True; AU7_823_1ML22_MIL_3 Channel 6.DependOnSlotGroup = False; AU7_823_1ML22_MIL_3 Channel 7.Index = 16#6630; AU7_823_1ML22_MIL_3 Channel 7.SubIndex = 7; AU7_823_1ML22_MIL_3 Channel 7.Size = 1; AU7_823_1ML22_MIL_3 Channel 7.Offset = 0; AU7_823_1ML22_MIL_3 Channel 7.DependOnSlot = True; AU7_823_1ML22_MIL_3 Channel 7.DependOnSlotGroup = False; AU7_823_1ML22_MIL_3 Channel 8.Index = 16#6630; AU7_823_1ML22_MIL_3 Channel 8.SubIndex = 8; AU7_823_1ML22_MIL_3 Channel 8.Size = 1; AU7_823_1ML22_MIL_3 Channel 8.Offset = 0;
            AU7_823_1ML22_MIL_3 Channel 8.DependOnSlot = True; AU7_823_1ML22_MIL_3 Channel 8.DependOnSlotGroup = False; AU7_823_1ML22_MIL_3 Channel 9.Index = 16#6630; AU7_823_1ML22_MIL_3 Channel 9.SubIndex = 9; AU7_823_1ML22_MIL_3 Channel 9.Size = 1; AU7_823_1ML22_MIL_3 Channel 9.Offset = 0; AU7_823_1ML22_MIL_3 Channel 9.DependOnSlot = True; AU7_823_1ML22_MIL_3 Channel 9.DependOnSlotGroup = False; AU7_823_1ML22_MIL_3 Channel 10.Index = 16#6630; AU7_823_1ML22_MIL_3 Channel 10.SubIndex = 10; AU7_823_1ML22_MIL_3 Channel 10.Size = 1; AU7_823_1ML22_MIL_3 Channel 10.Offset = 0; AU7_823_1ML22_MIL_3 Channel 10.DependOnSlot = True; AU7_823_1ML22_MIL_3 Channel 10.DependOnSlotGroup = False; AU7_823_1ML22_MIL_3 Channel 11.Index = 16#6630; AU7_823_1ML22_MIL_3 Channel 11.SubIndex = 11; AU7_823_1ML22_MIL_3 Channel 11.Size = 1; AU7_823_1ML22_MIL_3 Channel 11.Offset = 0; AU7_823_1ML22_MIL_3 Channel 11.DependOnSlot = True; AU7_823_1ML22_MIL_3 Channel 11.DependOnSlotGroup = False; AU7_823_1ML22_MIL_3 Channel 12.Index = 16#6630; AU7_823_1ML22_MIL_3 Channel 12.SubIndex = 12; AU7_823_1ML22_MIL_3 Channel 12.Size = 1; AU7_823_1ML22_MIL_3 Channel 12.Offset = 0; AU7_823_1ML22_MIL_3 Channel 12.DependOnSlot = True; AU7_823_1ML22_MIL_3 Channel 12.DependOnSlotGroup = False; AU7_823_1ML22_MIL_3 Channel 13.Index = 16#6630; AU7_823_1ML22_MIL_3 Channel 13.SubIndex = 13; AU7_823_1ML22_MIL_3 Channel 13.Size = 1; AU7_823_1ML22_MIL_3 Channel 13.Offset = 0; AU7_823_1ML22_MIL_3 Channel 13.DependOnSlot = True; AU7_823_1ML22_MIL_3 Channel 13.DependOnSlotGroup = False; AU7_823_1ML22_MIL_3 Channel 14.Index = 16#6630; AU7_823_1ML22_MIL_3 Channel 14.SubIndex = 14; AU7_823_1ML22_MIL_3 Channel 14.Size = 1; AU7_823_1ML22_MIL_3 Channel 14.Offset = 0; AU7_823_1ML22_MIL_3 Channel 14.DependOnSlot = True; AU7_823_1ML22_MIL_3 Channel 14.DependOnSlotGroup = False; AU7_823_1ML22_MIL_3 Channel 15.Index = 16#6630; AU7_823_1ML22_MIL_3 Channel 15.SubIndex = 15;
            AU7_823_1ML22_MIL_3 Channel 15.Size = 1; AU7_823_1ML22_MIL_3 Channel 15.Offset = 0; AU7_823_1ML22_MIL_3 Channel 15.DependOnSlot = True; AU7_823_1ML22_MIL_3 Channel 15.DependOnSlotGroup = False; AU7_823_1ML22_MIL_3 Channel 16.Index = 16#6630; AU7_823_1ML22_MIL_3 Channel 16.SubIndex = 16; AU7_823_1ML22_MIL_3 Channel 16.Size = 1; AU7_823_1ML22_MIL_3 Channel 16.Offset = 0; AU7_823_1ML22_MIL_3 Channel 16.DependOnSlot = True; AU7_823_1ML22_MIL_3 Channel 16.DependOnSlotGroup = False; RxTxPdo.NumberofExcludes = 4; RxTxPdo.NumberofEntries = 2; RxTxPdo.Index = 16#1A70; RxTxPdo.Fixed = True; RxTxPdo.Mandatory = False; RxTxPdo.Virtual = False; RxTxPdo.Sm = -1; RxTxPdo.Su = 0; RxTxPdo.Name = 'Digital Inputs(Byte)'; RxTxPdo.DependOnSlot = True; RxTxPdo.DependOnSlotGroup = False; RxTxPdo.OverwrittenByModule = True; Exclude = [16#1A6F,16#1A71,16#1A72,16#1A73]; AU7_823_1ML22_MIL_3 Channel 1-8.Index = 16#6631; AU7_823_1ML22_MIL_3 Channel 1-8.SubIndex = 1; AU7_823_1ML22_MIL_3 Channel 1-8.Size = 8; AU7_823_1ML22_MIL_3 Channel 1-8.Offset = 0; AU7_823_1ML22_MIL_3 Channel 1-8.DependOnSlot = True; AU7_823_1ML22_MIL_3 Channel 1-8.DependOnSlotGroup = False; AU7_823_1ML22_MIL_3 Channel 9-16.Index = 16#6631; AU7_823_1ML22_MIL_3 Channel 9-16.SubIndex = 2; AU7_823_1ML22_MIL_3 Channel 9-16.Size = 8; AU7_823_1ML22_MIL_3 Channel 9-16.Offset = 0; AU7_823_1ML22_MIL_3 Channel 9-16.DependOnSlot = True; AU7_823_1ML22_MIL_3 Channel 9-16.DependOnSlotGroup = False; RxTxPdo.NumberofExcludes = 4; RxTxPdo.NumberofEntries = 2; RxTxPdo.Index = 16#1A71; RxTxPdo.Fixed = True; RxTxPdo.Mandatory = False;
            RxTxPdo.Virtual = False; RxTxPdo.Sm = -1; RxTxPdo.Su = 0; RxTxPdo.Name = 'Digital Inputs(Arr 8Bit)'; RxTxPdo.DependOnSlot = True; RxTxPdo.DependOnSlotGroup = False; RxTxPdo.OverwrittenByModule = True; Exclude = [16#1A6F,16#1A70,16#1A72,16#1A73]; AU7_823_1ML22_MIL_3 Channel 1-8.Index = 16#6632; AU7_823_1ML22_MIL_3 Channel 1-8.SubIndex = 1; AU7_823_1ML22_MIL_3 Channel 1-8.Size = 8; AU7_823_1ML22_MIL_3 Channel 1-8.Offset = 0; AU7_823_1ML22_MIL_3 Channel 1-8.DependOnSlot = True; AU7_823_1ML22_MIL_3 Channel 1-8.DependOnSlotGroup = False; AU7_823_1ML22_MIL_3 Channel 9-16.Index = 16#6632; AU7_823_1ML22_MIL_3 Channel 9-16.SubIndex = 2; AU7_823_1ML22_MIL_3 Channel 9-16.Size = 8; AU7_823_1ML22_MIL_3 Channel 9-16.Offset = 0; AU7_823_1ML22_MIL_3 Channel 9-16.DependOnSlot = True; AU7_823_1ML22_MIL_3 Channel 9-16.DependOnSlotGroup = False; RxTxPdo.NumberofExcludes = 4; RxTxPdo.NumberofEntries = 1; RxTxPdo.Index = 16#1A72; RxTxPdo.Fixed = True; RxTxPdo.Mandatory = False; RxTxPdo.Virtual = False; RxTxPdo.Sm = -1; RxTxPdo.Su = 0; RxTxPdo.Name = 'Digital Inputs(Arr 16Bit)'; RxTxPdo.DependOnSlot = True; RxTxPdo.DependOnSlotGroup = False; RxTxPdo.OverwrittenByModule = True; Exclude = [16#1A6F,16#1A70,16#1A71,16#1A73]; AU7_823_1ML22_MIL_3 Channel 1-16.Index = 16#6633; AU7_823_1ML22_MIL_3 Channel 1-16.SubIndex = 1; AU7_823_1ML22_MIL_3 Channel 1-16.Size = 16; AU7_823_1ML22_MIL_3 Channel 1-16.Offset = 0; AU7_823_1ML22_MIL_3 Channel 1-16.DependOnSlot = True; AU7_823_1ML22_MIL_3 Channel 1-16.DependOnSlotGroup = False; RxTxPdo.NumberofExcludes = 4;
            RxTxPdo.NumberofEntries = 1; RxTxPdo.Index = 16#1A73; RxTxPdo.Fixed = True; RxTxPdo.Mandatory = False; RxTxPdo.Virtual = False; RxTxPdo.Sm = -1; RxTxPdo.Su = 0; RxTxPdo.Name = 'Digital Inputs(Word)'; RxTxPdo.DependOnSlot = True; RxTxPdo.DependOnSlotGroup = False; RxTxPdo.OverwrittenByModule = True; Exclude = [16#1A6F,16#1A70,16#1A71,16#1A72]; AU7_823_1ML22_MIL_3 Channel 1-16.Index = 16#6634; AU7_823_1ML22_MIL_3 Channel 1-16.SubIndex = 1; AU7_823_1ML22_MIL_3 Channel 1-16.Size = 16; AU7_823_1ML22_MIL_3 Channel 1-16.Offset = 0; AU7_823_1ML22_MIL_3 Channel 1-16.DependOnSlot = True; AU7_823_1ML22_MIL_3 Channel 1-16.DependOnSlotGroup = False; RxTxPdo.NumberofExcludes = 4; RxTxPdo.NumberofEntries = 16; RxTxPdo.Index = 16#1A74; RxTxPdo.Fixed = True; RxTxPdo.Mandatory = False; RxTxPdo.Virtual = False; RxTxPdo.Sm = 3; RxTxPdo.Su = 0; RxTxPdo.Name = 'Digital Inputs(Bit)'; RxTxPdo.DependOnSlot = True; RxTxPdo.DependOnSlotGroup = False; RxTxPdo.OverwrittenByModule = True; Exclude = [16#1A75,16#1A76,16#1A77,16#1A78]; AU7_823_1ML22_MIL_4 Channel 1.Index = 16#6640; AU7_823_1ML22_MIL_4 Channel 1.SubIndex = 1; AU7_823_1ML22_MIL_4 Channel 1.Size = 1; AU7_823_1ML22_MIL_4 Channel 1.Offset = 0; AU7_823_1ML22_MIL_4 Channel 1.DependOnSlot = True; AU7_823_1ML22_MIL_4 Channel 1.DependOnSlotGroup = False; AU7_823_1ML22_MIL_4 Channel 2.Index = 16#6640; AU7_823_1ML22_MIL_4 Channel 2.SubIndex = 2; AU7_823_1ML22_MIL_4 Channel 2.Size = 1;
            AU7_823_1ML22_MIL_4 Channel 2.Offset = 0; AU7_823_1ML22_MIL_4 Channel 2.DependOnSlot = True; AU7_823_1ML22_MIL_4 Channel 2.DependOnSlotGroup = False; AU7_823_1ML22_MIL_4 Channel 3.Index = 16#6640; AU7_823_1ML22_MIL_4 Channel 3.SubIndex = 3; AU7_823_1ML22_MIL_4 Channel 3.Size = 1; AU7_823_1ML22_MIL_4 Channel 3.Offset = 0; AU7_823_1ML22_MIL_4 Channel 3.DependOnSlot = True; AU7_823_1ML22_MIL_4 Channel 3.DependOnSlotGroup = False; AU7_823_1ML22_MIL_4 Channel 4.Index = 16#6640; AU7_823_1ML22_MIL_4 Channel 4.SubIndex = 4; AU7_823_1ML22_MIL_4 Channel 4.Size = 1; AU7_823_1ML22_MIL_4 Channel 4.Offset = 0; AU7_823_1ML22_MIL_4 Channel 4.DependOnSlot = True; AU7_823_1ML22_MIL_4 Channel 4.DependOnSlotGroup = False; AU7_823_1ML22_MIL_4 Channel 5.Index = 16#6640; AU7_823_1ML22_MIL_4 Channel 5.SubIndex = 5; AU7_823_1ML22_MIL_4 Channel 5.Size = 1; AU7_823_1ML22_MIL_4 Channel 5.Offset = 0; AU7_823_1ML22_MIL_4 Channel 5.DependOnSlot = True; AU7_823_1ML22_MIL_4 Channel 5.DependOnSlotGroup = False; AU7_823_1ML22_MIL_4 Channel 6.Index = 16#6640; AU7_823_1ML22_MIL_4 Channel 6.SubIndex = 6; AU7_823_1ML22_MIL_4 Channel 6.Size = 1; AU7_823_1ML22_MIL_4 Channel 6.Offset = 0; AU7_823_1ML22_MIL_4 Channel 6.DependOnSlot = True; AU7_823_1ML22_MIL_4 Channel 6.DependOnSlotGroup = False; AU7_823_1ML22_MIL_4 Channel 7.Index = 16#6640; AU7_823_1ML22_MIL_4 Channel 7.SubIndex = 7; AU7_823_1ML22_MIL_4 Channel 7.Size = 1; AU7_823_1ML22_MIL_4 Channel 7.Offset = 0; AU7_823_1ML22_MIL_4 Channel 7.DependOnSlot = True; AU7_823_1ML22_MIL_4 Channel 7.DependOnSlotGroup = False; AU7_823_1ML22_MIL_4 Channel 8.Index = 16#6640; AU7_823_1ML22_MIL_4 Channel 8.SubIndex = 8; AU7_823_1ML22_MIL_4 Channel 8.Size = 1; AU7_823_1ML22_MIL_4 Channel 8.Offset = 0; AU7_823_1ML22_MIL_4 Channel 8.DependOnSlot = True; AU7_823_1ML22_MIL_4 Channel 8.DependOnSlotGroup = False; AU7_823_1ML22_MIL_4 Channel 9.Index = 16#6640;
            AU7_823_1ML22_MIL_4 Channel 9.SubIndex = 9; AU7_823_1ML22_MIL_4 Channel 9.Size = 1; AU7_823_1ML22_MIL_4 Channel 9.Offset = 0; AU7_823_1ML22_MIL_4 Channel 9.DependOnSlot = True; AU7_823_1ML22_MIL_4 Channel 9.DependOnSlotGroup = False; AU7_823_1ML22_MIL_4 Channel 10.Index = 16#6640; AU7_823_1ML22_MIL_4 Channel 10.SubIndex = 10; AU7_823_1ML22_MIL_4 Channel 10.Size = 1; AU7_823_1ML22_MIL_4 Channel 10.Offset = 0; AU7_823_1ML22_MIL_4 Channel 10.DependOnSlot = True; AU7_823_1ML22_MIL_4 Channel 10.DependOnSlotGroup = False; AU7_823_1ML22_MIL_4 Channel 11.Index = 16#6640; AU7_823_1ML22_MIL_4 Channel 11.SubIndex = 11; AU7_823_1ML22_MIL_4 Channel 11.Size = 1; AU7_823_1ML22_MIL_4 Channel 11.Offset = 0; AU7_823_1ML22_MIL_4 Channel 11.DependOnSlot = True; AU7_823_1ML22_MIL_4 Channel 11.DependOnSlotGroup = False; AU7_823_1ML22_MIL_4 Channel 12.Index = 16#6640; AU7_823_1ML22_MIL_4 Channel 12.SubIndex = 12; AU7_823_1ML22_MIL_4 Channel 12.Size = 1; AU7_823_1ML22_MIL_4 Channel 12.Offset = 0; AU7_823_1ML22_MIL_4 Channel 12.DependOnSlot = True; AU7_823_1ML22_MIL_4 Channel 12.DependOnSlotGroup = False; AU7_823_1ML22_MIL_4 Channel 13.Index = 16#6640; AU7_823_1ML22_MIL_4 Channel 13.SubIndex = 13; AU7_823_1ML22_MIL_4 Channel 13.Size = 1; AU7_823_1ML22_MIL_4 Channel 13.Offset = 0; AU7_823_1ML22_MIL_4 Channel 13.DependOnSlot = True; AU7_823_1ML22_MIL_4 Channel 13.DependOnSlotGroup = False; AU7_823_1ML22_MIL_4 Channel 14.Index = 16#6640; AU7_823_1ML22_MIL_4 Channel 14.SubIndex = 14; AU7_823_1ML22_MIL_4 Channel 14.Size = 1; AU7_823_1ML22_MIL_4 Channel 14.Offset = 0; AU7_823_1ML22_MIL_4 Channel 14.DependOnSlot = True; AU7_823_1ML22_MIL_4 Channel 14.DependOnSlotGroup = False; AU7_823_1ML22_MIL_4 Channel 15.Index = 16#6640; AU7_823_1ML22_MIL_4 Channel 15.SubIndex = 15; AU7_823_1ML22_MIL_4 Channel 15.Size = 1; AU7_823_1ML22_MIL_4 Channel 15.Offset = 0; AU7_823_1ML22_MIL_4 Channel 15.DependOnSlot = True;
            AU7_823_1ML22_MIL_4 Channel 15.DependOnSlotGroup = False; AU7_823_1ML22_MIL_4 Channel 16.Index = 16#6640; AU7_823_1ML22_MIL_4 Channel 16.SubIndex = 16; AU7_823_1ML22_MIL_4 Channel 16.Size = 1; AU7_823_1ML22_MIL_4 Channel 16.Offset = 0; AU7_823_1ML22_MIL_4 Channel 16.DependOnSlot = True; AU7_823_1ML22_MIL_4 Channel 16.DependOnSlotGroup = False; RxTxPdo.NumberofExcludes = 4; RxTxPdo.NumberofEntries = 2; RxTxPdo.Index = 16#1A75; RxTxPdo.Fixed = True; RxTxPdo.Mandatory = False; RxTxPdo.Virtual = False; RxTxPdo.Sm = -1; RxTxPdo.Su = 0; RxTxPdo.Name = 'Digital Inputs(Byte)'; RxTxPdo.DependOnSlot = True; RxTxPdo.DependOnSlotGroup = False; RxTxPdo.OverwrittenByModule = True; Exclude = [16#1A74,16#1A76,16#1A77,16#1A78]; AU7_823_1ML22_MIL_4 Channel 1-8.Index = 16#6641; AU7_823_1ML22_MIL_4 Channel 1-8.SubIndex = 1; AU7_823_1ML22_MIL_4 Channel 1-8.Size = 8; AU7_823_1ML22_MIL_4 Channel 1-8.Offset = 0; AU7_823_1ML22_MIL_4 Channel 1-8.DependOnSlot = True; AU7_823_1ML22_MIL_4 Channel 1-8.DependOnSlotGroup = False; AU7_823_1ML22_MIL_4 Channel 9-16.Index = 16#6641; AU7_823_1ML22_MIL_4 Channel 9-16.SubIndex = 2; AU7_823_1ML22_MIL_4 Channel 9-16.Size = 8; AU7_823_1ML22_MIL_4 Channel 9-16.Offset = 0; AU7_823_1ML22_MIL_4 Channel 9-16.DependOnSlot = True; AU7_823_1ML22_MIL_4 Channel 9-16.DependOnSlotGroup = False; RxTxPdo.NumberofExcludes = 4; RxTxPdo.NumberofEntries = 2; RxTxPdo.Index = 16#1A76; RxTxPdo.Fixed = True; RxTxPdo.Mandatory = False; RxTxPdo.Virtual = False; RxTxPdo.Sm = -1; RxTxPdo.Su = 0;
            RxTxPdo.Name = 'Digital Inputs(Arr 8Bit)'; RxTxPdo.DependOnSlot = True; RxTxPdo.DependOnSlotGroup = False; RxTxPdo.OverwrittenByModule = True; Exclude = [16#1A74,16#1A75,16#1A77,16#1A78]; AU7_823_1ML22_MIL_4 Channel 1-8.Index = 16#6642; AU7_823_1ML22_MIL_4 Channel 1-8.SubIndex = 1; AU7_823_1ML22_MIL_4 Channel 1-8.Size = 8; AU7_823_1ML22_MIL_4 Channel 1-8.Offset = 0; AU7_823_1ML22_MIL_4 Channel 1-8.DependOnSlot = True; AU7_823_1ML22_MIL_4 Channel 1-8.DependOnSlotGroup = False; AU7_823_1ML22_MIL_4 Channel 9-16.Index = 16#6642; AU7_823_1ML22_MIL_4 Channel 9-16.SubIndex = 2; AU7_823_1ML22_MIL_4 Channel 9-16.Size = 8; AU7_823_1ML22_MIL_4 Channel 9-16.Offset = 0; AU7_823_1ML22_MIL_4 Channel 9-16.DependOnSlot = True; AU7_823_1ML22_MIL_4 Channel 9-16.DependOnSlotGroup = False; RxTxPdo.NumberofExcludes = 4; RxTxPdo.NumberofEntries = 1; RxTxPdo.Index = 16#1A77; RxTxPdo.Fixed = True; RxTxPdo.Mandatory = False; RxTxPdo.Virtual = False; RxTxPdo.Sm = -1; RxTxPdo.Su = 0; RxTxPdo.Name = 'Digital Inputs(Arr 16Bit)'; RxTxPdo.DependOnSlot = True; RxTxPdo.DependOnSlotGroup = False; RxTxPdo.OverwrittenByModule = True; Exclude = [16#1A74,16#1A75,16#1A76,16#1A78]; AU7_823_1ML22_MIL_4 Channel 1-16.Index = 16#6643; AU7_823_1ML22_MIL_4 Channel 1-16.SubIndex = 1; AU7_823_1ML22_MIL_4 Channel 1-16.Size = 16; AU7_823_1ML22_MIL_4 Channel 1-16.Offset = 0; AU7_823_1ML22_MIL_4 Channel 1-16.DependOnSlot = True; AU7_823_1ML22_MIL_4 Channel 1-16.DependOnSlotGroup = False; RxTxPdo.NumberofExcludes = 4; RxTxPdo.NumberofEntries = 1; RxTxPdo.Index = 16#1A78; RxTxPdo.Fixed = True;
            RxTxPdo.Mandatory = False; RxTxPdo.Virtual = False; RxTxPdo.Sm = -1; RxTxPdo.Su = 0; RxTxPdo.Name = 'Digital Inputs(Word)'; RxTxPdo.DependOnSlot = True; RxTxPdo.DependOnSlotGroup = False; RxTxPdo.OverwrittenByModule = True; Exclude = [16#1A74,16#1A75,16#1A76,16#1A77]; AU7_823_1ML22_MIL_4 Channel 1-16.Index = 16#6644; AU7_823_1ML22_MIL_4 Channel 1-16.SubIndex = 1; AU7_823_1ML22_MIL_4 Channel 1-16.Size = 16; AU7_823_1ML22_MIL_4 Channel 1-16.Offset = 0; AU7_823_1ML22_MIL_4 Channel 1-16.DependOnSlot = True; AU7_823_1ML22_MIL_4 Channel 1-16.DependOnSlotGroup = False; AU7_823_1ML22_MIL Channel 1.Name = 'AU7_823_1ML22_MIL Channel 1'; AU7_823_1ML22_MIL Channel 1.DataType = 'BOOL'; AU7_823_1ML22_MIL Channel 1.Default = ''; AU7_823_1ML22_MIL Channel 1.Comment = ''; AU7_823_1ML22_MIL Channel 2.Name = 'AU7_823_1ML22_MIL Channel 2'; AU7_823_1ML22_MIL Channel 2.DataType = 'BOOL'; AU7_823_1ML22_MIL Channel 2.Default = ''; AU7_823_1ML22_MIL Channel 2.Comment = ''; AU7_823_1ML22_MIL Channel 3.Name = 'AU7_823_1ML22_MIL Channel 3'; AU7_823_1ML22_MIL Channel 3.DataType = 'BOOL'; AU7_823_1ML22_MIL Channel 3.Default = ''; AU7_823_1ML22_MIL Channel 3.Comment = ''; AU7_823_1ML22_MIL Channel 4.Name = 'AU7_823_1ML22_MIL Channel 4'; AU7_823_1ML22_MIL Channel 4.DataType = 'BOOL'; AU7_823_1ML22_MIL Channel 4.Default = ''; AU7_823_1ML22_MIL Channel 4.Comment = ''; AU7_823_1ML22_MIL Channel 5.Name = 'AU7_823_1ML22_MIL Channel 5'; AU7_823_1ML22_MIL Channel 5.DataType = 'BOOL'; AU7_823_1ML22_MIL Channel 5.Default = ''; AU7_823_1ML22_MIL Channel 5.Comment = ''; AU7_823_1ML22_MIL Channel 6.Name = 'AU7_823_1ML22_MIL Channel 6'; AU7_823_1ML22_MIL Channel 6.DataType = 'BOOL'; AU7_823_1ML22_MIL Channel 6.Default = ''; AU7_823_1ML22_MIL Channel 6.Comment = ''; AU7_823_1ML22_MIL Channel 7.Name = 'AU7_823_1ML22_MIL Channel 7';
            AU7_823_1ML22_MIL Channel 7.DataType = 'BOOL'; AU7_823_1ML22_MIL Channel 7.Default = ''; AU7_823_1ML22_MIL Channel 7.Comment = ''; AU7_823_1ML22_MIL Channel 8.Name = 'AU7_823_1ML22_MIL Channel 8'; AU7_823_1ML22_MIL Channel 8.DataType = 'BOOL'; AU7_823_1ML22_MIL Channel 8.Default = ''; AU7_823_1ML22_MIL Channel 8.Comment = ''; AU7_823_1ML22_MIL Channel 9.Name = 'AU7_823_1ML22_MIL Channel 9'; AU7_823_1ML22_MIL Channel 9.DataType = 'BOOL'; AU7_823_1ML22_MIL Channel 9.Default = ''; AU7_823_1ML22_MIL Channel 9.Comment = ''; AU7_823_1ML22_MIL Channel 10.Name = 'AU7_823_1ML22_MIL Channel 10'; AU7_823_1ML22_MIL Channel 10.DataType = 'BOOL'; AU7_823_1ML22_MIL Channel 10.Default = ''; AU7_823_1ML22_MIL Channel 10.Comment = ''; AU7_823_1ML22_MIL Channel 11.Name = 'AU7_823_1ML22_MIL Channel 11'; AU7_823_1ML22_MIL Channel 11.DataType = 'BOOL'; AU7_823_1ML22_MIL Channel 11.Default = ''; AU7_823_1ML22_MIL Channel 11.Comment = ''; AU7_823_1ML22_MIL Channel 12.Name = 'AU7_823_1ML22_MIL Channel 12'; AU7_823_1ML22_MIL Channel 12.DataType = 'BOOL'; AU7_823_1ML22_MIL Channel 12.Default = ''; AU7_823_1ML22_MIL Channel 12.Comment = ''; AU7_823_1ML22_MIL Channel 13.Name = 'AU7_823_1ML22_MIL Channel 13'; AU7_823_1ML22_MIL Channel 13.DataType = 'BOOL'; AU7_823_1ML22_MIL Channel 13.Default = ''; AU7_823_1ML22_MIL Channel 13.Comment = ''; AU7_823_1ML22_MIL Channel 14.Name = 'AU7_823_1ML22_MIL Channel 14'; AU7_823_1ML22_MIL Channel 14.DataType = 'BOOL'; AU7_823_1ML22_MIL Channel 14.Default = ''; AU7_823_1ML22_MIL Channel 14.Comment = ''; AU7_823_1ML22_MIL Channel 15.Name = 'AU7_823_1ML22_MIL Channel 15'; AU7_823_1ML22_MIL Channel 15.DataType = 'BOOL'; AU7_823_1ML22_MIL Channel 15.Default = ''; AU7_823_1ML22_MIL Channel 15.Comment = ''; AU7_823_1ML22_MIL Channel 16.Name = 'AU7_823_1ML22_MIL Channel 16'; AU7_823_1ML22_MIL Channel 16.DataType = 'BOOL'; AU7_823_1ML22_MIL Channel 16.Default = ''; AU7_823_1ML22_MIL Channel 16.Comment = ''; AU7_823_1ML22_MIL Channel 1-8.Name = 'AU7_823_1ML22_MIL Channel 1-8';
            AU7_823_1ML22_MIL Channel 1-8.DataType = 'USINT'; AU7_823_1ML22_MIL Channel 1-8.Default = ''; AU7_823_1ML22_MIL Channel 1-8.Comment = ''; AU7_823_1ML22_MIL Channel 9-16.Name = 'AU7_823_1ML22_MIL Channel 9-16'; AU7_823_1ML22_MIL Channel 9-16.DataType = 'USINT'; AU7_823_1ML22_MIL Channel 9-16.Default = ''; AU7_823_1ML22_MIL Channel 9-16.Comment = ''; AU7_823_1ML22_MIL Channel 1-8.Name = 'AU7_823_1ML22_MIL Channel 1-8'; AU7_823_1ML22_MIL Channel 1-8.DataType = 'BIT'; AU7_823_1ML22_MIL Channel 1-8.Default = ''; AU7_823_1ML22_MIL Channel 1-8.Comment = ''; AU7_823_1ML22_MIL Channel 9-16.Name = 'AU7_823_1ML22_MIL Channel 9-16'; AU7_823_1ML22_MIL Channel 9-16.DataType = 'BIT'; AU7_823_1ML22_MIL Channel 9-16.Default = ''; AU7_823_1ML22_MIL Channel 9-16.Comment = ''; AU7_823_1ML22_MIL Channel 1-16.Name = 'AU7_823_1ML22_MIL Channel 1-16'; AU7_823_1ML22_MIL Channel 1-16.DataType = 'BIT'; AU7_823_1ML22_MIL Channel 1-16.Default = ''; AU7_823_1ML22_MIL Channel 1-16.Comment = ''; AU7_823_1ML22_MIL Channel 1-16.Name = 'AU7_823_1ML22_MIL Channel 1-16'; AU7_823_1ML22_MIL Channel 1-16.DataType = 'UINT'; AU7_823_1ML22_MIL Channel 1-16.Default = ''; AU7_823_1ML22_MIL Channel 1-16.Comment = ''; AU7_823_1ML22_MIL_1 Channel 1.Name = 'AU7_823_1ML22_MIL_1 Channel 1'; AU7_823_1ML22_MIL_1 Channel 1.DataType = 'BOOL'; AU7_823_1ML22_MIL_1 Channel 1.Default = ''; AU7_823_1ML22_MIL_1 Channel 1.Comment = ''; AU7_823_1ML22_MIL_1 Channel 2.Name = 'AU7_823_1ML22_MIL_1 Channel 2'; AU7_823_1ML22_MIL_1 Channel 2.DataType = 'BOOL'; AU7_823_1ML22_MIL_1 Channel 2.Default = ''; AU7_823_1ML22_MIL_1 Channel 2.Comment = ''; AU7_823_1ML22_MIL_1 Channel 3.Name = 'AU7_823_1ML22_MIL_1 Channel 3'; AU7_823_1ML22_MIL_1 Channel 3.DataType = 'BOOL'; AU7_823_1ML22_MIL_1 Channel 3.Default = ''; AU7_823_1ML22_MIL_1 Channel 3.Comment = ''; AU7_823_1ML22_MIL_1 Channel 4.Name = 'AU7_823_1ML22_MIL_1 Channel 4'; AU7_823_1ML22_MIL_1 Channel 4.DataType = 'BOOL'; AU7_823_1ML22_MIL_1 Channel 4.Default = ''; AU7_823_1ML22_MIL_1 Channel 4.Comment = ''; AU7_823_1ML22_MIL_1 Channel 5.Name = 'AU7_823_1ML22_MIL_1 Channel 5';
            AU7_823_1ML22_MIL_1 Channel 5.DataType = 'BOOL'; AU7_823_1ML22_MIL_1 Channel 5.Default = ''; AU7_823_1ML22_MIL_1 Channel 5.Comment = ''; AU7_823_1ML22_MIL_1 Channel 6.Name = 'AU7_823_1ML22_MIL_1 Channel 6'; AU7_823_1ML22_MIL_1 Channel 6.DataType = 'BOOL'; AU7_823_1ML22_MIL_1 Channel 6.Default = ''; AU7_823_1ML22_MIL_1 Channel 6.Comment = ''; AU7_823_1ML22_MIL_1 Channel 7.Name = 'AU7_823_1ML22_MIL_1 Channel 7'; AU7_823_1ML22_MIL_1 Channel 7.DataType = 'BOOL'; AU7_823_1ML22_MIL_1 Channel 7.Default = ''; AU7_823_1ML22_MIL_1 Channel 7.Comment = ''; AU7_823_1ML22_MIL_1 Channel 8.Name = 'AU7_823_1ML22_MIL_1 Channel 8'; AU7_823_1ML22_MIL_1 Channel 8.DataType = 'BOOL'; AU7_823_1ML22_MIL_1 Channel 8.Default = ''; AU7_823_1ML22_MIL_1 Channel 8.Comment = ''; AU7_823_1ML22_MIL_1 Channel 9.Name = 'AU7_823_1ML22_MIL_1 Channel 9'; AU7_823_1ML22_MIL_1 Channel 9.DataType = 'BOOL'; AU7_823_1ML22_MIL_1 Channel 9.Default = ''; AU7_823_1ML22_MIL_1 Channel 9.Comment = ''; AU7_823_1ML22_MIL_1 Channel 10.Name = 'AU7_823_1ML22_MIL_1 Channel 10'; AU7_823_1ML22_MIL_1 Channel 10.DataType = 'BOOL'; AU7_823_1ML22_MIL_1 Channel 10.Default = ''; AU7_823_1ML22_MIL_1 Channel 10.Comment = ''; AU7_823_1ML22_MIL_1 Channel 11.Name = 'AU7_823_1ML22_MIL_1 Channel 11'; AU7_823_1ML22_MIL_1 Channel 11.DataType = 'BOOL'; AU7_823_1ML22_MIL_1 Channel 11.Default = ''; AU7_823_1ML22_MIL_1 Channel 11.Comment = ''; AU7_823_1ML22_MIL_1 Channel 12.Name = 'AU7_823_1ML22_MIL_1 Channel 12'; AU7_823_1ML22_MIL_1 Channel 12.DataType = 'BOOL'; AU7_823_1ML22_MIL_1 Channel 12.Default = ''; AU7_823_1ML22_MIL_1 Channel 12.Comment = ''; AU7_823_1ML22_MIL_1 Channel 13.Name = 'AU7_823_1ML22_MIL_1 Channel 13'; AU7_823_1ML22_MIL_1 Channel 13.DataType = 'BOOL'; AU7_823_1ML22_MIL_1 Channel 13.Default = ''; AU7_823_1ML22_MIL_1 Channel 13.Comment = ''; AU7_823_1ML22_MIL_1 Channel 14.Name = 'AU7_823_1ML22_MIL_1 Channel 14'; AU7_823_1ML22_MIL_1 Channel 14.DataType = 'BOOL'; AU7_823_1ML22_MIL_1 Channel 14.Default = ''; AU7_823_1ML22_MIL_1 Channel 14.Comment = ''; AU7_823_1ML22_MIL_1 Channel 15.Name = 'AU7_823_1ML22_MIL_1 Channel 15';
            AU7_823_1ML22_MIL_1 Channel 15.DataType = 'BOOL'; AU7_823_1ML22_MIL_1 Channel 15.Default = ''; AU7_823_1ML22_MIL_1 Channel 15.Comment = ''; AU7_823_1ML22_MIL_1 Channel 16.Name = 'AU7_823_1ML22_MIL_1 Channel 16'; AU7_823_1ML22_MIL_1 Channel 16.DataType = 'BOOL'; AU7_823_1ML22_MIL_1 Channel 16.Default = ''; AU7_823_1ML22_MIL_1 Channel 16.Comment = ''; AU7_823_1ML22_MIL_1 Channel 1-8.Name = 'AU7_823_1ML22_MIL_1 Channel 1-8'; AU7_823_1ML22_MIL_1 Channel 1-8.DataType = 'USINT'; AU7_823_1ML22_MIL_1 Channel 1-8.Default = ''; AU7_823_1ML22_MIL_1 Channel 1-8.Comment = ''; AU7_823_1ML22_MIL_1 Channel 9-16.Name = 'AU7_823_1ML22_MIL_1 Channel 9-16'; AU7_823_1ML22_MIL_1 Channel 9-16.DataType = 'USINT'; AU7_823_1ML22_MIL_1 Channel 9-16.Default = ''; AU7_823_1ML22_MIL_1 Channel 9-16.Comment = ''; AU7_823_1ML22_MIL_1 Channel 1-8.Name = 'AU7_823_1ML22_MIL_1 Channel 1-8'; AU7_823_1ML22_MIL_1 Channel 1-8.DataType = 'BIT'; AU7_823_1ML22_MIL_1 Channel 1-8.Default = ''; AU7_823_1ML22_MIL_1 Channel 1-8.Comment = ''; AU7_823_1ML22_MIL_1 Channel 9-16.Name = 'AU7_823_1ML22_MIL_1 Channel 9-16'; AU7_823_1ML22_MIL_1 Channel 9-16.DataType = 'BIT'; AU7_823_1ML22_MIL_1 Channel 9-16.Default = ''; AU7_823_1ML22_MIL_1 Channel 9-16.Comment = ''; AU7_823_1ML22_MIL_1 Channel 1-16.Name = 'AU7_823_1ML22_MIL_1 Channel 1-16'; AU7_823_1ML22_MIL_1 Channel 1-16.DataType = 'BIT'; AU7_823_1ML22_MIL_1 Channel 1-16.Default = ''; AU7_823_1ML22_MIL_1 Channel 1-16.Comment = ''; AU7_823_1ML22_MIL_1 Channel 1-16.Name = 'AU7_823_1ML22_MIL_1 Channel 1-16'; AU7_823_1ML22_MIL_1 Channel 1-16.DataType = 'UINT'; AU7_823_1ML22_MIL_1 Channel 1-16.Default = ''; AU7_823_1ML22_MIL_1 Channel 1-16.Comment = ''; AU7_823_1ML22_MIL_2 Channel 1.Name = 'AU7_823_1ML22_MIL_2 Channel 1'; AU7_823_1ML22_MIL_2 Channel 1.DataType = 'BOOL'; AU7_823_1ML22_MIL_2 Channel 1.Default = ''; AU7_823_1ML22_MIL_2 Channel 1.Comment = ''; AU7_823_1ML22_MIL_2 Channel 2.Name = 'AU7_823_1ML22_MIL_2 Channel 2'; AU7_823_1ML22_MIL_2 Channel 2.DataType = 'BOOL'; AU7_823_1ML22_MIL_2 Channel 2.Default = ''; AU7_823_1ML22_MIL_2 Channel 2.Comment = ''; AU7_823_1ML22_MIL_2 Channel 3.Name = 'AU7_823_1ML22_MIL_2 Channel 3';
            AU7_823_1ML22_MIL_2 Channel 3.DataType = 'BOOL'; AU7_823_1ML22_MIL_2 Channel 3.Default = ''; AU7_823_1ML22_MIL_2 Channel 3.Comment = ''; AU7_823_1ML22_MIL_2 Channel 4.Name = 'AU7_823_1ML22_MIL_2 Channel 4'; AU7_823_1ML22_MIL_2 Channel 4.DataType = 'BOOL'; AU7_823_1ML22_MIL_2 Channel 4.Default = ''; AU7_823_1ML22_MIL_2 Channel 4.Comment = ''; AU7_823_1ML22_MIL_2 Channel 5.Name = 'AU7_823_1ML22_MIL_2 Channel 5'; AU7_823_1ML22_MIL_2 Channel 5.DataType = 'BOOL'; AU7_823_1ML22_MIL_2 Channel 5.Default = ''; AU7_823_1ML22_MIL_2 Channel 5.Comment = ''; AU7_823_1ML22_MIL_2 Channel 6.Name = 'AU7_823_1ML22_MIL_2 Channel 6'; AU7_823_1ML22_MIL_2 Channel 6.DataType = 'BOOL'; AU7_823_1ML22_MIL_2 Channel 6.Default = ''; AU7_823_1ML22_MIL_2 Channel 6.Comment = ''; AU7_823_1ML22_MIL_2 Channel 7.Name = 'AU7_823_1ML22_MIL_2 Channel 7'; AU7_823_1ML22_MIL_2 Channel 7.DataType = 'BOOL'; AU7_823_1ML22_MIL_2 Channel 7.Default = ''; AU7_823_1ML22_MIL_2 Channel 7.Comment = ''; AU7_823_1ML22_MIL_2 Channel 8.Name = 'AU7_823_1ML22_MIL_2 Channel 8'; AU7_823_1ML22_MIL_2 Channel 8.DataType = 'BOOL'; AU7_823_1ML22_MIL_2 Channel 8.Default = ''; AU7_823_1ML22_MIL_2 Channel 8.Comment = ''; AU7_823_1ML22_MIL_2 Channel 9.Name = 'AU7_823_1ML22_MIL_2 Channel 9'; AU7_823_1ML22_MIL_2 Channel 9.DataType = 'BOOL'; AU7_823_1ML22_MIL_2 Channel 9.Default = ''; AU7_823_1ML22_MIL_2 Channel 9.Comment = ''; AU7_823_1ML22_MIL_2 Channel 10.Name = 'AU7_823_1ML22_MIL_2 Channel 10'; AU7_823_1ML22_MIL_2 Channel 10.DataType = 'BOOL'; AU7_823_1ML22_MIL_2 Channel 10.Default = ''; AU7_823_1ML22_MIL_2 Channel 10.Comment = ''; AU7_823_1ML22_MIL_2 Channel 11.Name = 'AU7_823_1ML22_MIL_2 Channel 11'; AU7_823_1ML22_MIL_2 Channel 11.DataType = 'BOOL'; AU7_823_1ML22_MIL_2 Channel 11.Default = ''; AU7_823_1ML22_MIL_2 Channel 11.Comment = ''; AU7_823_1ML22_MIL_2 Channel 12.Name = 'AU7_823_1ML22_MIL_2 Channel 12'; AU7_823_1ML22_MIL_2 Channel 12.DataType = 'BOOL'; AU7_823_1ML22_MIL_2 Channel 12.Default = ''; AU7_823_1ML22_MIL_2 Channel 12.Comment = ''; AU7_823_1ML22_MIL_2 Channel 13.Name = 'AU7_823_1ML22_MIL_2 Channel 13';
            AU7_823_1ML22_MIL_2 Channel 13.DataType = 'BOOL'; AU7_823_1ML22_MIL_2 Channel 13.Default = ''; AU7_823_1ML22_MIL_2 Channel 13.Comment = ''; AU7_823_1ML22_MIL_2 Channel 14.Name = 'AU7_823_1ML22_MIL_2 Channel 14'; AU7_823_1ML22_MIL_2 Channel 14.DataType = 'BOOL'; AU7_823_1ML22_MIL_2 Channel 14.Default = ''; AU7_823_1ML22_MIL_2 Channel 14.Comment = ''; AU7_823_1ML22_MIL_2 Channel 15.Name = 'AU7_823_1ML22_MIL_2 Channel 15'; AU7_823_1ML22_MIL_2 Channel 15.DataType = 'BOOL'; AU7_823_1ML22_MIL_2 Channel 15.Default = ''; AU7_823_1ML22_MIL_2 Channel 15.Comment = ''; AU7_823_1ML22_MIL_2 Channel 16.Name = 'AU7_823_1ML22_MIL_2 Channel 16'; AU7_823_1ML22_MIL_2 Channel 16.DataType = 'BOOL'; AU7_823_1ML22_MIL_2 Channel 16.Default = ''; AU7_823_1ML22_MIL_2 Channel 16.Comment = ''; AU7_823_1ML22_MIL_2 Channel 1-8.Name = 'AU7_823_1ML22_MIL_2 Channel 1-8'; AU7_823_1ML22_MIL_2 Channel 1-8.DataType = 'USINT'; AU7_823_1ML22_MIL_2 Channel 1-8.Default = ''; AU7_823_1ML22_MIL_2 Channel 1-8.Comment = ''; AU7_823_1ML22_MIL_2 Channel 9-16.Name = 'AU7_823_1ML22_MIL_2 Channel 9-16'; AU7_823_1ML22_MIL_2 Channel 9-16.DataType = 'USINT'; AU7_823_1ML22_MIL_2 Channel 9-16.Default = ''; AU7_823_1ML22_MIL_2 Channel 9-16.Comment = ''; AU7_823_1ML22_MIL_2 Channel 1-8.Name = 'AU7_823_1ML22_MIL_2 Channel 1-8'; AU7_823_1ML22_MIL_2 Channel 1-8.DataType = 'BIT'; AU7_823_1ML22_MIL_2 Channel 1-8.Default = ''; AU7_823_1ML22_MIL_2 Channel 1-8.Comment = ''; AU7_823_1ML22_MIL_2 Channel 9-16.Name = 'AU7_823_1ML22_MIL_2 Channel 9-16'; AU7_823_1ML22_MIL_2 Channel 9-16.DataType = 'BIT'; AU7_823_1ML22_MIL_2 Channel 9-16.Default = ''; AU7_823_1ML22_MIL_2 Channel 9-16.Comment = ''; AU7_823_1ML22_MIL_2 Channel 1-16.Name = 'AU7_823_1ML22_MIL_2 Channel 1-16'; AU7_823_1ML22_MIL_2 Channel 1-16.DataType = 'BIT'; AU7_823_1ML22_MIL_2 Channel 1-16.Default = ''; AU7_823_1ML22_MIL_2 Channel 1-16.Comment = ''; AU7_823_1ML22_MIL_2 Channel 1-16.Name = 'AU7_823_1ML22_MIL_2 Channel 1-16'; AU7_823_1ML22_MIL_2 Channel 1-16.DataType = 'UINT'; AU7_823_1ML22_MIL_2 Channel 1-16.Default = ''; AU7_823_1ML22_MIL_2 Channel 1-16.Comment = ''; AU7_823_1ML22_MIL_3 Channel 1.Name = 'AU7_823_1ML22_MIL_3 Channel 1';
            AU7_823_1ML22_MIL_3 Channel 1.DataType = 'BOOL'; AU7_823_1ML22_MIL_3 Channel 1.Default = ''; AU7_823_1ML22_MIL_3 Channel 1.Comment = ''; AU7_823_1ML22_MIL_3 Channel 2.Name = 'AU7_823_1ML22_MIL_3 Channel 2'; AU7_823_1ML22_MIL_3 Channel 2.DataType = 'BOOL'; AU7_823_1ML22_MIL_3 Channel 2.Default = ''; AU7_823_1ML22_MIL_3 Channel 2.Comment = ''; AU7_823_1ML22_MIL_3 Channel 3.Name = 'AU7_823_1ML22_MIL_3 Channel 3'; AU7_823_1ML22_MIL_3 Channel 3.DataType = 'BOOL'; AU7_823_1ML22_MIL_3 Channel 3.Default = ''; AU7_823_1ML22_MIL_3 Channel 3.Comment = ''; AU7_823_1ML22_MIL_3 Channel 4.Name = 'AU7_823_1ML22_MIL_3 Channel 4'; AU7_823_1ML22_MIL_3 Channel 4.DataType = 'BOOL'; AU7_823_1ML22_MIL_3 Channel 4.Default = ''; AU7_823_1ML22_MIL_3 Channel 4.Comment = ''; AU7_823_1ML22_MIL_3 Channel 5.Name = 'AU7_823_1ML22_MIL_3 Channel 5'; AU7_823_1ML22_MIL_3 Channel 5.DataType = 'BOOL'; AU7_823_1ML22_MIL_3 Channel 5.Default = ''; AU7_823_1ML22_MIL_3 Channel 5.Comment = ''; AU7_823_1ML22_MIL_3 Channel 6.Name = 'AU7_823_1ML22_MIL_3 Channel 6'; AU7_823_1ML22_MIL_3 Channel 6.DataType = 'BOOL'; AU7_823_1ML22_MIL_3 Channel 6.Default = ''; AU7_823_1ML22_MIL_3 Channel 6.Comment = ''; AU7_823_1ML22_MIL_3 Channel 7.Name = 'AU7_823_1ML22_MIL_3 Channel 7'; AU7_823_1ML22_MIL_3 Channel 7.DataType = 'BOOL'; AU7_823_1ML22_MIL_3 Channel 7.Default = ''; AU7_823_1ML22_MIL_3 Channel 7.Comment = ''; AU7_823_1ML22_MIL_3 Channel 8.Name = 'AU7_823_1ML22_MIL_3 Channel 8'; AU7_823_1ML22_MIL_3 Channel 8.DataType = 'BOOL'; AU7_823_1ML22_MIL_3 Channel 8.Default = ''; AU7_823_1ML22_MIL_3 Channel 8.Comment = ''; AU7_823_1ML22_MIL_3 Channel 9.Name = 'AU7_823_1ML22_MIL_3 Channel 9'; AU7_823_1ML22_MIL_3 Channel 9.DataType = 'BOOL'; AU7_823_1ML22_MIL_3 Channel 9.Default = ''; AU7_823_1ML22_MIL_3 Channel 9.Comment = ''; AU7_823_1ML22_MIL_3 Channel 10.Name = 'AU7_823_1ML22_MIL_3 Channel 10'; AU7_823_1ML22_MIL_3 Channel 10.DataType = 'BOOL'; AU7_823_1ML22_MIL_3 Channel 10.Default = ''; AU7_823_1ML22_MIL_3 Channel 10.Comment = ''; AU7_823_1ML22_MIL_3 Channel 11.Name = 'AU7_823_1ML22_MIL_3 Channel 11';
            AU7_823_1ML22_MIL_3 Channel 11.DataType = 'BOOL'; AU7_823_1ML22_MIL_3 Channel 11.Default = ''; AU7_823_1ML22_MIL_3 Channel 11.Comment = ''; AU7_823_1ML22_MIL_3 Channel 12.Name = 'AU7_823_1ML22_MIL_3 Channel 12'; AU7_823_1ML22_MIL_3 Channel 12.DataType = 'BOOL'; AU7_823_1ML22_MIL_3 Channel 12.Default = ''; AU7_823_1ML22_MIL_3 Channel 12.Comment = ''; AU7_823_1ML22_MIL_3 Channel 13.Name = 'AU7_823_1ML22_MIL_3 Channel 13'; AU7_823_1ML22_MIL_3 Channel 13.DataType = 'BOOL'; AU7_823_1ML22_MIL_3 Channel 13.Default = ''; AU7_823_1ML22_MIL_3 Channel 13.Comment = ''; AU7_823_1ML22_MIL_3 Channel 14.Name = 'AU7_823_1ML22_MIL_3 Channel 14'; AU7_823_1ML22_MIL_3 Channel 14.DataType = 'BOOL'; AU7_823_1ML22_MIL_3 Channel 14.Default = ''; AU7_823_1ML22_MIL_3 Channel 14.Comment = ''; AU7_823_1ML22_MIL_3 Channel 15.Name = 'AU7_823_1ML22_MIL_3 Channel 15'; AU7_823_1ML22_MIL_3 Channel 15.DataType = 'BOOL'; AU7_823_1ML22_MIL_3 Channel 15.Default = ''; AU7_823_1ML22_MIL_3 Channel 15.Comment = ''; AU7_823_1ML22_MIL_3 Channel 16.Name = 'AU7_823_1ML22_MIL_3 Channel 16'; AU7_823_1ML22_MIL_3 Channel 16.DataType = 'BOOL'; AU7_823_1ML22_MIL_3 Channel 16.Default = ''; AU7_823_1ML22_MIL_3 Channel 16.Comment = ''; AU7_823_1ML22_MIL_3 Channel 1-8.Name = 'AU7_823_1ML22_MIL_3 Channel 1-8'; AU7_823_1ML22_MIL_3 Channel 1-8.DataType = 'USINT'; AU7_823_1ML22_MIL_3 Channel 1-8.Default = ''; AU7_823_1ML22_MIL_3 Channel 1-8.Comment = ''; AU7_823_1ML22_MIL_3 Channel 9-16.Name = 'AU7_823_1ML22_MIL_3 Channel 9-16'; AU7_823_1ML22_MIL_3 Channel 9-16.DataType = 'USINT'; AU7_823_1ML22_MIL_3 Channel 9-16.Default = ''; AU7_823_1ML22_MIL_3 Channel 9-16.Comment = ''; AU7_823_1ML22_MIL_3 Channel 1-8.Name = 'AU7_823_1ML22_MIL_3 Channel 1-8'; AU7_823_1ML22_MIL_3 Channel 1-8.DataType = 'BIT'; AU7_823_1ML22_MIL_3 Channel 1-8.Default = ''; AU7_823_1ML22_MIL_3 Channel 1-8.Comment = ''; AU7_823_1ML22_MIL_3 Channel 9-16.Name = 'AU7_823_1ML22_MIL_3 Channel 9-16'; AU7_823_1ML22_MIL_3 Channel 9-16.DataType = 'BIT'; AU7_823_1ML22_MIL_3 Channel 9-16.Default = ''; AU7_823_1ML22_MIL_3 Channel 9-16.Comment = ''; AU7_823_1ML22_MIL_3 Channel 1-16.Name = 'AU7_823_1ML22_MIL_3 Channel 1-16';
            AU7_823_1ML22_MIL_3 Channel 1-16.DataType = 'BIT'; AU7_823_1ML22_MIL_3 Channel 1-16.Default = ''; AU7_823_1ML22_MIL_3 Channel 1-16.Comment = ''; AU7_823_1ML22_MIL_3 Channel 1-16.Name = 'AU7_823_1ML22_MIL_3 Channel 1-16'; AU7_823_1ML22_MIL_3 Channel 1-16.DataType = 'UINT'; AU7_823_1ML22_MIL_3 Channel 1-16.Default = ''; AU7_823_1ML22_MIL_3 Channel 1-16.Comment = ''; AU7_823_1ML22_MIL_4 Channel 1.Name = 'AU7_823_1ML22_MIL_4 Channel 1'; AU7_823_1ML22_MIL_4 Channel 1.DataType = 'BOOL'; AU7_823_1ML22_MIL_4 Channel 1.Default = ''; AU7_823_1ML22_MIL_4 Channel 1.Comment = ''; AU7_823_1ML22_MIL_4 Channel 2.Name = 'AU7_823_1ML22_MIL_4 Channel 2'; AU7_823_1ML22_MIL_4 Channel 2.DataType = 'BOOL'; AU7_823_1ML22_MIL_4 Channel 2.Default = ''; AU7_823_1ML22_MIL_4 Channel 2.Comment = ''; AU7_823_1ML22_MIL_4 Channel 3.Name = 'AU7_823_1ML22_MIL_4 Channel 3'; AU7_823_1ML22_MIL_4 Channel 3.DataType = 'BOOL'; AU7_823_1ML22_MIL_4 Channel 3.Default = ''; AU7_823_1ML22_MIL_4 Channel 3.Comment = ''; AU7_823_1ML22_MIL_4 Channel 4.Name = 'AU7_823_1ML22_MIL_4 Channel 4'; AU7_823_1ML22_MIL_4 Channel 4.DataType = 'BOOL'; AU7_823_1ML22_MIL_4 Channel 4.Default = ''; AU7_823_1ML22_MIL_4 Channel 4.Comment = ''; AU7_823_1ML22_MIL_4 Channel 5.Name = 'AU7_823_1ML22_MIL_4 Channel 5'; AU7_823_1ML22_MIL_4 Channel 5.DataType = 'BOOL'; AU7_823_1ML22_MIL_4 Channel 5.Default = ''; AU7_823_1ML22_MIL_4 Channel 5.Comment = ''; AU7_823_1ML22_MIL_4 Channel 6.Name = 'AU7_823_1ML22_MIL_4 Channel 6'; AU7_823_1ML22_MIL_4 Channel 6.DataType = 'BOOL'; AU7_823_1ML22_MIL_4 Channel 6.Default = ''; AU7_823_1ML22_MIL_4 Channel 6.Comment = ''; AU7_823_1ML22_MIL_4 Channel 7.Name = 'AU7_823_1ML22_MIL_4 Channel 7'; AU7_823_1ML22_MIL_4 Channel 7.DataType = 'BOOL'; AU7_823_1ML22_MIL_4 Channel 7.Default = ''; AU7_823_1ML22_MIL_4 Channel 7.Comment = ''; AU7_823_1ML22_MIL_4 Channel 8.Name = 'AU7_823_1ML22_MIL_4 Channel 8'; AU7_823_1ML22_MIL_4 Channel 8.DataType = 'BOOL'; AU7_823_1ML22_MIL_4 Channel 8.Default = ''; AU7_823_1ML22_MIL_4 Channel 8.Comment = ''; AU7_823_1ML22_MIL_4 Channel 9.Name = 'AU7_823_1ML22_MIL_4 Channel 9';
            AU7_823_1ML22_MIL_4 Channel 9.DataType = 'BOOL'; AU7_823_1ML22_MIL_4 Channel 9.Default = ''; AU7_823_1ML22_MIL_4 Channel 9.Comment = ''; AU7_823_1ML22_MIL_4 Channel 10.Name = 'AU7_823_1ML22_MIL_4 Channel 10'; AU7_823_1ML22_MIL_4 Channel 10.DataType = 'BOOL'; AU7_823_1ML22_MIL_4 Channel 10.Default = ''; AU7_823_1ML22_MIL_4 Channel 10.Comment = ''; AU7_823_1ML22_MIL_4 Channel 11.Name = 'AU7_823_1ML22_MIL_4 Channel 11'; AU7_823_1ML22_MIL_4 Channel 11.DataType = 'BOOL'; AU7_823_1ML22_MIL_4 Channel 11.Default = ''; AU7_823_1ML22_MIL_4 Channel 11.Comment = ''; AU7_823_1ML22_MIL_4 Channel 12.Name = 'AU7_823_1ML22_MIL_4 Channel 12'; AU7_823_1ML22_MIL_4 Channel 12.DataType = 'BOOL'; AU7_823_1ML22_MIL_4 Channel 12.Default = ''; AU7_823_1ML22_MIL_4 Channel 12.Comment = ''; AU7_823_1ML22_MIL_4 Channel 13.Name = 'AU7_823_1ML22_MIL_4 Channel 13'; AU7_823_1ML22_MIL_4 Channel 13.DataType = 'BOOL'; AU7_823_1ML22_MIL_4 Channel 13.Default = ''; AU7_823_1ML22_MIL_4 Channel 13.Comment = ''; AU7_823_1ML22_MIL_4 Channel 14.Name = 'AU7_823_1ML22_MIL_4 Channel 14'; AU7_823_1ML22_MIL_4 Channel 14.DataType = 'BOOL'; AU7_823_1ML22_MIL_4 Channel 14.Default = ''; AU7_823_1ML22_MIL_4 Channel 14.Comment = ''; AU7_823_1ML22_MIL_4 Channel 15.Name = 'AU7_823_1ML22_MIL_4 Channel 15'; AU7_823_1ML22_MIL_4 Channel 15.DataType = 'BOOL'; AU7_823_1ML22_MIL_4 Channel 15.Default = ''; AU7_823_1ML22_MIL_4 Channel 15.Comment = ''; AU7_823_1ML22_MIL_4 Channel 16.Name = 'AU7_823_1ML22_MIL_4 Channel 16'; AU7_823_1ML22_MIL_4 Channel 16.DataType = 'BOOL'; AU7_823_1ML22_MIL_4 Channel 16.Default = ''; AU7_823_1ML22_MIL_4 Channel 16.Comment = ''; AU7_823_1ML22_MIL_4 Channel 1-8.Name = 'AU7_823_1ML22_MIL_4 Channel 1-8'; AU7_823_1ML22_MIL_4 Channel 1-8.DataType = 'USINT'; AU7_823_1ML22_MIL_4 Channel 1-8.Default = ''; AU7_823_1ML22_MIL_4 Channel 1-8.Comment = ''; AU7_823_1ML22_MIL_4 Channel 9-16.Name = 'AU7_823_1ML22_MIL_4 Channel 9-16'; AU7_823_1ML22_MIL_4 Channel 9-16.DataType = 'USINT'; AU7_823_1ML22_MIL_4 Channel 9-16.Default = ''; AU7_823_1ML22_MIL_4 Channel 9-16.Comment = ''; AU7_823_1ML22_MIL_4 Channel 1-8.Name = 'AU7_823_1ML22_MIL_4 Channel 1-8';
            AU7_823_1ML22_MIL_4 Channel 1-8.DataType = 'BIT'; AU7_823_1ML22_MIL_4 Channel 1-8.Default = ''; AU7_823_1ML22_MIL_4 Channel 1-8.Comment = ''; AU7_823_1ML22_MIL_4 Channel 9-16.Name = 'AU7_823_1ML22_MIL_4 Channel 9-16'; AU7_823_1ML22_MIL_4 Channel 9-16.DataType = 'BIT'; AU7_823_1ML22_MIL_4 Channel 9-16.Default = ''; AU7_823_1ML22_MIL_4 Channel 9-16.Comment = ''; AU7_823_1ML22_MIL_4 Channel 1-16.Name = 'AU7_823_1ML22_MIL_4 Channel 1-16'; AU7_823_1ML22_MIL_4 Channel 1-16.DataType = 'BIT'; AU7_823_1ML22_MIL_4 Channel 1-16.Default = ''; AU7_823_1ML22_MIL_4 Channel 1-16.Comment = ''; AU7_823_1ML22_MIL_4 Channel 1-16.Name = 'AU7_823_1ML22_MIL_4 Channel 1-16'; AU7_823_1ML22_MIL_4 Channel 1-16.DataType = 'UINT'; AU7_823_1ML22_MIL_4 Channel 1-16.Default = ''; AU7_823_1ML22_MIL_4 Channel 1-16.Comment = ''; ID.Name = 'ID'; ID.DataType = 'UINT'; ID.Default = ''; ID.Comment = ''; AU7_823_1ML22_MIL Channel 1.Name = 'AU7_823_1ML22_MIL Channel 1'; AU7_823_1ML22_MIL Channel 1.DataType = 'BOOL'; AU7_823_1ML22_MIL Channel 1.Default = ''; AU7_823_1ML22_MIL Channel 1.Comment = ''; AU7_823_1ML22_MIL Channel 2.Name = 'AU7_823_1ML22_MIL Channel 2'; AU7_823_1ML22_MIL Channel 2.DataType = 'BOOL'; AU7_823_1ML22_MIL Channel 2.Default = ''; AU7_823_1ML22_MIL Channel 2.Comment = ''; AU7_823_1ML22_MIL Channel 3.Name = 'AU7_823_1ML22_MIL Channel 3'; AU7_823_1ML22_MIL Channel 3.DataType = 'BOOL'; AU7_823_1ML22_MIL Channel 3.Default = ''; AU7_823_1ML22_MIL Channel 3.Comment = ''; AU7_823_1ML22_MIL Channel 4.Name = 'AU7_823_1ML22_MIL Channel 4'; AU7_823_1ML22_MIL Channel 4.DataType = 'BOOL'; AU7_823_1ML22_MIL Channel 4.Default = ''; AU7_823_1ML22_MIL Channel 4.Comment = ''; AU7_823_1ML22_MIL Channel 5.Name = 'AU7_823_1ML22_MIL Channel 5'; AU7_823_1ML22_MIL Channel 5.DataType = 'BOOL'; AU7_823_1ML22_MIL Channel 5.Default = ''; AU7_823_1ML22_MIL Channel 5.Comment = ''; AU7_823_1ML22_MIL Channel 6.Name = 'AU7_823_1ML22_MIL Channel 6';
            AU7_823_1ML22_MIL Channel 6.DataType = 'BOOL'; AU7_823_1ML22_MIL Channel 6.Default = ''; AU7_823_1ML22_MIL Channel 6.Comment = ''; AU7_823_1ML22_MIL Channel 7.Name = 'AU7_823_1ML22_MIL Channel 7'; AU7_823_1ML22_MIL Channel 7.DataType = 'BOOL'; AU7_823_1ML22_MIL Channel 7.Default = ''; AU7_823_1ML22_MIL Channel 7.Comment = ''; AU7_823_1ML22_MIL Channel 8.Name = 'AU7_823_1ML22_MIL Channel 8'; AU7_823_1ML22_MIL Channel 8.DataType = 'BOOL'; AU7_823_1ML22_MIL Channel 8.Default = ''; AU7_823_1ML22_MIL Channel 8.Comment = ''; AU7_823_1ML22_MIL Channel 9.Name = 'AU7_823_1ML22_MIL Channel 9'; AU7_823_1ML22_MIL Channel 9.DataType = 'BOOL'; AU7_823_1ML22_MIL Channel 9.Default = ''; AU7_823_1ML22_MIL Channel 9.Comment = ''; AU7_823_1ML22_MIL Channel 10.Name = 'AU7_823_1ML22_MIL Channel 10'; AU7_823_1ML22_MIL Channel 10.DataType = 'BOOL'; AU7_823_1ML22_MIL Channel 10.Default = ''; AU7_823_1ML22_MIL Channel 10.Comment = ''; AU7_823_1ML22_MIL Channel 11.Name = 'AU7_823_1ML22_MIL Channel 11'; AU7_823_1ML22_MIL Channel 11.DataType = 'BOOL'; AU7_823_1ML22_MIL Channel 11.Default = ''; AU7_823_1ML22_MIL Channel 11.Comment = ''; AU7_823_1ML22_MIL Channel 12.Name = 'AU7_823_1ML22_MIL Channel 12'; AU7_823_1ML22_MIL Channel 12.DataType = 'BOOL'; AU7_823_1ML22_MIL Channel 12.Default = ''; AU7_823_1ML22_MIL Channel 12.Comment = ''; AU7_823_1ML22_MIL Channel 13.Name = 'AU7_823_1ML22_MIL Channel 13'; AU7_823_1ML22_MIL Channel 13.DataType = 'BOOL'; AU7_823_1ML22_MIL Channel 13.Default = ''; AU7_823_1ML22_MIL Channel 13.Comment = ''; AU7_823_1ML22_MIL Channel 14.Name = 'AU7_823_1ML22_MIL Channel 14'; AU7_823_1ML22_MIL Channel 14.DataType = 'BOOL'; AU7_823_1ML22_MIL Channel 14.Default = ''; AU7_823_1ML22_MIL Channel 14.Comment = ''; AU7_823_1ML22_MIL Channel 15.Name = 'AU7_823_1ML22_MIL Channel 15'; AU7_823_1ML22_MIL Channel 15.DataType = 'BOOL'; AU7_823_1ML22_MIL Channel 15.Default = ''; AU7_823_1ML22_MIL Channel 15.Comment = ''; AU7_823_1ML22_MIL Channel 16.Name = 'AU7_823_1ML22_MIL Channel 16';
            AU7_823_1ML22_MIL Channel 16.DataType = 'BOOL'; AU7_823_1ML22_MIL Channel 16.Default = ''; AU7_823_1ML22_MIL Channel 16.Comment = ''; AU7_823_1ML22_MIL Channel 1-8.Name = 'AU7_823_1ML22_MIL Channel 1-8'; AU7_823_1ML22_MIL Channel 1-8.DataType = 'USINT'; AU7_823_1ML22_MIL Channel 1-8.Default = ''; AU7_823_1ML22_MIL Channel 1-8.Comment = ''; AU7_823_1ML22_MIL Channel 9-16.Name = 'AU7_823_1ML22_MIL Channel 9-16'; AU7_823_1ML22_MIL Channel 9-16.DataType = 'USINT'; AU7_823_1ML22_MIL Channel 9-16.Default = ''; AU7_823_1ML22_MIL Channel 9-16.Comment = ''; AU7_823_1ML22_MIL Channel 1-8.Name = 'AU7_823_1ML22_MIL Channel 1-8'; AU7_823_1ML22_MIL Channel 1-8.DataType = 'BIT'; AU7_823_1ML22_MIL Channel 1-8.Default = ''; AU7_823_1ML22_MIL Channel 1-8.Comment = ''; AU7_823_1ML22_MIL Channel 9-16.Name = 'AU7_823_1ML22_MIL Channel 9-16'; AU7_823_1ML22_MIL Channel 9-16.DataType = 'BIT'; AU7_823_1ML22_MIL Channel 9-16.Default = ''; AU7_823_1ML22_MIL Channel 9-16.Comment = ''; AU7_823_1ML22_MIL Channel 1-16.Name = 'AU7_823_1ML22_MIL Channel 1-16'; AU7_823_1ML22_MIL Channel 1-16.DataType = 'BIT'; AU7_823_1ML22_MIL Channel 1-16.Default = ''; AU7_823_1ML22_MIL Channel 1-16.Comment = ''; AU7_823_1ML22_MIL Channel 1-16.Name = 'AU7_823_1ML22_MIL Channel 1-16'; AU7_823_1ML22_MIL Channel 1-16.DataType = 'UINT'; AU7_823_1ML22_MIL Channel 1-16.Default = ''; AU7_823_1ML22_MIL Channel 1-16.Comment = ''; AU7_823_1ML22_MIL_1 Channel 1.Name = 'AU7_823_1ML22_MIL_1 Channel 1'; AU7_823_1ML22_MIL_1 Channel 1.DataType = 'BOOL'; AU7_823_1ML22_MIL_1 Channel 1.Default = ''; AU7_823_1ML22_MIL_1 Channel 1.Comment = ''; AU7_823_1ML22_MIL_1 Channel 2.Name = 'AU7_823_1ML22_MIL_1 Channel 2'; AU7_823_1ML22_MIL_1 Channel 2.DataType = 'BOOL'; AU7_823_1ML22_MIL_1 Channel 2.Default = ''; AU7_823_1ML22_MIL_1 Channel 2.Comment = ''; AU7_823_1ML22_MIL_1 Channel 3.Name = 'AU7_823_1ML22_MIL_1 Channel 3'; AU7_823_1ML22_MIL_1 Channel 3.DataType = 'BOOL'; AU7_823_1ML22_MIL_1 Channel 3.Default = ''; AU7_823_1ML22_MIL_1 Channel 3.Comment = ''; AU7_823_1ML22_MIL_1 Channel 4.Name = 'AU7_823_1ML22_MIL_1 Channel 4';
            AU7_823_1ML22_MIL_1 Channel 4.DataType = 'BOOL'; AU7_823_1ML22_MIL_1 Channel 4.Default = ''; AU7_823_1ML22_MIL_1 Channel 4.Comment = ''; AU7_823_1ML22_MIL_1 Channel 5.Name = 'AU7_823_1ML22_MIL_1 Channel 5'; AU7_823_1ML22_MIL_1 Channel 5.DataType = 'BOOL'; AU7_823_1ML22_MIL_1 Channel 5.Default = ''; AU7_823_1ML22_MIL_1 Channel 5.Comment = ''; AU7_823_1ML22_MIL_1 Channel 6.Name = 'AU7_823_1ML22_MIL_1 Channel 6'; AU7_823_1ML22_MIL_1 Channel 6.DataType = 'BOOL'; AU7_823_1ML22_MIL_1 Channel 6.Default = ''; AU7_823_1ML22_MIL_1 Channel 6.Comment = ''; AU7_823_1ML22_MIL_1 Channel 7.Name = 'AU7_823_1ML22_MIL_1 Channel 7'; AU7_823_1ML22_MIL_1 Channel 7.DataType = 'BOOL'; AU7_823_1ML22_MIL_1 Channel 7.Default = ''; AU7_823_1ML22_MIL_1 Channel 7.Comment = ''; AU7_823_1ML22_MIL_1 Channel 8.Name = 'AU7_823_1ML22_MIL_1 Channel 8'; AU7_823_1ML22_MIL_1 Channel 8.DataType = 'BOOL'; AU7_823_1ML22_MIL_1 Channel 8.Default = ''; AU7_823_1ML22_MIL_1 Channel 8.Comment = ''; AU7_823_1ML22_MIL_1 Channel 9.Name = 'AU7_823_1ML22_MIL_1 Channel 9'; AU7_823_1ML22_MIL_1 Channel 9.DataType = 'BOOL'; AU7_823_1ML22_MIL_1 Channel 9.Default = ''; AU7_823_1ML22_MIL_1 Channel 9.Comment = ''; AU7_823_1ML22_MIL_1 Channel 10.Name = 'AU7_823_1ML22_MIL_1 Channel 10'; AU7_823_1ML22_MIL_1 Channel 10.DataType = 'BOOL'; AU7_823_1ML22_MIL_1 Channel 10.Default = ''; AU7_823_1ML22_MIL_1 Channel 10.Comment = ''; AU7_823_1ML22_MIL_1 Channel 11.Name = 'AU7_823_1ML22_MIL_1 Channel 11'; AU7_823_1ML22_MIL_1 Channel 11.DataType = 'BOOL'; AU7_823_1ML22_MIL_1 Channel 11.Default = ''; AU7_823_1ML22_MIL_1 Channel 11.Comment = ''; AU7_823_1ML22_MIL_1 Channel 12.Name = 'AU7_823_1ML22_MIL_1 Channel 12'; AU7_823_1ML22_MIL_1 Channel 12.DataType = 'BOOL'; AU7_823_1ML22_MIL_1 Channel 12.Default = ''; AU7_823_1ML22_MIL_1 Channel 12.Comment = ''; AU7_823_1ML22_MIL_1 Channel 13.Name = 'AU7_823_1ML22_MIL_1 Channel 13'; AU7_823_1ML22_MIL_1 Channel 13.DataType = 'BOOL'; AU7_823_1ML22_MIL_1 Channel 13.Default = ''; AU7_823_1ML22_MIL_1 Channel 13.Comment = ''; AU7_823_1ML22_MIL_1 Channel 14.Name = 'AU7_823_1ML22_MIL_1 Channel 14';
            AU7_823_1ML22_MIL_1 Channel 14.DataType = 'BOOL'; AU7_823_1ML22_MIL_1 Channel 14.Default = ''; AU7_823_1ML22_MIL_1 Channel 14.Comment = ''; AU7_823_1ML22_MIL_1 Channel 15.Name = 'AU7_823_1ML22_MIL_1 Channel 15'; AU7_823_1ML22_MIL_1 Channel 15.DataType = 'BOOL'; AU7_823_1ML22_MIL_1 Channel 15.Default = ''; AU7_823_1ML22_MIL_1 Channel 15.Comment = ''; AU7_823_1ML22_MIL_1 Channel 16.Name = 'AU7_823_1ML22_MIL_1 Channel 16'; AU7_823_1ML22_MIL_1 Channel 16.DataType = 'BOOL'; AU7_823_1ML22_MIL_1 Channel 16.Default = ''; AU7_823_1ML22_MIL_1 Channel 16.Comment = ''; AU7_823_1ML22_MIL_1 Channel 1-8.Name = 'AU7_823_1ML22_MIL_1 Channel 1-8'; AU7_823_1ML22_MIL_1 Channel 1-8.DataType = 'USINT'; AU7_823_1ML22_MIL_1 Channel 1-8.Default = ''; AU7_823_1ML22_MIL_1 Channel 1-8.Comment = ''; AU7_823_1ML22_MIL_1 Channel 9-16.Name = 'AU7_823_1ML22_MIL_1 Channel 9-16'; AU7_823_1ML22_MIL_1 Channel 9-16.DataType = 'USINT'; AU7_823_1ML22_MIL_1 Channel 9-16.Default = ''; AU7_823_1ML22_MIL_1 Channel 9-16.Comment = ''; AU7_823_1ML22_MIL_1 Channel 1-8.Name = 'AU7_823_1ML22_MIL_1 Channel 1-8'; AU7_823_1ML22_MIL_1 Channel 1-8.DataType = 'BIT'; AU7_823_1ML22_MIL_1 Channel 1-8.Default = ''; AU7_823_1ML22_MIL_1 Channel 1-8.Comment = ''; AU7_823_1ML22_MIL_1 Channel 9-16.Name = 'AU7_823_1ML22_MIL_1 Channel 9-16'; AU7_823_1ML22_MIL_1 Channel 9-16.DataType = 'BIT'; AU7_823_1ML22_MIL_1 Channel 9-16.Default = ''; AU7_823_1ML22_MIL_1 Channel 9-16.Comment = ''; AU7_823_1ML22_MIL_1 Channel 1-16.Name = 'AU7_823_1ML22_MIL_1 Channel 1-16'; AU7_823_1ML22_MIL_1 Channel 1-16.DataType = 'BIT'; AU7_823_1ML22_MIL_1 Channel 1-16.Default = ''; AU7_823_1ML22_MIL_1 Channel 1-16.Comment = ''; AU7_823_1ML22_MIL_1 Channel 1-16.Name = 'AU7_823_1ML22_MIL_1 Channel 1-16'; AU7_823_1ML22_MIL_1 Channel 1-16.DataType = 'UINT'; AU7_823_1ML22_MIL_1 Channel 1-16.Default = ''; AU7_823_1ML22_MIL_1 Channel 1-16.Comment = ''; AU7_823_1ML22_MIL_2 Channel 1.Name = 'AU7_823_1ML22_MIL_2 Channel 1'; AU7_823_1ML22_MIL_2 Channel 1.DataType = 'BOOL'; AU7_823_1ML22_MIL_2 Channel 1.Default = ''; AU7_823_1ML22_MIL_2 Channel 1.Comment = ''; AU7_823_1ML22_MIL_2 Channel 2.Name = 'AU7_823_1ML22_MIL_2 Channel 2';
            AU7_823_1ML22_MIL_2 Channel 2.DataType = 'BOOL'; AU7_823_1ML22_MIL_2 Channel 2.Default = ''; AU7_823_1ML22_MIL_2 Channel 2.Comment = ''; AU7_823_1ML22_MIL_2 Channel 3.Name = 'AU7_823_1ML22_MIL_2 Channel 3'; AU7_823_1ML22_MIL_2 Channel 3.DataType = 'BOOL'; AU7_823_1ML22_MIL_2 Channel 3.Default = ''; AU7_823_1ML22_MIL_2 Channel 3.Comment = ''; AU7_823_1ML22_MIL_2 Channel 4.Name = 'AU7_823_1ML22_MIL_2 Channel 4'; AU7_823_1ML22_MIL_2 Channel 4.DataType = 'BOOL'; AU7_823_1ML22_MIL_2 Channel 4.Default = ''; AU7_823_1ML22_MIL_2 Channel 4.Comment = ''; AU7_823_1ML22_MIL_2 Channel 5.Name = 'AU7_823_1ML22_MIL_2 Channel 5'; AU7_823_1ML22_MIL_2 Channel 5.DataType = 'BOOL'; AU7_823_1ML22_MIL_2 Channel 5.Default = ''; AU7_823_1ML22_MIL_2 Channel 5.Comment = ''; AU7_823_1ML22_MIL_2 Channel 6.Name = 'AU7_823_1ML22_MIL_2 Channel 6'; AU7_823_1ML22_MIL_2 Channel 6.DataType = 'BOOL'; AU7_823_1ML22_MIL_2 Channel 6.Default = ''; AU7_823_1ML22_MIL_2 Channel 6.Comment = ''; AU7_823_1ML22_MIL_2 Channel 7.Name = 'AU7_823_1ML22_MIL_2 Channel 7'; AU7_823_1ML22_MIL_2 Channel 7.DataType = 'BOOL'; AU7_823_1ML22_MIL_2 Channel 7.Default = ''; AU7_823_1ML22_MIL_2 Channel 7.Comment = ''; AU7_823_1ML22_MIL_2 Channel 8.Name = 'AU7_823_1ML22_MIL_2 Channel 8'; AU7_823_1ML22_MIL_2 Channel 8.DataType = 'BOOL'; AU7_823_1ML22_MIL_2 Channel 8.Default = ''; AU7_823_1ML22_MIL_2 Channel 8.Comment = ''; AU7_823_1ML22_MIL_2 Channel 9.Name = 'AU7_823_1ML22_MIL_2 Channel 9'; AU7_823_1ML22_MIL_2 Channel 9.DataType = 'BOOL'; AU7_823_1ML22_MIL_2 Channel 9.Default = ''; AU7_823_1ML22_MIL_2 Channel 9.Comment = ''; AU7_823_1ML22_MIL_2 Channel 10.Name = 'AU7_823_1ML22_MIL_2 Channel 10'; AU7_823_1ML22_MIL_2 Channel 10.DataType = 'BOOL'; AU7_823_1ML22_MIL_2 Channel 10.Default = ''; AU7_823_1ML22_MIL_2 Channel 10.Comment = ''; AU7_823_1ML22_MIL_2 Channel 11.Name = 'AU7_823_1ML22_MIL_2 Channel 11'; AU7_823_1ML22_MIL_2 Channel 11.DataType = 'BOOL'; AU7_823_1ML22_MIL_2 Channel 11.Default = ''; AU7_823_1ML22_MIL_2 Channel 11.Comment = ''; AU7_823_1ML22_MIL_2 Channel 12.Name = 'AU7_823_1ML22_MIL_2 Channel 12';
            AU7_823_1ML22_MIL_2 Channel 12.DataType = 'BOOL'; AU7_823_1ML22_MIL_2 Channel 12.Default = ''; AU7_823_1ML22_MIL_2 Channel 12.Comment = ''; AU7_823_1ML22_MIL_2 Channel 13.Name = 'AU7_823_1ML22_MIL_2 Channel 13'; AU7_823_1ML22_MIL_2 Channel 13.DataType = 'BOOL'; AU7_823_1ML22_MIL_2 Channel 13.Default = ''; AU7_823_1ML22_MIL_2 Channel 13.Comment = ''; AU7_823_1ML22_MIL_2 Channel 14.Name = 'AU7_823_1ML22_MIL_2 Channel 14'; AU7_823_1ML22_MIL_2 Channel 14.DataType = 'BOOL'; AU7_823_1ML22_MIL_2 Channel 14.Default = ''; AU7_823_1ML22_MIL_2 Channel 14.Comment = ''; AU7_823_1ML22_MIL_2 Channel 15.Name = 'AU7_823_1ML22_MIL_2 Channel 15'; AU7_823_1ML22_MIL_2 Channel 15.DataType = 'BOOL'; AU7_823_1ML22_MIL_2 Channel 15.Default = ''; AU7_823_1ML22_MIL_2 Channel 15.Comment = ''; AU7_823_1ML22_MIL_2 Channel 16.Name = 'AU7_823_1ML22_MIL_2 Channel 16'; AU7_823_1ML22_MIL_2 Channel 16.DataType = 'BOOL'; AU7_823_1ML22_MIL_2 Channel 16.Default = ''; AU7_823_1ML22_MIL_2 Channel 16.Comment = ''; AU7_823_1ML22_MIL_2 Channel 1-8.Name = 'AU7_823_1ML22_MIL_2 Channel 1-8'; AU7_823_1ML22_MIL_2 Channel 1-8.DataType = 'USINT'; AU7_823_1ML22_MIL_2 Channel 1-8.Default = ''; AU7_823_1ML22_MIL_2 Channel 1-8.Comment = ''; AU7_823_1ML22_MIL_2 Channel 9-16.Name = 'AU7_823_1ML22_MIL_2 Channel 9-16'; AU7_823_1ML22_MIL_2 Channel 9-16.DataType = 'USINT'; AU7_823_1ML22_MIL_2 Channel 9-16.Default = ''; AU7_823_1ML22_MIL_2 Channel 9-16.Comment = ''; AU7_823_1ML22_MIL_2 Channel 1-8.Name = 'AU7_823_1ML22_MIL_2 Channel 1-8'; AU7_823_1ML22_MIL_2 Channel 1-8.DataType = 'BIT'; AU7_823_1ML22_MIL_2 Channel 1-8.Default = ''; AU7_823_1ML22_MIL_2 Channel 1-8.Comment = ''; AU7_823_1ML22_MIL_2 Channel 9-16.Name = 'AU7_823_1ML22_MIL_2 Channel 9-16'; AU7_823_1ML22_MIL_2 Channel 9-16.DataType = 'BIT'; AU7_823_1ML22_MIL_2 Channel 9-16.Default = ''; AU7_823_1ML22_MIL_2 Channel 9-16.Comment = ''; AU7_823_1ML22_MIL_2 Channel 1-16.Name = 'AU7_823_1ML22_MIL_2 Channel 1-16'; AU7_823_1ML22_MIL_2 Channel 1-16.DataType = 'BIT'; AU7_823_1ML22_MIL_2 Channel 1-16.Default = ''; AU7_823_1ML22_MIL_2 Channel 1-16.Comment = ''; AU7_823_1ML22_MIL_2 Channel 1-16.Name = 'AU7_823_1ML22_MIL_2 Channel 1-16';
            AU7_823_1ML22_MIL_2 Channel 1-16.DataType = 'UINT'; AU7_823_1ML22_MIL_2 Channel 1-16.Default = ''; AU7_823_1ML22_MIL_2 Channel 1-16.Comment = ''; AU7_823_1ML22_MIL_3 Channel 1.Name = 'AU7_823_1ML22_MIL_3 Channel 1'; AU7_823_1ML22_MIL_3 Channel 1.DataType = 'BOOL'; AU7_823_1ML22_MIL_3 Channel 1.Default = ''; AU7_823_1ML22_MIL_3 Channel 1.Comment = ''; AU7_823_1ML22_MIL_3 Channel 2.Name = 'AU7_823_1ML22_MIL_3 Channel 2'; AU7_823_1ML22_MIL_3 Channel 2.DataType = 'BOOL'; AU7_823_1ML22_MIL_3 Channel 2.Default = ''; AU7_823_1ML22_MIL_3 Channel 2.Comment = ''; AU7_823_1ML22_MIL_3 Channel 3.Name = 'AU7_823_1ML22_MIL_3 Channel 3'; AU7_823_1ML22_MIL_3 Channel 3.DataType = 'BOOL'; AU7_823_1ML22_MIL_3 Channel 3.Default = ''; AU7_823_1ML22_MIL_3 Channel 3.Comment = ''; AU7_823_1ML22_MIL_3 Channel 4.Name = 'AU7_823_1ML22_MIL_3 Channel 4'; AU7_823_1ML22_MIL_3 Channel 4.DataType = 'BOOL'; AU7_823_1ML22_MIL_3 Channel 4.Default = ''; AU7_823_1ML22_MIL_3 Channel 4.Comment = ''; AU7_823_1ML22_MIL_3 Channel 5.Name = 'AU7_823_1ML22_MIL_3 Channel 5'; AU7_823_1ML22_MIL_3 Channel 5.DataType = 'BOOL'; AU7_823_1ML22_MIL_3 Channel 5.Default = ''; AU7_823_1ML22_MIL_3 Channel 5.Comment = ''; AU7_823_1ML22_MIL_3 Channel 6.Name = 'AU7_823_1ML22_MIL_3 Channel 6'; AU7_823_1ML22_MIL_3 Channel 6.DataType = 'BOOL'; AU7_823_1ML22_MIL_3 Channel 6.Default = ''; AU7_823_1ML22_MIL_3 Channel 6.Comment = ''; AU7_823_1ML22_MIL_3 Channel 7.Name = 'AU7_823_1ML22_MIL_3 Channel 7'; AU7_823_1ML22_MIL_3 Channel 7.DataType = 'BOOL'; AU7_823_1ML22_MIL_3 Channel 7.Default = ''; AU7_823_1ML22_MIL_3 Channel 7.Comment = ''; AU7_823_1ML22_MIL_3 Channel 8.Name = 'AU7_823_1ML22_MIL_3 Channel 8'; AU7_823_1ML22_MIL_3 Channel 8.DataType = 'BOOL'; AU7_823_1ML22_MIL_3 Channel 8.Default = ''; AU7_823_1ML22_MIL_3 Channel 8.Comment = ''; AU7_823_1ML22_MIL_3 Channel 9.Name = 'AU7_823_1ML22_MIL_3 Channel 9'; AU7_823_1ML22_MIL_3 Channel 9.DataType = 'BOOL'; AU7_823_1ML22_MIL_3 Channel 9.Default = ''; AU7_823_1ML22_MIL_3 Channel 9.Comment = ''; AU7_823_1ML22_MIL_3 Channel 10.Name = 'AU7_823_1ML22_MIL_3 Channel 10';
            AU7_823_1ML22_MIL_3 Channel 10.DataType = 'BOOL'; AU7_823_1ML22_MIL_3 Channel 10.Default = ''; AU7_823_1ML22_MIL_3 Channel 10.Comment = ''; AU7_823_1ML22_MIL_3 Channel 11.Name = 'AU7_823_1ML22_MIL_3 Channel 11'; AU7_823_1ML22_MIL_3 Channel 11.DataType = 'BOOL'; AU7_823_1ML22_MIL_3 Channel 11.Default = ''; AU7_823_1ML22_MIL_3 Channel 11.Comment = ''; AU7_823_1ML22_MIL_3 Channel 12.Name = 'AU7_823_1ML22_MIL_3 Channel 12'; AU7_823_1ML22_MIL_3 Channel 12.DataType = 'BOOL'; AU7_823_1ML22_MIL_3 Channel 12.Default = ''; AU7_823_1ML22_MIL_3 Channel 12.Comment = ''; AU7_823_1ML22_MIL_3 Channel 13.Name = 'AU7_823_1ML22_MIL_3 Channel 13'; AU7_823_1ML22_MIL_3 Channel 13.DataType = 'BOOL'; AU7_823_1ML22_MIL_3 Channel 13.Default = ''; AU7_823_1ML22_MIL_3 Channel 13.Comment = ''; AU7_823_1ML22_MIL_3 Channel 14.Name = 'AU7_823_1ML22_MIL_3 Channel 14'; AU7_823_1ML22_MIL_3 Channel 14.DataType = 'BOOL'; AU7_823_1ML22_MIL_3 Channel 14.Default = ''; AU7_823_1ML22_MIL_3 Channel 14.Comment = ''; AU7_823_1ML22_MIL_3 Channel 15.Name = 'AU7_823_1ML22_MIL_3 Channel 15'; AU7_823_1ML22_MIL_3 Channel 15.DataType = 'BOOL'; AU7_823_1ML22_MIL_3 Channel 15.Default = ''; AU7_823_1ML22_MIL_3 Channel 15.Comment = ''; AU7_823_1ML22_MIL_3 Channel 16.Name = 'AU7_823_1ML22_MIL_3 Channel 16'; AU7_823_1ML22_MIL_3 Channel 16.DataType = 'BOOL'; AU7_823_1ML22_MIL_3 Channel 16.Default = ''; AU7_823_1ML22_MIL_3 Channel 16.Comment = ''; AU7_823_1ML22_MIL_3 Channel 1-8.Name = 'AU7_823_1ML22_MIL_3 Channel 1-8'; AU7_823_1ML22_MIL_3 Channel 1-8.DataType = 'USINT'; AU7_823_1ML22_MIL_3 Channel 1-8.Default = ''; AU7_823_1ML22_MIL_3 Channel 1-8.Comment = ''; AU7_823_1ML22_MIL_3 Channel 9-16.Name = 'AU7_823_1ML22_MIL_3 Channel 9-16'; AU7_823_1ML22_MIL_3 Channel 9-16.DataType = 'USINT'; AU7_823_1ML22_MIL_3 Channel 9-16.Default = ''; AU7_823_1ML22_MIL_3 Channel 9-16.Comment = ''; AU7_823_1ML22_MIL_3 Channel 1-8.Name = 'AU7_823_1ML22_MIL_3 Channel 1-8'; AU7_823_1ML22_MIL_3 Channel 1-8.DataType = 'BIT'; AU7_823_1ML22_MIL_3 Channel 1-8.Default = ''; AU7_823_1ML22_MIL_3 Channel 1-8.Comment = ''; AU7_823_1ML22_MIL_3 Channel 9-16.Name = 'AU7_823_1ML22_MIL_3 Channel 9-16';
            AU7_823_1ML22_MIL_3 Channel 9-16.DataType = 'BIT'; AU7_823_1ML22_MIL_3 Channel 9-16.Default = ''; AU7_823_1ML22_MIL_3 Channel 9-16.Comment = ''; AU7_823_1ML22_MIL_3 Channel 1-16.Name = 'AU7_823_1ML22_MIL_3 Channel 1-16'; AU7_823_1ML22_MIL_3 Channel 1-16.DataType = 'BIT'; AU7_823_1ML22_MIL_3 Channel 1-16.Default = ''; AU7_823_1ML22_MIL_3 Channel 1-16.Comment = ''; AU7_823_1ML22_MIL_3 Channel 1-16.Name = 'AU7_823_1ML22_MIL_3 Channel 1-16'; AU7_823_1ML22_MIL_3 Channel 1-16.DataType = 'UINT'; AU7_823_1ML22_MIL_3 Channel 1-16.Default = ''; AU7_823_1ML22_MIL_3 Channel 1-16.Comment = ''; AU7_823_1ML22_MIL_4 Channel 1.Name = 'AU7_823_1ML22_MIL_4 Channel 1'; AU7_823_1ML22_MIL_4 Channel 1.DataType = 'BOOL'; AU7_823_1ML22_MIL_4 Channel 1.Default = ''; AU7_823_1ML22_MIL_4 Channel 1.Comment = ''; AU7_823_1ML22_MIL_4 Channel 2.Name = 'AU7_823_1ML22_MIL_4 Channel 2'; AU7_823_1ML22_MIL_4 Channel 2.DataType = 'BOOL'; AU7_823_1ML22_MIL_4 Channel 2.Default = ''; AU7_823_1ML22_MIL_4 Channel 2.Comment = ''; AU7_823_1ML22_MIL_4 Channel 3.Name = 'AU7_823_1ML22_MIL_4 Channel 3'; AU7_823_1ML22_MIL_4 Channel 3.DataType = 'BOOL'; AU7_823_1ML22_MIL_4 Channel 3.Default = ''; AU7_823_1ML22_MIL_4 Channel 3.Comment = ''; AU7_823_1ML22_MIL_4 Channel 4.Name = 'AU7_823_1ML22_MIL_4 Channel 4'; AU7_823_1ML22_MIL_4 Channel 4.DataType = 'BOOL'; AU7_823_1ML22_MIL_4 Channel 4.Default = ''; AU7_823_1ML22_MIL_4 Channel 4.Comment = ''; AU7_823_1ML22_MIL_4 Channel 5.Name = 'AU7_823_1ML22_MIL_4 Channel 5'; AU7_823_1ML22_MIL_4 Channel 5.DataType = 'BOOL'; AU7_823_1ML22_MIL_4 Channel 5.Default = ''; AU7_823_1ML22_MIL_4 Channel 5.Comment = ''; AU7_823_1ML22_MIL_4 Channel 6.Name = 'AU7_823_1ML22_MIL_4 Channel 6'; AU7_823_1ML22_MIL_4 Channel 6.DataType = 'BOOL'; AU7_823_1ML22_MIL_4 Channel 6.Default = ''; AU7_823_1ML22_MIL_4 Channel 6.Comment = ''; AU7_823_1ML22_MIL_4 Channel 7.Name = 'AU7_823_1ML22_MIL_4 Channel 7'; AU7_823_1ML22_MIL_4 Channel 7.DataType = 'BOOL'; AU7_823_1ML22_MIL_4 Channel 7.Default = ''; AU7_823_1ML22_MIL_4 Channel 7.Comment = ''; AU7_823_1ML22_MIL_4 Channel 8.Name = 'AU7_823_1ML22_MIL_4 Channel 8';
            AU7_823_1ML22_MIL_4 Channel 8.DataType = 'BOOL'; AU7_823_1ML22_MIL_4 Channel 8.Default = ''; AU7_823_1ML22_MIL_4 Channel 8.Comment = ''; AU7_823_1ML22_MIL_4 Channel 9.Name = 'AU7_823_1ML22_MIL_4 Channel 9'; AU7_823_1ML22_MIL_4 Channel 9.DataType = 'BOOL'; AU7_823_1ML22_MIL_4 Channel 9.Default = ''; AU7_823_1ML22_MIL_4 Channel 9.Comment = ''; AU7_823_1ML22_MIL_4 Channel 10.Name = 'AU7_823_1ML22_MIL_4 Channel 10'; AU7_823_1ML22_MIL_4 Channel 10.DataType = 'BOOL'; AU7_823_1ML22_MIL_4 Channel 10.Default = ''; AU7_823_1ML22_MIL_4 Channel 10.Comment = ''; AU7_823_1ML22_MIL_4 Channel 11.Name = 'AU7_823_1ML22_MIL_4 Channel 11'; AU7_823_1ML22_MIL_4 Channel 11.DataType = 'BOOL'; AU7_823_1ML22_MIL_4 Channel 11.Default = ''; AU7_823_1ML22_MIL_4 Channel 11.Comment = ''; AU7_823_1ML22_MIL_4 Channel 12.Name = 'AU7_823_1ML22_MIL_4 Channel 12'; AU7_823_1ML22_MIL_4 Channel 12.DataType = 'BOOL'; AU7_823_1ML22_MIL_4 Channel 12.Default = ''; AU7_823_1ML22_MIL_4 Channel 12.Comment = ''; AU7_823_1ML22_MIL_4 Channel 13.Name = 'AU7_823_1ML22_MIL_4 Channel 13'; AU7_823_1ML22_MIL_4 Channel 13.DataType = 'BOOL'; AU7_823_1ML22_MIL_4 Channel 13.Default = ''; AU7_823_1ML22_MIL_4 Channel 13.Comment = ''; AU7_823_1ML22_MIL_4 Channel 14.Name = 'AU7_823_1ML22_MIL_4 Channel 14'; AU7_823_1ML22_MIL_4 Channel 14.DataType = 'BOOL'; AU7_823_1ML22_MIL_4 Channel 14.Default = ''; AU7_823_1ML22_MIL_4 Channel 14.Comment = ''; AU7_823_1ML22_MIL_4 Channel 15.Name = 'AU7_823_1ML22_MIL_4 Channel 15'; AU7_823_1ML22_MIL_4 Channel 15.DataType = 'BOOL'; AU7_823_1ML22_MIL_4 Channel 15.Default = ''; AU7_823_1ML22_MIL_4 Channel 15.Comment = ''; AU7_823_1ML22_MIL_4 Channel 16.Name = 'AU7_823_1ML22_MIL_4 Channel 16'; AU7_823_1ML22_MIL_4 Channel 16.DataType = 'BOOL'; AU7_823_1ML22_MIL_4 Channel 16.Default = ''; AU7_823_1ML22_MIL_4 Channel 16.Comment = ''; AU7_823_1ML22_MIL_4 Channel 1-8.Name = 'AU7_823_1ML22_MIL_4 Channel 1-8'; AU7_823_1ML22_MIL_4 Channel 1-8.DataType = 'USINT'; AU7_823_1ML22_MIL_4 Channel 1-8.Default = ''; AU7_823_1ML22_MIL_4 Channel 1-8.Comment = ''; AU7_823_1ML22_MIL_4 Channel 9-16.Name = 'AU7_823_1ML22_MIL_4 Channel 9-16';
            AU7_823_1ML22_MIL_4 Channel 9-16.DataType = 'USINT'; AU7_823_1ML22_MIL_4 Channel 9-16.Default = ''; AU7_823_1ML22_MIL_4 Channel 9-16.Comment = ''; AU7_823_1ML22_MIL_4 Channel 1-8.Name = 'AU7_823_1ML22_MIL_4 Channel 1-8'; AU7_823_1ML22_MIL_4 Channel 1-8.DataType = 'BIT'; AU7_823_1ML22_MIL_4 Channel 1-8.Default = ''; AU7_823_1ML22_MIL_4 Channel 1-8.Comment = ''; AU7_823_1ML22_MIL_4 Channel 9-16.Name = 'AU7_823_1ML22_MIL_4 Channel 9-16'; AU7_823_1ML22_MIL_4 Channel 9-16.DataType = 'BIT'; AU7_823_1ML22_MIL_4 Channel 9-16.Default = ''; AU7_823_1ML22_MIL_4 Channel 9-16.Comment = ''; AU7_823_1ML22_MIL_4 Channel 1-16.Name = 'AU7_823_1ML22_MIL_4 Channel 1-16'; AU7_823_1ML22_MIL_4 Channel 1-16.DataType = 'BIT'; AU7_823_1ML22_MIL_4 Channel 1-16.Default = ''; AU7_823_1ML22_MIL_4 Channel 1-16.Comment = ''; AU7_823_1ML22_MIL_4 Channel 1-16.Name = 'AU7_823_1ML22_MIL_4 Channel 1-16'; AU7_823_1ML22_MIL_4 Channel 1-16.DataType = 'UINT'; AU7_823_1ML22_MIL_4 Channel 1-16.Default = ''; AU7_823_1ML22_MIL_4 Channel 1-16.Comment = ''
          unmapped channels: %QX1.0 AU7_823_1ML22_MIL Channel 1, AU7_823_1ML22_MIL Channel 2, AU7_823_1ML22_MIL Channel 3, AU7_823_1ML22_MIL Channel 4, AU7_823_1ML22_MIL Channel 5, AU7_823_1ML22_MIL Channel 6, AU7_823_1ML22_MIL Channel 7, AU7_823_1ML22_MIL Channel 8, AU7_823_1ML22_MIL Channel 9, AU7_823_1ML22_MIL Channel 10, AU7_823_1ML22_MIL Channel 11, AU7_823_1ML22_MIL Channel 12, AU7_823_1ML22_MIL Channel 13, AU7_823_1ML22_MIL Channel 14, AU7_823_1ML22_MIL Channel 15, AU7_823_1ML22_MIL Channel 16, AU7_823_1ML22_MIL_1 Channel 1, AU7_823_1ML22_MIL_1 Channel 2, AU7_823_1ML22_MIL_1 Channel 3, AU7_823_1ML22_MIL_1 Channel 4, AU7_823_1ML22_MIL_1 Channel 5, AU7_823_1ML22_MIL_1 Channel 6, AU7_823_1ML22_MIL_1 Channel 7, AU7_823_1ML22_MIL_1 Channel 8, AU7_823_1ML22_MIL_1 Channel 9, AU7_823_1ML22_MIL_1 Channel 10, AU7_823_1ML22_MIL_1 Channel 11, AU7_823_1ML22_MIL_1 Channel 12, AU7_823_1ML22_MIL_1 Channel 13, AU7_823_1ML22_MIL_1 Channel 14, AU7_823_1ML22_MIL_1 Channel 15, AU7_823_1ML22_MIL_1 Channel 16, AU7_823_1ML22_MIL_2 Channel 1, AU7_823_1ML22_MIL_2 Channel 2, AU7_823_1ML22_MIL_2 Channel 3, AU7_823_1ML22_MIL_2 Channel 4, AU7_823_1ML22_MIL_2 Channel 5, AU7_823_1ML22_MIL_2 Channel 6, AU7_823_1ML22_MIL_2 Channel 7, AU7_823_1ML22_MIL_2 Channel 8,
            AU7_823_1ML22_MIL_2 Channel 9, AU7_823_1ML22_MIL_2 Channel 10, AU7_823_1ML22_MIL_2 Channel 11, AU7_823_1ML22_MIL_2 Channel 12, AU7_823_1ML22_MIL_2 Channel 13, AU7_823_1ML22_MIL_2 Channel 14, AU7_823_1ML22_MIL_2 Channel 15, AU7_823_1ML22_MIL_2 Channel 16, AU7_823_1ML22_MIL_3 Channel 1, AU7_823_1ML22_MIL_3 Channel 2, AU7_823_1ML22_MIL_3 Channel 3, AU7_823_1ML22_MIL_3 Channel 4, AU7_823_1ML22_MIL_3 Channel 5, AU7_823_1ML22_MIL_3 Channel 6, AU7_823_1ML22_MIL_3 Channel 7, AU7_823_1ML22_MIL_3 Channel 8, AU7_823_1ML22_MIL_3 Channel 9, AU7_823_1ML22_MIL_3 Channel 10, AU7_823_1ML22_MIL_3 Channel 11, AU7_823_1ML22_MIL_3 Channel 12, AU7_823_1ML22_MIL_3 Channel 13, AU7_823_1ML22_MIL_3 Channel 14, AU7_823_1ML22_MIL_3 Channel 15, AU7_823_1ML22_MIL_3 Channel 16, AU7_823_1ML22_MIL_4 Channel 1, AU7_823_1ML22_MIL_4 Channel 2, AU7_823_1ML22_MIL_4 Channel 3, AU7_823_1ML22_MIL_4 Channel 4, AU7_823_1ML22_MIL_4 Channel 5, AU7_823_1ML22_MIL_4 Channel 6, AU7_823_1ML22_MIL_4 Channel 7, AU7_823_1ML22_MIL_4 Channel 8, AU7_823_1ML22_MIL_4 Channel 9, AU7_823_1ML22_MIL_4 Channel 10, AU7_823_1ML22_MIL_4 Channel 11, AU7_823_1ML22_MIL_4 Channel 12, AU7_823_1ML22_MIL_4 Channel 13, AU7_823_1ML22_MIL_4 Channel 14, AU7_823_1ML22_MIL_4 Channel 15, AU7_823_1ML22_MIL_4 Channel 16,
            ID, %IX3.0 AU7_823_1ML22_MIL Channel 1, AU7_823_1ML22_MIL Channel 2, AU7_823_1ML22_MIL Channel 3, AU7_823_1ML22_MIL Channel 4, AU7_823_1ML22_MIL Channel 5, AU7_823_1ML22_MIL Channel 6, AU7_823_1ML22_MIL Channel 7, AU7_823_1ML22_MIL Channel 8, AU7_823_1ML22_MIL Channel 9, AU7_823_1ML22_MIL Channel 10, AU7_823_1ML22_MIL Channel 11, AU7_823_1ML22_MIL Channel 12, AU7_823_1ML22_MIL Channel 13, AU7_823_1ML22_MIL Channel 14, AU7_823_1ML22_MIL Channel 15, AU7_823_1ML22_MIL Channel 16, AU7_823_1ML22_MIL_1 Channel 1, AU7_823_1ML22_MIL_1 Channel 2, AU7_823_1ML22_MIL_1 Channel 3, AU7_823_1ML22_MIL_1 Channel 4, AU7_823_1ML22_MIL_1 Channel 5, AU7_823_1ML22_MIL_1 Channel 6, AU7_823_1ML22_MIL_1 Channel 7, AU7_823_1ML22_MIL_1 Channel 8, AU7_823_1ML22_MIL_1 Channel 9, AU7_823_1ML22_MIL_1 Channel 10, AU7_823_1ML22_MIL_1 Channel 11, AU7_823_1ML22_MIL_1 Channel 12, AU7_823_1ML22_MIL_1 Channel 13, AU7_823_1ML22_MIL_1 Channel 14, AU7_823_1ML22_MIL_1 Channel 15, AU7_823_1ML22_MIL_1 Channel 16, AU7_823_1ML22_MIL_2 Channel 1, AU7_823_1ML22_MIL_2 Channel 2, AU7_823_1ML22_MIL_2 Channel 3, AU7_823_1ML22_MIL_2 Channel 4, AU7_823_1ML22_MIL_2 Channel 5, AU7_823_1ML22_MIL_2 Channel 6, AU7_823_1ML22_MIL_2 Channel 7,
            AU7_823_1ML22_MIL_2 Channel 8, AU7_823_1ML22_MIL_2 Channel 9, AU7_823_1ML22_MIL_2 Channel 10, AU7_823_1ML22_MIL_2 Channel 11, AU7_823_1ML22_MIL_2 Channel 12, AU7_823_1ML22_MIL_2 Channel 13, AU7_823_1ML22_MIL_2 Channel 14, AU7_823_1ML22_MIL_2 Channel 15, AU7_823_1ML22_MIL_2 Channel 16, AU7_823_1ML22_MIL_3 Channel 1, AU7_823_1ML22_MIL_3 Channel 2, AU7_823_1ML22_MIL_3 Channel 3, AU7_823_1ML22_MIL_3 Channel 4, AU7_823_1ML22_MIL_3 Channel 5, AU7_823_1ML22_MIL_3 Channel 6, AU7_823_1ML22_MIL_3 Channel 7, AU7_823_1ML22_MIL_3 Channel 8, AU7_823_1ML22_MIL_3 Channel 9, AU7_823_1ML22_MIL_3 Channel 10, AU7_823_1ML22_MIL_3 Channel 11, AU7_823_1ML22_MIL_3 Channel 12, AU7_823_1ML22_MIL_3 Channel 13, AU7_823_1ML22_MIL_3 Channel 14, AU7_823_1ML22_MIL_3 Channel 15, AU7_823_1ML22_MIL_3 Channel 16, AU7_823_1ML22_MIL_4 Channel 1, AU7_823_1ML22_MIL_4 Channel 2, AU7_823_1ML22_MIL_4 Channel 3, AU7_823_1ML22_MIL_4 Channel 4, AU7_823_1ML22_MIL_4 Channel 5, AU7_823_1ML22_MIL_4 Channel 6, AU7_823_1ML22_MIL_4 Channel 7, AU7_823_1ML22_MIL_4 Channel 8, AU7_823_1ML22_MIL_4 Channel 9, AU7_823_1ML22_MIL_4 Channel 10, AU7_823_1ML22_MIL_4 Channel 11, AU7_823_1ML22_MIL_4 Channel 12, AU7_823_1ML22_MIL_4 Channel 13, AU7_823_1ML22_MIL_4 Channel 14, AU7_823_1ML22_MIL_4 Channel 15,
            AU7_823_1ML22_MIL_4 Channel 16
        AU7_823_1ML22_MIL : AU7 823-1ML22-MIL,16DI/16DO (24VDC,PNP/NPN,NPN), AUTO, order no. AU7 823-1ML22-MIL, version 0
        AU7_823_1ML22_MIL_4 : AU7 823-1ML22-MIL,16DI/16DO (24VDC,PNP/NPN,NPN), AUTO, order no. AU7 823-1ML22-MIL, version 0
        AU7_823_1ML22_MIL_3 : AU7 823-1ML22-MIL,16DI/16DO (24VDC,PNP/NPN,NPN), AUTO, order no. AU7 823-1ML22-MIL, version 0
        AU7_823_1ML22_MIL_2 : AU7 823-1ML22-MIL,16DI/16DO (24VDC,PNP/NPN,NPN), AUTO, order no. AU7 823-1ML22-MIL, version 0
        AU7_823_1ML22_MIL_1 : AU7 823-1ML22-MIL,16DI/16DO (24VDC,PNP/NPN,NPN), AUTO, order no. AU7 823-1ML22-MIL, version 0
      InoSV660N_8 : SV660_1Axis_00915, Inovance, order no. InoSV660N, version Revision=16#00010000
          settings: FunCodeList = H02;H02-01;H03;H03-03;H03-05;; WriteValueList = H02-01_8194_2_1_UINT_RW;H03-03_8195_4_1_UINT_RW;H03-05_8195_6_1_UINT_RW;; Number of Outputs = 6; Number of Inputs = 10; Number of Infos about Outputs = 6; Number of Infos about Inputs = 10; Configuration address of the slave = 10; Sync.Length = 18; Sync.Length = 32; FMMU.Length = 18; FMMU.Length = 32; AutoUpdate = False; DC sync0 cycletime = 4000; DC sync1 cycletime = 4000; Number of SDO = 10; Homing method.Index = 16#6098; Homing method.Subindex = 16#00; Homing method.Value = 26; Homing method.Size = 8; Homing method.AbortIfError = FALSE; Homing method.JumpToLine = FALSE; Homing method.Line = 0; Homing method.CompleteAccess = FALSE; Actual Position Calculation Method.Index = 16#60E6; Actual Position Calculation Method.Subindex = 16#00; Actual Position Calculation Method.Value = 0; Actual Position Calculation Method.Size = 8; Actual Position Calculation Method.AbortIfError = FALSE; Actual Position Calculation Method.JumpToLine = FALSE; Actual Position Calculation Method.Line = 0; Actual Position Calculation Method.CompleteAccess = FALSE; Speed during search for switch.Index = 16#6099; Speed during search for switch.Subindex = 16#01; Speed during search for switch.Value = 41943040; Speed during search for switch.Size = 32; Speed during search for switch.AbortIfError = FALSE; Speed during search for switch.JumpToLine = FALSE; Speed during search for switch.Line = 0; Speed during search for switch.CompleteAccess = FALSE; Homing acceleration.Index = 16#609A;
            Homing acceleration.Subindex = 16#00; Homing acceleration.Value = 139810133; Homing acceleration.Size = 32; Homing acceleration.AbortIfError = FALSE; Homing acceleration.JumpToLine = FALSE; Homing acceleration.Line = 0; Homing acceleration.CompleteAccess = FALSE; Speed during search for zero.Index = 16#6099; Speed during search for zero.Subindex = 16#02; Speed during search for zero.Value = 16777216; Speed during search for zero.Size = 32; Speed during search for zero.AbortIfError = FALSE; Speed during search for zero.JumpToLine = FALSE; Speed during search for zero.Line = 0; Speed during search for zero.CompleteAccess = FALSE; Time of home searching.Index = 16#2005; Time of home searching.Subindex = 16#24; Time of home searching.Value = 50000; Time of home searching.Size = 16; Time of home searching.AbortIfError = FALSE; Time of home searching.JumpToLine = FALSE; Time of home searching.Line = 0; Time of home searching.CompleteAccess = FALSE; Positive torque limit value.Index = 16#60E0; Positive torque limit value.Subindex = 16#00; Positive torque limit value.Value = 3500; Positive torque limit value.Size = 16; Positive torque limit value.AbortIfError = FALSE; Positive torque limit value.JumpToLine = FALSE; Positive torque limit value.Line = 0; Positive torque limit value.CompleteAccess = FALSE; Negative torque limit value.Index = 16#60E1; Negative torque limit value.Subindex = 16#00; Negative torque limit value.Value = 3500; Negative torque limit value.Size = 16; Negative torque limit value.AbortIfError = FALSE; Negative torque limit value.JumpToLine = FALSE; Negative torque limit value.Line = 0; Negative torque limit value.CompleteAccess = FALSE; Max profile velocity.Index = 16#607F;
            Max profile velocity.Subindex = 16#00; Max profile velocity.Value = 83886080; Max profile velocity.Size = 32; Max profile velocity.AbortIfError = FALSE; Max profile velocity.JumpToLine = FALSE; Max profile velocity.Line = 0; Max profile velocity.CompleteAccess = FALSE; RxTxPdo.NumberofEntries = 6; RxTxPdo.Sm = 2; Controlword.Index = 16#6040; Controlword.SubIndex = 0; Controlword.Size = 16; Controlword.DependOnSlot = false; Controlword.DependOnSlotGroup = false; Target position.Index = 16#607A; Target position.SubIndex = 0; Target position.Size = 32; Target position.DependOnSlot = false; Target position.DependOnSlotGroup = false; Touch probe function.Index = 16#60B8; Touch probe function.SubIndex = 0; Touch probe function.Size = 16; Touch probe function.DependOnSlot = false; Touch probe function.DependOnSlotGroup = false; Physical outputs.Index = 16#60FE; Physical outputs.SubIndex = 1; Physical outputs.Size = 32; Physical outputs.DependOnSlot = false; Physical outputs.DependOnSlotGroup = false; Target velocity.Index = 16#60FF; Target velocity.SubIndex = 0; Target velocity.Size = 32; Target velocity.DependOnSlot = false; Target velocity.DependOnSlotGroup = false; Target torque.Index = 16#6071; Target torque.SubIndex = 0; Target torque.Size = 16; Target torque.DependOnSlot = false; Target torque.DependOnSlotGroup = false; RxTxPdo.Sm = -1;
            RxTxPdo.NumberofEntries = 10; RxTxPdo.Sm = 3; Error code.Index = 16#603F; Error code.SubIndex = 0; Error code.Size = 16; Error code.DependOnSlot = false; Error code.DependOnSlotGroup = false; Statusword.Index = 16#6041; Statusword.SubIndex = 0; Statusword.Size = 16; Statusword.DependOnSlot = false; Statusword.DependOnSlotGroup = false; Position actual value.Index = 16#6064; Position actual value.SubIndex = 0; Position actual value.Size = 32; Position actual value.DependOnSlot = false; Position actual value.DependOnSlotGroup = false; Torque actual value.Index = 16#6077; Torque actual value.SubIndex = 0; Torque actual value.Size = 16; Torque actual value.DependOnSlot = false; Torque actual value.DependOnSlotGroup = false; Following error actual value.Index = 16#60F4; Following error actual value.SubIndex = 0; Following error actual value.Size = 32; Following error actual value.DependOnSlot = false; Following error actual value.DependOnSlotGroup = false; Touch probe status.Index = 16#60B9; Touch probe status.SubIndex = 0; Touch probe status.Size = 16; Touch probe status.DependOnSlot = false; Touch probe status.DependOnSlotGroup = false; Touch probe pos1 pos value.Index = 16#60BA; Touch probe pos1 pos value.SubIndex = 0; Touch probe pos1 pos value.Size = 32; Touch probe pos1 pos value.DependOnSlot = false; Touch probe pos1 pos value.DependOnSlotGroup = false; Touch probe pos2 pos value.Index = 16#60BC; Touch probe pos2 pos value.SubIndex = 0; Touch probe pos2 pos value.Size = 32;
            Touch probe pos2 pos value.DependOnSlot = false; Touch probe pos2 pos value.DependOnSlotGroup = false; Digital inputs.Index = 16#60FD; Digital inputs.SubIndex = 0; Digital inputs.Size = 32; Digital inputs.DependOnSlot = false; Digital inputs.DependOnSlotGroup = false; Velocity actual value.Index = 16#606C; Velocity actual value.SubIndex = 0; Velocity actual value.Size = 32; Velocity actual value.DependOnSlot = false; Velocity actual value.DependOnSlotGroup = false; RxTxPdo.Sm = -1; Controlword.Name = 'Controlword'; Controlword.DataType = 'UINT'; Target position.Name = 'Target position'; Target position.DataType = 'DINT'; Touch probe function.Name = 'Touch probe function'; Touch probe function.DataType = 'UINT'; Physical outputs.Name = 'Physical outputs'; Physical outputs.DataType = 'UDINT'; Target velocity.Name = 'Target velocity'; Target velocity.DataType = 'DINT'; Target torque.Name = 'Target torque'; Target torque.DataType = 'INT'; Error code.Name = 'Error code'; Error code.DataType = 'UINT'; Statusword.Name = 'Statusword'; Statusword.DataType = 'UINT'; Position actual value.Name = 'Position actual value'; Position actual value.DataType = 'DINT'; Torque actual value.Name = 'Torque actual value'; Torque actual value.DataType = 'INT'; Following error actual value.Name = 'Following error actual value'; Following error actual value.DataType = 'DINT'; Touch probe status.Name = 'Touch probe status'; Touch probe status.DataType = 'UINT'; Touch probe pos1 pos value.Name = 'Touch probe pos1 pos value'; Touch probe pos1 pos value.DataType = 'DINT'; Touch probe pos2 pos value.Name = 'Touch probe pos2 pos value';
            Touch probe pos2 pos value.DataType = 'DINT'; Digital inputs.Name = 'Digital inputs'; Digital inputs.DataType = 'UDINT'; Velocity actual value.Name = 'Velocity actual value'; Velocity actual value.DataType = 'DINT'
          unmapped channels: Controlword, Target position, Touch probe function, Physical outputs, Target velocity, Target torque, Error code, Statusword, Position actual value, Torque actual value, Following error actual value, Touch probe status, Touch probe pos1 pos value, Touch probe pos2 pos value, Digital inputs, Velocity actual value
        地轨轴11Y : Axis, Inovance, order no. 0, version 1.0.0.0
            settings: wDriveID = 8; dwRatioTechUnitsDenom = 4194304; iRatioTechUnitsNum = -5; iEncoderType = 1; iAbsEncoderOption = 2; HomingMode = 10; ZeroSignal = 0; StartDirction = 1; EndDirection = 1; PosLimitMode = 0; NegLimitMode = 0; HomingVelocity = 10; HomingApproachVelocity = 2; HomingAcceleration = 100; HomingDeceleration = 100; HomingJerk = 0; HomeMaskDistance = 0; HomePositionOffset = 0; HomePushTime = 0; HomeCompensation = 0; HomeTimeout = 0; HomeCompensationVelocity = 1000; 4000 = 1; 4001 = 0; 4003 = true; 4004 = 26; 4005 = 0; 4006 = 50.0; 4007 = 166.666666; 4008 = 20.0; 4009 = 50000; 4010 = 3500; 4011 = 3500; 4012 = 100.000000; ScalingIncs = 16#800000; InvertDirection = TRUE; 6005 = 10; AdrOffset_8010 = 2192; BitOffset_8010 = 0; BitLength_8010 = 16;
              Address_8010 = '%QW1096'; Type_8010 = 'UINT'; AddressPointer_8010 = ADR(%QW1096); AdrOffset_8020 = 2196; BitOffset_8020 = 0; BitLength_8020 = 32; Address_8020 = '%QD549'; Type_8020 = 'DINT'; AddressPointer_8020 = ADR(%QD549); AdrOffset_8030 = 2208; BitOffset_8030 = 0; BitLength_8030 = 32; Address_8030 = '%QD552'; Type_8030 = 'DINT'; AddressPointer_8030 = ADR(%QD552); AdrOffset_8040 = 2212; BitOffset_8040 = 0; BitLength_8040 = 16; Address_8040 = '%QW1106'; Type_8040 = 'INT'; AddressPointer_8040 = ADR(%QW1106); AdrOffset_8050 = 4294967295; BitOffset_8050 = 0; BitLength_8050 = 0; Address_8050 = ''; Type_8050 = ''; AddressPointer_8050 = 0; AdrOffset_8060 = 2200; BitOffset_8060 = 0; BitLength_8060 = 16; Address_8060 = '%QW1100'; Type_8060 = 'UINT'; AddressPointer_8060 = ADR(%QW1100); AdrOffset_8070 = 4294967295; BitOffset_8070 = 0; BitLength_8070 = 0; Address_8070 = ''; Type_8070 = ''; AddressPointer_8070 = 0; AdrOffset_8080 = 4294967295;
              BitOffset_8080 = 0; BitLength_8080 = 0; Address_8080 = ''; Type_8080 = ''; AddressPointer_8080 = 0; AdrOffset_8090 = 2204; BitOffset_8090 = 0; BitLength_8090 = 32; Address_8090 = '%QD551'; Type_8090 = 'UDINT'; AddressPointer_8090 = ADR(%QD551); AdrOffset_8100 = 4294967295; BitOffset_8100 = 0; BitLength_8100 = 0; Address_8100 = ''; Type_8100 = ''; AddressPointer_8100 = 0; AdrOffset_8510 = 2290; BitOffset_8510 = 0; BitLength_8510 = 16; Address_8510 = '%IW1145'; Type_8510 = 'UINT'; AddressPointer_8510 = ADR(%IW1145); AdrOffset_8520 = 2292; BitOffset_8520 = 0; BitLength_8520 = 32; Address_8520 = '%ID573'; Type_8520 = 'DINT'; AddressPointer_8520 = ADR(%ID573); AdrOffset_8530 = 2320; BitOffset_8530 = 0; BitLength_8530 = 32; Address_8530 = '%ID580'; Type_8530 = 'DINT'; AddressPointer_8530 = ADR(%ID580); AdrOffset_8540 = 2296; BitOffset_8540 = 0; BitLength_8540 = 16; Address_8540 = '%IW1148'; Type_8540 = 'INT';
              AddressPointer_8540 = ADR(%IW1148); AdrOffset_8550 = 4294967295; BitOffset_8550 = 0; BitLength_8550 = 0; Address_8550 = ''; Type_8550 = ''; AddressPointer_8550 = 0; AdrOffset_8560 = 2316; BitOffset_8560 = 0; BitLength_8560 = 32; Address_8560 = '%ID579'; Type_8560 = 'UDINT'; AddressPointer_8560 = ADR(%ID579); AdrOffset_8570 = 2304; BitOffset_8570 = 0; BitLength_8570 = 16; Address_8570 = '%IW1152'; Type_8570 = 'UINT'; AddressPointer_8570 = ADR(%IW1152); AdrOffset_8580 = 2308; BitOffset_8580 = 0; BitLength_8580 = 32; Address_8580 = '%ID577'; Type_8580 = 'DINT'; AddressPointer_8580 = ADR(%ID577); AdrOffset_8590 = 4294967295; BitOffset_8590 = 0; BitLength_8590 = 0; Address_8590 = ''; Type_8590 = ''; AddressPointer_8590 = 0; AdrOffset_8600 = 2312; BitOffset_8600 = 0; BitLength_8600 = 32; Address_8600 = '%ID578'; Type_8600 = 'DINT'; AddressPointer_8600 = ADR(%ID578); AdrOffset_8600 = 4294967295; BitOffset_8600 = 0; BitLength_8600 = 0;
              Address_8610 = ''; Type_8610 = ''; AddressPointer_8610 = 0; AdrOffset_8620 = 2288; BitOffset_8620 = 0; BitLength_8620 = 16; Address_8620 = '%IW1144'; Type_8620 = 'UINT'; AddressPointer_8620 = ADR(%IW1144); IsValid = True; AxisNumber = 9; IsHostHoming = False; PulseSelectIndex = 4; SERVO_MAX_ID = 83886080
      InoSV660N_5 : SV660_1Axis_00915, Inovance, order no. InoSV660N, version Revision=16#00010000
          settings: FunCodeList = H02;H02-01;H03;H03-03;H03-05;; WriteValueList = H02-01_8194_2_1_UINT_RW;H03-03_8195_4_1_UINT_RW;H03-05_8195_6_1_UINT_RW;; Number of Outputs = 6; Number of Inputs = 10; Number of Infos about Outputs = 6; Number of Infos about Inputs = 10; Configuration address of the slave = 7; Sync.Length = 18; Sync.Length = 32; FMMU.Length = 18; FMMU.Length = 32; AutoUpdate = False; DC sync0 cycletime = 4000; DC sync1 cycletime = 4000; Number of SDO = 10; Homing method.Index = 16#6098; Homing method.Subindex = 16#00; Homing method.Value = 27; Homing method.Size = 8; Homing method.AbortIfError = FALSE; Homing method.JumpToLine = FALSE; Homing method.Line = 0; Homing method.CompleteAccess = FALSE; Actual Position Calculation Method.Index = 16#60E6; Actual Position Calculation Method.Subindex = 16#00; Actual Position Calculation Method.Value = 0; Actual Position Calculation Method.Size = 8; Actual Position Calculation Method.AbortIfError = FALSE; Actual Position Calculation Method.JumpToLine = FALSE; Actual Position Calculation Method.Line = 0; Actual Position Calculation Method.CompleteAccess = FALSE; Speed during search for switch.Index = 16#6099; Speed during search for switch.Subindex = 16#01; Speed during search for switch.Value = 41943040; Speed during search for switch.Size = 32; Speed during search for switch.AbortIfError = FALSE; Speed during search for switch.JumpToLine = FALSE; Speed during search for switch.Line = 0; Speed during search for switch.CompleteAccess = FALSE; Homing acceleration.Index = 16#609A;
            Homing acceleration.Subindex = 16#00; Homing acceleration.Value = 139810133; Homing acceleration.Size = 32; Homing acceleration.AbortIfError = FALSE; Homing acceleration.JumpToLine = FALSE; Homing acceleration.Line = 0; Homing acceleration.CompleteAccess = FALSE; Speed during search for zero.Index = 16#6099; Speed during search for zero.Subindex = 16#02; Speed during search for zero.Value = 16777216; Speed during search for zero.Size = 32; Speed during search for zero.AbortIfError = FALSE; Speed during search for zero.JumpToLine = FALSE; Speed during search for zero.Line = 0; Speed during search for zero.CompleteAccess = FALSE; Time of home searching.Index = 16#2005; Time of home searching.Subindex = 16#24; Time of home searching.Value = 50000; Time of home searching.Size = 16; Time of home searching.AbortIfError = FALSE; Time of home searching.JumpToLine = FALSE; Time of home searching.Line = 0; Time of home searching.CompleteAccess = FALSE; Positive torque limit value.Index = 16#60E0; Positive torque limit value.Subindex = 16#00; Positive torque limit value.Value = 3500; Positive torque limit value.Size = 16; Positive torque limit value.AbortIfError = FALSE; Positive torque limit value.JumpToLine = FALSE; Positive torque limit value.Line = 0; Positive torque limit value.CompleteAccess = FALSE; Negative torque limit value.Index = 16#60E1; Negative torque limit value.Subindex = 16#00; Negative torque limit value.Value = 3500; Negative torque limit value.Size = 16; Negative torque limit value.AbortIfError = FALSE; Negative torque limit value.JumpToLine = FALSE; Negative torque limit value.Line = 0; Negative torque limit value.CompleteAccess = FALSE; Max profile velocity.Index = 16#607F;
            Max profile velocity.Subindex = 16#00; Max profile velocity.Value = 83886080; Max profile velocity.Size = 32; Max profile velocity.AbortIfError = FALSE; Max profile velocity.JumpToLine = FALSE; Max profile velocity.Line = 0; Max profile velocity.CompleteAccess = FALSE; RxTxPdo.NumberofEntries = 6; RxTxPdo.Sm = 2; Controlword.Index = 16#6040; Controlword.SubIndex = 0; Controlword.Size = 16; Controlword.DependOnSlot = false; Controlword.DependOnSlotGroup = false; Target position.Index = 16#607A; Target position.SubIndex = 0; Target position.Size = 32; Target position.DependOnSlot = false; Target position.DependOnSlotGroup = false; Touch probe function.Index = 16#60B8; Touch probe function.SubIndex = 0; Touch probe function.Size = 16; Touch probe function.DependOnSlot = false; Touch probe function.DependOnSlotGroup = false; Physical outputs.Index = 16#60FE; Physical outputs.SubIndex = 1; Physical outputs.Size = 32; Physical outputs.DependOnSlot = false; Physical outputs.DependOnSlotGroup = false; Target velocity.Index = 16#60FF; Target velocity.SubIndex = 0; Target velocity.Size = 32; Target velocity.DependOnSlot = false; Target velocity.DependOnSlotGroup = false; Target torque.Index = 16#6071; Target torque.SubIndex = 0; Target torque.Size = 16; Target torque.DependOnSlot = false; Target torque.DependOnSlotGroup = false; RxTxPdo.Sm = -1;
            RxTxPdo.NumberofEntries = 10; RxTxPdo.Sm = 3; Error code.Index = 16#603F; Error code.SubIndex = 0; Error code.Size = 16; Error code.DependOnSlot = false; Error code.DependOnSlotGroup = false; Statusword.Index = 16#6041; Statusword.SubIndex = 0; Statusword.Size = 16; Statusword.DependOnSlot = false; Statusword.DependOnSlotGroup = false; Position actual value.Index = 16#6064; Position actual value.SubIndex = 0; Position actual value.Size = 32; Position actual value.DependOnSlot = false; Position actual value.DependOnSlotGroup = false; Torque actual value.Index = 16#6077; Torque actual value.SubIndex = 0; Torque actual value.Size = 16; Torque actual value.DependOnSlot = false; Torque actual value.DependOnSlotGroup = false; Following error actual value.Index = 16#60F4; Following error actual value.SubIndex = 0; Following error actual value.Size = 32; Following error actual value.DependOnSlot = false; Following error actual value.DependOnSlotGroup = false; Touch probe status.Index = 16#60B9; Touch probe status.SubIndex = 0; Touch probe status.Size = 16; Touch probe status.DependOnSlot = false; Touch probe status.DependOnSlotGroup = false; Touch probe pos1 pos value.Index = 16#60BA; Touch probe pos1 pos value.SubIndex = 0; Touch probe pos1 pos value.Size = 32; Touch probe pos1 pos value.DependOnSlot = false; Touch probe pos1 pos value.DependOnSlotGroup = false; Touch probe pos2 pos value.Index = 16#60BC; Touch probe pos2 pos value.SubIndex = 0; Touch probe pos2 pos value.Size = 32;
            Touch probe pos2 pos value.DependOnSlot = false; Touch probe pos2 pos value.DependOnSlotGroup = false; Digital inputs.Index = 16#60FD; Digital inputs.SubIndex = 0; Digital inputs.Size = 32; Digital inputs.DependOnSlot = false; Digital inputs.DependOnSlotGroup = false; Velocity actual value.Index = 16#606C; Velocity actual value.SubIndex = 0; Velocity actual value.Size = 32; Velocity actual value.DependOnSlot = false; Velocity actual value.DependOnSlotGroup = false; RxTxPdo.Sm = -1; Controlword.Name = 'Controlword'; Controlword.DataType = 'UINT'; Target position.Name = 'Target position'; Target position.DataType = 'DINT'; Touch probe function.Name = 'Touch probe function'; Touch probe function.DataType = 'UINT'; Physical outputs.Name = 'Physical outputs'; Physical outputs.DataType = 'UDINT'; Target velocity.Name = 'Target velocity'; Target velocity.DataType = 'DINT'; Target torque.Name = 'Target torque'; Target torque.DataType = 'INT'; Error code.Name = 'Error code'; Error code.DataType = 'UINT'; Statusword.Name = 'Statusword'; Statusword.DataType = 'UINT'; Position actual value.Name = 'Position actual value'; Position actual value.DataType = 'DINT'; Torque actual value.Name = 'Torque actual value'; Torque actual value.DataType = 'INT'; Following error actual value.Name = 'Following error actual value'; Following error actual value.DataType = 'DINT'; Touch probe status.Name = 'Touch probe status'; Touch probe status.DataType = 'UINT'; Touch probe pos1 pos value.Name = 'Touch probe pos1 pos value'; Touch probe pos1 pos value.DataType = 'DINT'; Touch probe pos2 pos value.Name = 'Touch probe pos2 pos value';
            Touch probe pos2 pos value.DataType = 'DINT'; Digital inputs.Name = 'Digital inputs'; Digital inputs.DataType = 'UDINT'; Velocity actual value.Name = 'Velocity actual value'; Velocity actual value.DataType = 'DINT'
          unmapped channels: Controlword, Target position, Touch probe function, Physical outputs, Target velocity, Target torque, Error code, Statusword, Position actual value, Torque actual value, Following error actual value, Touch probe status, Touch probe pos1 pos value, Touch probe pos2 pos value, Digital inputs, Velocity actual value
        拍照轴8Y : Axis, Inovance, order no. 0, version 1.0.0.0
            settings: wDriveID = 5; dwRatioTechUnitsDenom = 4194304; iRatioTechUnitsNum = 5; iEncoderType = 1; iAbsEncoderOption = 2; HomingMode = 10; ZeroSignal = 0; StartDirction = 1; EndDirection = 1; PosLimitMode = 0; NegLimitMode = 0; HomingVelocity = 10; HomingApproachVelocity = 2; HomingAcceleration = 100; HomingDeceleration = 100; HomingJerk = 0; HomeMaskDistance = 0; HomePositionOffset = 0; HomePushTime = 0; HomeCompensation = 0; HomeTimeout = 0; HomeCompensationVelocity = 1000; 4000 = 1; 4001 = 0; 4003 = true; 4004 = 27; 4005 = 0; 4006 = 50.0; 4007 = 166.666666; 4008 = 20.0; 4009 = 50000; 4010 = 3500; 4011 = 3500; 4012 = 100.000000; ScalingIncs = 16#800000; 6005 = 10; AdrOffset_8010 = 2120; BitOffset_8010 = 0; BitLength_8010 = 16; Address_8010 = '%QW1060';
              Type_8010 = 'UINT'; AddressPointer_8010 = ADR(%QW1060); AdrOffset_8020 = 2124; BitOffset_8020 = 0; BitLength_8020 = 32; Address_8020 = '%QD531'; Type_8020 = 'DINT'; AddressPointer_8020 = ADR(%QD531); AdrOffset_8030 = 2136; BitOffset_8030 = 0; BitLength_8030 = 32; Address_8030 = '%QD534'; Type_8030 = 'DINT'; AddressPointer_8030 = ADR(%QD534); AdrOffset_8040 = 2140; BitOffset_8040 = 0; BitLength_8040 = 16; Address_8040 = '%QW1070'; Type_8040 = 'INT'; AddressPointer_8040 = ADR(%QW1070); AdrOffset_8050 = 4294967295; BitOffset_8050 = 0; BitLength_8050 = 0; Address_8050 = ''; Type_8050 = ''; AddressPointer_8050 = 0; AdrOffset_8060 = 2128; BitOffset_8060 = 0; BitLength_8060 = 16; Address_8060 = '%QW1064'; Type_8060 = 'UINT'; AddressPointer_8060 = ADR(%QW1064); AdrOffset_8070 = 4294967295; BitOffset_8070 = 0; BitLength_8070 = 0; Address_8070 = ''; Type_8070 = ''; AddressPointer_8070 = 0; AdrOffset_8080 = 4294967295; BitOffset_8080 = 0;
              BitLength_8080 = 0; Address_8080 = ''; Type_8080 = ''; AddressPointer_8080 = 0; AdrOffset_8090 = 2132; BitOffset_8090 = 0; BitLength_8090 = 32; Address_8090 = '%QD533'; Type_8090 = 'UDINT'; AddressPointer_8090 = ADR(%QD533); AdrOffset_8100 = 4294967295; BitOffset_8100 = 0; BitLength_8100 = 0; Address_8100 = ''; Type_8100 = ''; AddressPointer_8100 = 0; AdrOffset_8510 = 2182; BitOffset_8510 = 0; BitLength_8510 = 16; Address_8510 = '%IW1091'; Type_8510 = 'UINT'; AddressPointer_8510 = ADR(%IW1091); AdrOffset_8520 = 2184; BitOffset_8520 = 0; BitLength_8520 = 32; Address_8520 = '%ID546'; Type_8520 = 'DINT'; AddressPointer_8520 = ADR(%ID546); AdrOffset_8530 = 2212; BitOffset_8530 = 0; BitLength_8530 = 32; Address_8530 = '%ID553'; Type_8530 = 'DINT'; AddressPointer_8530 = ADR(%ID553); AdrOffset_8540 = 2188; BitOffset_8540 = 0; BitLength_8540 = 16; Address_8540 = '%IW1094'; Type_8540 = 'INT'; AddressPointer_8540 = ADR(%IW1094);
              AdrOffset_8550 = 4294967295; BitOffset_8550 = 0; BitLength_8550 = 0; Address_8550 = ''; Type_8550 = ''; AddressPointer_8550 = 0; AdrOffset_8560 = 2208; BitOffset_8560 = 0; BitLength_8560 = 32; Address_8560 = '%ID552'; Type_8560 = 'UDINT'; AddressPointer_8560 = ADR(%ID552); AdrOffset_8570 = 2196; BitOffset_8570 = 0; BitLength_8570 = 16; Address_8570 = '%IW1098'; Type_8570 = 'UINT'; AddressPointer_8570 = ADR(%IW1098); AdrOffset_8580 = 2200; BitOffset_8580 = 0; BitLength_8580 = 32; Address_8580 = '%ID550'; Type_8580 = 'DINT'; AddressPointer_8580 = ADR(%ID550); AdrOffset_8590 = 4294967295; BitOffset_8590 = 0; BitLength_8590 = 0; Address_8590 = ''; Type_8590 = ''; AddressPointer_8590 = 0; AdrOffset_8600 = 2204; BitOffset_8600 = 0; BitLength_8600 = 32; Address_8600 = '%ID551'; Type_8600 = 'DINT'; AddressPointer_8600 = ADR(%ID551); AdrOffset_8600 = 4294967295; BitOffset_8600 = 0; BitLength_8600 = 0; Address_8610 = '';
              Type_8610 = ''; AddressPointer_8610 = 0; AdrOffset_8620 = 2180; BitOffset_8620 = 0; BitLength_8620 = 16; Address_8620 = '%IW1090'; Type_8620 = 'UINT'; AddressPointer_8620 = ADR(%IW1090); IsValid = True; AxisNumber = 6; IsHostHoming = False; PulseSelectIndex = 4; SERVO_MAX_ID = 83886080
      InoSV660N_4 : SV660_1Axis_00915, Inovance, order no. InoSV660N, version Revision=16#00010000
          settings: FunCodeList = H02;H02-01;H03;H03-03;H03-05;; WriteValueList = H02-01_8194_2_1_UINT_RW;H03-03_8195_4_1_UINT_RW;H03-05_8195_6_1_UINT_RW;; Number of Outputs = 6; Number of Inputs = 10; Number of Infos about Outputs = 6; Number of Infos about Inputs = 10; Configuration address of the slave = 6; Sync.Length = 18; Sync.Length = 32; FMMU.Length = 18; FMMU.Length = 32; AutoUpdate = False; DC sync0 cycletime = 4000; DC sync1 cycletime = 4000; Number of SDO = 10; Homing method.Index = 16#6098; Homing method.Subindex = 16#00; Homing method.Value = 27; Homing method.Size = 8; Homing method.AbortIfError = FALSE; Homing method.JumpToLine = FALSE; Homing method.Line = 0; Homing method.CompleteAccess = FALSE; Actual Position Calculation Method.Index = 16#60E6; Actual Position Calculation Method.Subindex = 16#00; Actual Position Calculation Method.Value = 0; Actual Position Calculation Method.Size = 8; Actual Position Calculation Method.AbortIfError = FALSE; Actual Position Calculation Method.JumpToLine = FALSE; Actual Position Calculation Method.Line = 0; Actual Position Calculation Method.CompleteAccess = FALSE; Speed during search for switch.Index = 16#6099; Speed during search for switch.Subindex = 16#01; Speed during search for switch.Value = 41943040; Speed during search for switch.Size = 32; Speed during search for switch.AbortIfError = FALSE; Speed during search for switch.JumpToLine = FALSE; Speed during search for switch.Line = 0; Speed during search for switch.CompleteAccess = FALSE; Homing acceleration.Index = 16#609A;
            Homing acceleration.Subindex = 16#00; Homing acceleration.Value = 139810133; Homing acceleration.Size = 32; Homing acceleration.AbortIfError = FALSE; Homing acceleration.JumpToLine = FALSE; Homing acceleration.Line = 0; Homing acceleration.CompleteAccess = FALSE; Speed during search for zero.Index = 16#6099; Speed during search for zero.Subindex = 16#02; Speed during search for zero.Value = 16777216; Speed during search for zero.Size = 32; Speed during search for zero.AbortIfError = FALSE; Speed during search for zero.JumpToLine = FALSE; Speed during search for zero.Line = 0; Speed during search for zero.CompleteAccess = FALSE; Time of home searching.Index = 16#2005; Time of home searching.Subindex = 16#24; Time of home searching.Value = 50000; Time of home searching.Size = 16; Time of home searching.AbortIfError = FALSE; Time of home searching.JumpToLine = FALSE; Time of home searching.Line = 0; Time of home searching.CompleteAccess = FALSE; Positive torque limit value.Index = 16#60E0; Positive torque limit value.Subindex = 16#00; Positive torque limit value.Value = 3500; Positive torque limit value.Size = 16; Positive torque limit value.AbortIfError = FALSE; Positive torque limit value.JumpToLine = FALSE; Positive torque limit value.Line = 0; Positive torque limit value.CompleteAccess = FALSE; Negative torque limit value.Index = 16#60E1; Negative torque limit value.Subindex = 16#00; Negative torque limit value.Value = 3500; Negative torque limit value.Size = 16; Negative torque limit value.AbortIfError = FALSE; Negative torque limit value.JumpToLine = FALSE; Negative torque limit value.Line = 0; Negative torque limit value.CompleteAccess = FALSE; Max profile velocity.Index = 16#607F;
            Max profile velocity.Subindex = 16#00; Max profile velocity.Value = 83886080; Max profile velocity.Size = 32; Max profile velocity.AbortIfError = FALSE; Max profile velocity.JumpToLine = FALSE; Max profile velocity.Line = 0; Max profile velocity.CompleteAccess = FALSE; RxTxPdo.NumberofEntries = 6; RxTxPdo.Sm = 2; Controlword.Index = 16#6040; Controlword.SubIndex = 0; Controlword.Size = 16; Controlword.DependOnSlot = false; Controlword.DependOnSlotGroup = false; Target position.Index = 16#607A; Target position.SubIndex = 0; Target position.Size = 32; Target position.DependOnSlot = false; Target position.DependOnSlotGroup = false; Touch probe function.Index = 16#60B8; Touch probe function.SubIndex = 0; Touch probe function.Size = 16; Touch probe function.DependOnSlot = false; Touch probe function.DependOnSlotGroup = false; Physical outputs.Index = 16#60FE; Physical outputs.SubIndex = 1; Physical outputs.Size = 32; Physical outputs.DependOnSlot = false; Physical outputs.DependOnSlotGroup = false; Target velocity.Index = 16#60FF; Target velocity.SubIndex = 0; Target velocity.Size = 32; Target velocity.DependOnSlot = false; Target velocity.DependOnSlotGroup = false; Target torque.Index = 16#6071; Target torque.SubIndex = 0; Target torque.Size = 16; Target torque.DependOnSlot = false; Target torque.DependOnSlotGroup = false; RxTxPdo.Sm = -1;
            RxTxPdo.NumberofEntries = 10; RxTxPdo.Sm = 3; Error code.Index = 16#603F; Error code.SubIndex = 0; Error code.Size = 16; Error code.DependOnSlot = false; Error code.DependOnSlotGroup = false; Statusword.Index = 16#6041; Statusword.SubIndex = 0; Statusword.Size = 16; Statusword.DependOnSlot = false; Statusword.DependOnSlotGroup = false; Position actual value.Index = 16#6064; Position actual value.SubIndex = 0; Position actual value.Size = 32; Position actual value.DependOnSlot = false; Position actual value.DependOnSlotGroup = false; Torque actual value.Index = 16#6077; Torque actual value.SubIndex = 0; Torque actual value.Size = 16; Torque actual value.DependOnSlot = false; Torque actual value.DependOnSlotGroup = false; Following error actual value.Index = 16#60F4; Following error actual value.SubIndex = 0; Following error actual value.Size = 32; Following error actual value.DependOnSlot = false; Following error actual value.DependOnSlotGroup = false; Touch probe status.Index = 16#60B9; Touch probe status.SubIndex = 0; Touch probe status.Size = 16; Touch probe status.DependOnSlot = false; Touch probe status.DependOnSlotGroup = false; Touch probe pos1 pos value.Index = 16#60BA; Touch probe pos1 pos value.SubIndex = 0; Touch probe pos1 pos value.Size = 32; Touch probe pos1 pos value.DependOnSlot = false; Touch probe pos1 pos value.DependOnSlotGroup = false; Touch probe pos2 pos value.Index = 16#60BC; Touch probe pos2 pos value.SubIndex = 0; Touch probe pos2 pos value.Size = 32;
            Touch probe pos2 pos value.DependOnSlot = false; Touch probe pos2 pos value.DependOnSlotGroup = false; Digital inputs.Index = 16#60FD; Digital inputs.SubIndex = 0; Digital inputs.Size = 32; Digital inputs.DependOnSlot = false; Digital inputs.DependOnSlotGroup = false; Velocity actual value.Index = 16#606C; Velocity actual value.SubIndex = 0; Velocity actual value.Size = 32; Velocity actual value.DependOnSlot = false; Velocity actual value.DependOnSlotGroup = false; RxTxPdo.Sm = -1; Controlword.Name = 'Controlword'; Controlword.DataType = 'UINT'; Target position.Name = 'Target position'; Target position.DataType = 'DINT'; Touch probe function.Name = 'Touch probe function'; Touch probe function.DataType = 'UINT'; Physical outputs.Name = 'Physical outputs'; Physical outputs.DataType = 'UDINT'; Target velocity.Name = 'Target velocity'; Target velocity.DataType = 'DINT'; Target torque.Name = 'Target torque'; Target torque.DataType = 'INT'; Error code.Name = 'Error code'; Error code.DataType = 'UINT'; Statusword.Name = 'Statusword'; Statusword.DataType = 'UINT'; Position actual value.Name = 'Position actual value'; Position actual value.DataType = 'DINT'; Torque actual value.Name = 'Torque actual value'; Torque actual value.DataType = 'INT'; Following error actual value.Name = 'Following error actual value'; Following error actual value.DataType = 'DINT'; Touch probe status.Name = 'Touch probe status'; Touch probe status.DataType = 'UINT'; Touch probe pos1 pos value.Name = 'Touch probe pos1 pos value'; Touch probe pos1 pos value.DataType = 'DINT'; Touch probe pos2 pos value.Name = 'Touch probe pos2 pos value';
            Touch probe pos2 pos value.DataType = 'DINT'; Digital inputs.Name = 'Digital inputs'; Digital inputs.DataType = 'UDINT'; Velocity actual value.Name = 'Velocity actual value'; Velocity actual value.DataType = 'DINT'
          unmapped channels: Controlword, Target position, Touch probe function, Physical outputs, Target velocity, Target torque, Error code, Statusword, Position actual value, Torque actual value, Following error actual value, Touch probe status, Touch probe pos1 pos value, Touch probe pos2 pos value, Digital inputs, Velocity actual value
        点样轴7Y : Axis, Inovance, order no. 0, version 1.0.0.0
            settings: wDriveID = 4; dwRatioTechUnitsDenom = 4194304; iRatioTechUnitsNum = 5; iEncoderType = 1; iAbsEncoderOption = 2; HomingMode = 10; ZeroSignal = 0; StartDirction = 1; EndDirection = 1; PosLimitMode = 0; NegLimitMode = 0; HomingVelocity = 10; HomingApproachVelocity = 2; HomingAcceleration = 100; HomingDeceleration = 100; HomingJerk = 0; HomeMaskDistance = 0; HomePositionOffset = 0; HomePushTime = 0; HomeCompensation = 0; HomeTimeout = 0; HomeCompensationVelocity = 1000; 4000 = 1; 4001 = 0; 4003 = true; 4004 = 27; 4005 = 0; 4006 = 50.0; 4007 = 166.666666; 4008 = 20.0; 4009 = 50000; 4010 = 3500; 4011 = 3500; 4012 = 100.000000; ScalingIncs = 16#800000; 6005 = 10; AdrOffset_8010 = 2096; BitOffset_8010 = 0; BitLength_8010 = 16; Address_8010 = '%QW1048';
              Type_8010 = 'UINT'; AddressPointer_8010 = ADR(%QW1048); AdrOffset_8020 = 2100; BitOffset_8020 = 0; BitLength_8020 = 32; Address_8020 = '%QD525'; Type_8020 = 'DINT'; AddressPointer_8020 = ADR(%QD525); AdrOffset_8030 = 2112; BitOffset_8030 = 0; BitLength_8030 = 32; Address_8030 = '%QD528'; Type_8030 = 'DINT'; AddressPointer_8030 = ADR(%QD528); AdrOffset_8040 = 2116; BitOffset_8040 = 0; BitLength_8040 = 16; Address_8040 = '%QW1058'; Type_8040 = 'INT'; AddressPointer_8040 = ADR(%QW1058); AdrOffset_8050 = 4294967295; BitOffset_8050 = 0; BitLength_8050 = 0; Address_8050 = ''; Type_8050 = ''; AddressPointer_8050 = 0; AdrOffset_8060 = 2104; BitOffset_8060 = 0; BitLength_8060 = 16; Address_8060 = '%QW1052'; Type_8060 = 'UINT'; AddressPointer_8060 = ADR(%QW1052); AdrOffset_8070 = 4294967295; BitOffset_8070 = 0; BitLength_8070 = 0; Address_8070 = ''; Type_8070 = ''; AddressPointer_8070 = 0; AdrOffset_8080 = 4294967295; BitOffset_8080 = 0;
              BitLength_8080 = 0; Address_8080 = ''; Type_8080 = ''; AddressPointer_8080 = 0; AdrOffset_8090 = 2108; BitOffset_8090 = 0; BitLength_8090 = 32; Address_8090 = '%QD527'; Type_8090 = 'UDINT'; AddressPointer_8090 = ADR(%QD527); AdrOffset_8100 = 4294967295; BitOffset_8100 = 0; BitLength_8100 = 0; Address_8100 = ''; Type_8100 = ''; AddressPointer_8100 = 0; AdrOffset_8510 = 2146; BitOffset_8510 = 0; BitLength_8510 = 16; Address_8510 = '%IW1073'; Type_8510 = 'UINT'; AddressPointer_8510 = ADR(%IW1073); AdrOffset_8520 = 2148; BitOffset_8520 = 0; BitLength_8520 = 32; Address_8520 = '%ID537'; Type_8520 = 'DINT'; AddressPointer_8520 = ADR(%ID537); AdrOffset_8530 = 2176; BitOffset_8530 = 0; BitLength_8530 = 32; Address_8530 = '%ID544'; Type_8530 = 'DINT'; AddressPointer_8530 = ADR(%ID544); AdrOffset_8540 = 2152; BitOffset_8540 = 0; BitLength_8540 = 16; Address_8540 = '%IW1076'; Type_8540 = 'INT'; AddressPointer_8540 = ADR(%IW1076);
              AdrOffset_8550 = 4294967295; BitOffset_8550 = 0; BitLength_8550 = 0; Address_8550 = ''; Type_8550 = ''; AddressPointer_8550 = 0; AdrOffset_8560 = 2172; BitOffset_8560 = 0; BitLength_8560 = 32; Address_8560 = '%ID543'; Type_8560 = 'UDINT'; AddressPointer_8560 = ADR(%ID543); AdrOffset_8570 = 2160; BitOffset_8570 = 0; BitLength_8570 = 16; Address_8570 = '%IW1080'; Type_8570 = 'UINT'; AddressPointer_8570 = ADR(%IW1080); AdrOffset_8580 = 2164; BitOffset_8580 = 0; BitLength_8580 = 32; Address_8580 = '%ID541'; Type_8580 = 'DINT'; AddressPointer_8580 = ADR(%ID541); AdrOffset_8590 = 4294967295; BitOffset_8590 = 0; BitLength_8590 = 0; Address_8590 = ''; Type_8590 = ''; AddressPointer_8590 = 0; AdrOffset_8600 = 2168; BitOffset_8600 = 0; BitLength_8600 = 32; Address_8600 = '%ID542'; Type_8600 = 'DINT'; AddressPointer_8600 = ADR(%ID542); AdrOffset_8600 = 4294967295; BitOffset_8600 = 0; BitLength_8600 = 0; Address_8610 = '';
              Type_8610 = ''; AddressPointer_8610 = 0; AdrOffset_8620 = 2144; BitOffset_8620 = 0; BitLength_8620 = 16; Address_8620 = '%IW1072'; Type_8620 = 'UINT'; AddressPointer_8620 = ADR(%IW1072); IsValid = True; AxisNumber = 5; IsHostHoming = False; PulseSelectIndex = 4; SERVO_MAX_ID = 83886080
      Auto_1023 : AU7-1023-xxxx-ECT, AUTO, order no. Auto-1023, version Revision=16#00001000
          settings: Configuration address of the slave = 13; AutoUpdate = False; DC sync0 cycletime = 4000; DC sync1 cycletime = 4000
          output 展缸1气缸1 : BIT  // Channel 1
          output 展缸1气缸2 : BIT  // Channel 2
          output 展缸1气缸3 : BIT  // Channel 3
          output 展缸1气缸4 : BIT  // Channel 4
          output 展缸2气缸1 : BIT  // Channel 5
          output 展缸2气缸2 : BIT  // Channel 6
          output 展缸2气缸3 : BIT  // Channel 7
          output 展缸2气缸4 : BIT  // Channel 8
          output 收集下压气缸 : BIT  // Channel 9
          output 收集夹持气缸 : BIT  // Channel 10
          output 收集升降气缸 : BIT  // Channel 11
          output 收集伸缩气缸 : BIT  // Channel 12
          output 刮板拍照遮光气缸 : BIT  // Channel 13
          output 刮板拍照旋转气缸 : BIT  // Channel 14
          output 刮板拍照下压气缸 : BIT  // Channel 15
          unmapped channels: Channel 16, Channel 17, Channel 18, Channel 19, Channel 20, Channel 21, Channel 22, Channel 23, Channel 24, Channel 25, Channel 26, Channel 27, Channel 28, Channel 29, Channel 30, Channel 31, Channel 32, ID, Channel 1, Channel 2, Channel 3, Channel 4, Channel 5, Channel 6, Channel 7, Channel 8, Channel 9, Channel 10, Channel 11, Channel 12, Channel 13, Channel 14, Channel 15, Channel 16
        _1023_xxxx_Extended_IO_Modules_13
        _1023_xxxx_Extended_IO_Modules_2
        _1023_xxxx_Extended_IO_Modules_8
        _1023_xxxx_Extended_IO_Modules_10
        _1023_xxxx_Extended_IO_Modules_5
        _1023_xxxx_Extended_IO_Modules_4
        _1023_xxxx_Extended_IO_Modules_1
        _1023_xxxx_Extended_IO_Modules_7
        _1023_xxxx_Extended_IO_Modules_14
        _1023_xxxx_Extended_IO_Modules_3
        _1023_xxxx_Extended_IO_Modules_9
        _1023_xxxx_Extended_IO_Modules_12
        _1023_xxxx_Extended_IO_Modules_16
        _1023_xxxx_Extended_IO_Modules_11
        _1023_xxxx_Extended_IO_Modules_15
        _1023_xxxx_Extended_IO_Modules_6
    SoftMotion General Axis Pool
      SMC_FreeEncoder : SMC_FreeEncoder, 3S - Smart Software Solutions GmbH, order no. 1805, version 3.5.5.0
          settings: wDriveID = 11; dwRatioTechUnitsDenom = 131072
    HwConfiguratioinDevice : SystemConfig, Inovance, version 00.00.00.10
        settings: NetworkConfigArray.NetworkConfigArray.BusType = 10; NetworkConfigArray.NetworkConfigArray.RackSum = 1; NetworkConfigArray.NetworkConfigArray.HardwareConfigArray.HardwareConfigArray.RackNo = 1; NetworkConfigArray.NetworkConfigArray.HardwareConfigArray.HardwareConfigArray.ModuleNum = 1; EnableFun = 9
    MODBUS_TCP : ModbusTCP本地从站, inovance, version 00.00.00.10
    CAN : CAN总线, INOVANCE, version 00.00.00.10
    Local Bus
      GL20_1600END : GL20(GL20S) 16通道DI模块, Inovance, version 00.00.00.10
          settings: ModuleBaseInfoStruct.BusType = 10; ModuleBaseInfoStruct.RackNumber = 1; ModuleBaseInfoStruct.SlotNumber = 1
          unmapped channels: IB(I), IB(II)
*)

// Device/Application/10_数据结构/HMI_Servo
TYPE HMI_Servo :
STRUCT
	position: ARRAY[1..10] OF LREAL;
	write: ARRAY[1..10] OF BOOL;
	execute: ARRAY[1..10] OF BOOL;
END_STRUCT
END_TYPE

// Device/Application/10_数据结构/servo
TYPE servo :
STRUCT
	/// <GrpComment>
	/// <GrpComment_zh-cn>回原点命令</GrpComment_zh-cn>
	/// </GrpComment>
	// 回原点命令
 	xHome  : BOOL;
	/// <GrpComment>
	/// <GrpComment_zh-cn>正方向点动</GrpComment_zh-cn>
	/// </GrpComment>
	// 正方向点动
 	xJogPos  : BOOL;
	/// <GrpComment>
	/// <GrpComment_zh-cn>负方向点动</GrpComment_zh-cn>
	/// </GrpComment>
	// 负方向点动
 	xJogNeg: BOOL;
	/// <GrpComment>
	/// <GrpComment_zh-cn>停止命令</GrpComment_zh-cn>
	/// </GrpComment>
	// 停止命令
 	xStop  : BOOL;
	/// <GrpComment>
	/// <GrpComment_zh-cn>绝对运动启动</GrpComment_zh-cn>
	/// </GrpComment>
	// 绝对运动启动
 	xMoveAbs  : BOOL;
	/// <GrpComment>
	/// <GrpComment_zh-cn>相对运动启动</GrpComment_zh-cn>
	/// </GrpComment>
	// 相对运动启动
 	xMoveRel  : BOOL;
	/// <GrpComment>
	/// <GrpComment_zh-cn>轴复位</GrpComment_zh-cn>
	/// </GrpComment>
	//轴复位
 	XReset : BOOL;
	/// <GrpComment>
	/// <GrpComment_zh-cn>绝对位置目标</GrpComment_zh-cn>
	/// </GrpComment>
	// 绝对位置目标
 	fAbsTarget  : LREAL;
	/// <GrpComment>
	/// <GrpComment_zh-cn>相对运动距离</GrpComment_zh-cn>
	/// </GrpComment>
	// 相对运动距离
 	fRelTarget:LREAL;
	/// <GrpComment>
	/// <GrpComment_zh-cn>运行速度</GrpComment_zh-cn>
	/// </GrpComment>
	// 运行速度
 	fVelocity: LREAL;
	/// <GrpComment>
	/// <GrpComment_zh-cn>加速度</GrpComment_zh-cn>
	/// </GrpComment>
	// 加速度
 	fAcc : LREAL;
	/// <GrpComment>
	/// <GrpComment_zh-cn>减速度</GrpComment_zh-cn>
	/// </GrpComment>
	// 减速度
 	fDec:LREAL;
	/// <GrpComment>
	/// <GrpComment_zh-cn>点动速度</GrpComment_zh-cn>
	/// </GrpComment>
	// 点动速度 
 	fJogVel : LREAL;
	/// <GrpComment>
	/// <GrpComment_zh-cn>轴使能状态</GrpComment_zh-cn>
	/// </GrpComment>
	// 轴使能状态
 	bEnabled:BOOL;
	/// <GrpComment>
	/// <GrpComment_zh-cn>原点完成</GrpComment_zh-cn>
	/// </GrpComment>
	// 原点完成
 	bHomed: BOOL;
	/// <GrpComment>
	/// <GrpComment_zh-cn>轴忙状态</GrpComment_zh-cn>
	/// </GrpComment>
	// 轴忙状态
 	bBusy:BOOL;
	/// <GrpComment>
	/// <GrpComment_zh-cn>轴报警</GrpComment_zh-cn>
	/// </GrpComment>
	// 轴报警
 	bError : BOOL;
	/// <GrpComment>
	/// <GrpComment_zh-cn>错误代码</GrpComment_zh-cn>
	/// </GrpComment>
	// 错误代码
 	iErrorCode : DINT;
	/// <GrpComment>
	/// <GrpComment_zh-cn>实际位置</GrpComment_zh-cn>
	/// </GrpComment>
	// 实际位置
 	fActPos:LREAL;
	/// <GrpComment>
	/// <GrpComment_zh-cn>实际速度</GrpComment_zh-cn>
	/// </GrpComment>
	// 实际速度
 	fActVel:LREAL;
	/// <GrpComment>
	/// <GrpComment_zh-cn>运动完成</GrpComment_zh-cn>
	/// </GrpComment>
	// 绝对运动完成
	bAbMoveDone :BOOL;
	/// <GrpComment>
	/// <GrpComment_zh-cn>运动完成</GrpComment_zh-cn>
	/// </GrpComment>
	// 相对运动完成
	bReMoveDone: BOOL;
END_STRUCT
END_TYPE

// Device/Application/10_数据结构/EN_功能块状态
{attribute 'qualified_only'}
{attribute 'strict'}
TYPE EN_功能块状态 :
(
	停止 := 0,
	运行:= 1,
	故障:= 2,
	急停:= 3,
	初始化:= 4
);
END_TYPE

// Device/Application/20_变量Date/HMI_Date
VAR_GLOBAL
	// 手轮切换
	HMI_HandWheel_3Y: BOOL;
	HMI_HandWheel_4X: BOOL;
	HMI_HandWheel_5Z: BOOL;
	HMI_HandWheel_6X: BOOL;
	HMI_HandWheel_7Y: BOOL;
	HMI_HandWheel_8Y: BOOL;
	HMI_HandWheel_9X: BOOL;
	HMI_HandWheel_10Z: BOOL;
	HMI_HandWheel_11Y: BOOL;
	一键回原点: BOOL;
	伺服上料_Setp: INT;
	伺服下料_Setp: INT;
	收集流程: INT;
	收集计数: INT;
	展开流程: INT;
	上样点样流程: INT;
	拍照刮板流程: INT;
	机器人流程: INT;
	ECAT掉站报警: BOOL;
END_VAR

VAR_GLOBAL RETAIN PERSISTENT
	HMI_打样瓶上料轴3Y AT %MB132240: HMI_Servo;
	HMI_点样轴6X AT %MB132344: HMI_Servo;
	HMI_点样轴7Y AT %MB132448: HMI_Servo;
	HMI_地轨轴11Y AT %MB132552: HMI_Servo;
	HMI_上样轴4X轴 AT %MB132656: HMI_Servo;
	HMI_上样轴5Z轴 AT %MB132760: HMI_Servo;
	升降上料完成 AT %MB132040: BOOL;
	升降下料完成 AT %MB132041: BOOL;
END_VAR

// Device/Application/20_变量Date/cyinder_date
VAR_GLOBAL
	cyinderAlarm: INT;
	cyinderAlarm2: INT;
	展缸1气缸1手动: BOOL;
	展缸1气缸1自动: BOOL;
	展缸1气缸2手动: BOOL;
	展缸1气缸2自动: BOOL;
	展缸1气缸3手动: BOOL;
	展缸1气缸3自动: BOOL;
	展缸1气缸4手动: BOOL;
	展缸1气缸4自动: BOOL;
	展缸2气缸1手动: BOOL;
	展缸2气缸1自动: BOOL;
	展缸2气缸2手动: BOOL;
	展缸2气缸2自动: BOOL;
	展缸2气缸3手动: BOOL;
	展缸2气缸3自动: BOOL;
	展缸2气缸4手动: BOOL;
	展缸2气缸4自动: BOOL;
	收集下压气缸手动: BOOL;
	收集下压气缸自动: BOOL;
	收集夹持气缸手动: BOOL;
	收集夹持气缸自动: BOOL;
	收集升降气缸手动: BOOL;
	收集升降气缸自动: BOOL;
	收集伸缩气缸手动: BOOL;
	收集伸缩气缸自动: BOOL;
	刮板拍照遮光气缸手动: BOOL;
	刮板拍照遮光气缸自动: BOOL;
	刮板拍照旋转气缸手动: BOOL;
	刮板拍照旋转气缸自动: BOOL;
	刮板拍照下压气缸手动: BOOL;
	刮板拍照下压气缸自动: BOOL;
	展缸1进液电池阀1手动: BOOL;
	展缸1进液电池阀1自动: BOOL;
	展缸1进液电池阀2手动: BOOL;
	展缸1进液电池阀2自动: BOOL;
	展缸1进液电池阀3手动: BOOL;
	展缸1进液电池阀3自动: BOOL;
	展缸1进液电池阀4手动: BOOL;
	展缸1进液电池阀4自动: BOOL;
	展缸1排液电池阀1手动: BOOL;
	展缸1排液电池阀1自动: BOOL;
	展缸1排液电池阀2手动: BOOL;
	展缸1排液电池阀2自动: BOOL;
	展缸1排液电池阀3手动: BOOL;
	展缸1排液电池阀3自动: BOOL;
	展缸1排液电池阀4手动: BOOL;
	展缸1排液电池阀4自动: BOOL;
	展缸1吹气电池阀1手动: BOOL;
	展缸1吹气电池阀1自动: BOOL;
	展缸1吹气电池阀2手动: BOOL;
	展缸1吹气电池阀2自动: BOOL;
	展缸1吹气电池阀3手动: BOOL;
	展缸1吹气电池阀3自动: BOOL;
	展缸1吹气电池阀4手动: BOOL;
	展缸1吹气电池阀4自动: BOOL;
	大真空泵手动: BOOL;
	大真空泵自动: BOOL;
	展缸2进液电池阀1手动: BOOL;
	展缸2进液电池阀1自动: BOOL;
	展缸2进液电池阀2手动: BOOL;
	展缸2进液电池阀2自动: BOOL;
	展缸2进液电池阀3手动: BOOL;
	展缸2进液电池阀3自动: BOOL;
	展缸2进液电池阀4手动: BOOL;
	展缸2进液电池阀4自动: BOOL;
	展缸2排液电池阀1手动: BOOL;
	展缸2排液电池阀1自动: BOOL;
	展缸2排液电池阀2手动: BOOL;
	展缸2排液电池阀2自动: BOOL;
	展缸2排液电池阀3手动: BOOL;
	展缸2排液电池阀3自动: BOOL;
	展缸2排液电池阀4手动: BOOL;
	展缸2排液电池阀4自动: BOOL;
	展缸2吹气电池阀1手动: BOOL;
	展缸2吹气电池阀1自动: BOOL;
	展缸2吹气电池阀2手动: BOOL;
	展缸2吹气电池阀2自动: BOOL;
	展缸2吹气电池阀3手动: BOOL;
	展缸2吹气电池阀3自动: BOOL;
	展缸2吹气电池阀4手动: BOOL;
	展缸2吹气电池阀4自动: BOOL;
	收集进液手动: BOOL;
	收集进液自动: BOOL;
	收集排液手动: BOOL;
	收集排液自动: BOOL;
	收集正压排液手动: BOOL;
	收集正压排液自动: BOOL;
	溶液收集瓶定位手动: BOOL;
	溶液收集瓶定位自动: BOOL;
	上样定位手动: BOOL;
	上样定位自动: BOOL;
	上样点样三通电池阀手动: BOOL;
	上样点样三通电池阀自动: BOOL;
	刮板拍照真空手动: BOOL;
	刮板拍照真空自动: BOOL;
	刮板拍照无刷电机手动: BOOL;
	刮板拍照无刷电机自动: BOOL;
	刮板拍照定位气缸手动: BOOL;
	刮板拍照定位气缸自动: BOOL;
	粉末收集器定位手动: BOOL;
	粉末收集器定位自动: BOOL;
	上样吹气手动: BOOL;
	上样吹气自动: BOOL;
END_VAR

// Device/Application/20_变量Date/IO
VAR_GLOBAL
	A相 AT %IX0.0: BOOL;
	B相 AT %IX0.1: BOOL;
	急停 AT %IX0.3: BOOL;
	复位 AT %IX0.4: BOOL;
	启动 AT %IX0.5: BOOL;
	停止 AT %IX0.6: BOOL;
	手自动 AT %IX0.7: BOOL;
	倍率X1 AT %IX1.0: BOOL;
	倍率X10 AT %IX1.1: BOOL;
	倍率X100 AT %IX1.2: BOOL;
	选择轴1 AT %IX1.3: BOOL;
	选择轴2 AT %IX1.4: BOOL;
	选择轴3 AT %IX1.5: BOOL;
	选择轴4 AT %IX1.6: BOOL;
	三色灯红 AT %QX0.0: BOOL;
	三色灯黄 AT %QX0.1: BOOL;
	三色灯绿 AT %QX0.2: BOOL;
	蜂鸣器 AT %QX0.3: BOOL;
	展缸1进液电池阀1 AT %QX1.0: BOOL;
	展缸1进液电池阀2 AT %QX1.1: BOOL;
	展缸1进液电池阀3 AT %QX1.2: BOOL;
	展缸1进液电池阀4 AT %QX1.3: BOOL;
	展缸1排液电池阀1 AT %QX1.4: BOOL;
	展缸1排液电池阀2 AT %QX1.5: BOOL;
	展缸1排液电池阀3 AT %QX1.6: BOOL;
	展缸1排液电池阀4 AT %QX1.7: BOOL;
	展缸1吹气电池阀1 AT %QX2.0: BOOL;
	展缸1吹气电池阀2 AT %QX2.1: BOOL;
	展缸1吹气电池阀3 AT %QX2.2: BOOL;
	展缸1吹气电池阀4 AT %QX2.3: BOOL;
	大真空泵 AT %QX2.4: BOOL;
	展缸2进液电池阀1 AT %QX3.0: BOOL;
	展缸2进液电池阀2 AT %QX3.1: BOOL;
	展缸2进液电池阀3 AT %QX3.2: BOOL;
	展缸2进液电池阀4 AT %QX3.3: BOOL;
	展缸2排液电池阀1 AT %QX3.4: BOOL;
	展缸2排液电池阀2 AT %QX3.5: BOOL;
	展缸2排液电池阀3 AT %QX3.6: BOOL;
	展缸2排液电池阀4 AT %QX3.7: BOOL;
	展缸2吹气电池阀1 AT %QX4.0: BOOL;
	展缸2吹气电池阀2 AT %QX4.1: BOOL;
	展缸2吹气电池阀3 AT %QX4.2: BOOL;
	展缸2吹气电池阀4 AT %QX4.3: BOOL;
	收集平台进液2通电池阀 AT %QX5.0: BOOL;
	收集平台排液3通电池阀 AT %QX5.1: BOOL;
	收集平台正压排液阀 AT %QX5.2: BOOL;
	溶液收集瓶工位定位气缸 AT %QX5.3: BOOL;
	上样定位气缸 AT %QX7.0: BOOL;
	上样点样三通电池阀 AT %QX7.1: BOOL;
	刮板拍照真空阀 AT %QX7.2: BOOL;
	刮板拍照无刷电机 AT %QX7.3: BOOL;
	刮板拍照定位气缸 AT %QX7.4: BOOL;
	粉末收集器工位定位气缸 AT %QX7.5: BOOL;
	上样吹气二通阀 AT %QX7.6: BOOL;
	展缸1气缸1原点 AT %IX3.0: BOOL;
	展缸1气缸1动点 AT %IX3.1: BOOL;
	展缸1气缸2原点 AT %IX3.2: BOOL;
	展缸1气缸2动点 AT %IX3.3: BOOL;
	展缸1气缸3原点 AT %IX3.4: BOOL;
	展缸1气缸3动点 AT %IX3.5: BOOL;
	展缸1气缸4原点 AT %IX3.6: BOOL;
	展缸1气缸4动点 AT %IX3.7: BOOL;
	展缸1排液气泡传感器 AT %IX4.0: BOOL;
	展缸1溶剂废液检测传感器 AT %IX4.1: BOOL;
	展缸2气缸1原点 AT %IX5.0: BOOL;
	展缸2气缸1动点 AT %IX5.1: BOOL;
	展缸2气缸2原点 AT %IX5.2: BOOL;
	展缸2气缸2动点 AT %IX5.3: BOOL;
	展缸2气缸3原点 AT %IX5.4: BOOL;
	展缸2气缸3动点 AT %IX5.5: BOOL;
	展缸2气缸4原点 AT %IX5.6: BOOL;
	展缸2气缸4动点 AT %IX5.7: BOOL;
	展缸2排液气泡传感器 AT %IX6.0: BOOL;
	展缸2溶剂废液检测传感器 AT %IX6.1: BOOL;
	收集平台下压气缸原点 AT %IX7.0: BOOL;
	上料进料传感器 AT %IX7.1: BOOL;
	收集平台夹持气缸原点 AT %IX7.2: BOOL;
	收集平台夹持气缸动点 AT %IX7.3: BOOL;
	收集平台升降气缸原点 AT %IX7.4: BOOL;
	收集平台升降气缸动点 AT %IX7.5: BOOL;
	收集平台推出气缸原点 AT %IX7.6: BOOL;
	收集平台推出气缸动点 AT %IX7.7: BOOL;
	收集平台气泡传感器 AT %IX8.0: BOOL;
	收集平台瓶子有无传感器 AT %IX8.1: BOOL;
	收集平台暂存工位传感器 AT %IX8.2: BOOL;
	玻璃升降光电开关1 AT %IX8.3: BOOL;
	玻璃升降光电开关2 AT %IX8.4: BOOL;
	玻璃升降接近开关1 AT %IX8.5: BOOL;
	玻璃升降接近开关2 AT %IX8.6: BOOL;
	下料出料传感器 AT %IX8.7: BOOL;
	上样料架检测1 AT %IX9.0: BOOL;
	上样料架检测2 AT %IX9.1: BOOL;
	上样气泡传感器 AT %IX9.2: BOOL;
	点样气泡传感器 AT %IX9.3: BOOL;
	刮板拍照遮光气缸上位 AT %IX9.4: BOOL;
	刮板拍照遮光气缸下位 AT %IX9.5: BOOL;
	刮板拍照旋转气缸原点 AT %IX9.6: BOOL;
	刮板拍照旋转气缸动点 AT %IX9.7: BOOL;
	刮板拍照下压气缸上位 AT %IX10.0: BOOL;
	刮板拍照暂存工位传感器 AT %IX10.2: BOOL;
	料库检测1 AT %IX11.0: BOOL;
	料库检测2 AT %IX11.1: BOOL;
	料库检测3 AT %IX11.2: BOOL;
	料库检测4 AT %IX11.3: BOOL;
	料库检测5 AT %IX11.4: BOOL;
	料库检测6 AT %IX11.5: BOOL;
	料库检测7 AT %IX11.6: BOOL;
	料库检测8 AT %IX11.7: BOOL;
	料库检测9 AT %IX12.0: BOOL;
	料库检测10 AT %IX12.1: BOOL;
	料库检测11 AT %IX12.2: BOOL;
	料库检测12 AT %IX12.3: BOOL;
	机器人工具检测1 AT %IX12.4: BOOL;
	机器人工具检测2 AT %IX12.5: BOOL;
	机器人工具检测3 AT %IX12.6: BOOL;
END_VAR

// Device/Application/PersistentVars
{attribute 'qualified_only'}
VAR_GLOBAL PERSISTENT RETAIN
END_VAR

// Device/Application/20_变量Date/servoaxisdate
VAR_GLOBAL RETAIN PERSISTENT
	玻璃上料轴1ZDATE AT %MB131072: servo;
	玻璃上料轴2ZDATE AT %MB131160: servo;
	打样瓶上料轴3YDATE AT %MB131248: servo;
	点样轴6XDATE AT %MB131336: servo;
	点样轴7YDATE AT %MB131424: servo;
	拍照轴8YDATE AT %MB131512: servo;
	刮板轴9XDATE AT %MB131600: servo;
	刮板轴10ZDATE AT %MB131688: servo;
	地轨轴11YDATE AT %MB131776: servo;
	上样轴4X轴DATE AT %MB131864: servo;
	上样轴5Z轴DATE AT %MB131952: servo;
END_VAR

// Device/Application/20_变量Date/GVL
VAR_GLOBAL
	MODE_State: INT;
	// 0:停止  1:运行  2:故障  3:急停
	Alarm: INT;
	ManualAuto: BOOL;
	初始化: BOOL;
	CNC启动: BOOL;
	CNC停止: BOOL;
	CNC完成: BOOL;
	伺服报警: BOOL;
	bSysReset: BOOL;
	bCyInhibit: BOOL;
	bAutoHomeResetPulse: BOOL;
	回零完成1Z: BOOL;
	回零完成2Z: BOOL;
	回零完成3Y: BOOL;
	回零完成4X: BOOL;
	回零完成5Z: BOOL;
	回零完成6X: BOOL;
	回零完成7Y: BOOL;
	回零完成8Y: BOOL;
	回零完成9X: BOOL;
	回零完成10Z: BOOL;
	回零完成11Y: BOOL;
	伺服未回原点报警: BOOL;
	collect_prepare_OK: BOOL;
	collect_OK: BOOL;
	Camera_scraper_initialization_OK: BOOL;
	Photo_preparation_completed_OK: BOOL;
	Scraper_collection_completed: BOOL;
	Robot_completes_material_retrieval: BOOL;
	Sampling_initialization_OK: BOOL;
	Sampling_Cleaning_OK: BOOL;
	Sampling_preparation_OK: BOOL;
	Sampling_Place_materials_OK: BOOL;
	Sampling_liquid_absorption: BOOL;
	Sampling_Spray_sample_OK: BOOL;
	expand_initialization_OK: BOOL;
	Expand_Group_clean_OK: BOOL;
	Expand_up_liquid_OK: BOOL;
	Expand_silica_gel_plate_OK: BOOL;
	排液开始: BOOL;
	Collector_coordinates: INT;
	Collect_bottle_coordinates: INT;
	上样清洗位置: INT;
	取工具setp: INT;
	取工具完成: BOOL;
	取升降硅胶板step: INT;
	取升降硅胶板完成: BOOL;
	放点样硅胶板step: INT;
	放点样硅胶板完成: BOOL;
	取点样硅胶板step: INT;
	取点样硅胶板完成: BOOL;
	放展缸硅胶板完成: BOOL;
	放展缸硅胶板step: INT;
	取展缸硅胶板step: INT;
	取展缸硅胶板完成: BOOL;
	放拍照硅胶板完成: BOOL;
	放拍照硅胶板step: INT;
	取收集器组放暂存工位step: INT;
	取收集瓶组放暂存工位完成: BOOL;
	取暂存收集器放刮板位完成: BOOL;
	取暂存收集器放刮板位step: INT;
	取刮板收集器放到收集工位完成: BOOL;
	取刮板收集器放到收集工位step: INT;
	取暂存收集瓶放收集工位step: INT;
	取暂存收集瓶放收集工位完成: BOOL;
	取收集器放暂存工位完成: BOOL;
	取收集器放暂存工位step: INT;
	取刮板硅胶板放废料区step: INT;
	取刮板硅胶板放废料区完成: BOOL;
	取暂存收集器组放仓库完成: BOOL;
	取暂存收集器组放仓库step: INT;
	取收集器组放暂存工位完成: BOOL;
	取收集瓶组放暂存工位step: INT;
	取暂存收集瓶组放仓库完成: BOOL;
	取暂存收集瓶组放仓库step: INT;
	取收集瓶放暂存工位step: INT;
	取收集瓶放暂存工位完成: BOOL;
	B1: ARRAY[1..2000] OF SMC_GEOINFO;
	泵站位符: BOOL;
	B2: ARRAY[1..2000] OF SMC_GEOINFO;
	DR: INT;
	大真空泵站位: ARRAY[0..11] OF BOOL;
	取拍照硅胶完step: INT;
	取拍照硅胶板完成: BOOL;
	上样料架报警: BOOL;
	bParameterList1: ARRAY[1..8] OF BOOL;
	Z1JOG_pos: BOOL;
	Z1JOG_neg: BOOL;
	Z2JOG_POS: BOOL;
	Z2JOG_NEG: BOOL;
	ModbusTcpError: Modbus_SLAVE_DIAGNOSE;
	展开工位允许放硅胶板1: BOOL;
	收集瓶组站位符: BOOL;
	收集器组站位符: BOOL;
	刮板拍照工位站位符: BOOL;
END_VAR

VAR_GLOBAL RETAIN PERSISTENT
	转发转存 AT %MW1301: STRING(128);
	接收字符 AT %MW1001: STRING(128);
	点样测试 AT %MX20.5: BOOL;
END_VAR

// Device/Application/20_变量Date/Host_Computer
VAR_GLOBAL
	bOutput: BOOL;
	bEnable: BOOL := TRUE;
	bErrorReset: BOOL;
	bStepEnable: BOOL := TRUE;
	/// <GrpComment>
	/// <GrpComment_zh-cn>PLC 正在执行动作</GrpComment_zh-cn>
	/// </GrpComment>
	// PLC 正在执行动作 
	PLC_Busy: BOOL := FALSE;
	/// <GrpComment>
	/// <GrpComment_zh-cn>修改:动作执行完成</GrpComment_zh-cn>
	/// </GrpComment>
	// 修改:动作执行完成 
	collect_Done: BOOL := FALSE;
	/// <GrpComment>
	/// <GrpComment_zh-cn>新增：动作执行错误/急停</GrpComment_zh-cn>
	/// </GrpComment>
	// 新增：动作执行错误/急停 
	collect_Error: BOOL := FALSE;
	/// <GrpComment>
	/// <GrpComment_zh-cn>新增：急停</GrpComment_zh-cn>
	/// </GrpComment>
	// 新增：急停
	PLC_EStop: BOOL;
	/// <GrpComment>
	/// <GrpComment_zh-cn>新增：收集工位置位</GrpComment_zh-cn>
	/// </GrpComment>
	// 新增：收集工位置位
	collect_Reset: BOOL;
	/// <GrpComment>
	/// <GrpComment_zh-cn>修改：收集工位状态机</GrpComment_zh-cn>
	/// </GrpComment>
	// 修改：收集工位状态机
	collect_Step: INT;
	/// <GrpComment>
	/// <GrpComment_zh-cn>收集工位注射泵转发指令</GrpComment_zh-cn>
	/// </GrpComment>
	// 收集工位注射泵转发指令
	collect_forward_instructions: STRING(128);
	/// <GrpComment>
	/// <GrpComment_zh-cn>收集次数</GrpComment_zh-cn>
	/// </GrpComment>
	// 收集次数
	collect_count: INT;
	/// <GrpComment>
	/// <GrpComment_zh-cn>新增：收集工位启动</GrpComment_zh-cn>
	/// </GrpComment>
	// 新增：收集工位启动
	collect_Enable: BOOL;
	/// <GrpComment>
	/// <GrpComment_zh-cn>新增：收集工位忙</GrpComment_zh-cn>
	/// </GrpComment>
	// 新增：收集工位忙
	collect_Busy: BOOL;
	/// <GrpComment>
	/// <GrpComment_zh-cn>PC→PLC: TRUE 启动状态机</GrpComment_zh-cn>
	/// </GrpComment>
	// PC→PLC: TRUE 启动状态机
	Expand_Enable: BOOL;
	/// <GrpComment>
	/// <GrpComment_zh-cn>PLC→PC: 子步号 {0,10,20,30,40,90}</GrpComment_zh-cn>
	/// </GrpComment>
	// PLC→PC: 子步号 {0,10,20,30,40,90}
	Expand_Step: INT;
	/// <GrpComment>
	/// <GrpComment_zh-cn>PLC→PC: prep完成锁存（语义变更：prep完成非整流程完成）</GrpComment_zh-cn>
	/// </GrpComment>
	// PLC→PC: prep完成锁存（语义变更：prep完成非整流程完成）
	Expand_Done: BOOL;
	/// <GrpComment>
	/// <GrpComment_zh-cn>PLC→PC: 故障锁存（Step=90），Expand_Reset=TRUE 清零</GrpComment_zh-cn>
	/// </GrpComment>
	// PLC→PC: 故障锁存（Step=90），Expand_Reset=TRUE 清零
	Expand_Error: BOOL;
	/// <GrpComment>
	/// <GrpComment_zh-cn>PC→PLC: TRUE 清错误</GrpComment_zh-cn>
	/// </GrpComment>
	// PC→PLC: TRUE 清错误
	Expand_Reset: BOOL;
	/// <GrpComment>
	/// <GrpComment_zh-cn>PLC→PC: 派生 (Step∈[10,80]) AND NOT Done</GrpComment_zh-cn>
	/// </GrpComment>
	// PLC→PC: 派生 (Step∈[10,80]) AND NOT Done
	Expand_Busy: BOOL;
	/// <GrpComment>
	/// <GrpComment_zh-cn>0=缸模式润洗 / 1=管路模式润洗</GrpComment_zh-cn>
	/// </GrpComment>
	// 0=缸模式润洗 / 1=管路模式润洗
	Expand_Mode_Flag: INT;
	/// <GrpComment>
	/// <GrpComment_zh-cn>展开组号 (1 或 2)，由 PLC 自动推导</GrpComment_zh-cn>
	/// </GrpComment>
	// 展开组号 (1 或 2)，由 PLC 自动推导
	Expand_Group: INT;
	/// <GrpComment>
	/// <GrpComment_zh-cn>缸号在组内序号（1-4），由 PLC 自动推导</GrpComment_zh-cn>
	/// </GrpComment>
	// 缸号在组内序号（1-4），由 PLC 自动推导
	Expand_Number: INT;
	/// <GrpComment>
	/// <GrpComment_zh-cn>注射泵 DT 协议指令（合并后的单一变量）</GrpComment_zh-cn>
	/// </GrpComment>
	// 上液注射泵重复次数
	Expand_up_liquid_count: INT;
	/// <GrpComment>
	/// <GrpComment_zh-cn>注射泵 DT 协议指令（合并后的单一变量）</GrpComment_zh-cn>
	/// </GrpComment>
	// 润洗重复次数
	Expand_rinse_count: INT;
	/// <GrpComment>
	/// <GrpComment_zh-cn>注射泵 DT 协议指令（合并后的单一变量）</GrpComment_zh-cn>
	/// </GrpComment>
	// 注射泵 DT 协议指令（合并后的单一变量）
	Expand_forward_instructions: STRING(128);
	/// <GrpComment>
	/// <GrpComment_zh-cn>══════════════════════════════════════════════════════════════
	/// 【新增】展缸状态跟踪
	/// ══════════════════════════════════════════════════════════════</GrpComment_zh-cn>
	/// </GrpComment>
	// ══════════════════════════════════════════════════════════════
	// 【新增】展缸状态跟踪
	// ══════════════════════════════════════════════════════════════
	Tank_State: ARRAY[1..8] OF INT;
	/// <GrpComment>
	/// <GrpComment_zh-cn>PLC→PC: 每缸状态
	/// 0  = Idle（空闲，可分配）
	/// 10 = Prepping（准备中：润洗/上液/放板）
	/// 40 = Developing（展开中，等待视觉/延时触发排液）
	/// 50 = Draining（排液中）
	/// 99 = Done（排液完成，等待 PC 释放）
	/// 90 = Error（故障）</GrpComment_zh-cn>
	/// </GrpComment>
	// PLC→PC: 每缸状态
	//   0  = Idle（空闲，可分配）
	//   10 = Prepping（准备中：润洗/上液/放板）
	//   40 = Developing（展开中，等待视觉/延时触发排液）
	//   50 = Draining（排液中）
	//   99 = Done（排液完成，等待 PC 释放）
	//   90 = Error（故障）
	Tank_SampleID: ARRAY[1..8] OF DINT;
	/// <GrpComment>
	/// <GrpComment_zh-cn>PC→PLC: 绑定样品 ID（调试/溯源用，PLC 不使用此值做逻辑判断）
	/// ══════════════════════════════════════════════════════════════
	/// 【新增】Prep 目标参数
	/// ══════════════════════════════════════════════════════════════</GrpComment_zh-cn>
	/// </GrpComment>
	// PC→PLC: 绑定样品 ID（调试/溯源用，PLC 不使用此值做逻辑判断）
	// ══════════════════════════════════════════════════════════════
	// 【新增】Prep 目标参数
	// ══════════════════════════════════════════════════════════════
	Expand_Target_Tank: INT;
	/// <GrpComment>
	/// <GrpComment_zh-cn>PC→PLC: 目标缸号(1-8)，Enable 触发前写入
	/// PLC 读取后自动推导：
	/// Expand_Group  = (Target_Tank - 1) / 4 + 1
	/// Expand_Number = (Target_Tank - 1) MOD 4 + 1
	/// ══════════════════════════════════════════════════════════════
	/// 【新增】Per-tank 排液控制
	/// ══════════════════════════════════════════════════════════════</GrpComment_zh-cn>
	/// </GrpComment>
	// PC→PLC: 目标缸号(1-8)，Enable 触发前写入
	// PLC 读取后自动推导：
	//   Expand_Group  = (Target_Tank - 1) / 4 + 1
	//   Expand_Number = (Target_Tank - 1) MOD 4 + 1
	// ══════════════════════════════════════════════════════════════
	// 【新增】Per-tank 排液控制
	// ══════════════════════════════════════════════════════════════
	Tank_Drain_Enable: ARRAY[1..8] OF BOOL;
	/// <GrpComment>
	/// <GrpComment_zh-cn>PC→PLC: 触发第 i 缸排液（前置条件：Tank_State[i]=40）</GrpComment_zh-cn>
	/// </GrpComment>
	// PC→PLC: 触发第 i 缸排液（前置条件：Tank_State[i]=40）
	Tank_Drain_Done: ARRAY[1..8] OF BOOL;
	/// <GrpComment>
	/// <GrpComment_zh-cn>PLC→PC: 第 i 缸排液完成锁存
	/// PC 确认后写 Tank_Drain_Enable[i]=FALSE 进行复位
	/// ══════════════════════════════════════════════════════════════
	/// 【新增】排液子程序内部变量
	/// ══════════════════════════════════════════════════════════════</GrpComment_zh-cn>
	/// </GrpComment>
	// PLC→PC: 第 i 缸排液完成锁存
	// PC 确认后写 Tank_Drain_Enable[i]=FALSE 进行复位
	// ══════════════════════════════════════════════════════════════
	// 【新增】排液子程序内部变量
	// ══════════════════════════════════════════════════════════════
	DrainTimer: ARRAY[1..8] OF TON;
	/// <GrpComment>
	/// <GrpComment_zh-cn>每缸排液定时器（后续可替换为传感器判断）</GrpComment_zh-cn>
	/// </GrpComment>
	// 每缸排液定时器（后续可替换为传感器判断）
	DrainDuration: TIME := TIME#5s0ms;
	/// <GrpComment>
	/// <GrpComment_zh-cn>PC→PLC: TRUE 启动状态机</GrpComment_zh-cn>
	/// </GrpComment>
	// PC→PLC: TRUE 启动状态机
	Sampling_Enable: BOOL;
	/// <GrpComment>
	/// <GrpComment_zh-cn>PLC→PC: 子步号 {0,10,20,30,40,50,90}</GrpComment_zh-cn>
	/// </GrpComment>
	// PLC→PC: 子步号 {0,10,20,30,40,50,90}
	Sampling_Step: INT;
	/// <GrpComment>
	/// <GrpComment_zh-cn>PLC→PC: 完成锁存（Step 50 结束后置 TRUE）</GrpComment_zh-cn>
	/// </GrpComment>
	// PLC→PC: 完成锁存（Step 50 结束后置 TRUE）
	Sampling_Done: BOOL;
	/// <GrpComment>
	/// <GrpComment_zh-cn>PLC→PC: 故障锁存（Step=90），Sampling_Reset=TRUE 清零</GrpComment_zh-cn>
	/// </GrpComment>
	// PLC→PC: 故障锁存（Step=90），Sampling_Reset=TRUE 清零
	Sampling_Error: BOOL;
	/// <GrpComment>
	/// <GrpComment_zh-cn>PC→PLC: TRUE 清错误</GrpComment_zh-cn>
	/// </GrpComment>
	// PC→PLC: TRUE 清错误
	Sampling_Reset: BOOL;
	/// <GrpComment>
	/// <GrpComment_zh-cn>PLC→PC: 派生 (Step∈[10,80]) AND NOT Done</GrpComment_zh-cn>
	/// </GrpComment>
	// PLC→PC: 派生 (Step∈[10,80]) AND NOT Done
	Sampling_Busy: BOOL;
	/// <GrpComment>
	/// <GrpComment_zh-cn>PC→PLC: 清洗泵指令（1条DT协议）</GrpComment_zh-cn>
	/// </GrpComment>
	// PC→PLC: 清洗泵指令（1条DT协议）
	Sampling_clean_instructions: ARRAY[1..2] OF STRING(128);
	/// <GrpComment>
	/// <GrpComment_zh-cn>PC→PLC: 清洗次数（0=跳过清洗）</GrpComment_zh-cn>
	/// </GrpComment>
	// PC→PLC: 清洗次数（0=跳过清洗）
	Sampling_clean_count: INT;
	/// <GrpComment>
	/// <GrpComment_zh-cn>── Step 20 气泡准备 ──</GrpComment_zh-cn>
	/// </GrpComment>
	// 上样准备泵指令
	Sampling_prep_instructions: ARRAY[1..2] OF STRING(128);
	/// <GrpComment>
	/// <GrpComment_zh-cn>PC→PLC: 气泡序列指令数组，按 bubble_count 逐条执行
	/// 上位机 translate_sample_bubble_cmd() 生成，默认 Phase1=6条，上限 16</GrpComment_zh-cn>
	/// </GrpComment>
	// PC→PLC: 气泡序列指令数组，按 bubble_count 逐条执行
	// 上位机 translate_sample_bubble_cmd() 生成，默认 Phase1=6条，上限 16
	Sampling_bubble_count: INT;
	/// <GrpComment>
	/// <GrpComment_zh-cn>PC→PLC: 数组有效条目数（0=跳过气泡准备）</GrpComment_zh-cn>
	/// </GrpComment>
	// PC→PLC: 数组有效条目数（0=跳过气泡准备）
	Sampling_BubbleSensor: BOOL;
	/// <GrpComment>
	/// <GrpComment_zh-cn>PLC 物理输入 / OPC UA 可写（调试用）
	/// TRUE = 气泡传感器检测到气-液界面到达上样针位置
	/// TODO【实机集成点】映射为物理输入 AT %IXx.y</GrpComment_zh-cn>
	/// </GrpComment>
	// PLC 物理输入 / OPC UA 可写（调试用）
	// TRUE = 气泡传感器检测到气-液界面到达上样针位置
	// TODO【实机集成点】映射为物理输入 AT %IXx.y
	Sampling_phase2_instructions: STRING(128);
	/// <GrpComment>
	/// <GrpComment_zh-cn>PC→PLC: Phase 2 单次补液泵指令（循环执行直到传感器触发）
	/// 简化版未使用，实机需按 [pending]plc_spotting.txt Step 20 Phase 2 实现</GrpComment_zh-cn>
	/// </GrpComment>
	// PC→PLC: Phase 2 单次补液泵指令（循环执行直到传感器触发）
	// 简化版未使用，实机需按 [pending]plc_spotting.txt Step 20 Phase 2 实现
	Sampling_Phase2_MaxCycles: INT;
	/// <GrpComment>
	/// <GrpComment_zh-cn>PC→PLC: 上样 X 坐标（逻辑索引，PLC内部查表映射物理坐标）</GrpComment_zh-cn>
	/// </GrpComment>
	// PC→PLC: 上样 X 坐标（逻辑索引，PLC内部查表映射物理坐标）
	Sampling_X_coordinate: INT;
	/// <GrpComment>
	/// <GrpComment_zh-cn>PC→PLC: 上样 Y 坐标</GrpComment_zh-cn>
	/// </GrpComment>
	// PC→PLC: 上样 Y 坐标
	Sampling_Y_coordinate: INT;
	/// <GrpComment>
	/// <GrpComment_zh-cn>PC→PLC: 吸液泵指令（1条DT协议）</GrpComment_zh-cn>
	/// </GrpComment>
	// PC→PLC: 上样泵指令
	Sampling_sample_instructions: ARRAY[1..2] OF STRING(128);
	/// <GrpComment>
	/// <GrpComment_zh-cn>PC→PLC: 点样泵指令（1条DT协议）</GrpComment_zh-cn>
	/// </GrpComment>
	// PC→PLC: 点样泵指令（1条DT协议）
	Sampling_dispense_instructions: ARRAY[1..2] OF STRING(128);
	/// <GrpComment>
	/// <GrpComment_zh-cn>PC?PLC: ????? A0R ??????</GrpComment_zh-cn>
	/// </GrpComment>
	// PC?PLC: ????? A0R ??????
	Sampling_band_run_instruction: STRING(128);
	/// <GrpComment>
	/// <GrpComment_zh-cn>PC?PLC: ????????? T ??</GrpComment_zh-cn>
	/// </GrpComment>
	// PC?PLC: ????????? T ??
	Sampling_band_stop_instruction: STRING(128);
	/// <GrpComment>
	/// <GrpComment_zh-cn>PC?PLC: ????? 6X ??????(mm/s)</GrpComment_zh-cn>
	/// </GrpComment>
	Sampling_band_spot_speed: LREAL;
	/// <GrpComment>
	/// <GrpComment_zh-cn>PC?PLC: ????? 6X ???????(mm/s)</GrpComment_zh-cn>
	/// </GrpComment>
	Sampling_band_dry_speed: LREAL;
	/// <GrpComment>
	/// <GrpComment_zh-cn>PC?PLC: ??????????????</GrpComment_zh-cn>
	/// </GrpComment>
	Sampling_band_dry_cycles: INT;
	/// <GrpComment>
	/// <GrpComment_zh-cn>PC→PLC: TRUE 启动状态机；FALSE 清 Done 回 idle</GrpComment_zh-cn>
	/// </GrpComment>
	// PC→PLC: TRUE 启动状态机；FALSE 清 Done 回 idle
	scrape_Enable: BOOL;
	/// <GrpComment>
	/// <GrpComment_zh-cn>PLC→PC: 子步号 {0,10,15,20,30,40,90}</GrpComment_zh-cn>
	/// </GrpComment>
	// PLC→PC: 子步号 {0,10,15,20,30,40,90}
	scrape_Step: INT;
	/// <GrpComment>
	/// <GrpComment_zh-cn>PLC→PC: 完成锁存（Step 40 结束后置 TRUE）</GrpComment_zh-cn>
	/// </GrpComment>
	// PLC→PC: 完成锁存（Step 40 结束后置 TRUE）
	scrape_Done: BOOL;
	/// <GrpComment>
	/// <GrpComment_zh-cn>PLC→PC: 故障锁存（Step=90），scrape_Reset=TRUE 清零</GrpComment_zh-cn>
	/// </GrpComment>
	// PLC→PC: 故障锁存（Step=90），scrape_Reset=TRUE 清零
	scrape_Error: BOOL;
	/// <GrpComment>
	/// <GrpComment_zh-cn>PC→PLC: TRUE 清错误</GrpComment_zh-cn>
	/// </GrpComment>
	// PC→PLC: TRUE 清错误
	scrape_Reset: BOOL;
	/// <GrpComment>
	/// <GrpComment_zh-cn>PLC→PC: 派生 (Step∈[10,80]) AND NOT Done</GrpComment_zh-cn>
	/// </GrpComment>
	// PLC→PC: 派生 (Step∈[10,80]) AND NOT Done
	scrape_Busy: BOOL;
	/// <GrpComment>
	/// <GrpComment_zh-cn>PC→PLC: 乒乓确认信号</GrpComment_zh-cn>
	/// </GrpComment>
	// PC→PLC: 乒乓确认信号
	scrape_Confirm: BOOL;
	/// <GrpComment>
	/// <GrpComment_zh-cn>PC→PLC: G-code 刮取路径指令</GrpComment_zh-cn>
	/// </GrpComment>
	// PC→PLC: G-code 刮取路径指令
	scrape_gcode_instructions: STRING(128);
	/// <GrpComment>
	/// <GrpComment_zh-cn>PC→PLC: 拍照模式选择</GrpComment_zh-cn>
	/// </GrpComment>
	// PC→PLC: 拍照模式选择
	scrape_PhotoMode: INT;
	g_sx: ARRAY[1..400] OF REAL;
	g_sy: ARRAY[1..400] OF REAL;
	g_cx: ARRAY[1..400] OF REAL;
	g_cy: ARRAY[1..400] OF REAL;
	g_scrape_feed: INT;
	// 刮取次数
	g_pass_count: INT;
	// Z高度
	g_pass_z: REAL;
	IX0 AT %IB0: BYTE;
	IX1 AT %IB1: BYTE;
	IX2 AT %IB2: BYTE;
	IX3 AT %IB3: BYTE;
	IX4 AT %IB4: BYTE;
	IX5 AT %IB5: BYTE;
	IX6 AT %IB6: BYTE;
	IX7 AT %IB7: BYTE;
	IX8 AT %IB8: BYTE;
	IX9 AT %IB9: BYTE;
	IX10 AT %IB10: BYTE;
	IX11 AT %IB11: BYTE;
	IX12 AT %IB12: BYTE;
	// 允许拍照信号
	scrape_WaitConfirm: BOOL;
	// 收集瓶取库位号
	collect_Fetch_Rack_Plate: INT;
	// 收集器料库号
	scrape_Fetch_Rack_Plate: INT;
	// 取收集瓶料位号
	collect_Consume_Slot: INT;
	// 放收集器料位号
	collect_Powder_Return_Slot: INT;
	// 收集器取料位号
	scrape_Consume_Slot: INT;
	// 收集瓶放库位号
	collect_Old_Plate_Slot: INT;
	// 收集器放库位号
	scrape_Old_Plate_Slot: INT;
	// 最后一次刮板收集
	scrape_IsLast: BOOL;
	// 停止
	PLCStop: BOOL;
	// 启动
	PLCStart: BOOL;
	// PC→PLC：动作码
	Collect_L2_ActionCode: INT;
	// PC→PLC：请求序号
	Collect_L2_RequestSeq: DINT;
	// PC→PLC：启动信号
	Collect_L2_Start: BOOL;
	// PC→PLC：复位信号
	Collect_L2_Reset: BOOL;
	// PLC→PC：动作状态
	Collect_L2_State: INT;
	// PLC→PC：当前动作码
	Collect_L2_ActiveCode: INT;
	// PLC→PC：已接受序号
	Collect_L2_AcceptedSeq: DINT;
	// PLC→PC：已完成序号
	Collect_L2_CompletedSeq: DINT;
	// PLC→PC：内部步骤
	Collect_L2_Step: INT;
	// PLC→PC：错误码
	Collect_L2_ErrorCode: INT;
	// PLC→PC：安全状态
	Collect_L2_SafeState: INT;
	// PLC→PC：是否允许重试
	Collect_L2_Retryable: BOOL;
	// PC→PLC：动作码
	Sampling_L2_ActionCode: INT;
	// PC→PLC：请求序号
	Sampling_L2_RequestSeq: DINT;
	// PC→PLC：启动信号
	Sampling_L2_Start: BOOL;
	// PC→PLC：复位信号
	Sampling_L2_Reset: BOOL;
	// PLC→PC：动作状态
	Sampling_L2_State: INT;
	// PLC→PC：当前动作码
	Sampling_L2_ActiveCode: INT;
	// PLC→PC：已接受序号
	Sampling_L2_AcceptedSeq: DINT;
	// PLC→PC：已完成序号
	Sampling_L2_CompletedSeq: DINT;
	// PLC→PC：内部步骤
	Sampling_L2_Step: INT;
	// PLC→PC：错误码
	Sampling_L2_ErrorCode: INT;
	// PLC→PC：安全状态
	Sampling_L2_SafeState: INT;
	// PLC→PC：是否允许重试
	Sampling_L2_Retryable: BOOL;
	// PC→PLC：动作码
	Develop_L2_ActionCode: INT;
	// PC→PLC：请求序号
	Develop_L2_RequestSeq: DINT;
	// PC→PLC：启动信号
	Develop_L2_Start: BOOL;
	// PC→PLC：复位信号
	Develop_L2_Reset: BOOL;
	// PLC→PC：动作状态
	Develop_L2_State: INT;
	// PLC→PC：当前动作码
	Develop_L2_ActiveCode: INT;
	// PLC→PC：已接受序号
	Develop_L2_AcceptedSeq: DINT;
	// PLC→PC：已完成序号
	Develop_L2_CompletedSeq: DINT;
	// PLC→PC：内部步骤
	Develop_L2_Step: INT;
	// PLC→PC：错误码
	Develop_L2_ErrorCode: INT;
	// PLC→PC：安全状态
	Develop_L2_SafeState: INT;
	// PLC→PC：是否允许重试
	Develop_L2_Retryable: BOOL;
	// PC→PLC：动作码
	PhotoScrape_L2_ActionCode: INT;
	// PC→PLC：请求序号
	PhotoScrape_L2_RequestSeq: DINT;
	// PC→PLC：启动信号
	PhotoScrape_L2_Start: BOOL;
	// PC→PLC：复位信号
	PhotoScrape_L2_Reset: BOOL;
	// PLC→PC：动作状态
	PhotoScrape_L2_State: INT;
	// PLC→PC：当前动作码
	PhotoScrape_L2_ActiveCode: INT;
	// PLC→PC：已接受序号
	PhotoScrape_L2_AcceptedSeq: DINT;
	// PLC→PC：已完成序号
	PhotoScrape_L2_CompletedSeq: DINT;
	// PLC→PC：内部步骤
	PhotoScrape_L2_Step: INT;
	// PLC→PC：错误码
	PhotoScrape_L2_ErrorCode: INT;
	// PLC→PC：安全状态
	PhotoScrape_L2_SafeState: INT;
	// PLC→PC：是否允许重试
	PhotoScrape_L2_Retryable: BOOL;
	// PC→PLC：动作码
	FeedLift_L2_ActionCode: INT;
	// PC→PLC：请求序号
	FeedLift_L2_RequestSeq: DINT;
	// PC→PLC：启动信号
	FeedLift_L2_Start: BOOL;
	// PC→PLC：复位信号
	FeedLift_L2_Reset: BOOL;
	// PLC→PC：动作状态
	FeedLift_L2_State: INT;
	// PLC→PC：当前动作码
	FeedLift_L2_ActiveCode: INT;
	// PLC→PC：已接受序号
	FeedLift_L2_AcceptedSeq: DINT;
	// PLC→PC：已完成序号
	FeedLift_L2_CompletedSeq: DINT;
	// PLC→PC：内部步骤
	FeedLift_L2_Step: INT;
	// PLC→PC：错误码
	FeedLift_L2_ErrorCode: INT;
	// PLC→PC：安全状态
	FeedLift_L2_SafeState: INT;
	// PLC→PC：是否允许重试
	FeedLift_L2_Retryable: BOOL;
	// PC→PLC：动作码 (10=真空泵开/20=真空泵关)
	Pump_L2_ActionCode: INT;
	// PC→PLC：请求序号
	Pump_L2_RequestSeq: DINT;
	// PC→PLC：启动信号
	Pump_L2_Start: BOOL;
	// PC→PLC：复位信号
	Pump_L2_Reset: BOOL;
	// PLC→PC：动作状态
	Pump_L2_State: INT;
	// PLC→PC：当前动作码
	Pump_L2_ActiveCode: INT;
	// PLC→PC：已接受序号
	Pump_L2_AcceptedSeq: DINT;
	// PLC→PC：已完成序号
	Pump_L2_CompletedSeq: DINT;
	// PLC→PC：内部步骤
	Pump_L2_Step: INT;
	// PLC→PC：错误码
	Pump_L2_ErrorCode: INT;
	// PLC→PC：安全状态
	Pump_L2_SafeState: INT;
	// PLC→PC：是否允许重试
	Pump_L2_Retryable: BOOL;
	// ===== 连续伺服 B 方案: PC 写目标 (LREAL); 仿射/点表算出的绝对位置 =====
	Sampling_4X_Target  : LREAL;   // 上样4X 目标(mm), 按孔; 替代 position[Sampling_X_coordinate]
	Sampling_3Y_Target  : LREAL;   // 上样3Y(打样3Y) 目标(mm), 按孔; 替代 position[Sampling_Y_coordinate]
	Spot_6X_StartTarget : LREAL;   // 点样6X 起点(mm), 按带; 替代 position[2]
	Spot_6X_EndTarget   : LREAL;   // 点样6X 终点(mm), 按带; 替代 position[3]
	Spot_7Y_Target      : LREAL;   // 点样7Y(mm), 按带; 替代 position[2]
	Photo_8Y_Target     : LREAL;   // 拍照8Y 位(mm); 替代硬编码 420

	// ===== 连续伺服 B 方案: PLC 写实际位置镜像 (LREAL); 供上位机实时显示 + jog 标定采点 =====
	Sampling_4X_ActPos  : LREAL;
	Sampling_3Y_ActPos  : LREAL;
	Spot_6X_ActPos      : LREAL;
	Spot_7Y_ActPos      : LREAL;
	Photo_8Y_ActPos     : LREAL;
	{attribute 'symbol' := 'readwrite'}
	Rail_ActPos         : LREAL;   // 地轨11Y 实际位置(mm) 每扫描镜像; 供后端映射所在站
	{attribute 'symbol' := 'readwrite'}
	Rail_Homed          : BOOL;    // 地轨11Y 已回零; 未回零时实际位不可信

	// ===== Rail_L2 地轨派发通道 (第7通道; 时序与 Pump_L2/FeedLift_L2 一致) =====
	Rail_Target_Position : INT;    // 地轨目标位置码 1-6, PC 写
	Rail_Current_Position : INT;   // PLC 写: 地轨当前所在站位 1-6 (0=移动中/未知); Rail_L2 到位置位、开始清0
	Rail_L2_ActionCode   : INT;    // PC 写; 固定 10 = rail.move
	Rail_L2_RequestSeq   : DINT;   // PC 写; 每次请求 +1
	Rail_L2_Start        : BOOL;   // PC 写; 上升沿触发
	Rail_L2_Reset        : BOOL;   // PC 写; 复位
	Rail_L2_State        : INT;    // PLC 写; 0=IDLE,10=RUNNING,20=DONE,30=REJECTED,40=ERROR,50=INTERRUPTED
	Rail_L2_ActiveCode   : INT;    // PLC 写; 当前动作码
	Rail_L2_AcceptedSeq  : DINT;   // PLC 写; 已接受序号
	Rail_L2_CompletedSeq : DINT;   // PLC 写; 已完成序号 (=AcceptedSeq 即握手完成)
	Rail_L2_Step         : INT;    // PLC 写; 内部步
	Rail_L2_ErrorCode    : INT;    // PLC 写; 错误码
	Rail_L2_SafeState    : INT;    // PLC 写; 安全态
	Rail_L2_Retryable    : BOOL;   // PLC 写; 可重试标志
	
	// ===== 地轨 11Y 双源同步 (Rail_Sync POU; struct 离散位 PC<->HMI 对账) =====
	Rail_Pos_Target : ARRAY[1..6] OF LREAL;  // 仅 PC 写: 6 站点真源运行值 (派发器读 + PUSH 源); PLC 绝不回写
	Rail_Pos_HMI    : ARRAY[1..6] OF LREAL;  // 仅 PLC 写: 每扫描镜像 HMI position[] (PC 做 diff/pull 读, 不碰 struct)
	Rail_Sync_Req   : INT;   // PC 或 HMI 写: 0=空闲 1=PUSH 2=PULL
	Rail_Sync_Ack   : INT;   // PLC 写 (PULL 完成段由 PC 写): 0=空闲 1=完成 2=待PC提交 3=拒绝(限位)
	Rail_Sync_Src   : INT;   // 请求方写: 1=PC 2=HMI (审计 + 防误触)
	
	Sampling_4X_WashTarget : LREAL;   // 上样4X 清洗位(mm) 离散示教; 替代 HMI_上样轴4X轴.position[9]

	// ===== 孔板手动校准 去使能手推 (PC<->PLC; calibration_service 写 FreeMove / 读 Enabled) =====
	Sampling_Servo_FreeMove : BOOL;   // PC->PLC: TRUE=去使能上样4X/打样3Y 供手推标定 (PLC 仅 5Z 抬起<3 时放行)
	Sampling_Servo_Enabled  : BOOL;   // PLC->PC: 上样4X AND 打样3Y 实际使能镜像; 供标定页显示真状态

	// PC->PLC: parameterized two-state actuator targets (written before L2 Start)
	PhotoScrape_CamLocate_Target: BOOL := TRUE;          // TRUE=photo locate cylinder clamp, FALSE=release
	PhotoScrape_CamPress_Target: BOOL := TRUE;           // TRUE=press cylinder down, FALSE=release/up
	PhotoScrape_PowderCollectorLocate_Target: BOOL := TRUE; // TRUE=powder collector locator clamp, FALSE=release
	Collect_BottleLocate_Target: BOOL := TRUE;           // TRUE=bottle locator clamp, FALSE=release
END_VAR

// Device/Application/20_变量Date/RB_Date
VAR_GLOBAL
	// 0:FALSE  1:REUE  3100
	Execute: INT;
	// 0:FALSE  1:REUE   3101
	Reset: INT;
	// 0-255   3102
	FunctionID: INT;
	// 展开数据   3103
	ParameterList1: INT;
	// 3104
	ParameterList2: INT;
	// 3105
	ParameterList3: INT;
	// 3106
	ParameterList4: INT;
	// 3107
	ParameterList5: INT;
	// 3108
	ParameterList6: INT;
	ParameterList7: INT;
	ParameterList8: INT;
	// 0:Free 1:Busy 2:Complete 255:Error
	ParameterList9: INT;
	// 0:Free 1:Busy 2:Complete 255:Error
	ParameterList10: INT;
	// 0:Free 1:Busy 2:Complete 255:Error
	Status: INT;
	// 0:原点初始化 1-255 自定义
	Point: INT;
	/// <GrpComment>
	/// <GrpComment_zh-cn>0:无错误  255:不允许运行</GrpComment_zh-cn>
	/// </GrpComment>
	// 0:无错误  255:不允许运行  
	ErrorID: INT;
	RO_ParameterList1: INT;
	RO_ParameterList2: INT;
	RO_ParameterList3: INT;
	RO_ParameterList4: INT;
	RO_ParameterList5: INT;
	RO_ParameterList6: INT;
	RO_ParameterList7: INT;
	RO_ParameterList8: INT;
	RO_ParameterList9: INT;
	RO_ParameterList10: INT;
	收集工位允许放收集瓶: BOOL;
	收集工位允许放收集器: BOOL;
	收集工位放收集瓶完成: BOOL;
	收集工位放收集器到工位: BOOL;
	收集工位允许机器人退出工位: BOOL;
	收集工位机器人退出完成: BOOL;
	收集工位允许机器人取收集瓶放暂存工位: BOOL;
	收集工位机器人放收集瓶到暂存工位完成: BOOL;
	收集工位允许取收集器: BOOL;
	收集工位机器人到达收集器位置: BOOL;
	收集工位机器人取收集器放回暂存工位: BOOL;
	收集工位放收集器完成: BOOL;
	展开工位允许放硅胶板: BOOL;
	展开工位允许取硅胶板: BOOL;
	展开工位机器人到达准备点: BOOL;
	展开工位机器人放硅胶板完成: BOOL;
	展开工位取硅胶板完成: BOOL;
	上样点样允许放硅胶板: BOOL;
	上样点样允许取硅胶板: BOOL;
	上样点样放硅胶板完成: BOOL;
	拍照工位允许放硅胶板: BOOL;
	拍照工位放硅胶板完成: BOOL;
	拍照工位允许放收集器: BOOL;
	拍照工位机器人到达夹持位: BOOL;
	拍照工位机器人退出工位: BOOL;
	拍照工位机器人退出工位完成: BOOL;
	拍照工位允许取收集器: BOOL;
	拍照工位机器人到达收集器夹持位: BOOL;
	拍照工位机器人退出: BOOL;
	拍照工位机器人退出完成: BOOL;
	拍照工位允许取硅胶板放废料区: BOOL;
	拍照工位允许取硅胶板去展开: BOOL;
	拍照工位机器人取硅胶板完成: BOOL;
	升降上料伺服允许取料: BOOL;
	升降上料机器人已吸住物料: BOOL;
	升降上料伺服下降完成: BOOL;
	升降上料机器人取料完成: BOOL;
	升降上料机器人放料完成: BOOL;
	升降下料伺服允许放料: BOOL;
	升降下料机器人放废料完成: BOOL;
END_VAR

// Device/Application/40_Man/PLC_MainPRG
PROGRAM PLC_MainPRG
VAR
	PLC_Mode_0: FB_Mode;
	TON_1: TON;
	TON_0: TON;
	TON_2: TON;
	TON_3: TON;
	SysHC_ModbusTcpSlaveDiagnose_0: SysHC_ModbusTcpSlaveDiagnose;
	点样step: INT;
	打样伺服移动step: INT;
END_VAR

IF 点样测试 THEN
	CASE 打样伺服移动step OF
		
		0:
			点样轴6XDATE.fAbsTarget:=HMI_点样轴6X.position[2];        //起始位
			点样轴6XDATE.xMoveAbs:=TRUE;
			打样伺服移动step:=20;
		20:
			IF 点样轴6XDATE.bAbMoveDone THEN
				
				打样伺服移动step:=30;
				点样轴6XDATE.xMoveAbs:=FALSE;
			END_IF
		30:
			点样轴6XDATE.fAbsTarget:=HMI_点样轴6X.position[3];             //终点位
			点样轴6XDATE.xMoveAbs:=TRUE;
			打样伺服移动step:=40;
		40:
			IF 点样轴6XDATE.bAbMoveDone THEN
				
				打样伺服移动step:=0;
				点样轴6XDATE.xMoveAbs:=FALSE;
			END_IF
			
	END_CASE
ELSE
	打样伺服移动step:=0;
END_IF

A00_设备状态显示及控制 ();

%MW1000:=0;

PLC_Cyinder_气缸动作();
//开机窗口抑制气缸超时误报(等气压/传感器稳定); 窗口内强制清气缸报警位, HMI 不再成批刷报警
IF bCyInhibit THEN
	cyinderAlarm := 0;
END_IF
// ===== 连续伺服实际位置镜像 (B方案, PLC->PC, 每扫描无条件; 供实时显示+jog标定采点) =====
Sampling_4X_ActPos := 上样轴4X轴DATE.fActPos;
Sampling_3Y_ActPos := 打样瓶上料轴3YDATE.fActPos;
Spot_6X_ActPos     := 点样轴6XDATE.fActPos;
Spot_7Y_ActPos     := 点样轴7YDATE.fActPos;
Photo_8Y_ActPos    := 拍照轴8YDATE.fActPos;
Rail_ActPos := 地轨轴11YDATE.fActPos;   // 地轨11Y 实际位 -> 后端映射所在站 (每扫描无条件, 任意模式)
Rail_Homed  := 地轨轴11YDATE.bHomed;     // 地轨11Y 回零标志 -> 后端门控(未回零实际位不可信)
Rail_Sync();   // 地轨双源同步: 每扫描镜像 position[]->Rail_Pos_HMI[] + 处理 PUSH/PULL 邮箱

CASE MODE_State OF
	EN_功能块状态.运行:
		PLC_Pump_泵管理();
		Pump_L2();
		Rail_L2();
		FeedLift_L2();
		Sampling_L2();
		Collect_L2();
		Develop_L2();
		Develop_TankDrain();
		PhotoScrape_L2();
	IF NOT 上料进料传感器 THEN
		Alarm.2:=TRUE;
	END_IF
	IF NOT 下料出料传感器 THEN
		Alarm.3:=TRUE;
	END_IF
END_CASE

//所有状态复位
TON_3(IN:=复位,PT:=T#5S );
IF NOT 急停 OR TON_3.Q THEN
	A30_急停();
END_IF

//升降伺服流程
IF MODE_State<>1 THEN
	伺服上料_Setp:=0;
	伺服下料_Setp:=0;
END_IF


// //检测MODBUS通讯
// SysHC_ModbusTcpSlaveDiagnose_0(
// 	xEnable:=TRUE , 
// 	strSlaveIP:= '192.168.0.15', 
// 	xValid=> , 
// 	xBusy=> , 
// 	xError=> , 
// 	eErrorID=> , 
// 	stDiagData=>ModbusTcpError );

ACTION A10_上下料伺服流程:
//初始化
IF MODE_State =4 OR  初始化  THEN

		玻璃上料轴1ZDATE.fAbsTarget :=0;
		玻璃上料轴1ZDATE.xMoveAbs:=TRUE;
		玻璃上料轴1ZDATE.xJogPos :=FALSE;
		升降上料伺服允许取料 :=FALSE ;
		升降上料伺服下降完成 :=FALSE ;
		伺服上料_Setp:=0;
		伺服上料_Setp:=0;
		升降下料伺服允许放料  :=FALSE ;
		玻璃上料轴2ZDATE.xJogNeg :=FALSE;
		玻璃上料轴2ZDATE.xJogPos :=FALSE;
		升降上料机器人取料完成:=FALSE;
END_IF



//上料流程
IF MODE_State =1 THEN     //自动模式下
	IF 玻璃上料轴1ZDATE.bHomed AND 玻璃升降接近开关1 AND 上料进料传感器 AND 伺服上料_Setp=0 AND NOT Alarm.0 AND 升降上料完成 THEN
		伺服上料_Setp :=1;
	END_IF
	
    CASE 伺服上料_Setp OF
    	1 :
			IF NOT 玻璃升降光电开关1 AND 玻璃上料轴1ZDATE.fActPos<514  THEN
				Z1JOG_pos :=TRUE;
				ELSE
				Z1JOG_pos :=FALSE;
				伺服上料_Setp:=10;
			END_IF
   
	   10:
		   IF 玻璃升降光电开关1 THEN
		   	升降上料伺服允许取料 :=TRUE;
			伺服上料_Setp:=20;
		   END_IF
		   
	   20:
		   IF 升降上料机器人已吸住物料 THEN
		   	玻璃上料轴1ZDATE.fRelTarget :=-5.0;
			玻璃上料轴1ZDATE.xMoveRel :=TRUE;
			升降上料机器人已吸住物料:=FALSE;
			伺服上料_Setp:=30;
		   END_IF
	   30:
		   IF 玻璃上料轴1ZDATE .bReMoveDone  THEN
		   	升降上料伺服下降完成 :=TRUE ;
			玻璃上料轴1ZDATE.xMoveRel :=FALSE;
			伺服上料_Setp:=40;
		   END_IF
	   40:
		   IF 升降上料机器人取料完成  THEN
		   	升降上料伺服下降完成 :=FALSE ;
			升降上料伺服允许取料 :=FALSE ;
			升降上料机器人取料完成:=FALSE;
			伺服上料_Setp:=1;
		   END_IF 
    END_CASE
	
	IF 玻璃上料轴1ZDATE.fActPos>=510.0 AND  玻璃升降光电开关1 AND  NOT 玻璃升降接近开关1 THEN
		Alarm.0:=TRUE;                                             //上料机构无物料
		升降上料完成:=FALSE;
		玻璃上料轴1ZDATE.fAbsTarget :=0;
		玻璃上料轴1ZDATE.xMoveAbs:=TRUE;
		Z1JOG_pos :=FALSE;
		升降上料伺服允许取料 :=FALSE ;
		升降上料伺服下降完成 :=FALSE ;
		伺服上料_Setp:=0;
	END_IF
	IF 玻璃上料轴1ZDATE .bAbMoveDone  THEN
		玻璃上料轴1ZDATE.xMoveAbs:=FALSE;
		升降上料机器人放料完成:=FALSE;
    END_IF
	
	
END_IF
//下料流程
IF MODE_State =1 THEN     //自动模式下
	IF 玻璃上料轴2ZDATE.bHomed  AND 下料出料传感器 AND 伺服下料_Setp=0 AND NOT Alarm.1 AND 升降下料完成 THEN
		伺服下料_Setp :=1;
	END_IF
	
    CASE 伺服下料_Setp  OF
    	1 :
			IF NOT 玻璃升降光电开关2 AND 玻璃上料轴2ZDATE.fActPos<510  THEN
				Z2JOG_POS :=TRUE;
				
				ELSE
				Z2JOG_POS :=FALSE;
				伺服下料_Setp:=10;
			END_IF
   
	   10:
		   IF 玻璃升降光电开关2 THEN
			   Z2JOG_NEG :=TRUE;
			   伺服下料_Setp:=15;
		   END_IF
	   15:
		   IF NOT 玻璃升降光电开关2  THEN
				升降下料伺服允许放料  :=TRUE;
				Z2JOG_NEG :=FALSE;
				伺服下料_Setp:=20;
		   END_IF
			  
	   
	   20:
		   IF 升降下料机器人放废料完成 AND 玻璃升降光电开关2 AND 玻璃升降接近开关2 THEN
		   	Z2JOG_NEG :=TRUE;
			升降下料伺服允许放料  :=FALSE ;
			升降下料机器人放废料完成:=FALSE;
			伺服下料_Setp:=30;
		   END_IF
		  
	   30:
		   IF NOT 玻璃升降光电开关2 THEN
		   	Z2JOG_NEG :=FALSE;
			取刮板硅胶板放废料区完成:=FALSE;
			伺服下料_Setp:=15;
		   END_IF
	  
    END_CASE
	
	IF 玻璃上料轴2ZDATE.fActPos<=0 AND 玻璃升降光电开关1 THEN
		Alarm.1:=TRUE;                                           //下料机构已满料
		升降下料完成:=FALSE;
		伺服下料_Setp:=0;
		升降下料伺服允许放料  :=FALSE ;
		Z2JOG_NEG :=FALSE;
		Z2JOG_POS :=FALSE;
		玻璃上料轴2ZDATE.fAbsTarget :=0;
		玻璃上料轴2ZDATE.xMoveAbs:=TRUE;
		伺服下料_Setp:=0;
	END_IF
	IF 玻璃上料轴2ZDATE .bAbMoveDone  THEN
		玻璃上料轴2ZDATE.xMoveAbs:=FALSE;
		升降下料伺服允许放料  :=FALSE ;
    END_IF
END_IF
END_ACTION

ACTION A00_设备状态显示及控制:
//PLC模式切换
PLC_Mode_0(
    bWarning_alarm := cyinderAlarm<>0 OR Alarm<>0 OR 上样料架报警 OR ModbusTcpError.byDiagData>0, 

	xStart:= 启动 OR PLCStart, 
	xStop:=NOT  停止 OR PLCStop, 
	xReset:=复位 OR bAutoHomeResetPulse  , 
	xAutoMode:=手自动  , 
	xFault:=伺服报警 OR ECAT掉站报警 OR 伺服未回原点报警, 
	xEmergency:= 急停 , 
	bRed=>三色灯红  , 
	bYellow=> 三色灯黄, 
	bGreen=> 三色灯绿, 
	bBuzzer=> 蜂鸣器 , 
	iState=>MODE_STATE  , 
	bAuto=>ManualAuto  );
	
	//伺服报错
IF   玻璃上料轴1ZDATE.bError OR 玻璃上料轴2ZDATE.bError OR 打样瓶上料轴3YDATE.bError OR 点样轴6XDATE.bError OR 点样轴7YDATE.bError OR 拍照轴8YDATE.bError OR 刮板轴9XDATE.bError OR 刮板轴10ZDATE.bError OR 地轨轴11YDATE.bError OR 上样轴4X轴DATE.bError OR 上样轴5Z轴DATE.bError THEN
	伺服报警:=TRUE;
END_IF
   //伺服报错复位 复位按钮/启动自愈窗 bSysReset/自动回零完成脉冲 bAutoHomeResetPulse 自动清锁存
IF 复位 OR bSysReset OR bAutoHomeResetPulse THEN
	伺服报警:=FALSE;
	伺服未回原点报警:=FALSE;
	Alarm:=0;
	cyinderAlarm:=0;
	上样料架报警:=FALSE;
END_IF


IF NOT 玻璃上料轴1ZDATE.bHomed OR NOT 玻璃上料轴2ZDATE.bHomed OR NOT 打样瓶上料轴3YDATE.bHomed OR NOT 点样轴6XDATE.bHomed OR NOT 点样轴7YDATE.bHomed OR NOT 拍照轴8YDATE.bHomed OR NOT 刮板轴9XDATE.bHomed OR NOT 刮板轴10ZDATE.bHomed  OR NOT 地轨轴11YDATE.bHomed OR NOT 上样轴4X轴DATE.bHomed OR NOT 上样轴5Z轴DATE.bHomed THEN
	伺服未回原点报警:=TRUE ;
END_IF
END_ACTION

ACTION A20_机器人:
//机器人远程控制
// RB_Control_0(
//     PowerOn := RB_使能状态, 
//     PowerOnOut =>RB_上使能 , 
// 
//     ResetOut =>RB_复位 , 
// 
//     Reset := 复位, 
// 
//     StartCmd := 启动, 
//     StopCmd :=  TON_3.Q OR NOT 急停, 
//     PauseCmd := NOT 停止, 
//     RobotRunning := RB_运行中, 
//     RobotStopped :=RB_停止中 , 
//     RobotPaused :=RB_暂停中 , 
//     RobotAlarm :=RB_报警中 , 
//     StartOut =>RB_启动 , 
//     StopOut => RB_停止, 
//     PauseOut =>  RB_暂停, 
//     StatusRun => , 
//     StatusStop => , 
//     StatusPause => , 
//     StatusAlarm => , 
// 
// 	);
END_ACTION

ACTION A30_急停:

伺服上料_Setp:=0;
伺服下料_Setp:=0;
//收集工位
收集下压气缸手动:=FALSE;
收集下压气缸自动:=FALSE;
收集夹持气缸手动:=FALSE;
收集夹持气缸自动:=FALSE;
收集升降气缸手动:=FALSE;
收集升降气缸自动:=FALSE;
收集伸缩气缸手动:=FALSE;
收集伸缩气缸自动:=FALSE;
收集进液手动:=FALSE;
收集进液自动:=FALSE;
收集排液手动:=FALSE;
收集排液自动:=FALSE;
收集正压排液手动:=FALSE;
收集正压排液自动:=FALSE;
溶液收集瓶定位手动:=FALSE;
collect_prepare_OK:=FALSE;
collect_OK:=FALSE;



//展开工位
expand_initialization_OK:=FALSE;
Expand_Group_clean_OK:=FALSE;
Expand_up_liquid_OK:=FALSE;
Expand_silica_gel_plate_OK:=FALSE;
展缸1气缸1手动:=FALSE;
展缸1气缸1自动:=FALSE;
展缸1进液电池阀1手动:=FALSE;
展缸1进液电池阀1自动:=FALSE;
展缸1排液电池阀1手动:=FALSE;
展缸1排液电池阀1自动:=FALSE;
展缸1吹气电池阀1手动:=FALSE;
展缸1吹气电池阀1自动:=FALSE;
展缸1气缸2手动:=FALSE;
展缸1气缸2自动:=FALSE;
展缸1进液电池阀2手动:=FALSE;
展缸1进液电池阀2自动:=FALSE;
展缸1排液电池阀2手动:=FALSE;
展缸1排液电池阀2自动:=FALSE;
展缸1吹气电池阀2手动:=FALSE;
展缸1吹气电池阀2自动:=FALSE;
展缸1气缸3手动:=FALSE;
展缸1气缸3自动:=FALSE;
展缸1进液电池阀3手动:=FALSE;
展缸1进液电池阀3自动:=FALSE;	
展缸1排液电池阀3手动:=FALSE;
展缸1排液电池阀3自动:=FALSE;
展缸1吹气电池阀3手动:=FALSE;
展缸1吹气电池阀3自动:=FALSE;
展缸1气缸4手动:=FALSE;
展缸1气缸4自动:=FALSE;
展缸1进液电池阀4手动:=FALSE;
展缸1进液电池阀4自动:=FALSE;	
展缸1排液电池阀4手动:=FALSE;
展缸1排液电池阀4自动:=FALSE;
展缸1吹气电池阀4手动:=FALSE;
展缸1吹气电池阀4自动:=FALSE;
展缸2气缸1手动:=FALSE;
展缸2气缸1自动:=FALSE;
展缸2进液电池阀1手动:=FALSE;
展缸2进液电池阀1自动:=FALSE;
展缸2排液电池阀1手动:=FALSE;
展缸2排液电池阀1自动:=FALSE;
展缸2吹气电池阀1手动:=FALSE;
展缸2吹气电池阀1自动:=FALSE;
展缸2气缸2手动:=FALSE;
展缸2气缸2自动:=FALSE;
展缸2进液电池阀2手动:=FALSE;
展缸2进液电池阀2自动:=FALSE;
展缸2排液电池阀2手动:=FALSE;
展缸2排液电池阀2自动:=FALSE;
展缸2吹气电池阀2手动:=FALSE;
展缸2吹气电池阀2自动:=FALSE;
展缸2气缸3手动:=FALSE;
展缸2气缸3自动:=FALSE;
展缸2进液电池阀3手动:=FALSE;
展缸2进液电池阀3自动:=FALSE;	
展缸2排液电池阀3手动:=FALSE;
展缸2排液电池阀3自动:=FALSE;
展缸2吹气电池阀3手动:=FALSE;
展缸2吹气电池阀3自动:=FALSE;
展缸2气缸4手动:=FALSE;
展缸2气缸4自动:=FALSE;
展缸2进液电池阀4手动:=FALSE;
展缸2进液电池阀4自动:=FALSE;	
展缸2排液电池阀4手动:=FALSE;
展缸2排液电池阀4自动:=FALSE;
展缸2吹气电池阀4手动:=FALSE;
展缸2吹气电池阀4自动:=FALSE;
Expand_Step:=0;
//拍照刮板
刮板拍照真空自动:=FALSE;
刮板拍照真空手动:=FALSE;
刮板拍照无刷电机手动:=FALSE;
刮板拍照无刷电机自动:=FALSE;
刮板拍照定位气缸手动:=FALSE;
刮板拍照定位气缸自动:=FALSE;
粉末收集器定位手动:=FALSE;
粉末收集器定位自动:=FALSE;
刮板拍照遮光气缸手动:=FALSE;
刮板拍照遮光气缸自动:=FALSE;
刮板拍照旋转气缸手动:=FALSE;
刮板拍照旋转气缸自动:=FALSE;
刮板拍照下压气缸手动:=FALSE;
刮板拍照下压气缸自动:=FALSE;
 scrape_IsLast := FALSE;       // ★ 新增		
scrape_PhotoMode:=0;
scrape_Step:=0;
Camera_scraper_initialization_OK:=FALSE;
Photo_preparation_completed_OK:=FALSE;
Scraper_collection_completed:=FALSE;
Robot_completes_material_retrieval:=FALSE;	

//上样点样
上样定位手动:=FALSE;
上样定位自动:=FALSE;
上样点样三通电池阀手动:=FALSE;
上样点样三通电池阀自动:=FALSE;
上样吹气手动:=FALSE;
上样吹气自动:=FALSE;
打样瓶上料轴3YDATE.fAbsTarget:=0;
点样轴6XDATE.fAbsTarget:=0;
点样轴7YDATE.fAbsTarget:=0;
上样轴4X轴DATE.fAbsTarget:=0;
上样轴5Z轴DATE.fAbsTarget:=0;
点样轴7YDATE.xMoveAbs:=FALSE;
点样轴6XDATE.xMoveAbs:=FALSE;
上样轴5Z轴DATE.xMoveAbs:=FALSE;
上样轴4X轴DATE.xMoveAbs:=FALSE;
打样瓶上料轴3YDATE.xMoveAbs:=FALSE;
Sampling_Spray_sample_OK:=FALSE;
Sampling_liquid_absorption:=FALSE;
Sampling_preparation_OK:=FALSE;
大真空泵站位[11]:=FALSE;
大真空泵自动:=FALSE;
Sampling_Step:=0;

//机器人

泵站位符:=FALSE;
上样料架报警:=FALSE;
溶液收集瓶定位自动:=FALSE;
溶液收集瓶定位手动:=FALSE;
END_ACTION

END_PROGRAM

// Device/Application/40_Man/PLC_Cyinder_气缸动作
PROGRAM PLC_Cyinder_气缸动作
VAR
	cylinder_0: FB_cylinder;
	cylinder_1: FB_cylinder;
	cylinder_2: FB_cylinder;
	cylinder_3 :FB_cylinder ;
	cylinder_4 :FB_cylinder ;
	cylinder_5 :FB_cylinder ;
	cylinder_6 :FB_cylinder ;
	cylinder_7 :FB_cylinder ;
	cylinder_8 :FB_cylinder ;
	cylinder_9 :FB_cylinder ;
	cylinder_10 :FB_cylinder ;
	cylinder_11 :FB_cylinder ;
	cylinder_12 :FB_cylinder ;
	cylinder_13 :FB_cylinder ;
	cylinder_14 :FB_cylinder ;
	cylinder_15 :FB_cylinder ;
	cylinder_16 :FB_cylinder ;
	cylinder_17 :FB_cylinder ;
	cylinder_18 :FB_cylinder ;
	cylinder_19 :FB_cylinder ;
	cylinder_20 :FB_cylinder ;
	cylinder_21 :FB_cylinder ;
	cylinder_22 :FB_cylinder ;
	cylinder_23 :FB_cylinder ;
	cylinder_24 :FB_cylinder ;
	cylinder_25 :FB_cylinder ;
	cylinder_26 :FB_cylinder ;
	cylinder_27 :FB_cylinder ;
	cylinder_28 :FB_cylinder ;
	cylinder_29 :FB_cylinder ;
	cylinder_30 :FB_cylinder ;
	cylinder_31 :FB_cylinder ;
	cylinder_32 :FB_cylinder ;
	cylinder_33 :FB_cylinder ;
	cylinder_34 :FB_cylinder ;
	cylinder_35 :FB_cylinder ;
	cylinder_36 :FB_cylinder ;
	cylinder_37 :FB_cylinder ;
	cylinder_38 :FB_cylinder ;
	cylinder_39 :FB_cylinder ;
	cylinder_40 :FB_cylinder ;
	cylinder_41 :FB_cylinder ;
	cylinder_42 :FB_cylinder ;
	cylinder_43 :FB_cylinder ;
	cylinder_44 :FB_cylinder ;
	cylinder_45 :FB_cylinder ;
	cylinder_46 :FB_cylinder ;
	cylinder_47 :FB_cylinder ;
	cylinder_48 :FB_cylinder ;
	cylinder_49 :FB_cylinder ;
	cylinder_50 :FB_cylinder ;
END_VAR

//气缸动作
//展缸1气缸1
cylinder_0(
    xManualRetract := , 
    xAutoRetract := , 
    yValve2 => , 
    cylinder_type := 0, 

	xManualAuto:=ManualAuto  , 
	xManualExtend:=展缸1气缸1手动 , 
	xAutoExtend:= 展缸1气缸1自动, 
	xReset:=复位  , 
	xPosExtend:= 展缸1气缸1原点, 
	xPosRetract:= 展缸1气缸1动点 , 
	tTimeout:= T#5S, 
	yValve1=> 展缸1气缸1 , 
	bAlarm=> cyinderAlarm.0);
//展缸1气缸2
cylinder_1(
    xManualRetract := , 
    xAutoRetract := , 
    yValve2 => , 
    cylinder_type :=0 , 

	xManualAuto:=ManualAuto  , 
	xManualExtend:=展缸1气缸2手动 , 
	xAutoExtend:= 展缸1气缸2自动, 
	xReset:=复位  , 
	xPosExtend:= 展缸1气缸2原点, 
	xPosRetract:= 展缸1气缸2动点 , 
	tTimeout:= T#5S, 
	yValve1=> 展缸1气缸2, 
	bAlarm=> cyinderAlarm.1);
//展缸1气缸3
cylinder_2(
    xManualRetract := , 
    xAutoRetract := , 
    yValve2 => , 
    cylinder_type := 0, 

	xManualAuto:=ManualAuto  , 
	xManualExtend:=展缸1气缸3手动 , 
	xAutoExtend:= 展缸1气缸3自动, 
	xReset:=复位  , 
	xPosExtend:= 展缸1气缸3原点, 
	xPosRetract:= 展缸1气缸3动点 , 
	tTimeout:= T#5S, 
	yValve1=> 展缸1气缸3, 
	bAlarm=> cyinderAlarm.2);
//展缸1气缸4
cylinder_3(
    xManualRetract := , 
    xAutoRetract := , 
    yValve2 => , 
    cylinder_type :=0 , 

	xManualAuto:=ManualAuto  , 
	xManualExtend:=展缸1气缸4手动 , 
	xAutoExtend:= 展缸1气缸4自动, 
	xReset:=复位  , 
	xPosExtend:= 展缸1气缸4原点, 
	xPosRetract:= 展缸1气缸4动点 , 
	tTimeout:= T#5S, 
	yValve1=> 展缸1气缸4, 
	bAlarm=> cyinderAlarm.3);
//展缸2气缸1
cylinder_4(
    xManualRetract := , 
    xAutoRetract := , 
    yValve2 => , 
    cylinder_type := 0, 

	xManualAuto:=ManualAuto  , 
	xManualExtend:=展缸2气缸1手动 , 
	xAutoExtend:= 展缸2气缸1自动, 
	xReset:=复位  , 
	xPosExtend:= 展缸2气缸1原点, 
	xPosRetract:= 展缸2气缸1动点 , 
	tTimeout:= T#5S, 
	yValve1=> 展缸2气缸1, 
	bAlarm=> cyinderAlarm.4);
//展缸2气缸2
cylinder_5(
    xManualRetract := , 
    xAutoRetract := , 
    yValve2 => , 
    cylinder_type :=0 , 

	xManualAuto:=ManualAuto  , 
	xManualExtend:=展缸2气缸2手动 , 
	xAutoExtend:= 展缸2气缸2自动, 
	xReset:=复位  , 
	xPosExtend:= 展缸2气缸2原点, 
	xPosRetract:= 展缸2气缸2动点 , 
	tTimeout:= T#5S, 
	yValve1=> 展缸2气缸2, 
	bAlarm=> cyinderAlarm.5);
//展缸2气缸3
cylinder_6(
    xManualRetract := , 
    xAutoRetract := , 
    yValve2 => , 
    cylinder_type := 0, 

	xManualAuto:=ManualAuto  , 
	xManualExtend:=展缸2气缸3手动 , 
	xAutoExtend:= 展缸2气缸3自动, 
	xReset:=复位  , 
	xPosExtend:= 展缸2气缸3原点, 
	xPosRetract:= 展缸2气缸3动点 , 
	tTimeout:= T#5S, 
	yValve1=> 展缸2气缸3, 
	bAlarm=> cyinderAlarm.6);
//展缸2气缸4
cylinder_7(
    xManualRetract := , 
    xAutoRetract := , 
    yValve2 => , 
    cylinder_type := 0, 

	xManualAuto:=ManualAuto  , 
	xManualExtend:=展缸2气缸4手动 , 
	xAutoExtend:= 展缸2气缸4自动, 
	xReset:=复位  , 
	xPosExtend:= 展缸2气缸4原点, 
	xPosRetract:= 展缸2气缸4动点 , 
	tTimeout:= T#5S, 
	yValve1=> 展缸2气缸4, 
	bAlarm=> cyinderAlarm.7);
//大真空泵
cylinder_8(
    xManualRetract := , 
    xAutoRetract := , 
    yValve2 => , 
    cylinder_type :=0 , 

	xManualAuto:=ManualAuto  , 
	xManualExtend:= 大真空泵手动, 
	xAutoExtend:= 大真空泵自动, 
	xReset:=复位  , 
	xPosExtend:= , 
	xPosRetract:=  , 
	tTimeout:= , 
	yValve1=> 大真空泵, 
	bAlarm=> );
//收集平台下压气缸
cylinder_9(
    xManualRetract := , 
    xAutoRetract := , 
    yValve2 => , 
    cylinder_type := 0, 

	xManualAuto:=ManualAuto  , 
	xManualExtend:= 收集下压气缸手动, 
	xAutoExtend:= 收集下压气缸自动, 
	xReset:=复位  , 
	xPosExtend:=收集平台下压气缸原点 , 
	xPosRetract:= 收集下压气缸手动 OR 收集下压气缸自动, 
	tTimeout:= T#5S, 
	yValve1=> 收集下压气缸 , 
	bAlarm=> cyinderAlarm.8);
//收集平台夹持气缸
cylinder_10(
    xManualRetract := , 
    xAutoRetract := , 
    yValve2 => , 
    cylinder_type := 0, 

	xManualAuto:=ManualAuto  , 
	xManualExtend:= 收集夹持气缸手动, 
	xAutoExtend:= 收集夹持气缸自动, 
	xReset:=复位  , 
	xPosExtend:=收集平台夹持气缸原点 , 
	xPosRetract:= 收集平台夹持气缸动点, 
	tTimeout:= T#5S, 
	yValve1=> 收集夹持气缸  , 
	bAlarm=> cyinderAlarm.9);	
//收集平台升降气缸
cylinder_11(
    xManualRetract := , 
    xAutoRetract := , 
    yValve2 => , 
    cylinder_type := 0, 

	xManualAuto:=ManualAuto  , 
	xManualExtend:= 收集升降气缸手动, 
	xAutoExtend:= 收集升降气缸自动, 
	xReset:=复位  , 
	xPosExtend:=收集平台升降气缸原点 , 
	xPosRetract:= 收集平台升降气缸动点, 
	tTimeout:= T#5S, 
	yValve1=> 收集升降气缸   , 
	bAlarm=> cyinderAlarm.10);	
//收集平台伸缩气缸
cylinder_12(
    xManualRetract := , 
    xAutoRetract := , 
    yValve2 => , 
    cylinder_type :=0 , 

	xManualAuto:=ManualAuto  , 
	xManualExtend:= 收集伸缩气缸手动, 
	xAutoExtend:= 收集伸缩气缸自动, 
	xReset:=复位, 
	xPosExtend:=收集平台推出气缸原点, 
	xPosRetract:= 收集平台推出气缸动点, 
	tTimeout:= T#5S, 
	yValve1=> 收集伸缩气缸, 
	bAlarm=> cyinderAlarm.11);		
//刮板拍照遮光气缸
cylinder_13(
    xManualRetract := , 
    xAutoRetract := , 
    yValve2 => , 
    cylinder_type :=0 , 

	xManualAuto:=ManualAuto  , 
	xManualExtend:= 刮板拍照遮光气缸手动, 
	xAutoExtend:=刮板拍照遮光气缸自动 , 
	xReset:=复位  , 
	xPosExtend:=刮板拍照遮光气缸上位 , 
	xPosRetract:= 刮板拍照遮光气缸下位, 
	tTimeout:= T#5S, 
	yValve1=>  刮板拍照遮光气缸, 
	bAlarm=> cyinderAlarm.12);		
//刮板拍照旋转气缸
cylinder_14(
    xManualRetract := , 
    xAutoRetract := , 
    yValve2 => , 
    cylinder_type := 0, 

	xManualAuto:=ManualAuto  , 
	xManualExtend:= 刮板拍照旋转气缸手动 AND 刮板轴9XDATE.fActPos>330, 
	xAutoExtend:=刮板拍照旋转气缸自动 , 
	xReset:=复位  , 
	xPosExtend:=刮板拍照旋转气缸原点  , 
	xPosRetract:= 刮板拍照旋转气缸动点, 
	tTimeout:= T#5S, 
	yValve1=>  刮板拍照旋转气缸   , 
	bAlarm=> cyinderAlarm.13);		
//刮板拍照下压气缸
cylinder_15(
    xManualRetract := , 
    xAutoRetract := , 
    yValve2 => , 
    cylinder_type := 0, 

	xManualAuto:=ManualAuto  , 
	xManualExtend:= 刮板拍照下压气缸手动, 
	xAutoExtend:=刮板拍照下压气缸自动 , 
	xReset:=复位  , 
	xPosExtend:=刮板拍照下压气缸上位, 
	xPosRetract:=刮板拍照下压气缸手动 OR 刮板拍照下压气缸自动 , 
	tTimeout:= T#5S, 
	yValve1=>  刮板拍照下压气缸, 
	bAlarm=> cyinderAlarm.14);
//展缸1进液电池阀1
cylinder_17(
    xManualRetract := , 
    xAutoRetract := , 
    yValve2 => , 
    cylinder_type :=0 , 

	xManualAuto:=ManualAuto  , 
	xManualExtend:= 展缸1进液电池阀1手动, 
	xAutoExtend:= 展缸1进液电池阀1自动, 
	xReset:=复位  , 
	xPosExtend:=   , 
	xPosRetract:= , 
	tTimeout:= , 
	yValve1=> 展缸1进液电池阀1, 
	bAlarm=> );	
//展缸1进液电池阀2
cylinder_18(
    xManualRetract := , 
    xAutoRetract := , 
    yValve2 => , 
    cylinder_type := 0, 

	xManualAuto:=ManualAuto  , 
	xManualExtend:= 展缸1进液电池阀2手动, 
	xAutoExtend:= 展缸1进液电池阀2自动, 
	xReset:=复位  , 
	xPosExtend:=   , 
	xPosRetract:= , 
	tTimeout:= , 
	yValve1=> 展缸1进液电池阀2, 
	bAlarm=> );	
//展缸1进液电池阀3
cylinder_19(
    xManualRetract := , 
    xAutoRetract := , 
    yValve2 => , 
    cylinder_type := 0, 

	xManualAuto:=ManualAuto  , 
	xManualExtend:= 展缸1进液电池阀3手动, 
	xAutoExtend:= 展缸1进液电池阀3自动, 
	xReset:=复位  , 
	xPosExtend:=   , 
	xPosRetract:= , 
	tTimeout:= , 
	yValve1=> 展缸1进液电池阀3, 
	bAlarm=> );	
//展缸1进液电池阀4
cylinder_20(
    xManualRetract := , 
    xAutoRetract := , 
    yValve2 => , 
    cylinder_type := 0, 

	xManualAuto:=ManualAuto  , 
	xManualExtend:= 展缸1进液电池阀4手动, 
	xAutoExtend:= 展缸1进液电池阀4自动, 
	xReset:=复位  , 
	xPosExtend:=   , 
	xPosRetract:= , 
	tTimeout:= , 
	yValve1=> 展缸1进液电池阀4, 
	bAlarm=> );	
//展缸1排液电池阀1
cylinder_21(
    xManualRetract := , 
    xAutoRetract := , 
    yValve2 => , 
    cylinder_type := 0, 

	xManualAuto:=ManualAuto  , 
	xManualExtend:= 展缸1排液电池阀1手动, 
	xAutoExtend:= 展缸1排液电池阀1自动, 
	xReset:=复位  , 
	xPosExtend:=   , 
	xPosRetract:= , 
	tTimeout:= , 
	yValve1=> 展缸1排液电池阀1, 
	bAlarm=> );	
//展缸1排液电池阀2
cylinder_22(
    xManualRetract := , 
    xAutoRetract := , 
    yValve2 => , 
    cylinder_type :=0 , 

	xManualAuto:=ManualAuto  , 
	xManualExtend:= 展缸1排液电池阀2手动, 
	xAutoExtend:= 展缸1排液电池阀2自动, 
	xReset:=复位  , 
	xPosExtend:=   , 
	xPosRetract:= , 
	tTimeout:= , 
	yValve1=> 展缸1排液电池阀2, 
	bAlarm=> );	
//展缸1排液电池阀3
cylinder_23(
    xManualRetract := , 
    xAutoRetract := , 
    yValve2 => , 
    cylinder_type :=0 , 

	xManualAuto:=ManualAuto, 
	xManualExtend:= 展缸1排液电池阀3手动, 
	xAutoExtend:= 展缸1排液电池阀3自动, 
	xReset:=复位  , 
	xPosExtend:=   , 
	xPosRetract:= , 
	tTimeout:= , 
	yValve1=> 展缸1排液电池阀3, 
	bAlarm=> );	
//展缸1排液电池阀4
cylinder_24(
    xManualRetract := , 
    xAutoRetract := , 
    yValve2 => , 
    cylinder_type := 0, 

	xManualAuto:=ManualAuto, 
	xManualExtend:= 展缸1排液电池阀4手动, 
	xAutoExtend:= 展缸1排液电池阀4自动, 
	xReset:=复位  , 
	xPosExtend:=   , 
	xPosRetract:= , 
	tTimeout:= , 
	yValve1=> 展缸1排液电池阀4, 
	bAlarm=> );	
//展缸1吹气电池阀1
cylinder_25(
    xManualRetract := , 
    xAutoRetract := , 
    yValve2 => , 
    cylinder_type := 0, 

	xManualAuto:=ManualAuto, 
	xManualExtend:= 展缸1吹气电池阀1手动, 
	xAutoExtend:= 展缸1吹气电池阀1自动, 
	xReset:=复位  , 
	xPosExtend:=   , 
	xPosRetract:= , 
	tTimeout:= , 
	yValve1=> 展缸1吹气电池阀1, 
	bAlarm=> );	
//展缸1吹气电池阀2
cylinder_26(
    xManualRetract := , 
    xAutoRetract := , 
    yValve2 => , 
    cylinder_type := 0, 

	xManualAuto:=ManualAuto, 
	xManualExtend:= 展缸1吹气电池阀2手动, 
	xAutoExtend:= 展缸1吹气电池阀2自动, 
	xReset:=复位  , 
	xPosExtend:=   , 
	xPosRetract:= , 
	tTimeout:= , 
	yValve1=> 展缸1吹气电池阀2, 
	bAlarm=> );	
//展缸1吹气电池阀3
cylinder_27(
    xManualRetract := , 
    xAutoRetract := , 
    yValve2 => , 
    cylinder_type := 0, 

	xManualAuto:=ManualAuto  , 
	xManualExtend:= 展缸1吹气电池阀3手动, 
	xAutoExtend:= 展缸1吹气电池阀3自动, 
	xReset:=复位  , 
	xPosExtend:=   , 
	xPosRetract:= , 
	tTimeout:= , 
	yValve1=> 展缸1吹气电池阀3, 
	bAlarm=> );	
//展缸1吹气电池阀4
cylinder_28(
    xManualRetract := , 
    xAutoRetract := , 
    yValve2 => , 
    cylinder_type := 0, 

	xManualAuto:=ManualAuto, 
	xManualExtend:= 展缸1吹气电池阀4手动, 
	xAutoExtend:= 展缸1吹气电池阀4自动, 
	xReset:=复位  , 
	xPosExtend:=   , 
	xPosRetract:= , 
	tTimeout:= , 
	yValve1=> 展缸1吹气电池阀4, 
	bAlarm=> );	
//展缸2进液电池阀1
cylinder_29(
    xManualRetract := , 
    xAutoRetract := , 
    yValve2 => , 
    cylinder_type := 0, 

	xManualAuto:=ManualAuto, 
	xManualExtend:= 展缸2进液电池阀1手动, 
	xAutoExtend:= 展缸2进液电池阀1自动, 
	xReset:=复位  , 
	xPosExtend:=   , 
	xPosRetract:= , 
	tTimeout:= , 
	yValve1=> 展缸2进液电池阀1, 
	bAlarm=> );	
//展缸2进液电池阀2
cylinder_30(
    xManualRetract := , 
    xAutoRetract := , 
    yValve2 => , 
    cylinder_type := 0, 

	xManualAuto:=ManualAuto, 
	xManualExtend:= 展缸2进液电池阀2手动, 
	xAutoExtend:= 展缸2进液电池阀2自动, 
	xReset:=复位  , 
	xPosExtend:=   , 
	xPosRetract:= , 
	tTimeout:= , 
	yValve1=> 展缸2进液电池阀2, 
	bAlarm=> );	
//展缸2进液电池阀3
cylinder_31(
    xManualRetract := , 
    xAutoRetract := , 
    yValve2 => , 
    cylinder_type := 0, 

	xManualAuto:=ManualAuto, 
	xManualExtend:= 展缸2进液电池阀3手动, 
	xAutoExtend:= 展缸2进液电池阀3自动, 
	xReset:=复位  , 
	xPosExtend:=   , 
	xPosRetract:= , 
	tTimeout:= , 
	yValve1=> 展缸2进液电池阀3, 
	bAlarm=> );	
//展缸2进液电池阀4
cylinder_32(
    xManualRetract := , 
    xAutoRetract := , 
    yValve2 => , 
    cylinder_type := 0, 

	xManualAuto:=ManualAuto, 
	xManualExtend:= 展缸2进液电池阀4手动, 
	xAutoExtend:= 展缸2进液电池阀4自动, 
	xReset:=复位  , 
	xPosExtend:=   , 
	xPosRetract:= , 
	tTimeout:= , 
	yValve1=> 展缸2进液电池阀4, 
	bAlarm=> );	
//展缸2排液电池阀1
cylinder_33(
    xManualRetract := , 
    xAutoRetract := , 
    yValve2 => , 
    cylinder_type := 0, 

	xManualAuto:=ManualAuto, 
	xManualExtend:= 展缸2排液电池阀1手动, 
	xAutoExtend:= 展缸2排液电池阀1自动, 
	xReset:=复位  , 
	xPosExtend:=   , 
	xPosRetract:= , 
	tTimeout:= , 
	yValve1=> 展缸2排液电池阀1, 
	bAlarm=> );	
//展缸2排液电池阀2
cylinder_34(
    xManualRetract := , 
    xAutoRetract := , 
    yValve2 => , 
    cylinder_type := 0, 

	xManualAuto:=ManualAuto, 
	xManualExtend:= 展缸2排液电池阀2手动, 
	xAutoExtend:= 展缸2排液电池阀2自动, 
	xReset:=复位  , 
	xPosExtend:=   , 
	xPosRetract:= , 
	tTimeout:= , 
	yValve1=> 展缸2排液电池阀2, 
	bAlarm=> );	
//展缸2排液电池阀3
cylinder_35(
    xManualRetract := , 
    xAutoRetract := , 
    yValve2 => , 
    cylinder_type := 0, 

